(* IEC 61131-3 sources: ml2plc/benchmarks/st (part 7) *)

    weights_7 : ARRAY[0..191] OF REAL := [0.688684464, -0.251728266, -0.865464985, -0.106039852, -0.342710823, 0.691397548, 0.545316637, 0.451106936, -0.972581029, 1.01049495, -0.46521771, -0.194902733, 0.047600802, 0.219640687, -0.898541093, -1.06958103, 0.576955795, 0.662654877, -0.551774442, -0.393089443, 1.25733566, -0.102036051, -0.33817184, 0.573561192, 1.02358389, 0.0429671332, -0.451354206, 1.01461709, -0.512437761, -0.405483395, -0.904772937, 0.0525284261, 0.531825364, 1.37226915, -0.355399728, -0.68238759, 0.599305511, 0.39647612, -1.08820724, 1.2778101, -0.0734612197, -0.358505845, 0.813616991, 0.21143426, -0.601562083, -0.720784783, 0.119864009, 0.748160541, -0.00713000586, 0.244366869, -0.894774139, -0.781875014, -0.0933139026, 0.823451638, -1.0571214, 0.397565454, 0.221330047, 0.794143915, 0.0579137206, -0.834286153, -1.02714491, 0.4435018, 0.325868577, 0.0499007814, 0.244628534, -0.956271648, -0.811831295, 0.113917887, 0.623460889, -0.901144326, 0.656858027, 0.285817534, 0.424304128, -0.158880517, -1.02905571, 1.03020906, -0.499804497, -0.475916564, -0.337449938, -0.158021986, 1.40593672, 0.95926398, -0.595809937, -0.287213802, -0.47090137, -0.392327726, 1.09143257, -0.364193618, -0.291908026, 1.43915653, -1.03929389, 0.432665855, 0.234065458, 1.08598685, -0.368728101, -0.609597504, -0.233271882, -0.42965731, 0.926180065, 0.188584849, 0.223465264, -1.11406386, -0.50280422, -0.178945631, 1.10107863, -1.26540232, 0.234013259, 0.419472396, -0.618463218, -0.307608634, 1.32427752, 0.952789187, -0.563809812, -0.25738892, -1.16513908, 0.324054241, 0.353279918, -0.750201344, 0.0481031314, 0.692657232, 0.545174181, 0.144862831, -1.10333705, 0.573349059, 0.272133052, -1.33604789, -0.165077209, -0.424486279, 0.880616426, 0.664759457, 0.357302666, -1.25569296, -0.0329220407, 0.482446015, -0.317285031, 1.13552487, -0.381064355, -0.586573541, -0.733967721, 0.152410552, 0.860239148, 0.990790427, -0.491253883, -0.512532234, 1.046013, -0.51024735, -0.624616563, 0.882700682, -0.114194848, -0.756001472, 0.88511467, -0.404787958, -0.668740392, -0.692761958, -0.321748972, 1.15619385, -0.657764494, -0.166892812, 1.11973906, -1.07256877, 0.377563357, 0.286821365, 0.385569185, 0.258302331, -1.33617496, 1.14878833, -0.584546626, -0.583055913, -1.05693662, 0.504781961, 0.443913162, -0.114870973, -0.384501725, 0.897702992, 1.03910887, -0.165579304, -0.616232336, 0.463422328, 0.441405088, -0.974973619, 0.627231061, 0.212427795, -0.956863701, -0.648825645, -0.309565783, 1.04708552, 1.24038255, -0.20401369, -0.22858876, -0.200083375, -0.332850873, 0.897526622];
    bias_7 : ARRAY[0..2] OF REAL := [-0.0229109377, 0.115018375, -0.164126784];

END_VAR

VAR
    (* Merged variables from all regions *)
    buffer_0 : ARRAY[0..63] OF REAL;
    buffer_1 : ARRAY[0..63] OF REAL;
    h_new_0 : ARRAY[0..63] OF REAL;
    h_new_3 : ARRAY[0..63] OF REAL;
    h_state_0 : ARRAY[0..63] OF REAL;
    h_state_3 : ARRAY[0..63] OF REAL;
    r_gate_0 : ARRAY[0..63] OF REAL;
    r_gate_3 : ARRAY[0..63] OF REAL;
    u_gate_0 : ARRAY[0..63] OF REAL;
    u_gate_3 : ARRAY[0..63] OF REAL;

    (* Temporary computation variables *)
    i : DINT;
    j : DINT;
    t : DINT;
    sum : REAL;
    (* Computation helpers *)
    max_val : REAL;
    exp_val : REAL;
    exp_sum : REAL;
    (* Spatial loop variables *)
    oc : DINT;
    oh : DINT;
    ow : DINT;
    ic : DINT;
    kh : DINT;
    kw : DINT;
    ih : DINT;
    iw : DINT;
    (* Transpose loop variables *)
    t2_d0 : DINT;
    t2_d1 : DINT;
    t2_d2 : DINT;
END_VAR

(* Forward pass execution *)

(* Region: r0 [ACYCLIC] *)
(* Acyclic Region r0 *)
(* Layer 0: GRU (hidden_size=64, input_size=1, seq_len=1) *)
(* Generating output: Y, linear_before_reset=1 *)

(* Initialize states to zero *)
FOR j := 0 TO 63 DO
    h_state_0[j] := 0.0;
END_FOR;

(* Process 1 timesteps *)
FOR t := 0 TO 0 DO

    (* Reset Gate *)
    FOR j := 0 TO 63 DO
        sum := 0.0;
        FOR i := 0 TO 0 DO
            sum := sum + input_data * weights_0_r[j * 1 + i] ;
        END_FOR;
        FOR i := 0 TO 63 DO
            sum := sum + h_state_0[i] * recurrent_0_r[j * 64 + i] ;
        END_FOR;
    sum := sum + bias_0_r[j];
    r_gate_0[j] := 1.0 / (1.0 + EXP(-sum));
    END_FOR;

    (* Update Gate *)
    FOR j := 0 TO 63 DO
        sum := 0.0;
        FOR i := 0 TO 0 DO
            sum := sum + input_data * weights_0_u[j * 1 + i] ;
        END_FOR;
        FOR i := 0 TO 63 DO
            sum := sum + h_state_0[i] * recurrent_0_u[j * 64 + i] ;
        END_FOR;
    sum := sum + bias_0_u[j];
    u_gate_0[j] := 1.0 / (1.0 + EXP(-sum));
    END_FOR;

    (* Candidate (lbr=1): h'_t = tanh(Wx + r_t * (Rh + Rb_h) + Wb_h) *)
    FOR j := 0 TO 63 DO
        sum := 0.0;
        FOR i := 0 TO 0 DO
            sum := sum + input_data * weights_0_h[j * 1 + i] ;
        END_FOR;
        exp_val := 0.0;
        FOR i := 0 TO 63 DO
            exp_val := exp_val + h_state_0[i] * recurrent_0_h[j * 64 + i] ;
        END_FOR;
        sum := sum + r_gate_0[j] * (exp_val + bias_r_0_h[j]);
        sum := sum + bias_w_0_h[j];
    exp_val := EXP(2.0 * sum);
    h_new_0[j] := (exp_val - 1.0) / (exp_val + 1.0);
    END_FOR;

    (* Hidden state: h_t = u_t * h_{t-1} + (1 - u_t) * h'_t *)
    FOR j := 0 TO 63 DO
        h_state_0[j] := u_gate_0[j] * h_state_0[j] + (1.0 - u_gate_0[j]) * h_new_0[j];
    END_FOR;

    (* Y output: Full sequence *)
    FOR j := 0 TO 63 DO
        buffer_0[t * 64 + j] := h_state_0[j];
    END_FOR;
END_FOR;

(* Layer 1: Squeeze *)
FOR i := 0 TO 63 DO
    buffer_1[i] := buffer_0[i];
END_FOR;

(* Layer 2: Transpose perm=(1, 0, 2)  (1, 1, 64) -> (1, 1, 64) *)
FOR t2_d0 := 0 TO 0 DO
    FOR t2_d1 := 0 TO 0 DO
        FOR t2_d2 := 0 TO 63 DO
            buffer_0[t2_d0 * 64 + t2_d1 * 64 + t2_d2] := buffer_1[t2_d1 * 64 + t2_d0 * 64 + t2_d2];
        END_FOR;
    END_FOR;
END_FOR;

(* Layer 3: GRU (hidden_size=64, input_size=64, seq_len=1) *)
(* Generating output: Y, linear_before_reset=1 *)

(* Initialize states to zero *)
FOR j := 0 TO 63 DO
    h_state_3[j] := 0.0;
END_FOR;

(* Process 1 timesteps *)
FOR t := 0 TO 0 DO

    (* Reset Gate *)
    FOR j := 0 TO 63 DO
        sum := 0.0;
        FOR i := 0 TO 63 DO
            sum := sum + buffer_0[t * 64 + i] * weights_3_r[j * 64 + i] ;
        END_FOR;
        FOR i := 0 TO 63 DO
            sum := sum + h_state_3[i] * recurrent_3_r[j * 64 + i] ;
        END_FOR;
    sum := sum + bias_3_r[j];
    r_gate_3[j] := 1.0 / (1.0 + EXP(-sum));
    END_FOR;

    (* Update Gate *)
    FOR j := 0 TO 63 DO
        sum := 0.0;
        FOR i := 0 TO 63 DO
            sum := sum + buffer_0[t * 64 + i] * weights_3_u[j * 64 + i] ;
        END_FOR;
        FOR i := 0 TO 63 DO
            sum := sum + h_state_3[i] * recurrent_3_u[j * 64 + i] ;
        END_FOR;
    sum := sum + bias_3_u[j];
    u_gate_3[j] := 1.0 / (1.0 + EXP(-sum));
    END_FOR;

    (* Candidate (lbr=1): h'_t = tanh(Wx + r_t * (Rh + Rb_h) + Wb_h) *)
    FOR j := 0 TO 63 DO
        sum := 0.0;
        FOR i := 0 TO 63 DO
            sum := sum + buffer_0[t * 64 + i] * weights_3_h[j * 64 + i] ;
        END_FOR;
        exp_val := 0.0;
        FOR i := 0 TO 63 DO
            exp_val := exp_val + h_state_3[i] * recurrent_3_h[j * 64 + i] ;
        END_FOR;
        sum := sum + r_gate_3[j] * (exp_val + bias_r_3_h[j]);
        sum := sum + bias_w_3_h[j];
    exp_val := EXP(2.0 * sum);
    h_new_3[j] := (exp_val - 1.0) / (exp_val + 1.0);
    END_FOR;

    (* Hidden state: h_t = u_t * h_{t-1} + (1 - u_t) * h'_t *)
    FOR j := 0 TO 63 DO
        h_state_3[j] := u_gate_3[j] * h_state_3[j] + (1.0 - u_gate_3[j]) * h_new_3[j];
    END_FOR;

    (* Y output: Full sequence *)
    FOR j := 0 TO 63 DO
        buffer_1[t * 64 + j] := h_state_3[j];
    END_FOR;
END_FOR;

(* Layer 4: Squeeze *)
FOR i := 0 TO 63 DO
    buffer_0[i] := buffer_1[i];
END_FOR;

(* Layer 5: Slice starts=[0] ends=[1] axes=[0] steps=[1] *)
FOR i := 0 TO 63 DO
    buffer_1[i] := buffer_0[i];
END_FOR;

(* Layer 6: Squeeze *)
FOR i := 0 TO 63 DO
    buffer_0[i] := buffer_1[i];
END_FOR;

(* Layer 7: Fused Linear + SOFTMAX *)
FOR j := 0 TO 2 DO
    sum := 0.0;
    FOR i := 0 TO 63 DO
        sum := sum + buffer_0[i] * weights_7[i * 3 + j];
    END_FOR;
output_data[j] := sum + bias_7[j];
END_FOR;

(* Softmax: find max *)
max_val := output_data[0];
FOR i := 1 TO 2 DO
    IF output_data[i] > max_val THEN
        max_val := output_data[i];
    END_IF;
END_FOR;

(* Softmax: compute exponentials and sum *)
exp_sum := 0.0;
FOR i := 0 TO 2 DO
    output_data[i] := EXP(output_data[i] - max_val);
    exp_sum := exp_sum + output_data[i];
END_FOR;

(* Softmax: normalize *)
FOR i := 0 TO 2 DO
    output_data[i] := output_data[i] / exp_sum;
END_FOR;

END_FUNCTION_BLOCK

(* ---- GRU3_straton.st ---- *)
FUNCTION_BLOCK GRU3_FB

    (* Model Inputs/Outputs *)
VAR_INPUT
    input_data : REAL;
END_VAR

VAR_OUTPUT
    output_data : ARRAY[0..2] OF REAL;
END_VAR

VAR
    CONSTANT weights_0_u : ARRAY[0..63] OF REAL := [-0.439286172, -0.480953246, -0.870120704, -0.69075644, -0.657077134, -0.589701712, -0.481989682, 0.11155279, -0.595970333, -0.522424638, 0.066479668, -0.477147967, -0.548775792, -0.440251201, -0.581660211, -0.851885259, -0.447049588, -0.158783153, -0.671791077, -0.790636778, -0.670549393, -0.228230864, -0.573410928, -0.463102937, 0.294410557, -0.154226393, -0.428246915, -0.419357181, -0.580893517, -0.450942427, -0.434489578, -0.354421765, -0.500179946, -0.272357315, -0.211979702, -0.347913235, -0.509638548, -0.571337163, -0.666850746, -0.102425002, -0.464207053, -0.692536592, -0.576414764, -0.25179112, -0.587422669, 0.197722241, -0.440594107, -0.0186067764, -0.233214989, -0.485925347, -0.624329388, -0.464201093, -0.771930814, -0.648595512, -0.712386131, -0.865132749, 0.0861109644, -0.699016631, -0.64285028, -0.76548481, -0.601012945, -0.522387683, -0.408631802, -0.428571761];
    CONSTANT recurrent_0_u : ARRAY[0..4095] OF REAL := [-0.0650523901, -0.129474998, 0.0260338224, 0.0695474148, -0.0666072816, 0.0774139315, -0.0643586814, 0.0473090038, 0.0519357473, 0.0531803295, 0.0508824363, 0.156312734, 0.0510548055, -0.0783398449, 0.0161208138, -0.0254090969, -0.0333776586, 0.0407715552, 0.0384992361, -0.00284529058, 0.0996260718, -0.0809974, -0.0287103504, 0.0288348049, 0.121645145, 0.129295856, -0.121905953, -0.0567066036, -0.0332944021, 0.10126324, -0.0619100034, -0.0120835379, -0.0321507938, 0.152141571, 0.0557904243, 0.0295200478, 0.0753500834, 0.0523380376, -0.045079913, 0.0743025169, 0.03919724, -0.0464075021, 0.0460194834, 0.0400504917, -0.0186564252, -0.0811230615, 0.0205100551, -0.0494997241, -0.0123350881, -0.0521072671, 0.0318819955, 0.0125074722, 0.086325638, -0.14838697, 0.0729614198, -0.123611242, 0.0608778223, 0.136695266, -0.0275732893, 0.103986211, 0.0964937732, 0.0746636614, 0.0518375002, 0.0131850429, 0.0481536575, 0.080832839, 0.00456657633, -0.0930995643, -0.0926894546, -0.104142435, -0.0113655347, 0.0689256042, 0.0391013213, -0.145912498, 0.0662881434, -0.125198483, -0.0359372757, 0.0683884099, 0.0814840198, -0.0467883013, -0.0385110751, 0.0412478335, -0.026082132, 0.00598589424, -0.0733542442, -0.0616489351, 0.0599563681, 0.0975151584, -0.102699503, 0.0168768093, 0.0567795113, -0.109472096, 0.0479807556, -0.0641779676, 0.0252187103, 0.0170151237, 0.052396398, -0.00687042344, -0.0297337286, 0.052699931, 0.0299865901, 0.0428941771, 0.143816575, 0.0724755228, 0.0308377538, 0.0377355814, 0.073744677, 0.100715749, 0.0200833306, 0.00330035621, 0.0808146596, 0.0683915466, 0.00292335614, -0.0387148745, -0.0278775394, 0.0165898427, -0.0266524255, -0.0119600557, 0.0607938841, -0.171499431, 0.00670967251, -0.0278419442, -0.0198536664, -0.0489947647, -0.0504177436, -0.0603820346, -0.0319245569, 0.0403733216, -0.0657449737, -0.0835127532, 0.074783206, -0.0822283328, 0.0527420714, 0.025356207, 0.00193200377, 0.0403062142, 0.011863322, 0.0911065713, -0.0981498286, 0.0448010042, 0.00674223201, 0.0832657516, 0.0133088445, -0.0096457703, -0.126930133, 0.0133038349, -0.0605163276, 0.0315002874, 0.163095102, 0.0627945811, -0.0319333449, -0.0184467398, -0.0260825343, 0.1507947, 0.0180257969, -0.113473095, -0.00113128126, 0.034390863, 0.158128366, 0.0736147836, 0.00302845053, -0.0366435051, 0.0202366989, -0.0454519801, 0.027544789, 0.00827108417, -0.116445266, 0.136078835, -0.0322153643, 0.0859275237, -0.0495595485, -0.0305913445, -0.0528560281, -0.0197725855, 0.0479791425, -0.0321966782, -0.0912050977, 0.08009094, -0.131073937, -0.073050648, 0.0158983283, -0.0129424734, 0.0236992333, -0.0654924586, 0.00780409761, 0.0303560495, 0.0224402416, 0.195856482, 0.104409501, 0.00386209786, 0.0270838067, -0.0308708213, 0.0765376315, -0.144475698, -0.00663482724, -0.0773844719, -0.0756781921, 0.0114769517, 0.07947056, 0.0525699407, -0.0490815043, -0.0797774196, -0.0738181025, 0.00899818353, 0.00655652676, -0.0247584134, -0.142790094, -0.0536906458, 0.0891067088, 0.0319167599, 0.0273121186, -0.0111009832, 0.0738681182, -0.0465159416, 0.10495235, 0.0167910457, 0.0170945786, -0.0259337351, -0.0238404684, 0.105175085, 0.0262874551, -0.0252160784, 0.0407399312, 0.0396488942, -0.000441844575, 0.0779087767, -0.101633228, 0.00611562654, -0.138864547, 0.0793924779, 0.0318161361, 0.00487799011, -0.0742631257, 0.0282261875, -0.0452414677, 0.103862561, -0.233050048, 0.0166822113, -0.0502803773, -0.105138443, 0.00815397315, 0.075144209, -0.000656956807, 0.00553116389, -0.0327767022, 0.0563323051, 0.00168130081, -0.0347454548, 0.0447669849, 0.0809304044, 0.0181033891, 0.0829547346, 0.0445744358, 0.0685421899, -0.0522269495, 0.10767854, 0.0401147828, -0.0274171568, -0.0556086302, -0.0181052946, 0.0614649057, 0.15146631, -0.107644446, -0.0519810207, -0.0192557313, -0.050705526, -0.00130558573, -0.00449152011, 0.0586461015, -0.00949175656, -0.161170155, 0.0415757112, 0.0234208908, 0.0994374529, -0.107094176, 0.0798551813, 0.00859866291, 0.00905988738, 0.17884995, -0.052185487, -0.00788529217, -0.0128635718, 0.0425841771, -0.0781655982, 0.0738354772, -0.0700388551, -0.0454497337, -0.0581207834, 0.0587512478, -0.129331231, 0.089504689, 0.0157049354, 0.0867228657, 0.0273658019, -0.0242159963, -0.0269595832, -0.0785825849, -0.0127460342, 0.0726092383, -0.0813473612, 0.0418060534, -0.098036088, -0.0871397629, 0.12796244, 0.115513436, -0.0840419456, -0.0282502882, 0.0339900963, -0.0615085512, -0.0237938426, 0.14066948, 0.0103495289, 0.0563306212, 0.0128910914, 0.0566199236, -0.0431611128, 0.0414758436, -0.0598706417, -0.00455367938, 0.010008106, 0.0502123758, -0.0128066251, 0.119871259, 0.169338882, 0.0573619083, -0.00254678726, 0.0632556081, 0.0658841059, -0.0489678681, -0.0136197284, 0.0332296528, 0.0304199178, -0.0101228859, 0.0340865031, -0.1463456, -0.0561735369, -0.078145586, -0.105770409, 0.021583017, 0.0442470424, -0.0132950321, 0.0343763754, -0.131868333, -0.0834302157, 0.0234229043, 0.0955413878, -0.00966519676, 0.133738831, 0.0799299628, -0.0209413245, -0.0201649163, -0.078094773, 0.00760632753, 0.10674265, -0.0504244342, 0.130076349, -0.0765756071, 0.0406672917, -0.0677179396, 0.0489641167, 0.0178483911, 0.0639283434, -0.0072317142, 0.0689901859, 0.0284034405, 0.0447224788, 0.080589503, -0.0753613785, -0.0883018747, -0.209824249, -0.025372155, -0.0194213465, -0.121756315, -0.0405391641, 0.0252318978, -0.113081403, 0.00984102953, -0.0379814059, -0.0696330816, -0.0607138053, 0.00136227917, -0.0684736297, 0.084016636, 0.0580409989, 0.0783514529, 0.038732525, -0.110764012, -0.184509531, -0.0218135417, 0.0410628468, 0.0143347979, 0.0210808329, 0.0938048959, 0.0952843726, 0.0369632132, -0.036689274, 0.0596370548, -0.101092562, 0.021979671, -0.00666903984, -0.0002728533, -0.102687143, 0.101846725, -0.0270557068, -0.0740891248, 0.0451480709, 0.0244468898, 0.0135530774, -0.0656716228, 0.126964301, 0.046734333, -0.0135823097, 0.104897536, 0.0116401128, -0.0351510793, -0.0270920806, -0.0317737125, -0.0427896604, 0.0606436953, -0.055717431, 0.0877809376, 0.0525183901, 0.0816646814, -0.123816505, 0.0268022101, 0.0949827731, 0.0286988262, -1.17924064e-05, -0.107156947, -0.0325826406, -0.176235095, 0.0207939055, 0.140304744, 0.0597819574, -0.0181577466, 0.117161281, 0.0191873126, 0.0420570076, 0.0174266361, 0.0642305687, -0.0820301622, 0.0203213636, -0.0772711709, 0.0149432123, 0.078445442, -0.031391941, 0.0178297423, 0.0258787423, 0.105060086, -0.185030684, -0.0465904325, 0.033022128, -0.0522077605, 0.18817015, 0.17154251, 0.0908443928, -0.114609689, -0.0463253893, 0.179783046, -0.0138813183, -0.0250236578, -0.0397495851, -0.0401404127, 0.0414455384, 0.00421553105, 0.00501056761, -0.0355476104, -0.0948569328, -0.0180768073, -0.0929266214, -6.38996717e-05, 0.0402616151, -0.04017644, 0.0292976033, 0.122893214, -0.0101269074, 0.0949848741, 0.0924490988, -0.0142561533, 0.034249723, -0.0345417485, -0.0720876306, -0.116285995, 0.0757803917, 0.0925265029, 0.0501283891, 0.0556523763, -0.0871114284, 0.063929759, 0.111392535, -0.0113485595, -0.0560661219, 0.0588565171, 0.0202990752, 0.0169391409, 0.0079346532, -0.0346361771, -0.0971538872, -0.107799433, -0.0225640163, -0.104902133, 0.0540932752, -0.0481065586, 0.0236067846, -0.135952473, 0.105642021, 0.0632608011, -0.0237644296, 0.0115678804, 0.0341430977, 0.00839798432, 0.00526432134, 0.00430205092, 0.063617371, -0.0232296586, -0.0100963581, 0.0232974347, -0.00805089623, -0.0783473253, 0.0837393031, 0.0119392872, -0.171118468, 0.0533629246, 0.0270157438, -0.0287604984, -0.024254458, -0.0379126333, 0.0377461091, -0.129247546, -0.0196368489, 0.121421359, 0.141241029, -0.0185492001, -0.0607114322, -0.118905656, 0.0243493672, 0.00225942954, -0.02267823, -0.114327833, -0.00651719887, 0.0233639106, -0.0216970742, 0.181706235, 0.0208011288, 0.019147085, -0.046965789, -0.0224242695, 0.170098603, -0.0381373689, -0.0911064297, 0.0361324437, 0.0604973882, 0.0523151048, 0.00412818976, 0.0810551196, -0.0951434225, 0.0870590508, -0.0168896336, -0.128554851, -0.0098116193, -0.0513504371, 0.0390418544, -0.0403953195, -0.101676092, 0.0051176697, -0.00728737004, 0.0545737594, 0.0803038031, -0.106364466, 0.0805499181, -0.0291947313, -0.0313916355, 0.00281906407, -0.00804035645, 0.0905895531, 0.138566479, -0.0726417452, -0.0388255194, 0.0526182652, 0.0332292169, -0.0458627641, 0.0337294526, 0.00538110361, 0.140382588, 0.0673478395, -0.0970090628, -0.0075024087, -0.0495187268, -0.0802161619, 0.123421639, -0.0669697523, 0.0695282966, 0.0278533436, 0.0633659065, 0.00612806296, -0.0442293584, -0.0825438574, 0.102498822, -0.0788070858, -0.00543309376, 0.00251733419, -0.112787522, 0.0541282296, -0.167338938, 0.0514628179, -0.0181294475, 0.00405258778, -0.144672319, 0.0080318721, -0.0168379508, 0.0630492195, -0.0291489959, 0.0451016501, -0.0668138266, 0.0430565365, 0.0430122651, -0.0329513662, 0.000115959905, -0.155294836, 0.0717644468, -0.0975336134, 0.0627146736, 0.0671754926, -0.0245223772, -0.0847209394, 0.103243671, -0.0160844456, -0.0769205019, 0.0603941306, -0.0861880928, -0.124118626, -0.0407451317, -0.0479636192, 0.0243864693, 0.0225671809, 0.0300183278, 0.0491476469, 0.0137792621, -0.101849571, 0.0899749994, -0.147746086, 0.00454038568, 0.0589881316, -0.0145919751, 0.135418221, -0.0641773641, 0.00270533562, -0.0761346892, -0.0119857313, -0.0468325913, -0.0362873077, -0.131199926, 0.0103873778, 0.119403817, 0.0133330058, 0.0119966101, 0.0999416485, -0.0672517344, -0.0058638826, -0.00583216175, 0.0140269175, -0.068311438, 0.03253185, 0.103045583, -0.0298009366, -0.0424585715, 0.049341809, 0.0334219672, 0.0674507618, -0.0598343313, -0.0709823295, -0.00613911822, -0.0969725773, -0.114717588, 0.0991245732, 0.0570561923, -0.019426886, 0.052425161, -0.0514192283, 0.0795131326, -0.0747317523, -0.0695499405, 0.0674568191, 0.0873003826, 0.183561474, 0.0483771265, 0.00801333692, -0.0329486541, 0.118730754, -0.024188403, -0.00475108158, -0.102296896, 0.0118699996, -0.0566260032, -0.00249518454, 0.0371045657, -0.0271308124, 0.0527189821, 0.0894352719, 0.186274648, 0.0990155637, -0.0390276238, -0.102149099, 0.0725147501, 0.0395716839, -0.0627084598, 0.0174233504, -0.118221872, 0.057125818, 0.00148172863, -0.0975891799, 0.0914200917, -0.0564012453, -0.00408087857, -0.115551151, 0.0542268753, 0.019407969, -0.04010031, -0.0751183033, 0.0519157983, 0.0462308973, -0.00663706008, -0.0179555975, 0.128559679, -0.0160329398, -0.0250887014, 0.0124615263, -0.0278950725, 0.0723621994, -0.0639792681, 0.0245549679, -0.0128075834, 0.0482278317, -0.00473110611, -0.0172997359, 0.0275737233, 0.0381074212, -0.0479229614, 0.15075548, 0.236614883, -0.12308903, 0.0457972996, -0.0270488337, -0.0401842594, 0.0367866941, -0.0665339977, -0.124880955, 0.0096321106, -0.0183932558, -0.0149384877, -0.0207794402, -0.0273507237, 0.0092713302, -0.137307942, 0.124376148, -0.000531716272, -0.0697186887, 0.0233710855, -0.0879249945, -0.0595673844, -0.0753096193, -0.10940744, -0.0863983482, 0.0678732842, -0.0699944496, -0.0533968322, -0.0598150305, -0.109890275, -0.0255937222, 0.0414171703, -0.028406553, 0.0625951141, 0.0562955327, -0.040136572, 0.102456421, -0.094027251, 0.0563254878, 0.0507630631, -0.100891739, 0.0114759067, -0.0276399851, -0.0600263849, -0.0218528342, 0.0106363287, 0.0762119591, 0.0472210646, 0.0182249043, 0.0761318132, -0.0902465209, -0.0155644314, 0.0497058667, 0.00891689677, -0.0575596653, -0.063269861, -0.0369747803, -0.0418471023, -0.0446194261, 0.0618177094, 0.163427904, 0.0439322591, 0.0151975229, -0.139614716, 0.0382574834, 0.0647403747, 0.0044741584, 0.0366933271, -0.0847294405, -0.098235622, -0.102225974, 0.0730303079, 0.0709254742, 0.114724368, -0.058182843, -0.0275532752, 0.0699310824, 0.073567912, -0.118505709, -0.0922444239, 0.0654501319, -0.0442147106, -0.0973261297, 0.0649150908, 0.0473677218, -0.0438311286, -0.0123466263, -0.0506518409, -0.00112013146, 0.0114555079, -0.225004256, 0.0179542284, 0.00154356682, 0.0197916869, -0.0964033976, -0.0149603887, -0.0931083262, -0.0858175233, -0.0240392219, -0.0473877937, 0.0356729813, 0.0953858122, 0.0516837016, 0.000944763422, 0.000391166657, -0.0161546711, 0.0617823638, 0.0323178768, 0.0746243447, -0.0289416965, -0.132081941, 0.0347845852, -0.00957541913, -0.146093175, 0.00121896248, -0.088182658, -0.0529079251, 0.00144353509, -0.10963767, 0.0711052567, -0.130099729, -0.127687454, -0.0238898639, 0.0237303749, -0.0463271476, -0.0377245843, 0.146435305, 0.0406003967, -0.00347847119, 0.0402232558, 0.0606766082, -0.0170659591, 0.00456166919, -0.0581656583, -0.0257244669, -0.114303187, -0.109322034, -0.000124797225, 0.0906794146, 0.0998297706, -0.0660899505, -0.0273227766, 0.00623180624, -0.0511037856, 0.0518054552, -0.130383685, -0.104795009, 0.00977518409, 0.0961738452, 0.0406313278, 0.0335147977, -0.0768964514, -0.021825349, 0.114472322, -0.0201997422, -0.0598041527, -0.0629845262, 0.105795145, -0.0276378486, -0.0260668173, -0.0237419959, -0.0401881412, 0.0480453372, 0.0071930117, 0.00337004848, 0.0128219994, 0.067926839, 0.102826566, -0.0290449653, 0.123585209, 0.0586936176, -0.129759327, -0.0223709345, -0.116297573, -0.0687413886, 0.109364361, -0.016150102, 0.0699984133, 0.0204590037, -0.0488001369, -0.0933896229, 0.11484497, 0.146208376, -0.0152992923, 0.0223931447, 0.0693335161, -0.126214027, -0.0157451089, 0.020451, -0.0159052685, 0.0770635083, -0.165799066, -0.0527213998, -0.080435276, -0.0827942193, 0.0621753186, 0.00343356607, -0.0961636975, 0.0286911149, 0.0452868044, -0.0499980301, -0.0868136883, 0.050965365, -0.0764427632, -0.0663457513, 0.0639655739, -0.121900126, -0.0106822588, 0.0629351214, -0.0268343873, -0.0563602373, 0.0208010022, -0.0950316712, 0.0376925468, 0.0941148102, 0.0284186527, 0.0386470295, -0.0649496838, 0.00324150547, -0.0536398701, 0.0218845457, 0.101267442, 0.00504809991, -0.0866092741, 0.0529379621, 0.0938520655, 0.0396423154, 0.127945945, 0.11368385, -0.0549047142, 0.114498168, -0.0241714753, 0.0520189852, -0.0362896509, 0.0509226546, -0.165635839, 0.0881007984, 0.0160411, 0.024631137, 0.0659909099, -0.0762100443, 0.0427479185, -0.00694125425, 0.143184051, -0.149732918, 0.0110863149, -0.0155461309, -0.13748844, -0.0504982434, 0.025665462, -0.0429363698, -0.0277443547, -0.0475423895, 0.0285833944, -0.0735700205, -0.144904912, -0.0755529851, -0.0403888598, -0.0527475253, -0.000688489527, 0.101409346, 0.0988431573, -0.0909979939, 0.0660976842, 0.063818492, -0.00707271695, -0.00301229395, -0.0202014614, 0.0212209262, -0.0612271912, 0.142480314, -0.102822497, 0.121017784, -0.0435582623, 0.100066409, -0.0312062576, -0.0822519436, 0.057339862, 0.0568015501, 0.0269984789, -0.0163367614, -0.0477057099, -0.101986229, -0.00421534479, -0.179487348, -0.0764475316, -0.0430073664, -0.0425812863, 0.0527436584, -0.13650541, -0.00514466688, 0.00624288665, -0.0491546728, -0.0670409873, 0.0240444243, 0.035694059, -0.0549894422, -0.0163852815, -0.0803953186, -0.0258201156, -0.0284036025, 0.0236114748, -0.0177096128, 0.0899664611, -0.136392832, -0.0611273237, 0.0208600666, 0.0675291047, -0.033409629, 0.183402792, -0.0179462973, 0.0402268246, 0.0538903326, 0.0605378859, -0.00444559008, 0.00593124051, 0.0584437177, -0.0465901792, 0.0367346182, -0.00531690102, -0.0891991258, 0.108523466, -0.000754443929, 0.0853905827, 0.0139564294, -0.0571048073, -0.0341003574, 0.0744261444, -0.0160620511, 0.0420818552, -0.072983481, 0.105422221, 0.0132888965, -0.156731457, 0.0509976372, -0.00400068983, -0.0257125702, -0.010336509, -0.0466502346, -0.0191403441, -0.0370061398, -0.0619829483, 0.0589080006, 0.085831672, -0.0815126747, -0.148456261, 0.035992898, 0.00954711344, -0.0224743038, 0.0770518929, -0.0347290412, 0.0506613515, -0.0776980445, 0.0472105034, 0.206908733, 0.0290955547, -0.113211304, 0.146189138, 0.0581367761, -0.0555344708, 0.0266725048, 0.0476324111, -0.0754805133, 0.0204973966, 0.0354307257, -0.0414481908, 0.0941888317, -0.142457843, 0.01902714, 0.00608063489, -0.142902017, -0.00904501975, -0.0471438207, 0.0187765174, 0.0261135101, -0.0300621614, 0.0145887854, -0.0236850809, 0.0117516052, -0.0394856744, 0.0042070318, -0.094953917, -0.107410148, -0.0374321714, -0.0109713413, -0.0557455085, -0.0535232276, 0.0823234618, -0.0228107423, -0.145991802, -0.142637998, -0.0141612738, 0.0681499764, -0.0601133108, -0.048684977, 0.028852893, -0.0919774398, 0.0113884229, 0.0250541884, 0.108147934, 0.125753194, 0.040229924, -0.0862782151, 0.0393346809, -0.0627611578, -0.0139939766, -0.0519772731, 0.0389488079, -0.0385627151, -0.0904045478, -0.0797261447, -0.0159214437, -0.00528162252, 0.00593003258, -0.0402139761, -0.100702733, 0.0729726627, -0.0694422498, -0.101501249, 0.026667282, -0.0488509983, -0.0981456414, 0.0895740688, -0.0577398948, -0.0186711848, -0.00111833401, 0.000157465227, 0.070121713, 0.110388353, -0.0305795819, 0.00751299458, -0.159779117, -0.0279579163, 0.0977309942, -0.00896156579, 0.0305966716, 0.0786327869, 0.0876243636, -0.0386611111, -0.0101302303, -0.160905316, 0.105016418, -0.0753878355, -0.0497038662, -0.0164555032, -0.0430143699, -0.045727957, -0.0521295182, -0.00294361566, 0.0361426473, 0.00889566541, -0.0249266233, 0.0799256191, -0.0287304316, -0.0792678446, -0.0854634121, -0.050208319, 0.0208053384, -0.0348147191, -0.114404887, 0.0125034805, -0.0298862718, -0.0686926022, 0.0476176292, -0.0698538199, -0.0111048371, 0.0644094273, 0.0129547417, -0.0727717876, -0.0681286678, 0.13020657, -0.027219126, 0.0698305443, 0.0116916075, 0.14363949, -0.113594539, -0.000844738446, 0.0082028266, 0.0454428382, -0.00381363602, 0.0126697449, -0.187009782, -0.0268669054, -0.128417894, 0.0594988614, 0.0632686764, -0.138941869, 0.107257128, 0.112114236, 0.0334792137, -0.0564817488, 0.000689910725, 0.110511348, -0.116754688, 0.00211306289, 0.0736983195, -0.00167888403, -0.0343024731, 0.0968845412, 0.0107437428, -0.0036681965, -0.0132405106, 0.0795757398, -0.0983074009, -0.17490913, -0.0407146737, 0.129254073, -0.00595551729, -0.0102427769, -0.0578140169, -0.00301308557, -0.0852808505, -0.00178171322, -0.0460724831, 0.0447371192, -0.0961295962, 0.028552942, -0.0433705673, -0.0627188534, 0.0271210223, -0.0610382147, 0.0640244409, -0.00287532061, -0.0704336017, -0.145652339, -0.163796186, -0.157491252, 0.0173620582, 0.234602943, 0.0841561556, -0.00848647393, 0.0434717573, 0.148942828, 0.0672514886, 0.0184065942, 0.0249046497, 0.0132941119, -0.065047577, 0.0867860764, -0.0353404805, -0.0038694879, -0.00896554533, -0.030097058, -0.0858454853, 0.0279321168, -0.0583353005, -0.114406154, 0.0291701369, -0.103932366, 0.10427992, -0.0508416221, 0.0617097132, 0.0285572838, 0.035257943, 0.0155800534, -0.174241856, -0.0110836942, 0.0528832301, 0.170236602, -0.0480959341, 0.0568181984, 0.0429964401, -0.0398594141, 0.142875105, 0.0198408999, -0.0234815422, 0.0413020328, 0.0316126868, -0.0242498852, -0.085475266, 0.064656049, -0.091913268, 0.00903178845, 0.0966716036, 0.0519700944, 0.050653033, -0.171772823, -0.0414884649, 0.0218126774, 0.0484813899, -0.0342098139, 0.0431513302, -0.0775837302, -0.0194175802, 0.0608915053, -0.0958085358, -0.0525278524, 0.172223568, 0.0520742238, 0.0220057666, 0.108987883, 0.130237713, -0.107932687, 0.0317093804, -0.0324443653, 0.0835223198, 0.199562863, 0.148373321, 0.112411663, -0.0236171074, -0.0052724164, -0.0620609745, 0.0111017656, -0.0111301467, 0.0467493832, -0.0206472725, 0.00297360634, -0.0119733168, -0.0970944092, -0.0316341296, -0.0132295629, -0.0338335037, 0.0520780794, 0.12766394, 0.068843931, 0.195665359, 0.0558646694, -0.0955600888, -0.077448085, -0.0211934205, -0.0296740029, 0.00166139007, 0.0591102466, 0.0120509472, 0.0354253165, 0.157639459, 0.0244942661, -0.189979553, 0.0354224183, -0.0612734891, 0.0376649685, 0.205627829, 0.00432812702, -0.02739764, -0.0818298906, -0.120526254, 0.0180814825, -0.000375784934, -0.00592299784, 0.106825203, 0.0165459365, -0.0205880832, 0.111172318, 0.0138723217, 0.0164856389, 0.0165480785, 0.062894091, -0.0380115025, 0.0288346447, 0.0361645594, 0.0495932661, -0.0227110572, 0.075070098, -0.0742200911, 0.0544882938, -0.100449175, 0.0435093604, -0.0736430958, -0.037141487, 0.0257380009, -0.0985285342, -0.0582001545, 0.0263903867, -0.133239761, 0.105293542, 0.0509466119, 0.0149480924, 0.00264212303, -0.0803615153, 0.016234152, 0.059326943, 0.0166629646, 0.129690155, 0.00954441354, -0.089779377, 0.00573088974, -0.00493869651, 0.0591944307, 0.104186028, -0.0218419582, -0.00641731732, -0.0487543717, 0.0456377119, 0.0427142642, -0.0505627245, -0.0945144147, 0.0202183761, -0.0657929033, 0.0831303746, 0.0750920549, -0.0910624713, -0.0225744545, -0.124150276, -0.152486816, -0.0330677181, 0.0442869589, -0.0471795797, -0.134105518, -0.0558637902, 0.0834738016, 0.0108987726, 0.0160592347, 0.108882993, 0.0598439351, -0.0831453726, 0.0973557979, 0.0623315871, 0.0383794159, -0.00982961245, 0.0576453581, 0.0494841523, 0.0718243048, -0.0572519116, -0.0411631241, 0.0534142479, 0.0589003153, -0.0547911972, 0.0755654052, -0.0815965533, -0.0117946044, 0.103706859, 0.0667564943, 0.0903166533, -0.038736023, 0.018129129, 0.060453929, -0.0346493199, -0.0850336775, -0.00476394966, -0.046710752, 0.0143833831, -0.015953254, 0.0134185404, -0.0532437861, 0.017363999, -3.44109721e-05, -0.149937063, -0.0611102469, -0.0427428, -0.00926883332, 0.0374133512, -0.0711838678, 0.0258399993, -0.00872873422, 0.0366705805, -0.0147527959, 0.057190951, -0.0818497464, -0.0571168959, -0.0519183539, -0.0537600778, 0.0200558268, -0.0356059968, -0.0514560342, -0.115551762, 0.0614381582, 0.0904121846, 0.0550923347, 0.09433157, -0.0337151326, 0.0622163899, 0.0612645894, 0.0891919881, -0.0207224004, -0.0534750856, -0.0296462215, -0.0158423334, 0.0887120888, -0.0703074336, 0.00989756919, 0.130590975, 0.0778346881, 0.00399551541, 0.108989477, -0.00454995502, 0.0528934747, 0.121316366, 0.0511680767, 0.0755439252, -0.0733139291, 0.0752391368, 0.0770118833, -0.000957053155, 0.0114189107, 0.0590100586, 0.00575780775, -0.0877712369, -0.0187948812, -0.0657808185, 0.0406781025, 0.0595240593, 0.00684884563, 0.0149538293, 0.00922561437, 0.114996634, -0.0660880059, 0.00837289169, 0.0117377583, 0.0296314899, 0.0261435769, 0.14703317, -0.0287333839, -0.0299690161, 0.00223761285, -0.0870166644, 0.0896945298, 0.0500493981, 0.0744577274, 0.013104694, 0.0748228654, -0.0941333324, 0.0413618535, 0.0238855034, 0.0836726874, -0.0697423667, -0.121260516, 0.0637812093, 0.0396960527, 0.0819698572, 0.0435053259, 0.0501765572, 0.00983571447, 0.0299814939, -0.0600497648, 0.04743848, 0.0918345079, -0.192011252, 0.185129195, -0.132771015, -0.0218426287, 0.0106724147, 0.0418993495, 0.07511691, -0.0415916629, 0.0514673628, 0.0512605757, -0.101605847, 0.0378510244, 0.167794362, 0.0514133871, 0.0400778428, 0.0447239429, -0.0781334937, 0.0273859277, -0.0525638573, 0.0734867603, -0.0286831781, -0.0886658579, 0.0515142232, -0.117384307, -0.161638945, 0.110049561, 0.0852481127, 0.035481941, 0.0158129036, 0.088354513, -0.00556714088, 0.0537756681, -0.0467627533, -0.00163430907, 0.0605735257, 0.109923393, 0.0235946123, -0.0543056205, -0.0435014889, -0.0780219436, 0.0887052789, 0.0288573951, 0.0956314802, -0.119991414, -0.0950825363, -0.0577025861, -0.00233832374, 0.0321475305, -0.0296782143, -0.13685973, -0.0840527713, -0.115250856, -0.086614266, -0.0719218403, 0.0350063443, 0.0287500955, -0.0230677407, 0.13799727, 0.0648974031, -0.0969269872, 0.0105827358, 0.0187805891, -0.0817399919, 0.134309664, -0.0834898725, 0.0636503398, 0.0892517194, -0.0689574108, -0.0209724437, -0.00819023326, -0.00418700883, -0.0096282959, -0.0291463416, 0.0508619435, -0.0297213681, 0.0173015445, 0.00606717542, 0.0537274331, 0.041289378, 0.00145007065, 0.0465077683, 0.130988643, -0.0168933291, -0.0218317695, 0.0134224519, 0.00168778002, -0.00168193318, -0.0929443315, 0.0933136791, 0.0271413755, 0.0012512356, -0.0429633558, 0.00577729195, 0.0381182507, 0.0506631732, 0.0104230382, -0.0946019739, -0.146492317, -0.0122778527, 0.0851407722, -0.00430129794, 0.0286120772, 0.0544554926, 0.000575783662, 0.0418614075, 0.0509960353, 0.235207349, 0.0231721811, 0.03219245, 0.0219864137, 0.0771256983, -0.0475538969, 0.0167042073, 0.043224901, 0.0525902212, 0.0109413685, 0.0310349781, 0.0262097772, -0.0763660222, 0.0886459798, 0.0879353359, 0.0266202651, -0.012050109, 0.0364502966, 0.110469103, -0.0649368986, 0.137989163, -0.00345457532, -0.00076057855, 0.0495130271, 0.0963264555, 0.0292368587, -0.0136958137, -0.0916326419, -0.09134987, -0.143160895, 0.0552338138, 0.0943126529, -0.0341492742, -0.046550639, 0.0415712446, -0.190018594, -0.0170447789, 0.0271576829, -0.0791434646, -0.0259393826, -0.0358110107, 0.114700861, -0.0451665968, 0.00859330222, -0.0176053625, -0.0665916502, -0.10659565, -0.0103667611, 0.0607822947, -0.0335317552, -0.0578957722, -0.0600993, -0.0143982824, -0.0169818364, 0.0747436732, -0.0824175626, 0.0734613463, 0.0172847919, 0.0679807961, 0.0354374871, 0.0221069511, 0.0698141977, 0.103264622, -0.0643693283, -0.0904196575, 0.0209124722, 0.0533089563, 0.138175309, -0.0808143616, 0.0518090576, -0.04021056, 0.0328150876, 0.0717661381, 0.0629613996, 0.104841411, -0.0416442491, 0.0719090104, 0.059182696, -0.15314886, 0.0215544775, -0.0130644813, 0.114227138, 0.00902843848, -0.0153322266, -0.13713704, -0.0476132631, -0.119293369, -0.0679454356, 0.122949339, 0.0693741217, -0.0994557068, 0.0399324894, -0.0314740613, -0.000461213291, 0.00562566333, 0.140679166, 0.0478050821, 0.108278081, -0.0659516081, -0.00195731036, 0.0559609048, -0.0145426169, -0.0347096696, 0.0258138534, -0.0312658995, -0.0548630729, -0.0697729737, 0.0109880194, -0.0809436738, 0.0592633858, -0.00464516133, -0.107980013, -0.0189933032, 0.0685023963, -0.0257080533, 0.074374266, 0.0587298237, -0.056436114, 0.0454883464, 0.0601172373, -0.0381640494, -0.0409820527, 0.00114455202, 0.0928920731, -0.0341993608, 0.01902242, -0.0319391079, 0.0252930373, -0.0232422352, 0.00733191008, -0.0100106141, -0.056417428, -0.0364283621, -0.0677095577, -0.0730913579, -0.0449670255, -0.112897381, -0.0383246988, 0.0491045266, -0.00531547517, -0.069094345, -0.0260258541, -0.069829613, -0.0624606349, -0.133198172, 0.0081421202, 0.0548977219, -0.0505369082, -0.021252159, -0.0689540803, 0.0545859337, -0.00222222786, 0.0334032364, 0.0678267553, 0.0439778864, -0.0222215448, 0.0925648957, -0.0336760692, 0.0680503026, 0.067150943, 0.169242263, -0.127817169, 0.0840600431, 0.0119890599, 0.0408258699, -0.0424239263, 0.0234956034, -0.0822051615, 0.127012193, -0.018799413, -0.0460282192, 0.00472665858, 0.0129743032, 0.00426072115, 0.0703843161, 0.0145993857, 0.119512692, 0.0195069741, 0.0493210033, 0.0875848681, 0.100930437, -0.0486361198, -0.0475119352, 0.0138504477, 0.208870143, 0.0598653406, -0.120691441, -0.0283632614, 0.0474334285, 0.00298458477, 0.067226842, 0.150975302, -0.0541105792, 0.0256627742, -0.0438354947, -0.0542730018, -0.00181115232, -0.105021812, -0.0556066297, 0.0338146091, -0.0549245104, 0.0143369175, -0.0539371893, 0.0432943441, -0.0535181016, 0.0258672144, -0.0821818784, -0.0270294957, 0.0225534495, -0.0127259865, 0.0120830201, 0.0125242695, -0.0619680323, -0.087769866, -0.011979159, 0.15043509, -0.10600248, 0.0364335105, -0.061168395, 0.0152373658, -0.0460021645, -0.109346926, 0.0364494249, 0.00472447462, 0.102088474, 0.0257884748, 0.0533271991, 0.0729068294, 0.00768535864, 0.112634815, -0.0691387504, -0.0601366162, 0.0453425571, -0.0314094163, 0.0349893384, 0.0256387182, -0.00378753617, 0.0768208951, -0.0505088195, 0.0269892886, -0.00966024026, 0.043255616, 0.00924504176, -0.00864656642, -0.0591106378, 0.0949935094, 0.0487293713, -0.0323852487, 0.0252678767, -0.0076211039, 0.111468486, 0.0816216171, 0.037076585, 0.00846009329, -0.0315636173, 0.0731508285, 0.10651087, -0.034380503, 0.11133229, -0.00250713434, -0.0430554636, 0.165012404, -0.0231795907, 0.0274878461, 0.0483577475, -0.0599443391, 0.0668406785, -0.0761960298, 0.0266923569, 0.00958470255, -0.0702683628, 0.0497920513, 0.0786102861, 0.0636078268, 0.021653505, -0.0515439399, 0.0863124654, 0.0131225679, 0.054686375, -0.0462396704, -0.0317671299, -0.0549215488, 0.0526956804, 0.0599532798, 0.0697892085, -0.0464518778, 0.0786490142, 0.0801427364, 0.135556832, 0.0811728388, 0.0162178427, -0.100880146, -0.0164203923, -0.09579698, 0.00686951773, 0.0556715578, 0.154748037, -0.0384738967, -0.0697567761, -0.0658533126, 0.0563082471, -0.0837014914, -0.120353431, 0.0157528166, 0.11380288, -0.0509812795, -0.184196651, 0.140463933, 0.184002206, -0.0414622352, 0.156096339, -0.0566040725, 0.127726138, -0.135966212, 0.0285594333, -0.0718551874, -0.115175165, -0.0160157103, -0.0541006215, -0.0331212506, 0.0474987626, -0.0206688922, -0.0896792114, 0.0121970847, 0.0920595378, 0.0294709988, 0.00489335647, -0.0136370827, -0.0876406729, 0.0430216789, 0.040562436, 0.0644720495, -0.0303485282, 0.122684225, -0.165262386, 0.0237433817, 0.0427406877, -0.0989692509, 0.109646007, -0.00851122849, -0.00903640781, 0.0406889617, -0.0505370982, 0.0931062922, 0.0305767655, 0.062228322, -0.0525234826, -0.102460198, 0.0645387992, 0.0533145741, -0.206492513, 0.0133064939, 0.0559483878, 0.0906168297, -0.0595491901, -0.0381035544, -0.0209744722, 0.0858725533, -0.0881853476, -0.0829888582, -0.112644993, -0.0684021264, 0.0686395615, 0.0265239459, -0.131407306, 0.0274842456, -0.166530743, -0.0467720069, 0.01258785, -0.0204203501, -0.100700855, -0.110235199, 0.0999744534, -0.067055054, 0.0858595446, 0.0564401224, -0.0734795183, 0.0984800607, 0.000628214737, -0.100944236, 0.050260745, -0.0384647399, -0.117021114, -0.00581525033, -0.118169144, -0.0531625077, -0.110389993, -0.0503460653, 0.048195146, -0.0405612253, -0.0432871655, -0.0308589637, 0.0801219493, 0.022040328, 0.0507384911, 0.0382968932, 0.0698082075, 0.0641338974, 0.00569984969, 0.0396882296, 0.019232735, -0.0757699236, 0.0707999244, 0.0159386508, 0.0308304802, 0.0468344912, 0.0355247855, 0.0718743205, -0.0121067222, -0.0105456598, 0.0769912899, 0.0374626517, 0.0373739302, -0.0699928999, 0.0847563297, -0.0230606366, -0.0388202295, 0.103667095, -0.128558323, -0.046710927, -0.0857155696, -0.0199590083, 0.151113033, 0.121398017, -0.0511609092, 0.0720787272, 0.0295494981, 0.0245097131, 0.0487351418, 0.106066108, 0.0537618995, -0.0159866326, -0.156366274, 0.0242971852, 0.159070209, 0.00524867978, -0.0994271263, 0.0449088961, -0.0211867951, -0.0390554033, 0.077684395, 0.0779460743, 0.0523676053, 0.0588788539, 0.00485968869, -0.0598566197, 0.013074277, -0.0545727536, 0.0519137047, -0.0330678336, 0.0389791094, 0.0678062215, -0.125330731, 0.0168909654, -0.0826457739, 0.0725395679, 0.123465694, -0.0158160534, 0.111778371, 0.0435737222, -0.0315076187, -0.101733088, -0.0460981056, 0.109187216, 0.0352550186, -0.0129180942, 0.171947062, 0.0519051552, 0.0502665862, -0.0938540846, -0.0937337503, 0.0209997464, 0.019742392, -0.0841773972, 0.065202415, -0.0252768025, 0.0767172575, 0.132501423, -0.041324053, 0.013803497, -0.0191468094, -0.0501539335, -0.0029412359, 0.0496336222, -0.0182176437, -0.0242415741, -0.0769018009, -0.0222259574, -0.0599570423, -0.0785850957, 0.0483198538, -0.158214718, -0.102507047, 0.0461308062, -0.0683883056, -0.0411389247, -0.0950894877, 0.100902207, -0.00471645314, 0.00992084574, 0.0858963057, 0.0614297986, 0.117100388, -0.0240918137, 0.0707100406, 0.132806167, -0.116088726, 0.00466614868, 0.0599054582, -0.0183604769, 0.0550542325, 0.0614843927, 0.00322095677, 0.0649169087, -0.0379064046, 0.0497901775, 0.0719092637, -0.154971763, 0.117400832, -0.0427108631, -0.0316413231, 0.0339113027, -0.023429919, 0.0100743826, -0.0608712286, -0.0393153466, -0.0721224099, -0.019769663, 0.0305335447, -0.00641385559, -0.0616339706, 0.0896052122, -0.0450256616, -0.0206921622, 0.0356086567, -0.0749701783, -0.0147821922, 0.0112537732, 0.097909674, 0.0569019616, 0.0509603657, -0.072360158, -0.0678833127, 0.0768040866, -0.110155649, -0.0740643889, -0.094099097, -0.0108416183, 0.060312368, -0.0583655126, -0.104549289, -0.218230203, 0.0970755219, -0.0179643556, 0.100377582, -0.0316814184, 0.0642254949, -0.0426855683, -0.0397533514, -0.0256710351, 0.0136024654, -0.0055637476, -0.200856268, 0.0169277843, 0.078002885, -0.14920415, 0.0111826845, 0.0809670985, -0.052739054, 0.0624899492, 0.0306037925, -0.0699668303, -0.0787069276, 0.0403862, 0.0614282824, -0.00977569167, -0.0857097507, 0.103655919, 0.124205105, 0.0120967291, -0.0551354587, -0.042931851, -0.0854013264, -0.0685761273, 0.0644985661, -0.0383845717, -0.0024125278, -0.063759163, 0.0521320626, 0.124909475, 0.111597076, 0.0148241296, -0.0615106374, 0.0415096581, -0.0933477953, 0.0717638135, 0.0793121159, 0.0742387325, -0.0539873391, 0.00332836807, -0.0300874971, -0.0831861719, -0.0381114557, 0.0751383677, -0.113011718, -0.0112683401, 0.0606956668, -0.172200784, 0.00429096073, 0.0602080822, -0.137329713, -0.090002872, 0.0323414132, -0.0719932467, -0.140211582, -0.0128612556, 0.0361765325, 0.0980945751, -0.010059149, -0.0461915061, -0.0139733413, -0.0086908564, 0.0273868591, 0.0861311108, 0.0443583541, 0.0680558532, -0.0228823051, 0.0917587876, -0.100482099, -0.0359601751, 0.122452661, -0.0542502478, 0.027852837, 0.0694331974, 0.00141336536, -0.109030351, -0.131108165, -0.162553549, 0.0753331035, 0.0134982076, -0.0366807505, -0.0386078581, -0.00658005895, -0.0914643705, -0.0252701417, 0.0801979229, 0.0021053683, 0.0746067539, 0.0221132264, -0.00809657201, 0.12774621, 0.0647266284, 0.0584487692, -0.064717263, -0.0277714748, 0.0883828104, -0.110183463, 0.0370126292, -0.0138474237, 0.0159780867, -0.016058648, -0.0404856317, 0.0766953677, -0.10419903, -0.141589358, 0.144594938, -0.109949932, 0.0647953376, -0.0917214304, -0.0102576986, 0.0803454667, -0.0682678446, -0.0576918498, -0.00570382923, -0.0834980905, -0.00225776061, 0.0470857583, 0.0150479516, 0.042511303, 0.0727005824, -0.128937468, -0.0655451864, -0.0340349115, -0.0954819322, -0.0620098263, -0.172165602, 0.0282320231, -0.0634708181, 0.0287884995, -0.171313956, -0.152317584, -0.0844539329, -0.0112288594, 0.120956585, -0.0573068708, -0.0637781844, -0.0221945029, 0.0527748689, -0.0105367936, 0.0755724683, -0.0467769243, 0.0614911839, -0.135969311, 0.105225481, 0.156952262, 0.0370586067, 0.15616776, -0.0840421766, -0.0951181725, -0.0149632134, 0.0322490297, 0.0670348257, 0.130084842, 0.0266189165, -0.0625972375, 0.00457772799, 0.0979716629, -0.00742265768, 0.118027046, 0.0416464359, 0.0718041658, -0.0798822492, 0.0614944771, -0.091669254, 0.00349572115, 0.0355406329, -0.0315599367, -0.0384840742, 0.0917298421, -0.0112617295, -0.0501065403, 0.0413927324, -0.0128761344, 0.0815452337, -0.0172406044, 0.130260676, -0.0188278407, -0.0011760518, -0.0579140298, 0.0338388719, 0.112019926, 0.0727667958, -0.00672438648, 0.00536828581, -0.0465201363, 0.00503383111, -0.0678088143, 0.0614547953, -0.106527671, 0.108292408, -0.0248407945, -0.0236443058, -0.0199482255, 0.0271114185, -0.0999043509, 0.0715598539, -0.0604586042, 0.0159977283, 0.101002097, 0.0251209512, -0.0435456298, 0.0404220521, 0.0287586413, -0.00336176204, 0.00109383767, 0.188423753, -0.0121071227, 0.0344866551, 0.0340253003, 0.0281979404, -0.020309411, 0.112903818, -0.0353781506, 0.0142767709, -0.0821403638, 0.0994499773, -0.0324760824, 0.108188063, -0.000992564484, 0.0135587398, -0.13331835, 0.0263649207, 0.0262281783, -0.0107785314, 0.0589572713, -0.0244767591, 0.0194578413, 0.0756996647, -0.124957405, 0.0433721058, -0.0131629705, 0.00946621597, -0.0793711543, 0.0270108059, -0.0341884941, -0.0752030089, -0.104312092, 0.0887307227, 0.0835861564, -0.0330076404, 0.162407339, 0.0132059641, 0.0758589134, -0.0445123538, 0.0380469374, -0.000802192837, -0.0470603779, 0.135118589, -0.0318722017, 0.000692218542, -0.0302473344, 0.114358984, 0.00851656124, -0.126637205, 0.0359836593, -0.00687000901, -0.0121891778, 0.0134458765, 0.0366071984, 0.0142765157, 0.0222175159, 0.000126404688, -0.0124760196, -0.0359021425, -0.0431295522, -0.0966509655, -0.0100903204, -0.0353743173, 0.0715210587, -0.081053026, 0.0999638587, -0.019016372, -0.0239935089, 0.00648718514, 0.0153071349, 0.012509536, -0.0589868091, 0.0743578523, 0.0191438161, -0.0187446624, -0.0208187737, 0.00617905706, 0.160369337, -0.025553029, -0.164978892, 0.0432493463, 0.052146554, 0.00317490846, -0.0926495492, 0.0303232074, 0.125212759, -0.0296045784, 0.024818765, -0.0604889244, 0.0330986381, -0.0673882589, 0.0580419749, -0.103213176, 0.0422696471, 0.0958758742, -0.0965849459, -0.00950852036, 0.0918902084, -0.068486914, -0.12186332, 0.0030031316, 0.131197795, 0.00548650976, -0.00403932016, 0.0173820686, -0.0290936418, -0.0979100466, 0.0117043052, -0.118052997, 0.0237339474, 0.0828405619, -0.103721827, -0.0860361904, 0.065347068, -0.0213578418, -0.00391968619, 0.0236401204, 0.0144597851, 0.054736048, 0.0231402628, -0.0840564817, 0.0548789054, 0.130872041, 0.00752765685, 0.0240224563, -0.00454153167, 0.0319019519, 0.063471444, 0.0219805893, -0.0952587053, 0.0340296663, -0.00117000053, 0.0152508952, -0.0606811643, -0.047678858, -0.0131933, 0.0261857826, 0.0161818042, -0.0327050351, -0.000714013353, 0.062065091, -0.00254658936, 0.0433586389, -0.0278949924, -0.0263456665, -0.0698257834, -0.0431765653, -0.0144449733, 0.126253545, 0.0126124537, -0.0509497039, 0.000468326733, -0.00036503002, -0.0447247848, -0.0417972095, -0.0157134756, 0.025018584, 0.0699072331, 0.0882948413, -0.0929879695, 0.00265961373, 0.00323988311, 0.00498005841, 0.00374827161, 0.0459985994, -0.0181076191, 0.0145163927, -0.0408614576, 0.0804381892, 0.0233130399, 0.00467471313, -0.0549203008, -0.0559486635, -0.0105915256, 0.0502482392, 0.0795770064, -0.162366003, 0.000561785651, 0.00131846406, -0.0867253095, -0.0644728467, -0.0526860952, -0.0904279724, 0.0680651143, 0.0549977012, -0.0198836289, 0.0226633139, 0.124892376, -0.0483702384, 0.025002405, -0.00761365099, -0.193545878, 0.116730005, 0.0593729913, -0.0828391612, 0.159838334, 0.0629694685, 0.0573315881, 0.034116488, 0.122743621, 0.00297184102, 0.0652865767, 0.0233377926, 0.0117186205, 0.00482350402, 0.00210875086, -0.133521438, -0.00392506085, 0.0866617113, 0.0794988349, 0.0499842316, 0.123910151, 0.111768797, 0.00231364276, 0.0588010177, 0.0367658734, -0.0292860344, -0.0044385083, 0.0357940495, -0.000611573458, -0.0268944241, 0.0574458987, -0.0747600868, -0.095133923, -0.0577830747, -0.0673853606, -0.0535354726, -0.000596318394, -0.035483066, 0.0208486263, 0.0316488817, -0.195054889, 0.0611732341, -0.0187134333, -0.0486381464, -0.0301590897, 0.0133740138, 0.068864353, -0.140572727, -0.0387248173, -0.0527053252, 0.108385712, -0.0978539661, -0.0396942608, 0.055108171, 0.155904785, 0.128576532, -0.0461218059, -0.00189863332, 0.0483641289, 0.0793901011, 0.0244574696, -0.0248883814, 0.108808123, -0.118639104, 0.0368720591, 0.0476099178, -0.0547937602, -0.126454487, -0.10340786, -0.131127492, -0.0437266976, 0.0529951043, 0.0883525163, 0.0980372503, -0.0825529173, 0.102423966, 0.163403392, 0.0976418331, 0.0313921869, 0.0288433321, -0.0276666954, -0.0106668435, -0.00334626157, -0.0132831838, 0.0184611958, -0.0464694872, 0.0805625767, 0.0173439197, 0.0262606516, 0.126519099, 0.138395324, -0.00254166313, 0.119938344, 0.0573389977, 0.0542154163, 0.0692043006, 0.0597935244, -0.0188125204, 0.049818065, 0.0757564455, -0.0483031236, -0.193337351, -0.00217950717, -0.0817932785, -0.106830128, -0.0650802255, -0.0446323194, 0.0341032632, 0.080365479, -0.0988180935, -0.0450610071, -0.0722491369, 0.0166641083, 0.127055496, -0.103618376, 0.0380277, -0.0759299994, -0.0933069065, 0.0111208772, 0.155003533, -0.0709212944, -0.0932924896, 0.0226059556, 0.0122168204, -0.114529938, -0.103299066, 0.0415850468, 0.00406396575, 0.0625993013, 0.00801790785, 0.0511501096, -0.0501103476, 0.1241448, -0.0662367791, -0.00844532624, 0.177476555, 0.0625147074, -0.0147227608, -0.0120679624, 0.0353377983, -0.046898514, 0.0142605919, 0.056622006, 0.172268614, -0.0329496637, -0.231005609, 0.0563728623, 0.080097951, -0.00894291885, -0.151174337, 0.0251428112, -0.0579357818, -0.0256807655, 0.0514307618, 0.0262518115, 0.0426398553, -0.001229716, -0.0286666676, -0.0170986764, -0.125903815, -0.0690000802, 0.0786091909, 0.0171093177, -0.00777454674, -0.00667924713, -0.0768917128, 0.0167301055, -0.0605392531, -0.00799709186, 0.0590173975, 0.039383892, -0.0531835444, -0.0277832299, 0.0562856458, 0.0160953552, -0.103994332, 0.0460520945, 0.190410435, 0.122205824, 0.0989888832, 0.119691916, 0.142407835, -0.022124365, -0.00849366561, 0.0506508723, 0.0850793868, 0.0271743592, -0.0376036167, 0.0482522696, 0.102856554, -0.0496400036, 0.0277350806, 0.103806086, 0.0148996105, -0.0158420596, -0.0316775106, -0.0387260206, -0.0233267397, 0.0821134523, 0.0401642285, 0.0917946175, 0.0671747178, 0.0684598088, -0.000702465884, -0.0451893173, 0.0517121479, 0.00471234322, 0.0793196112, 0.00699635781, -0.131860629, -0.0368878245, 0.104009926, -0.0268972032, -0.0428332537, 0.113431826, 0.0198208876, -0.0664840862, -0.0546237454, -0.019905258, -0.00254343264, -0.036215134, -0.0554769486, -0.0181054473, 0.140997991, 0.0111484537, 0.0367606059, -0.0674065724, 0.0212049112, -0.0561227873, 0.0290108286, -0.00833883137, 0.00222712872, -0.0847283453, 0.0431756042, -0.109141119, -0.0129319951, 0.0333293751, 0.00531570101, 0.097147122, 0.0388240851, -0.0354440808, -0.0885681733, -0.213006049, 0.0727706179, 0.036135029, 0.102887303, -0.0465593152, 0.0640048981, -0.111603916, 0.094097659, -0.0586705655, -0.075268656, 0.052961275, -0.135893717, -0.0614549555, -0.0569578558, 0.0523011349, 0.0330762491, 0.0435143337, 0.0344756283, 0.0671566129, 0.10543716, 0.0944586769, 0.0153974276, -0.050820291, -0.0458775647, -0.0345414616, 0.0962239429, -0.096707724, -0.0452955365, -0.0182661228, -0.0212264918, 0.069447279, -0.0450920016, 0.100490421, 0.0278961621, 0.0882038102, -0.0678256229, 0.0138143562, -0.0689106062, -0.00360275386, 0.0663605928, -0.0607298799, -0.0621103942, -0.0543092974, 0.0128324572, -0.0431163646, 0.0219562948, 0.00678311661, -0.0441136137, 0.0982432887, -0.0705860108, 0.182194039, -0.108619966, 0.0207179412, -0.122581631, -0.0929343551, 0.0586816929, -0.0232572667, 0.00806567539, 0.0225188695, -0.0365971811, 0.102062739, -0.055163864, 0.0595620796, 0.193907857, -0.0719701275, -0.0325663052, 0.0913035646, -0.0724671558, -0.0490570292, 0.0606238581, -0.00221333839, -0.0208245013, -0.18978031, -0.0184468329, 0.0584079362, 0.0619091392, 0.0283486024, 0.00343166548, -0.0329216793, 0.102478705, 0.0746710822, 0.042023275, -0.00857234187, 0.02867046, -0.037411008, -0.00556871109, -0.0417560525, -0.123214625, -0.00407732744, 0.0280542225, -0.115010217, 0.0420889705, -0.0983415693, 0.033393234, 0.0291160401, 0.0999559239, -0.037810795, 0.0574650541, 0.0249308553, -0.0111770369, 0.0586905405, -0.0181362778, 0.129456714, -0.028140679, -0.0116888974, 0.0460940041, -0.183939517, -0.107369378, 0.0142709417, 0.0799058527, -0.0281989574, 0.00468265638, -0.00359648839, -0.00181956217, -0.00247250684, 0.0800077394, -0.0349083468, -0.0869949088, 0.030391261, 0.0290568061, 0.0480341166, 0.0350300148, -0.218458921, -0.0633597374, -0.00389631395, 0.0858308673, -0.165539861, -0.0115812551, 0.110183015, 0.0742593631, -0.0190524422, -0.0575886704, -0.0105343126, -0.0458830781, -0.0268041249, -0.0500699021, -0.0974797457, 0.142067999, 0.00756507739, -0.0139123565, -0.219773516, -0.192728773, 0.0831120834, 0.0301636811, 0.0989038795, -0.0733708888, -0.00122421142, -0.0823754147, 0.134696111, 0.064505741, 0.099184759, 0.0629062727, 0.215615958, -0.0425261408, -0.0731833428, 0.0291134324, 0.0813642889, 0.0460265577, -0.0210361108, 0.0383235291, -0.090638876, 0.00868848525, 0.0973384976, 0.0863050148, -0.126141474, -0.0671756789, 0.0142485201, -0.00345332734, 0.085107848, -0.0468325168, -0.0311242789, 0.0531625003, 0.0203431584, 0.0540217683, 0.0213960689, -0.0126134809, 0.0620418936, 0.0049791839, 0.094513759, -0.00577996671, 0.142208964, 0.0486403853, 0.00964468438, 0.0353494138, -0.0813095719, -0.0396264419, -0.0299608354, -0.0700816289, -0.0436064377, 0.0170924012, 0.0520251021, -0.0128122233, -0.0186763313, -0.0422864184, 0.0751069486, 0.0735050514, 0.0184059013, -0.14228113, -0.0401629582, -0.0588053875, 0.110950388, 0.113210753, 0.0271767527, -0.0060010571, -0.0826001614, -0.0834111571, 0.017040506, 0.0191633068, 0.0121653015, -0.0290833972, 0.0624605678, -0.0357175432, -0.0785514563, -0.0902193189, -0.0996724367, 0.0230609588, 0.0412896797, 0.0997388065, -0.0565732531, -0.00927331299, 0.138090402, 0.0513459668, 0.142254293, 0.128031746, -0.0142473355, -0.00695161195, -0.0359653533, 0.102160811, 0.0172250327, -0.0224740561, -0.0615768358, 0.0354183391, -0.141508907, 0.00267085433, 0.0222913697, -0.133883581, 0.0196404234, -0.0762126669, -0.0453807004, -0.0193437468, 0.0606390536, 0.140449613, -0.0485979468, -0.0578757189, 0.130762786, 0.0309764072, 0.0085640084, -0.0317615718, 0.0492270291, -0.04021018, 0.0889722332, -0.0266411975, 0.0901532173, 0.132348806, 0.0413502529, 0.0548291393, 0.0590111315, -0.0898910612, 0.0582996011, 0.065266408, -0.0744625032, -0.0377952904, -0.0368359089, 0.0469830334, -0.116807431, -0.115320541, -0.0879266933, 0.00238024257, 0.0103788227, -0.069691278, 0.00391908037, 0.024099797, 0.0738078877, 0.0303493738, 0.0550419018, -0.121972822, 0.0200210288, -0.0166991334, -0.0649560243, 0.0218866523, 0.0012789527, -0.071845673, 0.120481841, -0.219442159, -0.0388041958, -0.0489232615, 0.0408151038, 0.0525902323, -0.0625492558, -0.0334295034, -0.179259941, 0.0485134721, -0.00684842002, -0.172918841, 0.0152828321, -0.00353746861, 0.0797556043, 0.171828106, -0.0856639072, 0.0483391657, 0.106606655, -0.0346524417, -0.0662102997, 0.000548389042, -0.0723318458, -0.0226519592, -0.0298163742, -0.00970225781, -0.00914438255, 0.0463590994, -0.0031957943, 0.0499412045, -0.0235150084, -0.0300997011, 0.0376598649, 0.198073745, 0.0993624479, -0.0572848916, -0.109548002, 0.0868605822, -0.0564789772, -0.113025799, 0.0835291892, -0.0292221382, 0.0901703537, 0.108187534, -0.0882775038, 0.0816135556, 0.0239357501, 0.0677815974, 0.00296494737, 0.0748788863, -0.0120913768, 0.0256078783, 0.0664716363, 0.0385060161, 0.0163188521, -0.0646069273, -0.0842390433, -0.0362252221, 0.0761245117, 0.0370759107, 0.162758842, -0.119829409, -0.015496552, -0.0286020041, 0.127342939, -0.00396361947, 0.0463322103, 0.0827808231, -0.0372733176, -0.0234975945, -0.0555949658, -0.05986543, -0.0525532961, 0.0899257213, -0.0632371083, 0.00453333929, 0.139113203, 0.0346173048, -0.00875579193, 0.0369689353, 0.116822541, 0.000411467627, -0.0311805699, -0.0324053466, 0.042315729, 0.0325569808, 0.0705077425, -0.158490002, -0.0692853034, 0.014626611, 0.127531514, 0.085432902, -0.0120464228, 0.0703074709, 0.0510105826, 0.0701586604, -0.0554094948, 0.0482138582, 0.124873832, 0.0997996107, 0.00841645058, -0.0322865173, 0.00332034309, -0.0512876958, 0.00796328858, -0.0496845655, -0.0817840248, -0.0284804404, 0.207782403, -0.00811658893, 0.0207694601, -0.0552041009, -0.00310244411, 0.0468787253, -0.133973569, -0.155573621, -0.118333511, 0.0644147024, 0.0424428135, -0.0530001745, 0.0445820577, 0.0557935536, 0.0129037797, -0.0369238518, 0.127312809, -0.0277343579, -0.0698076189, 0.15275225, 0.0398202725, -0.0484452844, -0.0406120904, -0.0565820746, 0.00224541454, 0.0964962691, 0.00645267218, -0.0306327064, -0.118842952, 0.0958830044, 0.0555735417, -0.0384260118, -0.00305845402, -0.0558330007, 0.0854666829, -0.0205603279, -0.035670273, 0.0723932087, 0.0588418469, 0.0438152626, 0.0188954454, 0.101422183, 0.0711393803, 0.111880019, -0.0488751605, 0.013999437, -0.048159752, -0.0452164672, -0.0451781154, -0.00924299285, -0.158946276, 0.0276355017, -0.019252412, 0.050336957, 0.0381732211, 0.0468685105, -0.100663327, 0.0153418193, -0.0391150564, -0.057868544, 0.107873701, -0.00606214022, 0.0402068198, 0.112427071, 0.055900462, -0.00954103004, -0.0631262213, -0.0752608627, -0.121419631, 0.0537686422, 0.0702112317, -0.0317528136, 0.0155923311, 0.0643391088, 0.0823150501, 0.011424928, 0.0866788924, -0.0557377785, 0.0242005736, 0.0581678934, 0.0170797296, 0.0112792905, -0.029697597, 0.0732057691, -0.153560072, 0.0463197939, 0.00305291638, 0.187867433, 0.0859213769, -0.0525866076, 0.0788777024, 0.0505607501, -0.0339050591, 0.00377000868, -0.0081246607, -0.0502759106, -0.0199783258, -0.0896850973, 0.0376046449, -0.159608096, -0.0208158493, -0.0547869429, 0.140949667, 0.00822881982, 0.0426262915, -0.00746865384, -0.0208673328, -0.0236783735, 0.0556462817, 0.0360817984, 0.00203144737, 0.0328801721, 0.0383945853, 0.0120557062, 0.00986700132, 0.138688341, -0.0186713263, 0.0991785973, -0.0621830449, 0.102392785, 0.196683288, -0.113352746, 0.0307539217, 0.160915852, -0.00642421097, -0.0744954497, 0.0174026955, 0.0922159851, -0.00581721589, -0.104899362, 0.0780781731, -0.0671591014, -0.00771567598, 0.0277557056, -0.0648308918, 0.128763229, 0.0467619039, 0.035747759, -0.0413503721, 0.15562813, -0.0232945103, 0.125851959, -0.230834201, 0.0893382207, -0.0495846346, -0.0385772809, -0.0353227928, 0.0507783592, -0.035266526, -0.047131449, -0.0176881682, 0.0360539183, -0.0857599825, 0.0258405209, 0.0694242418, -0.00353942811, -0.0398704633, -0.0827132091, 0.0523384586, -0.117656805, 0.0172490813, -0.0411410183, -0.0999691635, -0.0979274511, -0.114667013, 0.0348461792, -0.0144496374, 0.058701843, 0.0706167221, -0.0642464906, 0.119065277, 0.131035864, -0.0304263122, -0.0137733072, -0.0363757685, 0.0266923793, -0.0455352701, 0.0286264122, 0.00583955739, 0.00585118961, 0.175062031, 0.00927729532, -0.0204659514, -0.0332344584, -0.0079884883, -0.0494965687, 0.0365244783, 0.0589441247, -0.0634012818, 0.0168215558, 0.00974214636, 0.0313278846, -0.0947920382, -0.0776266083, 0.0622960627, 0.0688989311, -0.0952006131, -0.0346632153, -0.0338409357, 0.0726115108, 0.197687849, 0.007835133, 0.00582121126, -0.00569648948, -0.00252835872, -0.0110833589, 0.0878808126, -0.00196283776, 0.165228099, 0.0459995419, -0.00982443895, -0.0796034783, 0.00905897189, -0.153510392, 0.108211473, 0.158081084, -0.0377744958, 0.0505883135, -0.0575247556, -0.075220719, 0.0338324197, -0.130541414, -0.0906890631, 0.0591744483, 0.0738413781, -0.149436235, -0.0250280201, -0.0346436054, -0.0141798705, -0.108943425, 0.00232343376, 0.00533589954, -0.127761394, -0.032311108, -0.0971097201, 0.0150812231, -0.0370598696, -0.00486735255, -0.0548874661, -0.0815641657, -0.0441496521, -0.130818218, -0.0627015531, 0.0333955213, -0.0187171474, 0.0680370629, 0.0568083078, 0.0401994251, 0.0638009235, 0.00617516972, -0.0177865513, 0.0456849448, 0.0413590893, -0.0400048085, -0.00927871279, 0.122263268, -0.0846701115, 0.0735645965, -0.0731005818, 0.0534018949, -0.0490769558, 0.07646323, -0.0171432532, 0.111487597, -0.0126327146, -0.0667313784, 0.0441563725, 0.0396787003, -0.0108370492, 0.0236835256, -0.0392706022, -0.102848731, -0.0621793605, -0.0423569158, -0.0354129225, 0.0208173264, 0.0364403203, -0.142889783, 0.0237936713, -0.0149820875, -0.145569399, -0.0394799598, 0.0969427079, -0.054175701, -0.134356916, 0.0276410729, 0.0506090187, 0.0710193217, 0.0870926604, -0.0606542602, -0.0026505813, -0.160247087, 0.0402680226, 0.0271979403, -0.0864291713, 0.0413569026, -0.0622934103, -0.0218009725, 0.089244321, 0.0332072489, 0.0657498166, -0.00505386665, -0.0492895395, -0.0890076309, 0.0782933906, 0.0204010755, -0.0450760461, -0.0718519688, 0.0547425337, 0.0627222061, 0.0665706843, 0.0384123474, -0.00860513374, 0.012388546, -0.0839210823, -0.0487274155, -0.0539148673, 0.0449279994, 0.078998886, -0.0950290188, -0.050470002, -0.0429880768, -0.0437469818, -0.048291862, 0.10736306, -0.0979295671, -0.0811112747, -0.0530942306, -0.153853074, -0.16854775, -0.0392187871, 0.0121662412, 0.00176871335, 0.0253451467, -0.0658509582, -0.0616914257, 0.0228686966, -0.10971415, 0.135989681, -0.0335242748, -0.000956429169, 0.0553396866, 0.126581058, 0.0474915504, 0.0211014152, -0.0707104206, 0.119461305, -0.0858744234, -0.0533777773, -0.206835583, 0.0496135354, -0.0852625817, 0.0548041314, 0.108932175, -0.0661319047, 0.00594475213, -0.0798635483, -0.00666934438, -0.00316115795, -0.0238929577, 0.0638570264, -0.0389510468, 0.0643313378, -0.0307526607, 0.0883754566, -0.0476251803, 0.00247806869, 0.0990912765, 0.0571272932, -0.0656959936, -0.0876581669, 0.0539998636, 0.0428763889, -0.0565429293, 0.0822702497, -0.0976557434, 0.0224922448, -0.137141794, 0.0516681969, -0.173518211, 0.00714187324, -0.0489615425, -0.0682698637, 0.0697755441, -0.0377197936, -0.0324800834, 0.0682256967, -0.0459169932, 0.16174911, -0.00530527253, 0.0351424366, -0.0741646439, 0.0660107434, -0.0197895616, -0.141294301, -0.07206662, 0.0847613141, -0.0939313322, 0.0219362117, -0.153947011, -0.0551418439, 0.154210478, 0.04822056, 0.0734988078, -0.0403701477, -0.138773963, 0.0329378285, -0.00727817742, 0.0566106662, -0.0855385438, -0.0894598365, -0.0608090162, 0.012729533, 0.0434634276, 0.0687907189, 0.148822874, -0.0516477674, -0.0554004386, -0.0936880261, -0.0658270121, 0.0839076266, 0.0431993119, -0.00819264818, 0.0264952667, -0.016709324, -0.00969122909, 0.138044655, -0.0653872341, -0.0255857483, -0.0257683992, 0.0354169458, -0.169573903, 0.0797453597, 0.0307036862, -0.0552977026, -0.136601239, -0.0300603788, 0.050477773, 0.070897989, -0.00995214283, -0.0248042196, -0.066885978, 0.0727180913, 0.0737626031, 0.0173303485, -0.025581304, 0.0635150671, -0.0901748165, -0.0042982474, -0.0772284865, -0.0734660327, -0.0484250672, -0.0562392324, -0.0777136534, -0.142158046, 0.118982479, -0.122404516, 0.0402211547, -0.0368508734, 0.029629685, 0.0634636134, -0.0273319464, 0.0272786859, 0.0352585874, -0.0379413068, -0.0257819872, -0.0336226448, -0.0354589596, -0.0424527749, 0.102676675, -0.0579748675, -0.0432516821, -0.0110586304, 0.123912379, -0.0254480392, 0.0900846422, -0.0209755339, -0.0430043302, -0.0256560706, -0.0365977176, 0.0179417226, 0.050363481, 0.127457201, 0.0994190574, 0.0845612884, -0.0200168267, -0.104750745, 0.239868566, 0.0186115988, 0.178199813, 0.0310933404, 0.062885955, -0.0562206246, -0.0392183103, -0.0526602902, -0.0727086812, -0.0366779007, -0.122839846, -0.0177269597, -0.020671878, -0.0447096899, 0.112125948, 0.0552616157, -0.0793292597, 0.11010053, 0.0566014536, 0.0105314925, 0.0649300516, 0.0124685336, -0.065028511, -0.0814464539, -0.0535159707, 0.075172931, 0.0512848869, 0.124607354, -0.0304890964, -0.0202325247, -0.0133397505, 0.00607856037, 0.0542979315, 0.0357338227, 0.0694069266, -0.0883907303, -0.0505184866, -0.0274258684, -0.0451109298, 0.0880140737, 0.0571361668, 0.0118459854, 0.0533859767, 0.101867095, 0.00520355441, 0.12812005, 0.200060204, 0.120280221, -0.0197006054, -0.0587520935, 0.0717615932, 0.166860014, -0.0882551745, -0.0660146177, -0.0328773782, -0.137794584, -0.0938184783, -0.00144285941, -0.118490122, 0.023691915, 0.0282468814, -0.0695485622, -0.0863662213, -0.104297206, 0.0190177113, -0.00720984489, 0.0746551752, -0.054489132, 0.16164881, 0.127069384, 0.0143358847, 0.0857696831, 0.0835655481, -0.0396123752, -0.116242573, -0.0264006965, -0.0861118883, -0.0320002288, -0.0515784696, 0.0245875269, -4.10219654e-05, -0.0561805964, 0.0511259586, 0.0491109192, -0.0950999707, 0.0726895705, -0.108802855, 0.018060118, -0.133699417, -0.00267339405, 0.0589299276, 0.0167818218, 0.0702794045, 0.000833958387, 0.0499559194, 0.0545615032, 0.162329838, -0.0680439919, -0.0699060559, -0.15240258, -0.0243935026, -0.00303140096, 0.00623072311, -0.020528052, 0.00236353464, 0.0902205631, -0.0367763489, 0.0199145116, 0.0212102402, -0.0352000743, -0.00631831959, 0.0320474952, 0.0281665921, 0.0808550641, 0.0251082182, 0.0282254033, 0.0036831554, -0.0160769746, 0.0233788732, 0.0261787195, 0.0226513185, -0.0150998672, 0.0153304236, 0.0188213531, 0.0503936633, -0.045406118, 0.0820774511, 0.0189963859, -0.0735352412, 0.0783244967, 0.0159697533, 0.123810753, 0.0472124331, 0.0501417145, 0.0643201843, -0.0742305368, -0.0364033878, -0.054758314, 0.0295691304, -0.00533509441, -0.0248704236, 0.0944912434, 0.0813809186, 0.0800662935, 0.0420621634, -0.104065731, -0.00707397517, 0.0386740789, 0.168509588, -0.0944282636, 0.0742100775, 0.121663205, 0.0613658726, 0.0363074765, 0.138406873, -0.078356795, 0.0452519581, -0.0600139759, 0.150149718, 0.023582831, 0.0457559377, -0.0855897516, 0.0482263267, 0.00215817336, 0.00113095716, 0.0506576933, 0.0123284925, 0.0568627268, 0.00802153349, 0.133727148, 0.0333910063, -0.023536358, 0.141339049, 0.0279657394, -0.105808012, -0.00864004344, -0.012913486, 0.0723010227, -0.0580282882, -0.0980359167, -0.121762902, 0.0335033461, 0.0492193848, -0.00799391884, 0.0229605138, -0.0465496927, 0.0366377011, -0.0190207548, -0.0344992056, -0.0638491586, 0.19049722, -0.0673196018, 0.163322881, 0.0370728299, 0.0201039165, -0.117321387, -0.0258302167, -0.021659717, -0.0786858648, -0.042272266, 0.082426101, 0.0618773587, -0.00105269952, 0.0102046933, -0.0235174112, -0.0510242581, -0.116305858, 0.0226745121, 0.0556324944, 0.120265208, 0.0731783137, 0.0661707222, -0.0280066542, -0.0199447945, 0.0128385788, 0.0226939432, 0.0104000568, 0.00935876649, -0.213882118, 0.043200016, 0.0241836477, -0.13518852, 0.140135095, 0.0253206324, -0.089445211, 0.00240788609, -0.0890551805, -0.0191624686, 0.0517471433, -0.0367655568, 0.0598453246, 0.112564206, -0.116867706, -0.0396824777, -0.0163099933, -0.118076362, 0.11046911, 0.0247966498, 0.0313623138, -0.108059898, 0.0364985466, -0.0730506554, -0.0836252645, 0.0544317178, 0.0144574177, 0.0365974307, -0.0178850703, -0.055263631, 0.130582184, 0.0158302486, 0.0212825127, 0.0239027031, -0.0166860893, -0.0275060162, 0.0294779949, 0.0809956118, 0.0361995175, 0.0210323408, -0.0460734852, -0.0791156143, 0.0205498245, -0.0106738573, -0.00989503041, 0.0165876858, -0.0203668587, 0.0815822035, -0.0239934083, 0.0604061931, -0.00175664946, 0.0208463781, 0.0540469699, 0.174571007, -0.0146036129, 0.0423222333, 0.0977733657, -0.0425417535, -0.0710100755, 0.0760513246, 0.113821641, -0.0535171703, -0.00542533398, -0.0697968975, -0.0428297296, 0.0674038902, -0.0297512412, -0.066744484, 0.0181291327, -0.00508406153, -0.0266535934, -0.0606855378, -0.0260272212, -0.029811386, -0.107172653, -0.150785118, -0.0542859547, 0.0356353149, -0.122487269, 0.0750695467, -0.0401163846, -0.0629263371, -0.0792647377, 0.104086034, -0.0047227107, 0.103974536, 0.0502419882, 0.0476147234, 0.052882392, 0.081533879, 0.0924756974, -0.0315656103, -0.0200783983, 0.130904391, -0.0245863274, 0.0448258296, -0.0867705271, -0.0143366829, -0.0240080208, 0.0499560311, -0.00190844573, 0.0032625813, -0.000506900251, -0.0229720958, 0.0386845991, -0.0575748906, 0.00777366385, 0.0670741051, 0.065418154, 0.149928927, 0.0400025733, 0.124139905, 0.0728096142, 0.00236796588, -0.120325178, 0.16046533, -0.0657965019, -0.0568519235, -0.00610711426, 0.0497483648, -0.00804714486, 0.0444892272, 0.0504619479, -0.133039102, 0.00865272805, 0.0114317089, -0.00698417053, 0.0169084482, -0.0348446779, -0.0723827779, 0.0108677205, -0.00218051486, 0.0390979648];
    CONSTANT bias_0_u : ARRAY[0..63] OF REAL := [-0.931392431, -0.669652343, -1.55073643, -1.15129042, -0.928060949, -0.835326016, -1.05773425, -0.809125721, -1.0343436, -1.36020243, -0.812485695, -0.596730828, -0.800589681, -0.83492893, -1.23361444, -1.4201777, -1.06900442, -1.04275012, -1.86629462, -1.68873703, -1.34019673, -0.945544183, -0.886029959, -0.729185879, -0.675665855, -0.875132143, -0.690106928, -0.763296306, -0.747061849, -1.10096192, -0.758312643, -1.23618972, -1.4139967, -1.28251481, -0.887215853, -1.12884796, -1.17651927, -1.66531849, -1.57700455, -1.01120985, -0.878331959, -0.872978032, -0.621329427, -1.0162462, -0.99940753, -0.698668599, -1.47800922, -0.852591813, -0.93049854, -0.788715541, -0.874885857, -0.572944462, -1.31330848, -0.807830811, -0.895757496, -1.79783428, -0.845625222, -1.08024359, -1.43994868, -1.82642233, -1.50900924, -0.701206744, -1.07954109, -1.05142236];
    CONSTANT weights_0_r : ARRAY[0..63] OF REAL := [-0.301351488, 0.191772759, -0.403094679, -0.385009229, -0.325696975, -0.344430864, -0.430924505, -0.490683407, -0.380927861, -0.361935526, -0.291825026, 0.270645022, -0.557896674, -0.624442339, -0.570287347, -0.547084689, -0.328458816, -0.604146957, -0.345501393, -0.616985977, -0.625005603, -0.563085496, -0.468810678, -0.398420662, -0.227860957, -0.486180753, 0.0191694256, -0.046916645, 0.234420627, -0.389543176, -0.00718040438, -0.374701381, -0.612858176, -0.358533949, -0.574734867, -0.603802323, -0.283780545, -0.357478797, -0.447851956, -0.458725035, -0.410655737, -0.376305223, 0.303187847, -0.553753257, -0.386509717, -0.504178882, -0.474493176, -0.238366574, -0.448695511, -0.551571906, -0.411650151, 0.404194504, -0.465952367, -0.147349313, -0.468469918, -0.304423511, -0.4342767, -0.47622183, -0.525499105, -0.457058758, -0.439959496, 0.0408562459, -0.552530468, -0.292028844];
    CONSTANT recurrent_0_r : ARRAY[0..4095] OF REAL := [-0.0834894925, 0.0467989594, -0.0922519863, 0.0892271101, -0.0968513042, 0.0679784194, -0.0419990122, -0.0955153108, -0.0172851142, -0.0447769873, 0.0400388502, -0.0478489809, 0.0498131029, 0.0975087509, 0.103417948, -0.0618524924, 0.138862789, -0.0484442562, -0.106181331, -0.132875144, 0.0242299326, 0.0707813576, -0.0631774291, 0.0927816704, 0.146799028, -0.0673606545, 0.0149163306, 0.158295408, -0.0541859716, -0.0671267807, -0.00778596848, 0.000831183046, 0.0179751236, 0.0616365261, 0.0552535653, -0.11939618, 0.00227971375, 0.0860660523, 0.0384575725, 0.0739784613, 0.00518694334, -0.0637862906, -0.00229425658, -0.0886000842, 0.119190097, -0.0505612381, -0.100778803, -0.11373806, -0.046051234, 0.0172212869, 0.00996381789, 0.0867178142, 0.00406045653, 0.0659313872, 0.0901537985, 0.00407537259, -0.155829459, -0.0182549451, -0.0341455899, 0.124589838, -0.0760684684, 0.0296373926, 0.00549710728, 0.0332801342, 0.0679366067, -0.0555260926, 0.0819408521, -0.0728703663, 0.020875264, -0.0447206348, -0.024039913, 0.0543668233, 0.0924990252, -0.0224341024, 0.0680758804, -0.0131752398, 0.0171246715, -0.0379354954, -0.118314825, -0.0296662319, 0.0103624333, -0.150564685, 0.0755786151, -0.0666730851, -0.0181739815, -0.0342114717, 0.0339080915, -0.0595367178, 0.0309331622, -0.0153474286, 0.0614931062, -0.0788206384, -0.0491645597, -0.0551766492, 0.110275842, -0.0309414417, -0.087802209, -0.0610899068, -0.00560984015, 0.0977157503, 0.00970546156, -0.156553969, -0.0635337755, 0.00846432708, -0.0481569208, -0.156108454, -0.0311011374, 0.0380924568, 0.0604931377, -0.106866658, 0.0386045091, 0.0167547446, -0.0975543559, -0.0810313448, -0.00664621964, -0.0154656004, 0.0141974762, -0.0400947481, 0.0326277912, -0.0616046824, -0.0670897216, 0.163002104, 0.01041748, 0.0679064617, -0.0368735157, -0.0427763127, -0.0614703819, -0.0516258851, -0.0362892523, -0.0502930507, -0.0644264519, 0.040134564, 0.163039222, 0.0453167073, 0.0265058093, 0.0309302956, -0.0310254358, -0.0870743915, 0.0869462565, -0.0102094412, 0.02950841, -0.0191445109, 0.0157393347, 0.112097934, 0.142738387, -0.0986512154, 0.101732939, 0.0275557972, -0.0516387671, -0.024218658, -0.00215544179, 0.0165637061, 0.0156634506, 0.0115557984, -0.0915465057, -0.0172377117, 0.0396726206, -0.0412831642, 0.0991871059, -0.0850381553, 0.122572176, 0.059342213, -0.0229966789, -0.0314630009, 0.00477001816, -0.0216304138, -0.0459695496, -0.0558857583, 0.0364166088, 0.0599161908, -0.0168819502, 0.155651927, 0.141873583, 0.126577303, 0.0584061071, -0.0245434716, 0.07191585, -0.125751734, -0.096313253, 0.0990332961, 0.0953751877, 0.0237817224, 0.0773518533, -0.0857243687, 0.138499305, 0.0413452238, -0.00136547722, 0.0418496765, -0.00384547003, 0.0725840926, 0.0687962323, -0.221241683, -0.0535463355, -0.0130795371, -0.152106091, 0.00108890608, -0.0629126653, -0.109754905, 0.0672944188, 0.0458643995, -0.127328977, 0.0779956579, -0.0260329992, -0.0222704634, 0.0060250815, 0.0342492759, 0.0469465703, 0.0682547241, 0.0466573387, -0.0317380279, 0.118174516, 0.0363855176, 0.0165183749, 0.216430724, 0.0503736399, -0.0601224527, 0.047193028, 0.131177261, -0.0908262208, -0.15726164, 0.0594424009, -0.0204188749, -0.0278644171, 0.101016611, -0.0298268441, -0.080154486, -0.0577925071, -0.106108546, 0.00219925866, 0.0538200289, -0.000312333927, -0.0564782694, 0.0101036718, 0.00516057666, 0.00766485184, 0.0177538376, 0.00237444974, -0.0577772781, -0.127201959, 0.0181556642, -0.00818925537, -0.0185058136, -0.0378008261, -0.0132604018, 0.0929510295, 0.0808474272, -0.0706657469, -0.113311686, -0.0553113446, 0.0279085524, -0.105972864, -0.0372796655, -0.0130742528, 0.0488647111, 0.0226176027, 0.0247713439, 0.0545698255, -0.0249881856, -0.0808280632, 0.0343040675, 0.0220307633, 0.0778453946, 0.00909530744, 0.00474842079, 0.0245809406, 0.027137503, -0.0232185125, 0.140213117, 0.0256274082, 0.0719716772, -0.0154388361, -0.0446083136, 0.0152545236, -0.0324217938, 0.0500168242, -0.114832193, 0.0540725663, -0.201761976, 0.0459797718, 0.0488682203, -0.0374526232, -0.0756408647, 0.0282250922, 0.0548831299, -0.151702717, 0.0439265333, 0.0316746458, 0.0101707652, 0.0837145448, 0.0808735639, 0.0973392278, -0.0686043128, -0.0390135162, -0.037535198, -0.0250067096, -0.0664628521, 0.0204570256, 0.0354304649, -0.057973817, 0.0578858256, 0.0356692336, 0.0886768922, 0.0543263741, 0.0420739315, 0.084652096, 0.180876732, -0.0387669355, 0.0118383123, 0.0290507115, -0.0599402376, 0.0485393032, -0.0703626052, -0.0345942751, -0.0286344141, 0.0617277063, -0.0411391258, -0.0778558925, -0.0121396091, 0.0011215657, 0.0436940789, 0.000647306093, 0.0169583671, 0.0537803844, 0.0782520995, -0.0194653235, -0.0218962058, 0.00249565719, -0.010981407, -0.0674014688, -0.0330897793, 0.018824378, 0.157535002, 0.0308090374, -0.0746396407, -0.0875643045, -0.00356309139, 0.00969221443, 0.0921113268, -0.0434736833, 0.0130275963, -0.0466789939, -0.0251713507, 0.10718137, 0.155800402, 0.0190462153, -0.0899385735, 0.137247831, -0.0866682157, -0.0320754685, -0.0946900174, -0.0161404721, 0.0882564411, -0.112924516, -0.088722147, 0.192345887, -0.0126325535, -0.0174161885, -0.0645587966, 0.0146739678, -0.0393769257, 0.0789906681, -0.0809244365, 0.0494276024, 0.0675513595, 0.0875197873, 0.168436021, 0.0236752108, -0.0369569995, 0.0797938108, -0.119467117, -0.0492167324, 0.0533705875, -0.000214729458, 0.0990879759, 0.0621759742, 0.0427966863, 0.0239031687, 0.0799559504, -0.0621714219, 0.0745402873, 0.0781922266, 0.0327110179, 0.0261501111, 0.011958912, 0.106199577, -0.0313672908, 0.0454588458, 0.0187561624, -0.0123822438, 0.0570373051, -0.0774810463, -0.0445477366, 0.195391595, -0.0160081312, -0.0467466153, -0.15215385, 0.0304640979, 0.0530834794, 0.0519628152, -0.142502248, 0.0521924794, -0.0213847924, 0.137605369, -0.0943483561, -0.0639615729, 0.0294855349, -0.000336129218, -0.104782604, 0.0927328095, -0.028684549, 0.132814825, -0.0141541846, 0.0926760733, 0.0494773462, -0.0836238563, 0.0119094858, 0.0856154338, -0.139292598, 0.0450100079, 0.0095192045, 0.0648575351, 0.0879206955, -0.0362641513, 0.0149863679, -0.093047604, 0.0910623372, -0.0729507431, 0.099900797, 0.00975495018, 0.10402672, -0.0265085027, 0.00896766782, -0.0797617286, 0.0680103824, -0.00225491449, -0.111769781, -0.0673333183, -0.107364029, 0.0766148716, 0.0842316598, 0.0189867634, -0.139816821, -0.0133126192, -0.125086024, 0.0900506675, 0.107696734, 0.0128689855, -0.0446564034, 0.0704938099, -0.0910163745, 0.120799132, -0.0846302807, -0.0124115273, 0.010663012, 0.0126034543, -0.0300969128, 0.0170655474, 0.0514482073, 0.0689900517, -0.00158789381, 0.149908528, -0.0603792854, 0.0131468186, -0.0535668321, -0.118181631, -0.025183931, -0.109207809, 0.00673588412, -0.124501571, 0.0124984011, 0.0683000535, -0.0511983112, -0.0355482064, 0.0124112274, -0.105003238, -0.0914214924, -0.037354432, -0.0406142324, 0.0181756504, -0.0504919142, -0.0960488319, -0.0375996903, 0.0391708873, -0.0349344909, 0.0847899988, -0.0085113775, -0.0851751342, -0.0951333269, 0.0153997168, -0.0674072206, 0.0236242227, 0.0501294322, -0.0528307669, 0.131298378, 0.0220658295, -0.0347023904, 0.029442694, 0.0483123884, -0.16232118, 0.0271872394, 0.0621333644, -0.0257400814, 0.0729334578, -0.0658665001, -0.105266467, -0.171774209, -0.0453840047, -0.0155880339, 0.0938720107, 0.0879871398, 0.0643682331, 0.0427748635, -0.0361816436, -0.0438858196, 0.0104101989, -0.134780109, 0.0869414657, 0.00118048675, -0.00513844192, 0.0182014499, -0.0240692645, -0.0398045331, -0.0146628786, 0.0358414315, -0.0180199072, -0.0287214592, 0.0866206288, -0.0701739937, 0.000415597111, 0.0721387342, -0.0679822639, 0.171161994, 0.0371262208, -0.0477780961, 0.0761367232, 0.00384224392, 0.130283386, -0.0281605236, -0.0999097824, 0.00152361393, -0.0915167928, -0.0212306529, 0.0126610585, 0.0154684512, -0.0978761613, 0.0650571138, 0.107376486, 0.0881768167, 0.0337237157, 0.054977864, 0.0540641472, -0.134753376, -0.131919801, 0.0537733622, -0.0841272324, -0.0393206924, 0.0709122196, 0.102772944, 0.156615913, 0.0902129337, -0.0831259787, 0.0207677744, -0.0577425808, 0.0763535425, 0.0751461163, 0.0386200547, 0.0937433094, -0.0476259813, -0.0373367108, 0.0155079169, -0.0248294845, -0.120135389, -0.0352638401, 0.145516515, -0.100795284, -0.0410206988, -0.141030952, -0.0106899496, -0.0759382918, -0.0494840071, -0.0805307701, -0.0583564751, 0.0285217259, -0.0824788734, -0.000849559903, 0.0188932419, -0.0336842611, -0.0506386012, 0.0203082673, 0.0773929581, -0.0287808534, -0.06769678, -0.0738249421, 0.155622259, 0.0350486711, 0.0308453329, -0.0915696025, 0.0791843161, -0.0964923128, -0.00887560379, -0.0208047107, -0.133802965, 0.0323152542, -0.026939515, -0.0812889114, 0.0496312641, 0.0404926501, -0.1019504, -0.0131298713, 0.100097105, 0.115483843, -0.00638710242, 0.163589418, -0.0991462022, -0.0362230949, -0.0176009014, -0.0313397944, -0.0212460831, -0.0176329389, 0.0253308993, -0.0264203008, -0.0197697654, 0.0765542611, -0.0138612632, 0.0492661186, 0.00846538972, -0.0992811099, 0.120879501, 0.0574992225, 0.0359927192, -0.0615425259, -0.0063858442, 0.0557737239, 0.0424413607, 0.130089223, -0.0444395095, 0.107088849, -0.0397110581, -0.053124819, 0.011124542, -0.0532939099, 0.0410669371, 0.0292511564, -0.101436161, -0.0138421534, 0.261617333, 0.0745773017, -0.00261045154, -0.0530744269, 0.0931384563, -0.041711852, 0.0388382412, -0.0277338717, -0.137989819, 0.0612927973, 0.104822055, 0.0361424498, -0.081897676, 0.082424067, -0.0292748399, -0.0650308207, -0.0574782565, -0.0816696733, 0.115542442, 0.108364627, 0.150625765, 0.0555263087, 0.000987943262, 0.0676554143, -0.0174685903, -0.019615002, -0.095944263, -0.0548800603, -0.0220668316, 0.0540091395, 0.040932171, 0.0198501125, -0.0563352332, -0.0535954833, 0.0527449995, 0.157754645, 0.00486304238, -0.177564219, -0.0268895626, -0.0191486217, -0.0552683026, -0.0416013673, -0.147009224, 0.0570645519, 0.114052191, 0.0689847618, -0.00186852366, -0.0354810581, -0.0787176266, -0.0754320398, -0.0211988557, 0.00642943941, -0.0388428755, -0.0820757076, -0.0232652538, -0.0523139276, -0.192835316, -0.0925032943, 0.0320784673, 0.0165662523, -0.050621748, 0.048093807, -0.0466006622, -0.0441171862, -0.0852081925, 0.0172305536, -0.0356022976, 0.125120699, 0.00274382625, 0.0296839103, 0.0180109572, -0.00339450128, -0.200602382, -0.0330988802, 0.00348684168, -0.143698916, 0.0309801847, -0.0543181002, -0.0799558908, 0.190914512, -0.0614015609, 0.00774812885, 0.0226198081, 0.0531787537, -0.0618811138, -0.0585327186, -0.0788292214, -0.00366556738, 0.0347583294, -0.0325671248, -0.134057224, -0.0463110805, 0.0597175434, 0.0521154925, 0.00114774657, -0.0531816185, 0.019560026, 0.0392225087, -0.00842877384, -0.101296403, 0.14710924, 0.0299691372, -0.0620323084, 0.10974852, -0.0141659304, -0.0494842306, -0.0295206457, 0.0119519308, -0.0382294469, -0.139502227, -0.131658226, 0.0115597174, 0.0770779178, -0.0218290314, -0.0121306516, -0.0382104144, 0.060878098, 0.142750472, -0.0589798763, 0.0676200837, 0.0185247324, -0.0410691239, 0.0299137048, -0.127572939, -0.0378006473, -0.100536868, -0.0363167077, 0.00676896796, -0.167191088, 0.0212077759, 0.0868244767, -0.132884994, 0.0342110395, -0.0611182749, -0.0260481872, 0.102945745, 0.0365496017, 0.0234432518, -0.0248310417, 0.175976261, 0.0216019899, -0.00532627665, 0.00764858723, 0.027753979, 0.0405078456, -0.0206162166, -0.00527708791, 0.0114256972, 0.0365030132, 0.0336980522, 0.0692263246, -0.0243159756, 0.0986577272, 0.10393206, -0.0943767056, 0.00742093101, 0.0436499268, 0.0341592506, 0.0456877351, 0.0279276185, -0.039765738, 0.135489181, 0.233778447, -0.0658682585, -0.0471731834, 0.000448940322, 0.00922876596, 0.117229208, 0.011610589, 0.0243017413, 0.031091243, -0.0900265202, 0.0601132065, 0.00408360083, 0.0275879912, -0.118830316, -0.0615517758, 0.0681044236, 0.158631369, -0.0484357812, 0.124020174, -0.0326664746, 0.0409314819, -0.00422460213, -0.0324111953, 0.0290527269, -0.103400938, -0.107562162, 0.0932063311, 0.0250069126, -0.124122925, 0.03050589, 0.102034807, 0.138139054, -0.0296162739, 0.0276926365, -0.0569745451, 0.129586026, 0.0547338687, -0.116471387, -0.0195134766, 0.0506814942, 0.0076626474, -0.0558482297, -0.101829417, 0.069013834, 0.0300411563, 0.0648475587, 0.166248247, 0.101213507, 0.0444345027, 0.147666112, 0.0086207306, 0.0374275669, 0.0151421484, -0.0581510216, -0.0248833448, -0.0628596321, -0.133901253, -0.0859556645, -0.0856730938, 0.045230452, -0.0480204336, 0.033454746, 0.0220677182, 0.054104574, -0.0845751017, -0.00932334457, 0.0160639696, -0.0344653763, 0.0510070175, -0.0676326752, -0.034518566, 0.00499220565, 0.0302092172, -0.0518940836, -0.00955612399, 0.00382014737, -0.0239019413, -0.115307562, -0.0828005672, 0.0636793822, -0.0738432407, 0.0954737216, -0.109313734, -0.0578072183, -0.012398852, -0.0527146682, 0.0275513027, -0.0815594122, 0.00507738208, 0.045145262, -0.0461822748, 0.0274811871, 0.0118764099, 0.0133302175, 0.133594975, -0.0398499705, 0.065370582, 0.0196005814, -0.114700183, -0.107491247, -0.030636169, -0.0373892598, -0.00918629952, 0.129107028, 0.0423830003, 0.0965084732, -0.100005589, -0.115171194, 0.00263285707, 0.060572587, 0.0379161015, -0.0931825787, -0.116522536, 0.0266920701, -0.0241217595, 0.00282175466, 0.0295968801, 0.000478329137, -0.110135563, -0.0414175317, -0.0636743531, 0.0197038241, -0.00920526311, 0.0625352487, -0.0236603841, -0.138025969, -0.0883734673, 0.0917572156, -0.11933253, 0.0258444548, 0.0710579157, -0.0780234337, -0.0148170441, 0.0312691033, -0.00566856563, -0.0145191867, -0.0349283367, -0.00670860149, 0.105804041, -0.0641736388, -0.0366437323, 0.0522898138, 0.115683272, -0.0386916995, -0.215895638, 0.0518536642, 0.0728991702, 0.0477389321, 0.0112064974, 0.0782056302, 0.0881057382, 0.024451958, 0.120363623, -0.0709322169, 0.06867598, -0.0660766438, 0.00340095931, 0.149231806, 0.0184066538, -0.0856160894, -0.0739547834, 0.0312558375, -0.0619605556, 0.0516609736, 0.0347899199, -0.15554671, -0.0294578224, -0.0578455925, 0.0576982014, 0.036413908, 0.0532127656, -0.0513671227, -0.030536525, -0.0260005239, -0.0207533687, -0.01641028, -0.116865128, 0.124191687, 0.114527084, 0.0870671272, 0.119564414, -0.0358877964, 0.0894882455, -0.0142037831, 0.0589610264, -0.00495830178, 0.0118975155, -0.0367976651, -0.106736168, 0.0531613529, 0.00647791289, 0.0446007475, -0.0617889166, -0.0287456177, -0.124598369, 0.0289232414, 0.128152966, 0.0362791494, -0.0292951427, -0.0408745706, -0.0576321818, -0.0480503216, 0.161305472, -0.00748889893, -0.0536159575, -0.019543618, 0.0229161847, 0.038694039, -0.00959399343, -0.036313355, -0.0360907875, -0.0258969292, 0.0174424201, 0.005995363, 0.0753622204, -0.0476423204, -0.0331449658, 0.0135375774, 0.0225478727, 0.079924807, -0.0982389003, 0.100322366, 0.0484079532, 0.0593880564, -0.104930677, -0.0233237967, -0.121263564, -0.047104951, 0.0493723154, 0.0864522606, -0.00893124938, 0.0428383239, 0.0720678344, -0.0713310167, -0.00386607088, 0.093112953, 0.00370634254, -0.0390104242, 0.0295266621, 0.184043735, -0.00185719877, 0.0377220772, -0.0604721606, -0.0894271433, -0.10692969, -0.0459658429, 0.00398916379, -0.0968620628, 0.0383661166, -0.0810789838, -0.0860629678, -0.109189242, 0.169216365, 0.1289244, 0.0566616319, -0.0316038765, -0.0574379712, 0.0202376135, -0.0542436466, -0.025901895, -0.018552348, -0.00465473533, 0.0463921055, 0.00306424685, 0.0593580268, -0.0218768641, 0.0863000751, -0.00658572465, -0.0336344652, 0.0975641906, 0.0272094943, -0.167632833, 0.0712785348, 0.0234816838, 0.0755730569, 0.121718504, -0.0777702406, 0.0686770678, -0.050026767, 0.0416301936, -0.0960736573, 0.0664560124, 0.102550723, 0.0625562221, 0.110591643, -0.113259137, 0.0022691451, 0.0703474581, 0.0666949004, -0.0071596792, 0.061394833, 0.0293247029, -0.0631409734, 0.020673316, -0.0263614226, 0.0982172564, 0.00699460227, -0.0455927588, 0.0802026019, -0.10190887, 0.0846148133, -0.11210525, -0.0350118726, -0.0242762193, -0.000193818472, 0.0546705574, 0.0366264507, 0.134070396, -0.0260837413, -0.0177230798, 0.0196370408, 0.0894785747, -0.0395769067, -0.107305057, 0.0529573187, -0.081204012, -0.152088001, 0.0303028487, 0.0674561337, -0.0395990945, 0.0461127982, -0.0541351065, 0.00466474006, 0.00836414658, 0.104049645, -0.00101429038, 0.13354446, -0.0696410462, -0.0254141055, 0.00835372508, 0.000807271339, -0.0187259577, -0.0563195646, 0.105594195, 0.0708100349, -0.0317827202, 0.0994293988, -0.0434136167, 0.102707855, -0.0394269079, 0.0146331284, -0.00732005015, -0.0310396105, -0.0530030057, -0.0496953093, -0.0778527483, 0.00890290551, 0.023694545, -0.0329473205, -0.0327186771, 0.023676496, 0.0597901158, -0.0215158965, -0.0325211063, 0.0834325701, 0.0684324652, -0.0814330131, -0.0691422001, -0.0356172249, -0.0329068005, 0.0185153484, -0.0137839317, -0.0288640819, 0.136546835, -0.037425831, -0.0333168395, 0.0422376283, -0.0332692713, 0.0755482465, 0.0192054361, -0.0823622718, -0.0410633124, -0.0412313119, 0.138509929, 0.0316699706, 0.132271022, 0.0183287039, 0.0480044708, 0.147155046, -0.0573583022, -0.0365737379, 0.107809931, 0.0909634158, -0.0412379578, -0.123732083, 0.0469360687, 0.111640856, 0.0569434911, 0.0930527151, 0.140695393, -0.0894969255, 0.00256445911, 0.0125999935, -0.0562401563, -0.114302367, -0.0382896215, 0.0104759187, -0.0232379213, 0.0542952791, -0.034059599, -0.146358714, 0.066709727, -0.0732627437, -0.00571516529, -0.0198372602, 0.120803088, -0.105709523, -0.100433663, -0.0215995014, -0.0400962122, -0.0655378699, -0.0331503414, 0.0164581686, -0.0318296552, -0.100893125, -0.181700885, 0.120456025, -0.0762417614, 0.0831995532, -0.00903397053, 0.143906787, 0.0352139436, -0.0112549327, 0.0669031441, -0.0417459607, 0.00541909691, 0.0642425418, 0.116839305, -0.179413512, -0.067691505, -0.00389492046, -0.00482019968, 0.00230792724, -0.0782617629, 0.0633524507, 0.0558453351, 0.0827809349, 0.108852305, -0.0359224975, 0.0284109451, -0.0222191606, -0.101449154, -0.127913833, -0.109366447, 0.146415055, -0.0545229688, 0.157297999, -0.0392694511, -0.136351794, 0.0631641373, 0.0868870541, -0.047785867, 0.128236473, -0.0711336285, -0.0256616995, 0.125207156, 0.073627241, -0.0366111249, 0.0887460783, -0.139744967, -0.0566972345, 0.0924156308, -0.00253159087, 0.0565007627, 0.0418369919, -0.119484343, 0.0318732932, -0.0316493884, 0.00976659823, -0.0111968163, -0.123742029, 0.0509138629, 0.0725260526, -0.0395703204, -0.00607385579, -0.00724574691, -0.0408083349, 0.0192282572, -0.0687208474, 0.00142038311, -0.125461325, 0.0599353909, 0.084194988, -0.057588283, 0.00553785916, 0.0209137872, 0.00708530564, -0.064549908, 0.000950800255, 0.0361906178, 0.106690891, -0.0902081355, -0.010964714, -0.0176610649, -0.0183612779, -0.0169377495, 0.0292202812, -0.00526601076, -0.0592814647, -0.0923140794, 0.0702977553, -0.0418194905, -0.00336346775, 0.0736140683, 0.0709515214, -0.0671726838, 0.119039156, -0.044654049, -0.0310713947, -0.058872927, -0.0735617876, 0.111595832, -0.000629011542, 0.0473766737, -0.0703351051, -0.103621587, -0.062163122, 0.0484706573, 0.0491833352, -0.0284291729, 0.120324776, 0.0621699095, 0.0961769968, -0.112067148, 0.0347730964, -0.126400009, 0.0318991877, -0.0962366164, -0.0341994688, 0.0218884982, 0.0080213882, -0.0774020925, -0.0732281432, 0.00689242594, 0.0167558584, -0.0840547979, 0.0384579897, 0.0810027942, -0.145067349, -0.100323461, 0.00845299568, 0.0601886511, 0.0302432552, 0.0088377092, -0.153663918, -0.0154264988, 0.00787600968, 0.0539445095, -0.164799377, -0.0100836325, 0.00179879088, -0.0612194575, 0.0524255112, 0.0441213287, 0.042193003, -0.0278313346, 0.0382799134, -0.00075703254, -0.0351711512, -0.00383648649, 0.0892538652, -0.120289706, 0.0880583376, 0.0809447318, -0.0352157615, -0.0152201615, 0.0262710433, -0.108669877, 0.0415507369, 0.019583337, 0.161030442, 0.0468844399, 0.00803215057, 0.00341675803, -0.0586863384, -0.127230674, 0.0464866236, 0.020540949, -0.0430138856, -0.194104955, 0.00367502496, -0.0318855755, -0.134010583, 0.0450272001, 0.0145560429, -0.246621549, 0.0988970846, 0.0510415658, 0.0687515289, -0.0536560044, -0.0625091419, -0.0327615403, 0.0907914191, 0.0783033073, 0.0203253068, 0.0194462538, 0.0553661026, -0.0425359383, 0.0350326747, 0.128417015, 0.0408646986, 0.026424367, -0.105355956, -0.113743819, 0.126335546, -0.00976781547, -0.0702449083, 0.0934237987, -0.0495629832, -0.120837845, 0.140801162, -0.0129696168, -0.0515523106, 0.0654594451, 0.0878215879, 0.00559131615, -0.0391941629, -0.110382959, -0.0833658129, -0.0678980723, -0.121550776, -0.0277186874, -0.0747896284, -0.0528696813, 0.062489666, 0.0258378275, 0.14689526, 0.0139871612, -0.0774390623, -0.0257221013, -0.133306846, -0.027471479, -0.0779962316, -0.0114445668, -0.0644760877, 0.0602955893, 0.0901463851, -0.0512889475, 0.0411484092, -0.0123691522, -0.0285694972, 0.0619165599, -0.0283145756, 0.0895031691, -0.0317250974, 0.0182393733, 0.0494113527, 0.0265502576, 0.0284394547, -0.109676167, 0.106926247, -0.00997429341, 0.0960271582, -0.0780220181, 0.0630786344, 0.0139888963, -0.0320418403, 0.0691434443, 0.0730710551, 0.0373421013, 0.109231554, -0.0456483439, 0.188781306, 0.0167414919, 0.0248027481, 0.0556567833, -0.131824747, 0.0671918541, -0.0238614921, 0.0298387464, 0.0921626911, -0.043094404, 0.078622967, -0.0343140215, 0.0269713774, -0.0172435343, -0.0108120041, 0.0982474908, 0.0519196466, 0.0162194744, 0.118766591, 0.0149338562, 0.0667814463, 0.032377176, -0.115251333, 0.0373098627, -0.0259436853, -0.0307341777, -0.11223197, -0.091855742, -0.115036793, -0.0118110599, -0.0412412398, -0.104448631, 0.0298828408, 0.054202266, 0.0600945503, -0.0280554015, 0.0998843983, -0.0229049902, -0.0153931035, -0.0195422284, 0.0835999846, -0.00953147747, -0.0565470383, 0.107559517, -0.0194214284, -0.0247669406, -0.0479892194, -0.0300220288, -0.0323037095, 0.0216859505, 0.0141581837, -0.0876181722, -0.00716956332, -0.16756773, -0.0205360614, -0.046861358, 0.0352517217, -0.0290013291, 0.124769107, 0.0261376947, 0.0112239327, -0.0346608944, 0.062852174, -0.0236231424, -0.153502658, -0.19097279, -0.106461793, -0.0408299826, -0.125152305, -0.0721943304, 0.0340681151, -0.0453003272, -0.061441943, -0.102795735, -0.0569854006, 0.034737654, 0.0421225093, -0.0153091736, -0.0218936522, -0.146173477, -0.00829258747, 0.184158102, 0.122241288, -0.084177345, 0.168531835, -0.00641076453, 0.0334824249, -0.0122941528, 0.032062754, 0.059957698, 0.0355172753, 0.107312627, 0.0144212283, 0.0861650929, 0.0188808516, 0.0193134509, -0.145267516, -0.0889582932, -0.0842778534, 0.0916769803, 0.0411723703, 0.00554753607, 0.0037490651, -0.10848517, 0.051846154, 0.0776569173, 0.101116732, 0.112386301, -0.0098252669, -0.0481179878, -0.0171496551, 0.0795148313, -0.0189479142, -0.018890053, 0.178836018, 0.0138866231, -0.0821822882, 0.0711538345, 0.0129677355, 0.146517605, -0.0250943117, 0.0803776085, 0.0770965517, -0.0571847223, -0.00601102784, -0.0542757064, -0.0443117172, -0.0133484909, -0.102817506, 0.0237798542, 0.00735295052, 0.0711276382, -0.0795218721, -0.0454166718, 0.0172596034, 0.0610119589, 0.0483013652, 0.0160205476, 0.0464293063, -0.0604674481, -0.0779783204, -0.089457497, 0.0523129627, -0.0215199031, -0.0400521234, 0.125532493, 0.00734655932, -0.0142266527, 0.17185384, 0.0890401602, 0.0309686381, -0.00859410036, -0.00727661327, 0.0869946256, 0.0273250788, 0.0912422165, 0.0242036991, 0.0311453603, -0.020802971, 0.16884917, 0.023390457, -0.011494942, 0.0450326912, -0.0799407959, -0.0613714755, 0.0293006413, -0.0254077837, 0.0961817577, 0.0673164576, -0.106642745, 0.0756556317, -0.119609937, 0.00969868712, -0.0904721096, -0.0404048115, -0.0239201784, -0.0613796264, -0.0403573252, 0.00890928507, -0.0665615574, -0.026793398, 0.00395689905, 0.00609805994, -0.0335235782, 0.0222840495, 0.0283607394, -0.0275544729, 0.080691807, -0.0175271239, 0.0861111283, -0.101052701, -0.0350018553, -0.0074343998, 0.0489694923, -0.04479919, -0.0272994488, -0.000515452353, 0.11313732, 0.00529505312, 0.0637723953, -0.0843197331, -0.0343549028, 0.0817853212, 0.0610746928, -0.0720800161, -0.0684199333, 0.0722889081, 0.0581635833, 0.0892965198, 0.0583080053, -0.000900680199, 0.0381048024, -0.0110369334, 0.0662589222, 0.059857443, 0.0375354849, -0.0301726814, -0.0731346235, -0.0929167867, 0.054312624, -0.0291669834, 0.0284009241, -0.0290024541, 0.0465549082, -0.11410591, -0.139297336, 0.0127172079, -0.0130840633, -0.0452667475, 0.12527664, 0.00445348769, 0.112321369, 0.109566353, -0.0398729518, 0.0398472846, 0.151911288, 0.0120465476, 0.0567985326, -0.0720740855, -0.0592865236, -0.0561313517, -0.163934529, -0.0104121789, 0.0304081552, -0.0932850093, -0.0522189215, 0.045732826, -0.066893436, 0.0734580308, -0.0794622451, -0.00772430375, 0.0656402558, -0.00430299528, 0.0265939385, -0.0601608455, -0.0750281513, 0.00693067675, -0.00672144443, -0.0678872094, 0.0953256115, 0.121188894, -0.0479607396, -0.000628431328, 0.0833768621, -0.044921536, 0.0608398728, -0.0442973524, -0.0231449939, -0.0572286695, -0.0221622698, -0.0162954461, -0.041878514, -0.192133889, -0.0224961266, -0.0339366198, -0.0900944024, 0.0720057562, -0.0412492082, -0.0521879941, 0.00318414159, 0.028346613, -0.0885099247, -0.000461629592, 0.103174105, 0.0511165485, -0.0606587902, -0.033228077, 0.0603607632, -0.06066975, 0.00644999929, 0.0252265558, -0.0471164212, 0.0586018898, -0.0240608919, -0.0429954156, 0.166241214, 0.0847603455, -0.0853525251, 0.11635372, 0.0768302977, 0.0145210586, -0.12955749, 0.00712409057, -0.0659702271, 0.0281008687, 0.0699765086, -0.013855814, -0.0146459248, -0.0388546735, -0.00915924273, 0.0566541813, -0.0674254894, -0.0491815172, 0.0648297444, 0.0113611426, 0.00847549736, -0.00886135548, 0.0137894098, 0.0638384819, 0.00420870353, 0.090354532, -0.0619390905, 0.171965525, 0.187458158, 0.0527163669, -0.043487113, -0.147247821, 0.033757668, 0.0188759882, 0.00401037186, 0.0405628979, 0.0586508065, 0.0865700543, -0.152879521, 0.0159267597, 0.0652434751, 0.0097250808, -0.0354112461, 0.084558472, 0.0526328981, -0.0632263646, -0.00106894691, -0.00946753658, -0.100315794, 0.0185935926, -0.14264448, 0.0788547918, 0.0478432029, -0.0242307168, -0.0160921402, 0.0731759369, -0.112183109, 0.0706517175, -0.0978575125, 0.0518998057, 0.0293896683, -0.00136082526, 0.120696381, -0.0453348346, 0.091407612, -0.0290567577, 0.074232772, 0.0126435924, 0.0418775305, -0.0812566578, 0.105791613, 0.0246349741, -0.0152652264, 0.018106509, -0.0737674311, 0.150271326, -0.215129614, 0.0300735831, -0.113408081, 0.0650518909, 0.0222016051, -0.0797848776, 0.0827352777, -0.00763365626, -0.0335478373, 0.0528862737, -0.0798040032, -0.0421789326, -0.0122761875, 0.0529228002, -0.0549547821, 0.100646958, -0.00234978111, -0.00746429106, -0.0555395149, -0.173543662, 0.0105401687, 0.00531535782, -0.0594168641, -0.129437089, -0.00683795381, 0.108063489, -0.00755071267, -0.109399363, 0.114717439, 0.104691789, -0.0698268041, 0.028761737, -0.0772326216, -0.044201903, 0.0836420134, -0.0357559994, -0.0959446877, 0.016582489, 0.104911201, 0.0475973561, 0.0710235164, 0.0856918842, -0.0608736686, -0.00993047655, -0.0893506557, 0.0339855142, -0.0493616611, -0.137649253, 0.130620331, 0.0248426832, 0.034240786, -0.0214420035, -0.0842188001, -0.0435745195, 0.115031354, 0.0328332856, -0.0987135395, 0.0862497985, -0.0302738771, -0.0708632991, 0.0572016239, -0.0762674138, 0.0691025257, -0.037434496, 0.0217761323, -0.0370992795, -0.0456319712, -0.0147401839, 0.0181538314, 0.0726551414, 0.00899257138, -0.0270052366, -0.0836559385, 0.0980546325, 0.061095994, 0.000828944147, -0.057132408, -0.0950826257, -0.0256363545, -0.0929112732, 0.0425492786, -0.0024689571, -0.0306376722, -0.0523114949, 0.101528853, -0.0523844846, 0.0640822276, -0.0737137944, -0.137838081, -0.0076995492, 0.136963502, -0.0478355587, 0.0325510614, 0.111381933, 0.117927238, 0.10202948, -0.0806948617, -0.0648256764, 0.133120418, -0.00224611163, -0.0104684122, -0.000627145171, -0.0603796095, -0.0283243842, 0.0665622652, -0.142835289, -0.0274916962, 0.00142771378, 0.0558498278, -0.0643476769, -0.00676162913, -0.053988494, -0.00484051928, 0.0715775266, 0.0154943559, -0.00997336302, -0.0383435152, -0.0402208492, -0.0872833431, -0.0233834311, 0.145907968, -0.0435767137, 0.0957608968, -0.028151758, 0.0649675578, 0.190936983, 0.06481345, -0.000855347142, 0.162423104, 0.0394274928, -0.0496312082, -0.0455062985, -0.222967058, 0.0792990401, -0.137906283, 0.149159878, -0.0124643315, -0.0468844511, -0.102703512, -0.0351455733, 0.117990598, 0.106325418, 0.0819974691, 0.0866898969, -0.0903978422, -0.0957485512, 0.0534124188, -0.0865085721, -0.0171378478, -0.0201135948, 0.065308623, -0.0143852551, -0.102555662, 0.0376451202, 0.00103474874, 0.0305470023, -0.0194290355, 0.0443652645, 0.0108052883, -0.050805755, -0.0560781658, -0.0568571538, 0.0239526071, 0.0536852479, 0.0659016892, -0.00530015863, -0.113984883, 0.00188809633, -0.00598471193, -0.0527855679, -0.00734733976, 0.0682486147, 0.0730547756, 0.074361369, -0.0592212304, 0.123616904, -0.0555166192, 0.0351577625, 0.0318785086, -0.0688275099, -0.0140260011, -0.113746852, 0.0592081994, 0.0959497392, 0.0216836743, 0.0712018013, -0.0673099607, 0.103493616, -0.0469349474, -0.0424249321, 0.0547314994, 0.111671314, 0.0592016429, 0.0379485413, 0.083008185, 0.0462957546, -0.00969570689, 0.14310959, 0.0635819286, -0.120568633, -0.105409615, -0.0384053178, -0.0211726725, 0.0320640057, 0.0474545248, 0.00662817247, 0.0142514175, -0.0209808461, 0.0332401618, -0.048783768, -0.0646389797, -0.0202070791, 0.0606515482, -0.0727318227, -0.0261643417, 0.0628451109, 0.011384422, 0.0278099049, 0.0245810207, -0.0205679573, -0.080847986, 0.0436471552, -0.0715225264, -0.0238368548, 0.0790551603, -0.00950204767, -0.0530045927, 0.105068803, -0.00632932503, -0.0153049761, -0.0635962635, -0.00862434041, -0.0106838793, -0.0973426327, -0.0257954448, -0.124228589, 0.0763272569, 0.211909845, -0.0236179382, -0.0810620636, 0.0319620222, -0.002163684, -0.0705077499, -0.014357605, 0.0262934938, -0.0343292169, 0.0361409076, -0.103956789, -0.0340285748, -0.0602297559, 0.174030885, 0.0790194348, 0.0161414575, -0.0282022953, -0.0180360191, 0.0213341229, -0.00993218832, 0.0482341982, -0.0360355154, -0.0160495229, -0.0549918339, -0.0281617641, -0.215279579, -0.0329001322, -0.13107945, -0.0194422733, -0.0811705217, 0.0703393519, 0.0948659852, 0.0860955417, 0.00298020244, 0.0174867325, 0.104314342, 0.00757317059, 0.0873776898, -0.109705932, -0.00641422626, 0.0342337042, -0.0431328341, 0.140281439, -0.0141475201, -0.00715182908, -0.0821413025, -0.166424349, 0.0175308995, -0.00971734151, -0.0294843055, 0.024879612, -0.0663464367, 0.0145991985, -0.113094434, 0.0108234081, -0.0424563773, 0.0702047348, 0.146885216, 0.0739716291, 0.0807786584, -0.0294531658, 0.0644897372, 0.0465509035, -0.140208289, 0.0105558988, 0.061719127, 0.119625054, 0.122069746, -0.00659644231, -0.0888892189, 0.0391467549, 0.0318171196, 0.0392123535, -0.0693224147, 0.03465968, -0.0476835184, 0.0632190555, 0.00752518512, -0.0693088621, 0.0556228012, -0.034609288, -0.0562940314, -0.0935908407, 0.0894165337, 0.0460318811, 0.0946106911, 0.0970253497, -0.0378115699, -0.0580373146, 0.00685130805, -0.0240787845, -0.0655495301, 0.0920475721, -0.0572968684, 0.0907118097, -0.000337135047, 0.0958020017, -0.00220216811, -0.105195656, -0.00343512697, 0.135109693, -0.0170508716, -0.0159937311, 0.0629626587, 0.038738329, 0.043182198, -0.149704367, -0.0275805071, 0.0830653906, 0.135414079, -0.0911396965, 0.0255063958, 0.0678325221, 0.117846638, -0.0977108777, -0.0146968234, 0.0410707369, -0.0079479944, 0.00758772902, -0.0975005254, -0.0584881231, -0.0411358178, -0.0954357386, 0.0131467246, 0.0884373337, 0.0314341597, -0.0540474504, -0.131020159, 0.00755074248, 0.00428653974, -0.0513308756, -0.144464895, -0.0465611182, -0.0106990952, 0.166800812, 0.0565037616, 0.0638967529, 0.0368259996, -0.00591901131, 0.0741597861, -0.0822639316, -0.0216166861, -0.0142547525, -0.105811425, -0.129464537, 0.00880646706, -0.124055475, 0.0486171208, -0.0312933289, 0.0335986391, -0.0956721902, 0.0666646883, 0.00134075899, -0.0241167396, 0.0286073964, -0.0168476515, 0.0488022156, -0.204614803, 0.119252726, 0.0173368528, 0.0164972693, 0.0484212488, -0.00370501354, -0.0814251751, 0.0140291722, 0.0981728882, 0.0892434344, -0.0246675052, 0.0102536585, -0.0505557954, -0.0823860988, -0.132501259, 0.0507950634, -0.0830733478, -0.0402466208, -0.121927015, 0.0505604818, -0.0569023155, -0.217993006, 0.0493810214, -0.069898285, -0.109336302, -0.00529927202, -0.0074481531, 0.00809708796, 0.0706185475, -0.0761374906, 0.0308077484, -0.0390697792, -0.0364637785, -0.120178454, 0.0378564, -0.014556909, -0.0459425524, 0.0791534483, 0.00495853275, 0.100030519, -0.0384478159, 0.0553810075, 0.0197767988, 0.0948791057, 0.0416829251, -0.0923174024, 0.0716896504, -0.0207008142, -0.128450945, -0.00730367564, 0.0726294816, -0.0313276686, -0.143590629, 0.0255806707, 0.0434266813, -0.0224328507, -0.0891770571, -0.0527072251, 0.0488626324, -0.0659937114, 0.0346077457, 0.00469872728, 0.0800054744, 0.0616751239, 0.133224607, -0.0785946772, 0.0515422523, -0.0605530702, -0.0692069903, 0.0869517401, -0.113503605, -0.0688326433, -0.0344808921, 0.0939441845, -0.0693285838, -0.129364058, 0.0331576131, 0.00330016902, -0.060806904, -0.0473938957, -0.0382475108, 0.163586751, -0.0755013227, -0.00396516128, -0.0122583583, 0.0928661376, -0.0399830714, -0.0281913932, -0.0356783494, -0.0565432012, -0.174874783, 0.00862659141, -0.0120314248, -0.10457021, -0.0178394355, -0.0528360493, 0.0537608564, 0.00123192556, 0.00244560465, 0.12382669, -0.119202323, 0.0578210056, 0.0637606233, 0.00625109719, 0.0115161706, -0.0988153443, 0.056037128, 0.0449979082, 0.0104337549, -0.0543784313, 0.0196551364, -0.0442993864, 0.0959204882, -0.10798794, -0.116974369, 0.0091380924, -0.0100636166, -0.0393831953, -0.0654226393, -0.0669216812, 0.0244851075, 0.0065101916, 0.00610528141, -0.106983304, -0.106025919, 0.00486871041, -0.0126079768, -0.0479022302, 0.023387013, 0.0537120663, -0.0453917272, -0.0491301902, 0.0628812015, -0.00236194581, -0.00814808439, 0.0227814056, 0.0942559615, 0.020572044, -0.116628557, 0.025704002, 0.0473104045, 0.00108542852, -0.0587278195, 0.0383057073, -0.0542852655, -0.0688491538, -0.0918664262, 0.00669162348, -0.10958086, 0.122720167, 0.0522697493, 0.0986699238, 0.106197536, -0.0432841703, 0.169561595, 0.117332898, -0.101258755, 0.0558797084, -0.125172824, 0.0544885956, -0.0112890974, 0.0185600091, 0.0578551888, -0.0466390587, 0.0376987047, 0.0864820108, -0.00115627423, -0.103971407, -0.00704975054, -0.0842340961, -0.204760641, -0.0627957657, 0.0418024473, -0.0980946198, -0.0473582223, -0.165247455, 0.0316605121, -0.00382990995, -0.0291041918, 0.0644813552, 0.0037751901, -0.0172346979, -0.0422124676, -0.0885811895, 0.0166758206, -0.0435407236, -0.0773774311, -0.0941780284, -0.0396579728, 0.0649015829, 0.0159331262, -0.0516304076, 0.0835015997, 0.00978837535, 0.0443133749, 0.0297001377, 0.02662565, -0.0238366965, -0.0462984852, 0.102302514, 0.0762243196, -0.0488283187, 0.0705497861, -0.0327157043, -0.11041598, -0.131304458, -0.0191016868, 0.0133641809, 0.0544066913, -0.0260483604, -0.0965383798, 0.0911923945, -0.0630287379, 0.0826769471, 0.133001104, -0.00473366678, 0.117705062, -0.0240012761, -0.00132794864, 0.0508191586, 0.0196961872, 0.159875497, -0.130224124, 0.0234762207, -0.0394301713, 0.018752683, -0.126942426, -0.0310703404, -0.0265759863, 0.0904723406, 0.0263345651, 0.000180898234, -0.00895390101, -0.139537156, -0.00722809602, 0.00720465649, -0.0559882782, -0.0860758871, 0.127098158, -0.0140588926, -0.0518677309, -0.0136835892, -0.0306002814, -0.0346528962, -0.0281581506, 0.0666721463, -0.115534246, -0.0981145948, -0.0289623868, -0.042298682, 0.0434158035, 0.0336587578, 0.0614327639, 0.0575813316, 0.0614780337, 0.0796466991, -0.0453872308, -0.0191985294, 0.135225505, 0.123685859, -0.0242740791, 0.0496836677, -0.0200163014, -0.00225748867, -0.0373399705, 0.00826786831, -0.014817981, 0.0557427146, -0.0234015342, 0.0436130874, -0.00313477032, 0.0691500381, 0.0741273835, 0.0460153595, 0.0242686737, -0.104999177, -0.0285043865, -0.171705365, 0.145800456, 0.0221375152, -0.00735259522, 0.0132935327, 0.0232473984, -0.112734877, -0.0114636961, -0.0499154553, 0.0371822603, 0.144290581, -0.0236323997, 0.0746450275, -0.00084541738, 0.0358160064, -0.0982175469, 0.0101916995, 0.0164498053, -0.0282862056, 0.112586729, -0.0157094374, -0.0454060249, 0.0233968291, -0.048598811, -0.071312651, 0.0603617281, -0.0299381651, -0.001147056, 0.0363889188, 0.0820527822, 0.0915727168, 0.00140509382, -0.0425595418, 0.0359408632, 0.0342875011, -0.0242629163, -0.0147682372, -0.0239619911, -0.0616740361, -0.106484808, -0.00417627115, -0.0359819755, 0.178155974, 0.0617378056, 0.00666147145, 0.07771945, -0.128619179, -0.063391149, -0.0276715122, 0.02143934, 0.112703092, -0.048061125, 0.0585327521, -0.0517405607, -0.0120576713, -0.0157191195, -0.14012593, -0.0363316238, -0.0819730535, 0.027305495, 0.0567959249, -0.00592879578, 0.0371960476, 0.0609055422, 0.0134695498, -0.0132031692, -0.0557713658, 0.015527321, 0.0689506158, 0.104819506, -0.014489511, -0.0784410834, 0.0254593417, 0.0180023275, -0.0046950113, -0.147947267, -0.0200401265, 0.106144421, -0.0275860094, -0.0517215878, 0.0516379327, 0.112819403, 0.0810719505, 0.034373235, -0.0147770941, 0.0814909488, -0.119913943, -0.0797332674, 0.018588502, -0.0902142748, 0.0192847736, 0.0663855523, -0.00207715854, -0.0844640508, 0.0395605639, -0.0880021155, 0.0426400639, 0.0728933513, 0.0677083433, -0.0474901125, 0.00312681869, -0.14532721, -0.111008584, -0.0410129428, 0.0849896818, -0.0987597853, 0.0398582518, 0.0964793861, -0.0304511748, -0.153164774, 0.00261903834, -0.0031320611, -0.0169175528, 0.014321099, -0.0595640317, 0.0555091128, -0.0140340831, -0.134952247, 0.00902788155, -0.108637534, -0.0187828317, 0.115464345, -0.0165707469, 0.119169354, -0.0362934433, 0.00672626123, 0.0907325149, -0.00682189502, 0.146521851, -0.0830077678, -0.120897137, 0.127929941, -0.115087472, 0.0116726132, 0.0962724537, -0.045083411, -0.15104124, 0.0840260535, 0.0407922938, 0.0877076387, 0.0777267292, 0.0350440107, -0.0656366274, 0.0713185966, 0.0618479177, -0.10615126, 0.0526302494, -0.0329756998, 0.160746917, 0.0684841126, -0.0272260159, 0.0634056702, -0.1046855, -0.0855556726, -0.0170933641, 0.000779412687, 0.0131857395, 0.0752171651, -0.048603531, -0.0176196843, -0.021763932, -0.0501052067, 0.0336745158, -0.0360268988, -0.0449153185, 4.29404899e-05, 0.0571754873, -0.0033179298, 0.0603400432, 0.168848693, -0.0462715253, 0.0458389819, 0.029579103, -0.0101604685, 0.033889018, 0.0622398555, 0.051276058, -0.0375341959, -0.0438668318, 0.0143896788, -0.0366873965, -0.00446784124, 0.0593102835, 0.0402583517, -0.0951602682, -0.180572614, -0.0796765611, -0.190664366, -0.0470530353, -0.0576060265, -0.0824119672, 0.0122747859, -0.110321932, 0.03454623, -0.0523498654, 0.0735493973, -0.0132928854, -0.00104576163, -0.0827548802, 0.0604652017, 0.0155662512, -0.0757914558, -0.0429328866, 0.0148150176, -0.0697317421, 0.0528019294, -0.0969544649, 0.111104771, -0.196005717, -0.0987585634, 0.0712072104, 0.00649388041, -0.0332998447, -0.0260967277, -0.0369820669, 0.0213686749, 0.0171974748, 0.123341791, 0.000567279756, -0.056413956, 0.0690545887, -0.0805647224, 0.00467581116, -0.0327795148, 0.0471625067, -0.0631929487, -0.0601705611, -0.0225944482, 0.0228578821, -0.0516695455, -0.0419914871, -0.0148608834, 0.196023926, -0.0900745094, -0.0365177616, 0.0983268544, -0.0211878717, -0.00590895489, 0.0804941356, 0.0306762606, -0.0259889401, 0.0064141457, -0.0201188475, 0.045681648, 0.116616346, 0.031765677, -0.056428425, 0.0712942854, -0.0335800052, 0.124227926, 0.135445073, -0.103780881, -0.0415219292, 0.0239031091, 0.0332115144, -0.0683033392, -0.112730265, -0.013637932, -0.0741279274, 0.1100403, -0.0143038603, 0.111749701, 0.0307638887, 0.0331706181, 0.0272779148, 0.0609667897, -0.055300042, 0.0078124404, -0.0154411234, -0.0340315588, 0.0390034989, 0.107351936, 0.0303496346, 0.00232033804, 0.0530956686, 0.0861958787, -0.0758782923, -0.015927013, 0.0752552003, -0.00799689069, -0.0265250653, -0.010232335, -0.0755146593, -0.0187492482, 0.0497631207, 0.0227313042, 0.086643979, -0.0903109387, 0.0361445211, 0.0851439014, -0.0371047631, 0.0125641655, -0.0443306118, 0.0184564423, 0.0641649738, -0.00154084526, -0.0506638959, -0.0268343985, -0.0993898287, -0.132515728, -0.0298210531, 0.031581834, -0.0476533435, -0.0211789683, -0.0385781489, -0.0643052086, -0.102327302, -0.0622971244, -0.0804271996, 0.0161505565, -0.083058618, -0.0220388602, 0.0415044576, 0.00775893964, 0.100917056, 0.0302919801, 0.0594701506, -0.032192573, -0.109479927, 0.00380911306, 0.0257576611, -0.0429031029, -0.0120052826, 0.0295684189, 0.132145762, 0.0901322439, -0.0651533455, 0.0392933302, 0.0356644392, -0.0225292798, -0.1250287, 0.0637708455, -0.12362133, -0.0713968426, -0.00440163491, -0.129764214, 0.0308040008, -0.123995245, 0.0727155209, 0.0359779857, 0.0557515621, -0.00788295828, -0.0418291837, -0.0556169599, 0.0073938407, -0.0131131299, -0.09903799, 8.13147053e-05, 0.0302125141, -0.0278899334, 0.0535467304, -0.0798689798, -0.0573887378, -0.0173641667, -0.00622116029, 0.0335880443, -0.0624668077, 0.0515625998, 0.11595048, -0.0661625415, 0.10432899, -0.11084725, 0.0875949562, 0.0392709337, -0.0364517421, -0.0743830502, 0.00235208124, 4.60073352e-05, -0.0377354324, -0.0205002762, 0.139248654, -0.00987232476, 0.0279238559, -0.0376371965, -0.0748126581, -0.14912799, 0.0279988665, -0.0754584074, 0.0367791727, -0.0684543997, -0.120797753, 0.210929647, -0.0683470666, 0.0416743346, -0.00167389307, -0.03560495, -0.0740633756, 0.0182297807, 0.0579238199, -0.0464916304, 0.0312767625, 0.0230260603, 0.00420898199, -0.00905129593, -0.0361692533, 0.0551778674, 0.0748246461, 0.0900884718, 0.106486678, 0.046182286, -0.0436386056, 0.0318417326, -0.0593780093, -0.0390714593, -0.00232599862, 0.0168671533, -0.00128097087, -0.0234770365, -0.207413524, 0.091397658, 0.0404496193, -0.0955121964, -0.0953916684, 0.0376782902, 0.0643178821, 0.0802147463, -0.069396995, -0.00916909426, 0.0369172953, 0.0255105644, -0.0491899848, -0.032136552, -0.107756861, 0.0107436292, 0.019768646, 0.0980418399, 0.0568639934, 0.0204656459, 0.0187228061, -0.00544637628, 0.0828665942, -0.00240248069, -0.0522129759, 0.0143650025, 0.0482954122, 0.0405194908, 0.117483482, 0.0239349958, 0.00080441311, -0.0541618094, 0.0940204933, -0.105444238, 0.118430451, -0.0870203078, -0.123753317, 0.0329259448, 0.0420681946, 0.132282391, -0.0484123155, 0.000465761404, 0.146358669, 0.177483767, -0.0771356225, -0.0731008649, 0.0138120726, -0.0384135433, 0.0724786445, -0.0743359923, -0.034141764, -0.0258353278, 0.0891263932, -0.0614453405, 0.149894118, -0.0627272725, -0.0523161069, 0.0335989147, -0.041771844, 0.0213093907, 0.0459769294, -0.00445639715, -0.0234814584, 0.103136525, 0.0533659272, -0.022723956, -0.0382430181, 0.0330411904, -0.147755891, -0.0439336523, -0.10285791, 0.0145746469, -0.0746227801, 0.0824759454, -0.067650646, -0.11463163, -0.136612028, -0.0311640576, 0.00981829129, 0.00207894668, -0.0804388374, 0.0687851235, -0.00379346497, 0.0771161541, -0.130354851, -0.0437753089, 0.00205173716, 0.0463164002, -0.0175507255, 0.0375224687, 0.10031689, -0.0767227262, 0.0601984486, 0.0444888584, -0.0265136808, -0.084761098, -0.000143888872, 0.0326584131, -0.0210909694, -0.0118333716, 0.118986979, -0.00320465397, -0.0930535793, -0.0411692336, -0.0462614559, -0.0252511725, -0.0238584261, 0.0695445091, -0.00723118708, 0.0638550073, -0.0812215209, -0.171835899, 0.055236809, -0.0854737982, 0.00169022381, 0.108785376, 0.0245490521, -0.0220617913, -0.121044368, 0.0211217031, -0.0161820352, 0.151667625, -0.092914477, -0.110812977, -0.0416993797, 0.0688993037, 0.0716673583, 0.0323226042, 0.0435284115, 0.0607336052, -0.048121959, -0.0266444664, -0.0232259948, -0.012700025, -0.107227765, -0.0672004223, -0.207843721, 0.037615329, -0.0249993652, -0.0910415351, 0.157347187, -0.0610164329, 0.191035032, -0.0491201542, -0.0428905301, -0.0213949382, -0.0874956697, 0.10035333, 0.0531928726, 0.0230856277, -0.0840579718, -0.0603243746, 0.0622626655, -0.0587715544, 0.0670978352, 0.0656613708, 0.00271900184, -0.0609509796, -0.0492823869, -0.0401115902, -0.0509398505, -0.0496883169, 0.065441981, -0.0381773636, 0.0243011992, -0.00364368455, -0.00995516777, 0.0427191481, -0.127105564, 0.0633584261, -0.0931454301, 0.049144771, 0.0516123921, 0.0413496122, 0.00990300626, 0.048000738, -0.0535469465, -0.0971256196, -0.0142761804, 0.0540780574, 0.0527291261, -0.0447016656, 0.081862554, -0.0444602482, 0.0722750202, -0.0399135537, -0.0010391192, -0.0163113624, 0.0631549135, 0.0347271562, -0.0251329131, -0.0387175083, 0.0111792628, -0.0346063338, -0.071156919, -0.046510119, 0.107706293, 0.0824263543, 0.0127300788, 0.127644643, 0.016475996, -0.0238917824, 0.151583269, 0.114829041, 0.0530352108, -0.0179952569, 0.0800536871, -0.070317775, -0.152198091, -0.04821942, -0.0494440272, -0.024356192, -0.0940830857, 0.0912103504, -0.119127162, 0.066063486, 0.00056592375, -0.011524695, -0.00827786606, 0.0117728822, -0.0889376029, -0.00546765141, -0.0990630835, 0.145165592, -0.00199469179, 0.12126606, -0.0608006977, -0.124840729, -0.0649535656, -0.144844249, 0.0948657542, 0.0110113937, 0.0435435511, 0.0776191503, 0.0173303783, -0.0691903085, -0.0406034701, 0.0872050077, -0.0880143195, 0.021160692, 0.114508845, 0.157790467, 0.0701552182, -0.140762731, 0.0232453775, 0.0812149644, 0.0195620134, 0.0553476885, 0.00700753927, 0.0144191021, 0.0325794406, 0.00836092979, 0.00485529378, -0.150897592, 0.137030959, -0.0338992923, -0.00199312624, 0.0158948619, 0.0711862817, 0.0803703815, 0.00394163653, 0.0166742392, -0.0637132823, 0.0576172471, 0.0989794806, 0.0588038862, -0.017602291, 0.0131374076, -0.103191964, 0.149016008, 0.0303576104, -0.00741250627, 0.0757397935, -0.014678305, -0.0112621728, 0.03361753, 0.0766832829, 0.0150260366, 0.0720072687, 0.140976176, 0.0125573575, 0.0717029348, 0.00362505531, 0.0787613168, -0.084628731, 0.044434987, 0.0376896113, -0.0569761284, -0.0480788872, 0.0425903611, 0.0584106147, 0.149757862, -0.00124625303, 0.0625538826, 0.0381772146, 0.00189108262, -0.0102716405, 0.147797242, -0.0874876529, -0.0679499805, -0.00844030268, 0.0668255314, -0.0102202641, 0.0443724021, 0.00881034881, -0.0599477515, 0.0419975035, -0.109376848, 0.031993825, 0.175400287, 0.0698224381, 0.0410628542, -0.150160089, -0.0284209065, 0.022347793, 0.00905410666, -0.0653152615, -0.0166206267, 0.21127218, 0.0454411879, 0.103180595, -0.0458617359, -0.0995125696, -0.0363291949, -0.0063140206, 0.0859165043, 0.0356240943, 0.0178990569, 0.0507258661, -0.0424911156, 0.032425534, 0.0798085704, 0.013637729, -0.072872974, 0.0755365044, -0.15487203, 0.0912024528, -0.121919304, -0.0774344206, 0.0649062693, -0.047781039, -0.0749223232, 0.114782691, 0.0160173289, -0.00308426097, -0.0619944185, 0.0919422507, -0.0676485077, -0.0958780199, -0.0106051993, 0.10275393, -0.0781324804, 0.0431928039, 0.00466829911, -0.0837497413, -0.017176494, 0.0481531695, 0.138138577, 0.105663054, 0.00645310851, -0.0261352975, 0.0743861869, 0.0354747064, -0.0858714581, -0.109296694, 0.069152981, 0.029206302, -0.17600356, 0.0795082301, -0.0715349987, -0.0060289707, 0.0259194784, -0.0387955941, 0.0371407866, 0.170553535, 0.0257288963, -0.0508159474, -0.0873826891, 0.0374071039, 0.0141317174, 0.00928837713, -0.0462122709, -0.0323836878, -0.111822888, -0.0685174242, -0.11734613, -0.0474074483, -0.0817076787, 0.0350165591, -0.154563427, 0.0498186871, -0.0998867452, 0.0855002999, 0.0407505259, -0.0847005695, 0.126987442, 0.00445590727, 0.148815557, 0.0157598257, -0.0677889213, 0.0678885877, 0.103936262, -0.0291266404, 0.108563244, -0.0531429797, 0.0151067507, -0.0193862207, 0.0237437859, -0.0711940601, 0.0665370151, 0.0799864382, 0.0235979799, 0.0302098636, -0.0391180962, 0.109693781, -0.0150751481, -0.0459537059, -0.123312064, -0.0431641638, 0.101107523, 0.0692357495, -0.0784172863, 0.0979446694, -0.029822316, -0.0326684006, 0.058933042, 0.0962768197, 0.0850250125, 0.032953918, 0.0947572589, -0.0437288508, 0.0137972319, -0.016414253, -0.00187447667, -0.0200755466, 0.0115629043, -0.0379117168, -0.0243147463, -0.0448954776, 0.0678378791, 0.000306433998, 0.0608597174, -0.0208371188, -0.0125763938, 0.00191673636, -0.0388574079, 0.0198504198, -0.0477382392, 0.0470644236, -0.0107967202, 0.173992619, -0.102686241, 0.0256157219, -0.0265013464, -0.163954511, -0.155132473, 0.12658456, 0.0500281639, 0.113883637, -0.00256442651, 0.0142556829, -0.0291736908, 0.0763308406, 0.0677200407, 0.0141491592, -0.0876829028, -0.0043666102, 0.0281589571, 0.0958286226, 0.0770577639, 0.0776152313, -0.0528775752, -0.0903838351, 0.0163058825, 0.00771669205, -0.0348566175, 0.0437220633, -0.0509710833, 0.0560960732, -0.00657285191, -0.0746331811, 0.0848636627, -0.0706262589, 0.104398347, -0.00784252677, -0.0019404497, 0.0469817668, -0.0435572118, -0.00113693834, -0.0457589179, 0.010874318, -0.0671563074, 0.024623489, 0.0105352551, 0.132269993, -0.0817873329, -0.0788935944, -0.040544644, -0.0617846958, -0.045770146, -0.0200390257, -0.145366877, -0.125423431, 0.0690955371, 0.0694849268, 0.0396142192, -0.0329445079, 0.0800578892, 0.0373657644, -0.0451677516, -0.0645712614, -0.0983189866, 0.00463890284, 0.0835429803, -0.0858966112, -0.0550517738, 0.0273464136, 0.0102375317, 0.0260891337, 0.0637064651, 0.00832006708, 0.0627907887, 0.0263583213, -0.0573627055, -0.0497084148, -0.123706594, -0.0853701085, 0.00854441524, 0.0208358113, -0.00285715237, 0.00765209273, -0.0266407281, -0.011619661, 0.0538106933, -0.120938472, 0.0332855321, -0.00340719614, -0.0140140066, -0.0576705113, 0.0325996391, 0.00708473613, 0.0657776147, 0.125871018, -0.0396783389, -0.0111825448, -0.0575863793, 0.101352975, -0.00209203176, 0.0176176727, -0.0766469836, 0.0313168392, 0.117277868, -0.0965819955, -0.103153199, -0.12177901, 0.0318619497, 0.0340569839, 0.0417677611, 0.205428436, -0.0218155142, 0.0979215279, -0.0488391891, 0.0437722132, 0.0320034884, -0.176868066, 0.0120335966, 0.0552526861, 0.13601996, 0.00721526891, 0.0537095554, -0.00682887249, 0.066698432, -0.0331088603, 0.058147911, -0.00401602685, 0.122633085, -0.0158447456, 0.142422378, -0.0176462829, -0.0290186554, 0.0217498466, 0.094007045, 0.0252387803, 0.00824793242, -0.0841873437, 0.122685328, 0.0434680283, 0.0487815365, -0.00721960329, 0.0800359696, 0.104408838, -0.0127684064, 0.0803305358, 0.0346615277, -0.032716807, -0.011786636, -0.0229381695, -0.0916494429, 0.0812630504, 0.0130644422, 0.027639389, -0.0231682099, 0.0505290926, 0.0093316352, 0.11424952, 0.0581807382, -0.0550244935, 0.0636840761, -0.0720747635, 0.10009405, -0.0246030726, -0.0192512758, 0.00266349874, -0.0312189572, -0.0594217815, 0.0872601718, -0.0480652973, -0.122673392, 0.0865379944, 0.137365401, 0.037465483, 0.0619018823, -0.0269445628, -0.0328418948, 0.110974364, 0.0480593592, 0.0864270777, 0.0263310969, 0.00914893672, -0.00284557976, -0.0217671227, -0.208772793, 0.0288814195, 0.082782194, 0.0077932477, -0.079423517, 0.0557791069, -0.003898561, -0.0291814711, 0.0399448611, -0.212592274, -0.126046807, -0.0656942427, -0.00784858316, -0.0898812488, -0.038078744, 0.00671042874, 0.0882877707, -0.106805675, 0.0206672121, 0.041465424, -0.0600041747, 0.0516393073, -0.0254743993, -0.00919895619, -0.0451346785, 0.0543551184, -0.0814894438, 0.0576454438, -0.0658828095, 0.104196236, 0.104056939, 0.0577372834, 0.0187297054, -0.1470038, 0.0328220278, 0.170873776, 0.0212486815, 0.00120717101, 0.0415091738, 0.0503896177, 0.0504891835, -0.114958778, 0.0143279154, 0.0389872454, -0.13502562, 0.104704447, 0.0744781494, 0.0312258564, 0.033509139, 0.00126305455, 0.0864359662, 0.0316561647, 0.0597085692, 0.111281879, -0.106449686, 0.0440641195, -0.0202647336, -0.0856270716, 0.0558689423, -0.0269347504, 0.0359246768, -0.00160080194, 0.125313014, -0.0114528965, 0.00402942672, -0.00101586059, 0.137872115, 0.0583958626, 0.00933099166, 0.124417253, -0.139215901, -0.0709310174, -0.147631377, -0.0317863114, -0.0459677838, -0.0470133126, 0.0606892928, 0.00546924025, 0.00531811826, -0.0243411474, 0.103531994, -0.0519852005, 0.0847287029, -0.044240281, 0.0635881126, -0.0433895402, 0.0413641483, 0.0175644141, 0.00655454025, 0.0130689368, 0.0702279434, 0.0816664398, -0.048228085, 0.13485229, -0.0109039508, 0.103604622, -0.0530207232, 0.048280403, 0.0366703942, -0.139046192, 0.0208499897, 0.0570953153, 0.0474857166, -0.0780786127, 0.0406286307, -0.023971118, -0.0951811895, 0.00127734989, -0.0205095876, -0.0751637295, -0.0296861902, 0.0369220525, -0.0240838528, 0.0758907795, 0.0400747061, 0.0179445073, 0.00428873487, 0.0070068296, -0.0846178532, 0.00317023322, -0.133584976, -0.0213891938, -0.010071286, -0.0526180975, -0.0439036749, -0.0216051992, -0.121510625, 0.0654005706, -0.0649946854, 0.0866615921, -0.00906985719, -0.11152412, 0.112167574, -0.0759050325, 0.0826534778, 0.0364894494, -0.0107544642, 0.0045947358, -0.0329279341, 0.159991831, -0.0640158802, -0.0484168828, 0.00337100029, -0.0512236133, 0.0678056479, -0.0402449071, 0.0908964649, 0.0604753233, 0.0151774399, -0.0899197906, -0.0495723039, 0.213968858, -0.00480384473, 0.0268741772, -0.107549869, 0.0347231999, 0.0437693372, -0.0361597687, 0.0470806845, -0.044883579, 0.0238408744, -0.0446516797, 0.0489419661, -0.0254730321, -0.0200302601, -0.104077362, 0.062718153, -0.0531329736, 0.0116707636, -0.117419451, 0.0254259072, 0.0750542581, -0.00397553854, -0.0665199682, -0.0184707958, -0.00270925183, 0.0763828158, 0.0337355435, 0.0279260315, -0.0583564714, -0.0531061068, 0.0229404271, 0.0293381512, 0.0615486503, 0.0824794471, 0.0113682449, -0.0790008307, 0.00741539523, 0.0823355466, -0.0864413232, -0.116274506, -0.000888613984, 0.0231170058, 0.0744010955, -0.000226739794, -0.0138292881, -0.0131120011, -0.0975422934, -0.0224729143, -0.0196888447, -0.140870899, 0.0356945992, -0.0985943973, 0.123549551, -0.000760247931, -0.0291051362, 0.0804991275, -0.0239255689, -0.0181377307, -0.0692903325, -0.0611725226, -0.0522443131, -0.134671256, 0.18177627, -0.110332564, -0.144453228, -0.106152989, -0.0792289972, -0.052244164, 0.00281627057, 0.0507592373, 0.0200824514, -0.0920186713, -0.142175823, 0.0308848098, -0.0685959309, -0.0735030398, -0.0047179726, 0.0742548928, 0.0716363564, -0.051056657, -0.000936691533, -0.0247088131, 0.0673220307, -0.103734247, 0.113195941, -0.0123151951, -0.0716323107, 0.0879234299, -0.0706144571, 0.0800992474, -0.116462201, 0.0710284188, -0.0274224319, 0.0911740512, -0.0591697395, 0.128571212, 0.00942194462, 0.0112342853, 0.0594393238, 0.122481525, 0.0518759452, 0.00391112827, 0.00459925085, -0.00107023492, -0.0406995639, 0.0181504153, 0.0787359923, 0.0413333066, -0.0773825496, 0.134060547, 0.105162509, 0.100520976, -0.0857238472, -0.0685628951, 0.0463460349, -0.128627837, -0.0599386021, 0.109882325, -0.00504093058, -0.0323709436, 0.0150102321, 0.039100565, 0.00190809369, 0.033697173, 0.00305089541, 0.00202031806, -0.146391481, 0.0123923076, -0.0165218934, 0.0793899894, 0.0192385539, -0.0389196128, -0.0517317243, 0.0559310243, -0.0768021494, 0.0226306207, 0.121306881, -0.0522455648, 0.00339139812, -0.0556291714, -0.0995496213, -0.0963014066, -0.0816042349, -0.11229635, 0.0557814501, -0.0740598366, -0.0173649304, 0.139369071, -0.0306224898, -0.0580060631, -0.091436848, -0.1747071, 0.118114039, 0.02228209, -0.0473897681, 0.0664613992, 0.0720168129, 0.0845688134, 0.0528362468, 0.000815280247, -0.102460355, 0.0476971269, -0.0671160519, 0.0525707528, -0.0415160656, -0.102914102, 0.0113827325, -0.083965674, -0.0490029082, -0.0314759016, -0.0968770608, -0.0548568815, -0.104666732, -0.0537175536, -0.0062415353, 0.10947898, -0.0233759973, -0.117974564, -0.0366625525, 0.0608506501, 0.0428013578, -0.0998068377, -0.118065089, -0.0119977761, 0.124744356, 0.0283070784, -0.0802738294, 0.0655657947, -0.0954824314, 0.0362423845, 0.0332849324, -0.0834430009, 0.0715879798, 0.0472209863, -0.0373611376, -0.0470067151, -0.0612793155, 0.0413198546, 0.0846912786, -0.0206781477, 0.148907751, 0.0997918695, -0.0374904834, 0.0923477262, -0.164048508, 0.0363637581, 0.12508589, 0.0251565874, 0.0373173356, -0.0349174105, -0.0210640188, -0.0291269049, 0.0575178042, -0.0673399717, -0.111204684, 0.000690751011, -0.0608374774, 0.0883233175, 0.0703906566, 0.00799492467, -0.0885908753, 0.0663681254, 0.00513501652, -0.0683957562, -0.0635244995, 0.0509348921, -0.045457378, 0.067822583, -0.0514202528, 0.0347993821, -0.105504952, 0.0464331098, -0.0200170074, 0.124304675, 0.00249845907, -0.139286578, 0.0419195741, 0.138129503, -0.137769043, -0.0693240017, -0.144727841, -0.0269639567, -0.0316476636, -0.00926445797, 0.0155554442, 0.0988779292, 0.0360196903, -0.11852254, -0.146118566, -0.141063496, 0.0180321112, 0.044023633, 0.0607468039, 0.0902918354, -0.0553643666, -0.0225360487, -0.0291328467, 0.120564714, 0.00701142848, 0.0940650702, 0.0386316068, -0.066673629, 0.0376338474, 0.0764669105, -0.0897704884, -0.0251525287, -0.00749431085, -0.0358690172, 0.0398492031, 0.0265903752, -0.0361888818, 0.125865638, 0.054716222, 0.0339330956, -0.0974758416, -0.0556336716, 0.0554950386, 0.0709042475, -0.0551284701, -0.150779456, 0.0356293619, -0.0151905287, -0.0415148139, 0.0461233035, -0.0375088528, 0.0776319429, 0.078568168, 0.0219056439, -0.0641739443, 0.0184024908, -0.0559999272, 0.00853113644, -0.0582099259, 0.0130015435, -0.000109020621, 0.0413256809, -0.0175708272, 0.00443046819, 0.0459968075, -0.0424706116, 0.00485516898, -0.139668763, -0.107954606, -0.033286605, 0.000858554617, 0.0112799844, 0.0316995755, -0.00445954315, 0.0098643275, 0.00362277031, -0.176973119, 0.0289542675, 0.0964407027, 0.0178754423, -0.0725989938, 0.0330223516, -0.0307930931, -0.136516929, -0.0208547302, 0.0932566077, -0.0433047451, 0.127082095, 0.0337875597, -0.0496471711, 0.0266216137, -0.0302028675, -0.0671077296, -0.069399491, -0.194116816, 0.107985169, 0.119947314, 0.116231322, -0.00947291963, -0.0721068382, -0.119167857, 0.0993771553, 0.0410175882, 0.0651499629, 0.113678746, -0.0722037777, 0.0489135459, -0.0615688562, 0.00746499747, -0.0885654688, 0.00774631463, -0.00619787909, 0.0144832283, -0.00118065253, -0.0396787487, -0.000157682225, -0.138799325, -0.094255127, 0.135156259, 0.0337659083, 0.0495264307, -0.00455174129, -0.098026149, 0.13226442, -0.00644892734, -0.0126878396, -0.119426385, 0.106981225, 0.0939402208, 0.0869578496, 0.0459269434, -0.0357407071, 0.0646807551, 0.067193076, -0.0493923053, 0.0898668766, 0.0236707926, 0.00805385411, -0.079227671, -0.087250486, 0.00157636264, -0.091030851, -0.0203078557, 0.0409940705, 0.0134612247, -0.0116334986, 0.0569527075, 0.0660834983, -0.13612771, -0.0281860009, -0.0982794464, -0.0445884764, 0.0251589492, 0.0647347793, 0.0288546849, 0.0464992821, 0.0603758171, -0.0300618839, 0.0956698805, -0.129332364, 0.0559479222];
    CONSTANT bias_0_r : ARRAY[0..63] OF REAL := [-0.173484892, -0.0675045773, 0.0491046086, 0.0463505276, -0.0815096349, -0.110554256, -0.0473120436, 0.437425762, -0.00653401855, 0.176917329, 0.370717168, 0.0396423079, -1.08117795, -0.0953554064, 0.150914401, 0.0577960424, -0.0104229543, 0.249676898, 0.0947834998, 0.126156241, 0.072207287, 0.261239588, -0.102599576, -0.646232307, 0.596568823, 0.280415773, -0.238218173, -0.300266802, -0.174425423, 0.181508452, -0.275678068, 0.177939966, 0.170858145, 0.144983739, 0.305772722, 0.21602802, -0.058799278, 0.16263026, 0.152120188, 0.226213232, -0.139869258, -0.26692462, -8.2628685e-06, 0.244418189, -0.0422431342, 0.486167401, 0.180008084, 0.371829987, 0.247329235, -0.39782384, -0.508523405, 0.0987078175, -0.00799489487, -0.575995445, -0.137379125, 0.00688174972, 0.359871328, -0.0202121828, 0.147642806, 0.0532373562, 0.141280323, -0.153836474, 0.204907924, -0.00387164229];
    CONSTANT weights_0_h : ARRAY[0..63] OF REAL := [0.511881709, 0.529895723, -0.477809012, -0.506132901, 0.537910998, -0.527767479, 0.491260558, -0.324178755, -0.548811018, 0.494253427, 0.363518178, -0.522180617, 0.508872926, -0.535762608, -0.393660396, 0.486902118, -0.543106973, 0.495763212, 0.534182966, -0.454969078, 0.549818516, 0.410422921, -0.523729563, 0.518692791, -0.241631955, 0.380803972, -0.511416197, 0.452509254, 0.450534821, 0.378833294, -0.505145967, -0.454468369, -0.521197736, -0.407331824, -0.358680755, -0.488305509, 0.447431266, 0.542436302, -0.509502351, -0.401503712, -0.546306491, -0.521000624, 0.419856697, -0.42881614, -0.506078959, 0.265747756, 0.523313284, 0.384962797, -0.367372096, -0.544435382, -0.486974597, 0.513249099, 0.413192004, -0.513616383, 0.459577471, -0.420617849, -0.35950458, 0.482437223, -0.450004786, 0.459671527, 0.469759375, 0.540518165, -0.404790819, 0.54321909];
    CONSTANT recurrent_0_h : ARRAY[0..4095] OF REAL := [0.0151014654, 0.0315691419, -0.00384554872, -0.105252482, 0.0954181105, -0.0486003868, 0.0757943094, -0.0748094544, 0.103059046, 0.0163525231, -0.0429565907, -0.0707249939, -0.123956338, -0.0394361317, -0.146633834, -0.103257373, 0.0837373883, 0.0299536027, 0.0506832749, -0.0691065937, -0.0754909143, -0.0278890803, -0.156872854, -0.0413584113, -0.137698248, 0.0687828958, 0.0563442335, 0.018389143, 0.0312211905, -0.0644816086, -0.0680799186, 0.102891371, -0.121650897, -0.0529458225, 0.092071712, -0.00170892943, -0.0130693149, 0.12133313, -0.124405108, 0.15404433, 0.0598416552, 0.0570201501, -0.0286285356, -0.0331414379, 0.0462406948, 0.0842860341, -0.0477161668, 0.0449983403, -0.0474944636, -0.0678177997, -0.0183854587, -0.0297140516, 0.106223077, -0.00322339637, -0.0999261439, -0.0824365318, 0.0240056701, 0.0590381622, -0.0936049968, 0.0295491889, 0.107780747, 0.080072917, 0.0176341012, -0.17420283, 0.0588149242, -0.0870779753, -0.134306341, -0.0692487508, -0.157706246, -0.0270572938, 0.0707601011, 0.149820372, 0.110426478, -0.00743779354, -0.0465169512, 0.0691735372, 0.111401349, -0.0139408177, 0.0205599926, -0.0962041765, 0.0503444895, 0.0740744546, -0.0419505239, 0.0196950305, -0.0837824196, 0.0464542881, -0.0288814493, -0.0535249971, 0.0254174136, -0.0666553527, 0.0397340655, -0.0178836547, 0.0203624424, -0.0447266363, -0.0661628321, 0.0150283603, -0.122055553, 0.0711871386, 0.0188331716, -0.109750815, -0.0493549854, -0.0550094284, -0.00762387738, -0.0353097506, 0.135499761, -0.015370369, 0.0184302274, -0.0249744803, 0.2203383, -0.0442610495, 0.0065962784, 0.0633476973, 0.0377533771, -0.0880632102, -0.0339279845, -0.0212823916, -0.0435293168, 0.0181129221, -0.0127849532, 0.110028744, 0.0964113325, -0.0344761126, -0.0126675069, 0.00523473881, -0.108181819, 0.129458338, -0.154461205, -0.0144926272, -0.0874574408, -0.0518219285, 0.0588002875, 0.014298114, 0.0187594295, -0.0174597241, 0.199162781, 0.134521887, -0.0472685322, -0.0397187695, -0.0142858475, 0.0857593864, -0.0718451291, -0.0385252982, -0.0189274848, -0.0534091666, -0.00660294015, -0.0306221731, 0.0354711525, -0.0566619001, -0.0506171137, 0.0256853756, -0.0265512876, -0.0473412536, -0.0894344822, -0.116834685, -0.0509595014, 0.0759056807, 0.0700788572, 0.00462372554, 0.089258492, -0.0152192153, 0.0457421429, -0.0269401558, -0.0140602961, 0.106877066, 0.123079993, -0.0989074409, 0.0320937112, 0.0529134832, -0.00390504859, 0.0247814283, 0.0754490569, -0.121886, 0.145266309, -0.121950209, -0.0752653405, -0.0901928097, 0.00366103277, 0.0372722931, 0.0210407581, -0.0174527131, -0.0353134423, -0.00717110001, -0.0354144573, 0.0215394534, 0.0330921113, 0.0686442032, -0.0344005786, 0.0645818338, -0.0111237355, 0.0727535784, 0.0465916693, -0.0652130917, 0.106176965, 0.0119006718, -0.0605614632, 0.0079497043, 0.0370872803, 0.00775675802, 0.0357049927, -0.126892924, -0.0222051032, 0.0738216713, 0.0740928352, 0.0294515938, 0.0681039169, -0.0378874578, 0.0758690089, 0.0175420642, -0.0628558099, -0.0672130585, 0.0307014622, -0.0804512277, 0.176019937, 0.132123068, -0.0889720023, -0.0831062198, -0.135356486, -0.143481523, -0.0899433345, -0.0380111784, -0.0449125469, -0.0193431079, -0.0362437889, -0.0266001876, -0.0325177684, 0.0157292224, 0.0499577671, 0.0174572486, 0.0536411963, 0.121578008, -0.0687552541, 0.0890867636, 0.0383188464, 0.0148758721, -0.0303913709, -0.00649094395, 0.0854870602, -0.102338418, -0.0666316673, -0.0281381235, 0.0549249165, 0.0424676798, 0.0872980133, -0.0456232056, 0.022293983, -0.148441434, 0.0569621846, -0.0632671192, -0.0296576694, 0.118491352, 0.0409092493, -0.054831367, -0.105856366, 0.0819140747, -0.128674701, 0.0155766308, -0.00430044997, 0.0650782585, -0.08370094, 0.0713149831, 0.0574905761, 0.0671258867, -0.0950446203, -0.0663676858, 0.0711896271, 0.00114663318, -0.00647407491, -0.119475968, 0.160537824, 0.0439400226, -0.0349544063, -0.012381129, 0.0524228588, 0.138963565, -0.100225538, 0.00670948718, -8.71550292e-05, 0.160157681, 0.0178130865, 0.02238499, 0.0803312287, -0.00828377903, 0.00724661164, 0.0321915038, 0.0242249686, 0.0313558206, 0.00169815496, -0.042619694, -0.0616292879, -0.0522229746, -0.0935247093, 0.153820843, 0.0857300758, -0.172498316, -0.021524474, -0.0319245197, 0.0929623768, 0.0532867275, 0.0314655602, -0.0274347682, -0.0879180729, 0.0986205786, -0.0337646529, 0.0416346788, 0.0332635641, 0.0381301343, 0.079621613, 0.0737273619, -0.0366122052, 0.119512878, 0.0474161692, -0.211196274, 0.0176645368, 0.0787715167, 0.0302956551, 0.0390346721, 0.00925036147, -0.0182805713, -0.041102685, -0.0138021689, -0.0270654373, 0.0491370782, -0.0514427237, -0.0751671568, 0.0477790311, 0.0277377404, -0.0619665608, 0.0156615973, 0.00482634781, -0.00682761334, 0.00939017069, 0.067990765, 0.137770802, 0.0574506521, 0.0701330528, -0.0982482061, -0.0862303302, 0.0904136226, 0.0466973111, -0.0325784385, -0.000851515681, 0.0318356156, 0.0433966741, 0.00800497457, -0.00970953703, -0.0271797776, 0.0797721297, -0.118577689, 0.0206320807, 0.017929947, 0.0955219716, 0.17246969, -0.0278012976, 0.0755585432, 0.079024449, -0.0478332341, -0.06807217, 0.0914565176, 0.20822309, 0.0121487696, 0.0471593961, 0.0288373716, -0.00932216831, -0.149716005, -0.0538578369, 0.0268720426, -0.0361705907, 0.117366888, 0.0253876261, -0.0262836274, 0.0496964678, -0.0192397106, -0.0702153593, -0.0391614847, -0.161675587, -0.136856928, 0.0672038645, -0.0700094998, -0.00911142305, 0.038635321, 0.0767850429, -0.0122583732, 0.183748305, 0.0132101532, 0.0678323731, -0.211896747, 0.0235066377, 0.0453544036, -0.0898434073, 0.103501424, -0.0940179378, -0.016603183, -0.00502588693, 3.42298299e-05, -0.013213018, 0.0565248802, -0.0319322944, 0.0672975481, -0.0400523022, -0.134900898, -0.0601539873, 0.0332695991, -0.0905719399, 0.0467153937, -0.0810768381, 0.127729416, -0.0900901854, 0.0902750939, 0.0299907867, 0.0586670302, 0.0495708399, 0.1158012, 0.0336007997, 0.00532219745, 0.123860262, -0.0363541022, 0.0275619552, -0.00662331656, 0.109502621, 0.0298098996, -0.00811201707, 0.0412303284, -0.0805860385, -0.0472148471, 0.102457054, 0.0257757008, 0.0102556758, -0.0890942737, -0.0421103425, 0.0365854949, -0.0659021437, 0.111958601, 0.0964360982, -0.046282202, -0.0126719587, -0.0458573662, 0.116932459, -0.0212433711, -0.0881072953, -0.00770005584, -0.0857032984, 0.0025970079, 0.0132948514, 0.0339403749, -0.0626496002, -0.0146684814, 0.0161503572, 0.000780121423, -0.032719072, 0.0686777085, 0.0906086937, -0.0502825528, 0.0462821573, -0.180640206, 0.00406896137, -0.0251903422, -0.11153277, -0.0614060163, 0.0169649497, -0.00545855705, 0.0387234055, 0.061546132, -0.0173524842, -0.0139072761, 0.0299902521, 0.00907874666, -0.00572424382, -0.0507996082, -0.0923170522, 0.0297425594, 0.0514120758, -0.0830440968, 0.0198585112, 0.0656371266, -0.0585631095, 0.0178769249, -0.0531284511, -0.0271281898, -0.140999585, -0.0196059793, 0.119963646, 0.111532696, -0.103885248, -0.100702703, -0.010400556, 0.0219070762, -0.0126086501, 0.0240438357, -0.060223829, 0.0423679128, -0.00986079872, 0.0329693109, -0.0818725005, -0.0714677423, -0.0257736444, 0.0543711409, 0.0940362662, -0.119938776, -0.0633669943, -0.116895951, -0.0374297909, 0.0153847542, 0.0372343957, -0.0610368811, 0.113813013, -0.0170616098, 0.00195942726, 0.00671724509, -0.0389183983, -0.0128870467, -0.113415472, -0.0129363602, -0.0356861092, 0.0534268841, -0.0288733747, 0.0418036468, -0.153400227, 0.0296305232, 0.0245947726, 0.066393964, -0.00165655045, -0.122910373, 0.0488593057, 0.0413906798, -0.0627416894, 0.0645338818, -0.026778372, -0.0406190902, -0.0442537032, -0.00246794894, 0.0225111302, -0.00398455374, -0.0284111463, 0.124458574, 0.130251542, 0.113397017, -0.0720993355, -0.0414232314, 0.0428066999, 0.0329683721, -0.0125187151, 0.115253933, -0.0684984401, 0.0104852254, -0.136497185, 0.00998436473, 0.0500208177, -0.0262930356, 0.0352597348, 0.0552926809, -0.134685189, 0.100826129, 0.0628324151, 0.0390063636, 0.010178389, 0.0558182113, -0.00302903913, -0.0310565364, 0.0949583054, -0.153061911, 0.0321237296, -0.051590357, 0.0456893779, -0.023379581, 0.0882194489, -0.0808342993, 0.093459636, 0.00758528709, -0.106659807, 0.00587938726, -0.0590616018, -0.0399960913, 0.00719778053, 0.108343609, 0.0468838401, 0.0391731933, -0.016234532, 0.0277812388, -0.0368827656, 0.00372426142, 0.0314919986, -0.0181080867, 0.0381364822, 0.112079777, 0.157007411, -0.0116896331, -0.0103837289, -0.155438438, 0.030527778, -0.114068605, 0.108232319, -0.0308927819, 0.117109597, 0.00867082179, -0.0103414804, -0.0227078237, -0.0242070407, 0.0158710014, 0.0176119618, -0.0023907884, 0.02301763, -0.172001734, -0.0185527913, 0.066018872, -0.00374495611, 0.00550355855, 0.0396729745, 0.0719289333, 0.0583389513, 0.228415847, 0.0289598331, 0.0523797348, -0.0487385169, -0.038304951, -0.0288884249, -0.0958547294, 0.0831411406, 0.00722385664, -0.0514185987, 0.0281225797, -0.0335371867, -0.0953213423, 0.0357710347, -0.00273016654, -0.0733452439, 0.0190322548, 0.0579749383, -0.0754311532, 0.0323413908, 0.130112335, 0.0591265336, 0.0263809413, -0.0889221877, 0.0362376422, 0.00274141366, 0.0602396727, -0.00956112519, -0.0633085221, -0.0705631971, -0.00269171223, -0.0227907635, -0.0692018792, 0.0450100601, -8.21100548e-05, 0.085006319, -0.0117384307, -0.178841949, 0.00916172564, -0.0331595391, 0.0488371365, 0.0309088267, -0.0520205721, 0.0543855466, -0.0609956905, -0.0151451491, -0.119706556, 0.0521327071, -0.0239361376, 0.0619983524, -0.0344233587, 0.0928516462, 0.123764999, -0.0510081723, 0.051918298, 0.134016812, 0.00433373079, -0.0399642885, -0.0476095639, 0.058590617, 0.0102138538, 0.0473462418, 0.0685652196, -0.00715079717, 0.0423923582, -0.123237118, -0.0599423945, -0.0193803404, 0.0810124949, 0.0482463613, 0.010171093, 0.0322510414, -0.0855225101, -0.0134441592, 0.0353776589, 0.0357695967, 0.0157995224, 0.00592060806, 0.0427856967, 0.019695485, -0.120965153, 0.0518125519, -0.025982812, 0.00440140441, -0.101803318, -0.00751397945, -0.0489026457, -0.110446945, 0.0387411118, -0.0329769477, -0.026433032, -0.0734259188, -0.0359849557, 0.0301200077, 0.0163871422, 0.00114649849, -0.10535416, 0.0533666052, 0.0522046946, -0.00681710057, -0.0213999078, -0.0203455649, -0.063229993, 0.0781266317, 0.0768756866, -0.0961050317, -0.065041244, -0.133748487, 0.0100543723, -0.0106222974, -0.0259819292, -0.0329633467, 0.0461320877, -0.0447794944, 0.003435269, 0.0207778122, 0.065288499, -0.028659109, 0.0149778146, 0.0349693224, 0.0478700735, 0.014303416, -0.0856329799, 0.10475678, 0.0338214226, -0.154605776, 0.00877577253, -0.132177755, -0.0806690902, -0.00436068373, -0.0136294104, -0.0454847552, -0.108277924, -0.0509702489, -0.10566017, 0.0186794251, 0.0360619947, 0.0443202034, 0.0150199682, 0.197757751, -0.0792406127, 0.126476422, -0.0556568801, -0.0213381834, 0.140827551, 0.0756311268, 0.0323015526, -0.0986557081, -0.0878089145, 0.0130598582, 0.0204975531, 0.0466922373, -0.0937384889, 0.0174807832, 0.0393661335, -0.0838654786, 0.014209413, 0.0197430924, 0.0545310043, 0.0844336376, -0.00396912917, 0.093169868, -0.159154788, 0.0605714992, -0.00325722061, -0.0306225698, -0.0325894691, 0.0413154587, 0.0223213788, 0.0820711106, 0.0751379952, -0.087409243, 0.0902555585, -0.0316079296, 0.00693639787, -0.0477129482, 0.0698177144, 0.0563609712, 0.150307685, -0.0405079909, 0.0418194234, 0.00745331962, -0.044603765, -0.0868503079, 0.0228795428, 0.0951327384, 0.145075753, -0.00281672552, 0.0819790065, 0.100366093, 0.120265633, -0.12336693, 0.097921811, -0.0526711382, 0.0146113727, 0.0517357066, -0.00685218349, -0.0323748961, -0.0437289886, -0.00333631411, -0.0126014203, -0.0984798595, -0.114890754, 0.0288062505, -0.0771140903, 0.0382514372, -0.0117044989, 0.126339108, -0.00630878564, 0.0530857854, -0.104100645, -0.00805898756, -0.0305066146, 0.105314784, 0.048034966, -0.00172337517, 0.0301087871, 0.165835604, 0.0267596543, -0.142763242, 0.181588918, 0.0551236197, 0.0679461434, 0.101056561, 0.0339270458, -0.073371917, 0.0601740666, -0.0367997475, 0.0108242445, 0.0693133548, -0.0234897546, 0.102104969, -0.0528279245, -0.0597027726, -0.0566084348, 0.0335544311, -0.205662742, -0.0541634336, 0.00158093637, 0.0658201575, 0.0301372595, 0.0693942308, 0.107268907, 0.0292246621, 0.128294975, 0.0263936706, 0.0309509225, -0.0775180459, 0.116698608, -0.0734690353, -0.0131640136, -0.0256189536, -0.062963888, -0.126585558, 0.0140708741, -0.0230707563, 0.109207697, 0.11241141, 0.0451781824, -0.0347523019, 0.0550954714, 0.0766290501, -0.0519221164, 0.0437252149, 0.102785774, -0.105436176, 0.10736078, 0.0210221633, -0.0217525065, 0.100014761, 0.0385276638, 0.0546158366, 0.0585203208, -0.0420682579, -0.171221569, -0.142569944, 0.0215001479, -0.023452919, 0.0635518059, 0.0205523521, -0.0221534446, -0.09596131, -0.0570831373, -0.0364792533, -0.117802076, 0.0533068553, 0.0692519322, 0.0763008073, -0.0444405191, -0.141365409, -0.0190920215, -0.0462770239, -0.116279766, -0.0336749479, 0.0318626389, 0.0286726728, -0.0309933089, 0.00509904884, -0.117549956, -0.0551077612, 0.00944215711, -0.0124984551, -0.0347758941, -0.0253979862, -0.0476573743, -0.0240106434, 0.0761979371, -0.00755198859, 0.000757890753, 0.0146143194, -0.0430316068, -0.105958819, -0.0228075683, -0.0752149299, -0.0152789466, 0.0252250638, 0.00773550943, 0.147780925, -0.0151827568, 0.0613514408, -0.0986682922, -0.0442262664, -0.0455808938, 0.0428584889, -0.0703783184, 0.0335962176, 0.022636719, 0.000310000032, -0.0391520672, -0.0628906041, -0.0938398689, -0.0734697208, -0.0291133802, 0.179060459, -0.0784291476, 0.0768223926, -0.0370093696, -0.0368609205, -0.0792517066, 0.0696835145, 0.0456825048, 0.0358340479, 0.0434729829, -0.0668236166, -0.0652068704, -0.183176398, -0.0633447096, 0.0550470129, 0.0324314684, -0.131186828, 0.00050502643, 0.0845886469, 0.0555002876, -0.0492061079, -0.201960742, -0.0906325206, -0.0749930367, 0.050311245, -0.0290989503, -0.0318274796, 0.0245478377, 0.0217907615, 0.0250097271, -0.0652556121, -0.0649409145, 0.0265176073, 0.0243124366, -0.0689618066, -0.107658178, -0.0692645833, -0.054567121, -0.0179806706, 0.0172811598, -0.13332127, 0.0765545368, -0.0310513452, -0.0622933619, 0.0652891845, -0.0139535349, -0.00840768591, -0.0719554275, -0.103346743, -0.205132723, 0.047608614, -0.00250128657, -0.000518750399, 0.0459744036, -0.108746588, -0.0344416574, -0.09308438, 0.0268362872, 0.0715449229, -0.059631139, -0.0216482393, -0.0235823784, -0.0962414742, 0.0395797528, 0.0250034407, 0.0147794839, 0.016083248, 0.0418951213, -0.0584590547, 0.0527435131, 0.0311591234, 0.130391851, 0.150298372, -0.0433518961, 0.0115818251, -0.103978656, -0.00348509476, -0.0824357718, -0.071391426, 0.00255766511, 0.0320981182, -0.22617498, -0.0560468659, -0.0822790861, -0.219181985, 0.00953684561, -0.0300233066, 0.111459889, 0.0274805464, -0.140019536, 0.0153040197, 0.0539604127, -0.0157690719, 0.0947029889, -0.070151329, 0.00172157213, 0.0609328263, -0.0234152079, 0.0360128805, -0.114299558, -0.0119139217, -0.0178148597, -0.0278276093, -0.0883894339, 0.064821586, -0.15142858, 0.0802713782, 0.0321872979, -0.0716421828, -0.122801922, -0.0259564184, 0.123508014, 0.0335269272, 0.0583531, 0.043163009, -0.0497357398, -0.0202746131, 0.0915562809, -0.0884398818, 0.00746741146, 0.0121395029, 0.0458049811, 0.0897039324, -0.0835799426, 0.00104040024, 0.0218561664, -0.0829297453, 0.0716589317, 0.00597879291, 0.00369991735, 0.0972465575, 0.0318837091, 0.0861498266, -0.125971302, -0.0046215672, 0.039220728, -0.0331700929, -0.0022045821, 0.0141417515, 0.00824223831, 0.100044392, -0.0323052891, -0.00785260275, 0.0707256421, 0.0591015667, -0.00800828263, -0.0836099014, 0.0224461854, -0.00758463563, -0.0430032499, -0.0993371308, 0.0381070673, -0.0292616654, -0.0305680539, -0.0527784973, 0.0147669194, -0.0452954806, 0.00313056516, -0.0710692182, 0.0366714299, 0.154665232, -0.132521346, -0.115051359, 0.0153902564, -0.0508783571, 0.0555030368, -0.0203189589, 0.0208809953, 0.0317924544, 0.0976715684, -0.163995042, -0.0313210711, 0.0696517229, -0.0985373706, 0.0176254176, -0.0817904994, -0.111890033, 0.0534250289, 0.0213724207, 0.0842697173, -0.0279486086, -0.00327455997, -0.0896307826, -0.00842390582, -0.0768062845, -0.106076509, -0.074272871, 0.0391257666, 0.0854253918, 0.0249287318, 0.00916362368, 0.0300335549, -0.0668060482, -0.100941926, -0.075986661, -0.00613939017, 0.0470039733, -0.0999038219, -0.0575053319, 0.019524131, 0.0361823663, 0.131882608, -0.0096709393, 0.0882648826, 0.041786477, 0.034654133, 0.0255509745, -0.0886439085, 0.00837724656, -0.0773778856, 0.0229398739, 0.0581588559, -0.0465174727, 0.0858686119, -0.0553110354, -0.0148559269, -0.0410864353, -0.00901198946, -0.00128553924, -0.0114130266, 0.0124721397, 0.0549827255, -0.007832665, -0.0482536331, -0.0951088592, -0.0759178251, 0.0608368292, -0.0407103449, -0.0283425767, 0.0321998298, 0.126301706, 0.067398712, 0.139780685, 0.0905814394, 0.00255679712, -0.00767655671, -0.00840915833, 0.088301219, -0.048137214, 0.0148405693, 0.00380565645, 0.0106215859, 0.089731425, 0.034143839, -0.0650838614, -0.0764127225, 0.13296175, -0.177675739, -0.0525807329, -0.104725361, 0.064101845, 0.10076917, -0.0463725515, -0.0662362948, -0.0379772894, -0.074941963, -0.141431734, 0.000464164652, 0.0287206192, -0.0947588235, -0.0683050156, -0.0300985053, 0.0466467403, 0.104172662, -0.134927958, 0.0471047983, -0.0949884206, -0.0951971039, 0.0283831507, 0.0657143593, 0.0462317839, 0.0435468554, 0.0596275926, -0.0388186611, -0.0583273657, -0.0233254395, 0.0902210325, -0.0985154659, -0.0384789072, 0.0537803955, 0.104289338, -0.0677582994, 0.0276348703, 0.0171381459, -0.0307430662, -0.0552040786, -0.0401273668, 0.00251147803, -0.0259028301, -0.128685653, 0.0270089079, -0.0281825364, 0.0558626354, -0.0426816903, -0.0650866926, 0.0326622389, -0.0483125076, -0.055412095, -0.0244423784, 0.0109835584, 0.0196121559, 0.0430874974, 0.0266159214, 0.00617672317, -0.107649848, 0.0332261026, 0.123890027, 0.067306675, -0.0808168426, 0.101745799, -0.0675554276, -0.0669053793, 0.0962668732, -0.104982689, 0.0697224736, 0.0392863825, 0.0293577798, 0.0433183499, 0.0401539989, -0.0264592841, -0.124858037, -0.0245554093, -0.071433872, 0.0490507632, -0.0315658227, 0.0505969934, 0.040864408, -0.000168052502, -0.0109752379, 0.0373206735, -0.145048499, -0.0239026174, -0.0684744939, -0.0636875778, -0.0114831738, 0.139179409, -0.00155177619, -0.15342024, -0.033083193, 0.000420395285, -0.117142901, 0.00887246989, 0.122661121, 0.113508984, 0.0204033777, 0.00637237635, 0.0819063187, 0.00776152499, -0.106520936, 0.0975836441, 0.0585022047, 0.0782554224, 0.046391435, -0.022785807, -0.0304160044, -0.0622793511, -0.0942288488, -0.0606903024, -0.00904364698, 0.0629969984, 0.0954230279, -0.12778683, -0.0284533855, -0.0272438936, 0.0757961869, 0.028047964, 0.0972610638, 0.0580233596, -0.0828812718, 0.119468622, 0.0710946023, 0.0221559331, -0.0590557754, -0.0555966273, -0.0606284887, -0.0115851667, -0.0940932408, 0.0262915269, 0.0135664009, -0.00717134774, -0.0664277151, -0.0882107168, 0.0916490331, 0.0246482864, 0.103041373, -0.123946175, -0.0915629715, 0.00223686872, -0.073600322, -0.0802451596, 0.108621851, 0.0714537129, 0.0417542085, 0.134732231, 0.0369990319, -0.082304731, 0.052722007, -0.0231204405, -0.00113231316, -0.0775985718, -0.0870465413, -0.0127883479, 0.0597468019, 0.0681404546, -0.0372708365, -0.00268130354, 0.0848922282, -0.0623495802, -0.00645769248, -0.117754631, 0.0372559428, -0.0158301927, 0.0494583473, -0.0121700251, 0.0199690834, -0.0330053344, 0.0689561367, -0.0206274483, -0.0206134468, 0.0432984717, -0.0370494798, -0.0341483019, 0.0488845222, -0.0686890259, 0.179095566, 0.0062625967, -0.0568772294, -0.091103442, 0.0186275057, 0.0290343128, 0.115588844, -0.0852092206, 0.0256224014, 0.0983831733, -0.00113785639, 1.40275806e-05, 0.0457989648, 0.0426610336, 0.152750835, -0.0321622267, 0.138436332, 0.0073488988, 0.0764992163, -0.0264629424, -0.0250669904, -0.00355184451, -0.0162453055, 0.0607386976, -0.125566661, -0.0264021866, -0.0892097577, 0.0325158015, -0.0342464149, -0.108295441, 0.0783299357, -0.0384992883, -0.045980528, -0.0264427215, -0.0641009584, 0.0916307718, -0.160485119, 0.101107836, -0.124456659, -0.0714205652, -0.0165864844, -0.0105503872, -0.0963487178, -0.00333322771, 0.0448205657, -0.0510514453, -0.0136782899, -0.096345827, 0.0154198436, 0.0299618877, -0.0672173873, -0.102037974, 0.0483165756, -0.0276720915, 0.130227983, 0.0581221469, -0.072762236, 0.047728993, -0.0352324732, -0.0594642349, -0.002675422, 0.139455602, 0.00566758122, -0.0134287253, -0.0688176528, 0.0625232831, 0.140319631, 0.0563304573, 0.0567270331, 0.0983596072, 0.150661379, -0.0800207555, -0.0853598565, 0.0336976275, 0.0131315533, -0.0819277465, 0.057536494, 0.00667545758, -0.0457928032, -0.038779866, -0.00723124668, 0.00690400228, 0.0680176616, -0.0253968798, -0.172183186, -0.0330998711, 0.0270697325, 0.0356532708, -0.0886402205, 0.0234502219, -0.0174542684, 0.0187187009, 0.00804674998, -0.0369820781, 0.00467156246, -0.0236953069, 0.104239531, -0.0260523707, -0.0250848345, 0.0440467596, -0.0172335394, 0.0141086634, 0.114409156, -0.0390056148, -0.143985286, -0.0538066439, 0.066485323, 0.0168812945, -0.0859410539, -0.00942959171, -0.0697698146, 0.15309763, -0.143645525, -0.191575617, -0.0842180029, 0.0131736286, -0.0419890843, -0.0355420783, 0.0517604202, 0.0332058445, -0.0892739147, 0.107086726, -0.047652822, 0.0188595317, 0.131176427, 0.0565858409, -0.021854572, -0.110475987, 0.0490295179, 0.118606359, 0.0701356754, -0.0754051432, 0.014309682, -0.00493702851, 0.00770587474, -0.00327124819, -0.00881879777, -0.0423447676, 0.010203043, 0.0713135451, -0.148224965, 0.00333502889, -0.0559453182, 0.0410412326, 0.0759655833, 0.0172477216, 0.0831833854, -0.0297368802, 0.111099362, 0.0883169025, -0.0722597763, 0.0131261591, 0.0140464399, 0.0175292101, -0.0339123756, -0.0285929143, 0.108016133, -0.0652214736, 0.0378189981, -0.05128555, 0.124187529, -0.0402831659, 0.0293531604, 0.00742054172, 0.00414653495, 0.0328657441, 0.00383558497, 0.0537207313, -0.0284183696, -0.0582612269, 0.0320823602, -0.0386008807, 0.0356729515, -0.0504770167, 0.0652536973, -0.098795183, 0.120945551, -0.0412323773, -0.113359623, -0.168529689, -0.044518292, 0.0557504669, 0.0932161137, 0.0808147937, 0.0658239126, 0.061269097, -0.0194292106, -0.0816457719, -0.122028135, 0.161170825, -0.0266123172, 0.000504847616, -0.10841462, 0.0521031097, -0.0749769509, 0.146326363, 0.085672766, 0.0806948692, -0.0364968404, 0.051602222, 0.00282965973, 0.015352767, -0.0605669692, -0.0158483312, 0.0319661647, 0.0238912627, 0.0661585629, 0.0638670698, 0.115828492, -0.15485394, -0.0117736533, 0.108005427, -0.0221562441, -0.0248847492, -0.00074852258, 0.0295029134, 0.0192475319, 0.0617187917, -0.0633570254, -0.0326333679, 0.109099194, -0.0391615331, 0.0408077464, 0.104218476, 0.0296367407, 0.141252548, -0.0425838605, 0.0149380863, -0.0466234013, 0.00988053158, 0.0613031909, -0.0232185572, -0.0452623069, 0.0944167376, -0.0354872383, -0.0408066846, -0.0227842871, 0.0703361928, 0.139385894, -0.095162794, -0.0230612122, -0.00723451842, 0.0986850411, -0.119977117, -0.00739560928, 0.112956479, 0.15224497, 0.0479522869, -0.0886996239, 0.105766222, -0.141112834, 0.028072454, 0.0646339506, -0.0836297721, 0.00408888934, 0.0167465769, -0.046307411, 0.0784704909, 0.103682615, -0.058488939, -0.0245305765, -0.180317387, 0.0136912018, -0.0455013961, 0.0150855631, 0.0137447789, -0.0616712347, -0.0202290341, -0.0954892188, -0.080296129, 0.0467284843, -0.0212473609, -0.0775994211, -0.00118725002, -0.0782555565, 0.0178641155, -0.0689989477, -0.0248651691, 0.0331919342, -0.0804729313, 0.147161454, -0.0213274248, 0.0495033935, 0.0764237717, 0.0679708943, 0.0652758181, -0.00163454004, 0.0484560132, -0.0121581219, -0.0294768251, -0.0991435349, 0.0434749015, 0.041380845, -0.0336263925, -0.00684622675, 0.00642223284, 0.113141291, 0.00063541159, 0.0797164962, 0.00572476164, 0.00803749915, 0.00497916713, 0.0753425732, 0.0550090857, 0.0912253633, 0.0515357107, -0.0963370577, 0.0212445389, 0.110619225, 0.0104701724, 0.038355682, 0.0566010661, -0.0528693311, -0.0188960116, -0.00828725286, 0.00950297341, 0.013510732, -0.00288709812, 0.036969047, 0.0287468154, -0.0306389034, -0.0461689308, 0.0143044386, 0.10684415, 0.0850169808, 0.0378084108, -0.0764039159, -0.11663378, 0.0441069901, 0.0465431176, -0.111619808, 0.161576584, 0.0282414705, 0.0527949333, -0.084071584, -0.0209491625, 0.0541457981, 0.0392391868, -0.0112208202, 0.131430283, 0.0981135964, -0.0509605333, 0.0122558931, 0.000687881373, 0.0265618041, -0.0195218176, 0.0836447179, 0.0750810206, 0.0458138585, 0.146810755, 0.112280034, -0.0652331486, -0.0341970846, 0.0334284902, 0.0540269427, 0.041710116, 0.00432903506, 0.00225922838, 0.0864569694, -0.0504702739, 0.0638329089, -0.103701279, -0.0741944537, 0.0245679785, -0.00566792488, -0.0840940848, -0.109055251, -0.092332907, 0.0407088175, 0.0101407645, 0.00827308837, 0.0545968898, 0.0400347561, -0.0566380098, 0.056541197, 0.17530027, -0.0367391258, -0.0958183855, -0.00934026763, -0.158351377, -0.155936778, 0.118473843, 0.0447239876, 0.0262825079, 0.0385334156, -0.109556459, -0.0255446192, -0.110488355, 0.00124787726, -0.0593225025, -0.00273051858, -0.119895019, 0.0221740324, 0.0167334601, -0.00351163605, -0.113927417, -0.0656535029, -0.0626883954, -0.104976065, 0.0191272385, -0.0353834517, -0.00768600404, 0.070701763, 0.0799218565, 0.0391910449, 0.00603917427, -0.059693262, -0.0492252111, 0.00577678531, 0.0442071334, -0.030128587, 0.066669561, 0.0311337113, -0.0896128789, -0.0929164663, -0.0267600212, -0.0353194922, -0.0334425792, 0.0913329497, 0.150555521, -0.028989261, 0.0309862904, -0.0615032986, -0.0679526925, 0.127847388, -0.050558269, 0.0688756928, -0.0219995752, -0.0388680398, -0.0246833228, 0.0794024989, 0.0578956082, -0.122922733, -0.00071552489, -0.0139164357, -0.030640576, 0.04551965, 0.0506845452, 0.0188603736, 0.0150425369, -0.0802400485, -0.154520959, 0.08918643, -0.0576012246, -0.0230565853, -0.0639366955, 0.0376155786, -0.00303743314, 0.0425109267, 0.0585362539, -0.0916770697, 0.0326580703, -0.0483011715, -0.0244255308, 0.00619422412, 0.0650111437, -0.0211275108, -0.0167442448, -0.0301489234, -0.0189132728, 0.0992666334, 0.099879846, -0.0303247832, -0.00238152314, 0.0860659778, 0.041869022, -0.0518088713, -0.116496213, 0.0370620675, -0.0484162308, 0.104685262, -0.10294643, -0.0191542041, 0.0183966011, 0.067674771, -0.0119359214, -0.0921194628, -0.0441772528, -0.0722718909, 0.0796230286, 0.0795891881, 0.061415635, 0.0472054407, 0.00711930217, -0.0801173747, 0.0219572019, 0.117652074, 0.0209528711, 0.0392731838, -0.0209772401, -0.14853999, 0.129064411, -0.0459602326, -0.0507139154, -0.0590851903, 0.0681848675, -0.0333252326, 0.0525169, 0.0554127023, 0.00368930586, 0.085702166, -0.0775162429, 0.00429337425, -0.0587444566, -0.113069221, 0.000643355772, 0.00562279858, 0.03658548, 0.052098155, 0.107099369, 0.0667936131, -0.0185411349, 0.054342512, -0.0529061705, 0.0734526962, -0.0151351551, -0.0273972377, -0.00876887143, 0.0737391412, -0.0285417158, -0.0303514209, 0.165578246, 0.0638718382, -0.117830209, 0.0496585406, 0.041049473, -0.041145876, 0.00240243599, -0.134060368, -0.0371007062, 0.156852558, -0.038457267, 0.117742702, -0.109646179, -0.0261033438, -0.0273322314, 0.0502961725, -0.00987560581, -0.176500574, 0.10560666, -0.0534770451, 0.0755180418, 0.073453106, -0.00855196454, 0.0408811681, 0.0972820148, 0.00222174916, -0.0196923241, 0.0295872837, 0.045618359, -0.0173810925, -0.0635485649, -0.05865952, 0.0125012361, -0.117654167, 0.0167404786, 0.00176727842, 0.0445348695, -0.110756509, -0.0411797725, 0.060854964, -0.0363162272, 0.0225862637, 0.148795485, -0.0943279639, -0.00545653328, 0.0138726663, -0.0828919411, -0.035351567, -0.0137856416, -0.0302281063, 0.00956151262, -0.000997079536, 0.0637324005, -0.124670953, -0.135817915, -0.0111148534, 0.0395183228, 0.0349599272, -0.0692137033, 0.0396531895, 0.0560348853, 0.0915048048, -0.0951796025, 0.104822598, 0.0226972662, -0.0891933069, 0.0428549908, 0.0416089669, -0.0720485374, 0.0193011872, -0.0514923371, 0.0840799958, -0.0275733396, -0.143871188, 0.0486096255, -0.120800242, -0.014725361, 0.0171756092, 0.0356361233, -0.0434459001, -0.0433174782, 0.0299344528, -0.0154602686, -0.0220428221, -0.0309799686, -0.0465802662, -0.00123932632, 0.01409504, 0.0529759042, 0.0602477156, -0.086191386, 0.0324929543, 0.128435671, -0.10888043, 0.000272087753, 0.0894615874, -0.0358649753, 0.166124359, -0.0133904777, 0.109172203, -0.0641209632, -0.107063599, -0.0110514136, 0.041730687, -0.0877945274, -0.142711118, -0.0765860453, -0.0497560874, 0.0428826585, 0.0574328303, -0.0130979903, 0.125451609, -0.0108842459, -0.0494310446, 0.109787889, 0.0778675824, 0.0823265761, -0.0133256987, -0.103071883, 0.0263200104, -0.0636986345, -0.0152745089, -0.0770010874, 0.0953732282, -0.0105203716, 0.0261606909, 0.027641397, 0.00574612617, 0.0131082274, 0.0553812869, -0.0236430056, 0.0110867014, -0.062127091, -0.0989792496, -0.0495412424, -0.0565992408, 0.0525233187, 0.0198662262, -0.179235637, 0.0898453221, 0.0248485431, 0.0347248986, -0.127199203, 0.0660550743, -0.0934803188, 0.00469446182, 0.00628458615, -0.015294848, 0.0112601621, 0.0915097445, 0.0121056205, -0.00299266726, -0.0751530081, -0.0402411073, -0.0411809869, -0.117185861, -0.0398585685, 0.083669208, -0.040651612, -0.0212481618, 0.0913396031, 0.0123984385, 0.0395914689, -0.0734995976, 0.0387141407, -0.0307631381, 0.0512015224, -0.0166006796, 0.0476839878, -0.00363002811, -0.044824414, -0.0565983057, 0.0472218171, -0.103720374, -0.0252437219, -0.0110661779, -0.0145094479, 0.0776091963, 0.132596031, 0.165300861, 0.105620116, -0.00800295733, 0.134556919, -0.0709809735, 0.0141896494, -0.0762698054, -0.0081240423, -0.0925129652, -0.0793496817, -0.0711927637, -0.0323574767, 0.0483066738, 0.0424038321, -0.0841650516, -0.0245392136, 0.0438334122, 0.0510460362, -0.0362881906, 0.0453605168, 0.0559055582, -0.0746992081, -0.0399772748, 0.0465168618, -0.141152978, 0.00446203956, 0.108306855, -0.0510297939, -0.0421319678, -0.0211320929, 0.0714860559, 0.104075775, -0.0466121845, 0.0498371385, -0.0711495504, -0.0451222062, 0.0821564347, 0.0265221037, -0.0201894213, -0.0309638102, -0.0375229344, 0.108002588, 0.1360026, -0.041354008, 0.0148476101, -0.136250153, -0.111906879, -0.114485517, -0.0318824686, -0.0298597962, 0.083672829, 0.0479454696, 0.0930844545, -0.060877461, 0.0467161275, 0.0868022069, -0.134293407, 0.00406222977, -0.0133788846, 0.00992775895, 0.0371012837, 0.000178516842, 0.0635174811, 0.0686589777, -0.0874956846, 0.0660264939, 0.0604191311, 0.0928163305, 0.00827313028, -0.0172130056, -0.0890372694, 0.0775875002, 0.0471425802, 0.0283339173, 0.0665764511, 0.121209987, 0.00305609987, -0.0121471994, 0.0831000879, 0.0268709604, -0.0201124046, 0.138248697, 0.100675456, 0.0173395015, -0.0172923226, 0.123695709, 0.0999183804, -0.0625192374, 0.193295047, 0.0205619447, -0.0610130019, -0.0741292834, 0.00925136171, -0.0755780712, 0.0248802584, 0.0684561953, -0.0357257873, 0.0628755689, -0.0676857382, 0.149378628, 0.078054443, -0.017178461, 0.0729198828, 0.0285188742, -0.0298199169, -0.107661113, -0.000575106591, -0.0742195025, 0.0206028353, -0.015194552, 0.0513066649, 0.0439567007, 0.11916057, 0.0410906821, -0.101361863, 0.00873067416, 0.0579848811, -0.00293635204, 0.0556497499, -0.0703574941, -0.0211555995, -0.0211676806, 0.0805090666, 0.0674633011, -0.0395794064, 0.0116857458, 0.0380934738, 0.0536395274, -0.0107757486, 0.0702201724, -0.0111099351, -0.0208020341, 0.0421061739, 0.015531511, 0.0450606272, 0.139781103, -0.0504179224, -0.151396498, 0.104282871, 0.168288693, 0.0592916235, -0.104686722, 0.077467382, 0.0554249324, 0.168543816, -0.0889628679, 0.0860685781, -0.075816907, -0.00723795965, -0.0432170518, 0.0212600082, 0.049996458, -0.0394047275, -0.0971770585, 0.0513941944, 0.0137694366, -0.0819444507, -0.0508803576, -0.09034881, 0.0181277636, -0.0112295821, -0.0214229617, -0.0297272354, -0.0584390461, 0.0124653149, 0.0346170813, -0.0422079898, 0.124681838, -0.126552731, -0.0979950204, -0.0617791265, -0.0607632399, 0.0271472353, 0.0653879493, 0.0878731906, 0.0700205639, -0.0435249135, -0.056338612, 0.0412846953, 0.0253047347, 0.027021125, 0.105870433, -0.0201928541, 0.0810924619, 0.0396603718, 0.0434814692, -0.0732205659, 0.152788639, -0.0767242163, -0.057194937, 0.0340616703, 0.0693667531, -0.0196612254, -0.0826099664, 0.0341789797, -0.0540570468, 0.0862257481, 0.155302301, 0.0740946457, -0.0832137838, -0.0889928043, -0.0929092243, 0.105825774, 0.110529013, -0.0169815123, 0.0412914976, -0.120870762, 0.0653953329, 0.0719392151, 0.0856548399, -0.0752637684, -0.0918144956, -0.0356733054, 0.0593351759, 0.0192785952, 0.134731516, 0.0298854578, -0.22963056, -0.089094311, 0.0390513539, 0.0759049505, -0.0633867681, -0.0268667713, -0.00343836844, -0.0256426632, 0.0398066193, 0.022945866, 0.0420098975, -0.00350727141, -0.014944654, 0.101577669, -0.108422257, -0.200207785, -0.00578112528, -0.139163405, -0.08182697, 0.0119988667, -0.0297275037, 0.0233182143, -0.103024743, -0.00383697683, -0.0522182137, -0.0818012059, 0.181222022, 0.0674812645, -0.0762788802, 0.0478710756, 0.0257269125, 0.0580434762, 0.00955753028, 0.0505937375, 0.0182330348, 0.0231178608, 0.0381997339, 0.0372849107, 0.0418353304, 0.0989421234, 0.0434807688, 0.0115981149, 0.0344024263, -0.0854934603, -0.00655464642, -0.0535590649, 0.11046946, -0.0398580283, 0.0241416339, 0.0115565509, -0.0263186991, 0.021106042, -0.00454965793, 0.00473457016, -0.0293057654, 0.00974595081, -0.153997883, 0.0386386216, -0.0189007111, -0.0384422429, -0.0820041448, -0.000343965366, -0.101367287, 0.158929065, -0.167421445, 0.0100682098, -0.0276947729, 0.127314717, 0.109571099, -0.0979896188, -0.00764027238, 0.0627418682, -0.062974833, 0.0021440573, 0.0187398717, -0.116322875, -0.0296423174, -0.0309300087, 0.0427315794, 0.0603606105, 0.0492910594, -0.0101312613, 0.0403695591, -0.122192383, -0.0596618354, -0.006468195, -0.00582188414, 0.0456683524, 0.08462248, -0.0642502531, 0.0695199221, 0.104578532, -0.0763068423, -0.0383230411, -0.115195557, 0.0805008113, 0.0371084101, 0.0499783009, -0.0620879009, 0.110976398, -0.0233650394, 0.178990453, 0.00924512744, -0.0522588454, -0.0252414644, -0.0995525867, 0.0605548769, 0.041917529, -0.0127279628, -0.0714572221, 0.0253617242, -0.113619633, 0.0571864396, 0.0421477221, -0.0455778614, -0.0354776122, 0.0346949771, -0.0156272464, 0.0213422589, 0.00892110169, -0.0124027561, -0.0183743574, -0.0407236591, -0.0177347586, 0.0878833383, -0.0695776194, 0.052132871, -0.0773894116, -0.144517958, 0.00482582301, -0.0226116925, 0.0160243455, -0.0286830291, -0.11305742, 0.101025783, -0.0856631398, -0.0672385097, -0.063888438, 0.134303913, 0.0549882837, -0.10768798, 0.0699498281, -0.00243488327, -0.0660401583, 0.0233532116, -0.0300203152, 0.0456442125, 0.101627544, 0.0769642889, 0.126996264, 0.000388812274, 0.0238995105, 0.0611703172, 0.161981046, 0.0104111126, -0.0210280977, 0.054599572, -0.163943604, -0.0888782218, 0.0246563032, -0.0952074975, 0.0669457465, -0.028490793, 0.124237835, -0.0327320583, 0.0467088819, 0.00436432566, 0.0165604576, 0.0425928347, 0.0523858219, 0.0352160819, -0.0192053169, -0.0619856268, 0.00652379543, 0.0649601892, -0.0250049718, -0.0268743802, -0.1220228, -0.04697432, -0.107010745, 0.0142582282, -0.1341566, 0.112670496, 0.0275352411, 0.0738019124, 0.0107060857, -0.132511884, -0.0193026438, -0.110272646, 0.0176010579, 0.0456731617, 0.0540217906, 0.101229809, -0.0176883563, -0.0548925437, 0.0111844558, 0.0977346152, -0.0939161479, -0.120759696, 0.00728588551, 0.0550565235, -0.029833205, 0.0463131741, 0.0199479777, 0.0799656361, 0.024923414, -0.0735116154, 0.133153856, 0.00860225316, -0.0625157654, -0.0283735283, 0.0827504992, 0.0140353963, 0.0028263703, 0.0391749628, -0.0747612491, 0.0264509879, 0.0634570345, -0.0968047306, 0.0735668764, -0.01932019, 0.0665857419, -0.0885678008, 0.0111907255, -0.0831329077, -0.0440419391, -0.0322117545, 0.0892609581, -0.0616574325, -0.0200462975, 0.0808087736, 0.0819935501, -0.0530164167, -0.0429007262, -0.00939739309, -0.0263765268, -0.137593597, -0.00815229025, 0.0761511475, -0.0534029752, 0.0863740742, 0.0341856666, 0.0761782378, 0.0798772946, -0.0981286988, -0.0827985257, 0.0168975629, 0.093077831, -0.168395638, -0.0431145653, 0.016699478, -0.00326111913, 0.015668232, 0.0981467217, -0.000121034682, -0.00150727481, 0.00911068171, -0.194074079, 0.14716652, -0.0177265238, -0.0327950604, -0.0578373149, 0.0473306887, -0.0268291067, 0.00913901348, 0.0758189857, 0.00338140503, 0.0992139801, 0.0170033798, 0.0540252551, 0.00315051153, 0.160677493, 0.0503151082, -0.0142692998, -0.0541427769, -0.0480790213, -0.141287893, -0.0236011781, 0.0220742133, 0.00780775771, 0.0283384491, 0.0634254366, 0.0844219178, 0.117850721, 0.0364065841, -0.00560771488, -0.0684203058, 0.0683472604, -0.0800958723, -0.024984628, 0.0593558885, 0.0699148774, 0.0657431185, -0.0415165834, 0.111496188, 0.0136796553, -0.00992874987, 0.0449885093, -0.0500408486, 0.00715490058, 0.0617081225, -0.0271681473, 0.0663627312, 0.0376835912, 0.00175093859, 0.0915442854, 0.105019227, 0.0400546379, -0.00614744518, 0.0322519839, -0.0272529051, 0.0788775086, 0.0287162662, -0.0435082987, 0.0217745118, 0.0680316836, -0.0822205916, -0.00315487385, -0.176027328, -0.121989861, 0.0802285671, 0.068146795, -0.168543041, -0.00805228017, 0.0575836152, 0.0659630448, 0.00027151301, -0.184287474, -0.077234745, 0.0259619169, -0.0104427869, 8.8326633e-06, -0.0462127365, -0.0143509647, 0.0386136211, -0.0137817906, -0.094456248, -0.159782857, 0.0176643096, 0.0408019051, -0.205906004, 0.0498316512, -0.0390802771, -0.00614602491, 0.0377606116, -0.0166628994, -0.0740462244, 0.0353523642, 0.180034012, -0.00229755789, -0.0284066554, 0.028490454, 0.0382132977, -0.0177712403, 0.00686036982, -0.030679781, -0.125406608, 0.0881356671, 0.0438567437, 0.117961451, -0.00673158048, -0.0559261478, 0.130192861, 0.189995065, 0.000300833955, -0.0918848291, -0.0665715709, -0.0063006077, 0.0395032689, 0.0745402798, -0.0587377436, -0.13368988, -0.180422559, 0.00515289791, 0.0346100554, -0.0216367804, -0.0543315858, -0.0574583523, 0.00970618054, -0.0398748443, 0.0254109539, 0.114461258, -0.121243052, -0.0534580722, 0.017572619, -0.0689000115, -0.0722096637, 0.0707206577, 0.0562217236, 0.0416003615, 0.110389158, -0.00586797949, 0.109078795, 0.0627859309, -0.0746139437, -0.178598255, -0.0356704518, -0.00472285412, 0.107308924, 0.0908543617, 0.0450132415, -0.0254008416, -0.00743856747, 0.0904664099, 0.0640947297, 0.0863719136, -0.0958629251, -0.0241381582, 0.0598428063, -0.0499173477, -0.0409107246, -0.0345571712, -0.0390259549, 0.0102475435, -0.0146067096, 0.0161825232, -0.150251925, -0.0792580172, -0.0553167947, -0.0292260703, -0.0188379996, 0.000643459149, 0.0435580686, -0.084482573, -0.0985249802, -0.0343088098, -0.0382055268, -0.0432224087, 0.0883175135, 0.0756114796, -0.107673466, -0.134927794, 0.156511784, -0.0245051514, -0.0353129432, 0.00829586387, -0.00211312249, -0.108969897, -0.00366004184, 0.0100791585, 0.0278191306, 0.0497515127, 0.0214323848, -0.178656191, -0.0619581416, -0.0192200616, -0.0922988132, -0.0254442655, -0.0353798307, -0.00773616694, -0.0958243981, -0.0667599365, -0.0184887256, 0.00128525868, -0.00953026954, -0.0225979239, -0.108141951, 0.0378866009, -0.00547851995, -0.0586479455, 0.0130515173, 0.0227658413, 0.0219786353, -0.202414721, -0.0952945799, 0.0276389942, -0.0366673917, 0.200630739, -0.0574049354, 0.219369635, -0.00560873933, -0.0660076439, -0.0390148684, -0.031058291, -0.0553637519, -0.0270704888, 0.0335120894, 0.0195704568, 0.150406182, 0.0333154984, 0.0506328456, -0.0182577893, 0.0639431775, -0.0194490161, -0.00723955827, 0.0276241396, 0.0438724533, 0.00639448036, 0.122798778, 0.143087864, -0.0388212763, -0.0141448826, 0.0388008952, -0.144713074, -0.0721375495, 0.0446854755, 0.109467804, 0.120496161, 0.00206460478, -0.0913183168, -0.0142692104, -0.0134913214, -0.0455319732, 0.0245725252, 0.0421691984, 0.0899413675, 0.102732658, -0.0451376662, 0.00271292776, -0.0701145157, -0.000515389256, -0.00187888183, 0.123769432, -0.0278835259, 0.000219712034, 0.0368434861, -0.0115500763, 0.0699552074, 0.0782960579, -0.00789592229, -0.0588972867, 0.015475966, -0.0345260911, 0.0453729257, -0.0503094792, 0.0914688855, -0.0559914261, 0.0229284205, -0.0123081263, -0.032612633, 0.0111059695, 0.0172873586, -0.0874353051, 0.0297923144, 0.0108721172, 0.0613508858, -0.00696083298, 0.0901359767, -0.0355426744, 0.0571047217, -0.0433449, -0.0547627285, 0.0374375358, -0.241334602, 0.00544045493, 0.0808352008, 0.0276897345, -0.0174633767, 0.071427986, 0.0266567338, 0.0054734163, 0.0435120538, -0.015824059, 0.123210691, -0.0259859301, 0.079398334, -0.0699486658, -0.0321526751, 0.0427672118, 0.107578516, 0.0229987837, 0.112871855, -0.0395532139, 0.00172494003, -0.129916966, -0.117473572, 0.118357927, -0.061017476, -0.0727849305, 0.0315671861, -0.0112778656, 0.00469734892, -0.106646806, -0.0425762646, -0.0328396969, 0.0200689025, -0.126754105, 0.0516137779, -0.00969748292, 0.0385525115, 0.0171331055, 0.0715736002, 0.0561930761, -0.0456623957, -0.0544602834, 0.0509038232, -0.0235189423, 0.0454678312, -0.0445984229, -0.0730791166, -0.0636863112, -0.0429399535, 0.0852165446, -0.00184737332, -0.0186565965, -0.0110966153, 0.162937522, -0.0437614545, 0.0861722082, -0.072525084, 0.0506918468, 0.0179148056, -0.0612825491, -0.0275459439, 0.0272253174, -0.0334783643, -0.0732806772, -0.0769508258, -0.0695436373, 0.0133161955, 0.0472069159, -0.0879593343, -0.0580082238, -0.0633575395, 0.0257822312, 0.030667264, -0.0600329526, 0.10595277, -0.0886051506, 0.092257075, 0.00813044235, 0.013223296, -0.0289506428, -0.00761445984, 0.107809797, 0.0216514673, 0.0489909947, 0.0685153082, -0.104536615, -0.154011056, -0.0122282058, -0.100846365, 0.00166160613, -0.00527038006, 0.0229451079, -0.169116393, 0.00357444584, 0.130249828, 0.0318445526, 0.0451219939, -0.0985371321, 0.077016972, -0.0675574839, -0.0485341214, 0.0892937258, -0.0119261499, 0.11686936, -0.0256366096, -0.064719893, -0.138646811, -0.0230368841, -0.0518703535, 0.0107466932, 0.0913660228, -0.0292170253, -0.00676173903, -0.161402151, 0.0616877712, -0.00999165885, -0.138042018, -0.0479046628, 0.109722525, -0.020709455, 0.00616726419, 0.0622854307, 0.0453955196, 0.0129737593, -0.0028758687, -0.0481419265, -0.0273242481, -0.0312653147, 0.0190724395, -0.102354854, 0.133722231, 0.0744988471, -0.0438664332, -0.118296951, -0.060179811, 0.0385666713, -0.0278032012, 0.0657609701, 0.0827093944, 0.0629360303, -0.0218015127, 0.0498604961, 0.0824899077, 0.00780756585, -0.121808678, -0.023255948, 0.018228665, 0.0122035956, -0.0136935897, 0.0258074179, 0.0411146283, 0.021556396, -0.0242421646, 0.0856881812, -0.0653296635, 0.0157615319, 0.0421842411, 0.0580450147, -0.00777962804, -0.0839014277, -0.151935533, 0.0329401083, -0.0699129552, 0.0765977055, 0.0439387038, -0.0685167909, -0.0831892118, -0.0514106527, -0.028607633, 0.061502032, 0.086351648, -0.00262156688, -0.0871760249, 0.12683478, -0.159808025, -0.163172737, 0.033106152, 0.00390011352, -0.0290324241, -0.0548253208, -0.0273482688, 0.11500749, 0.202738315, -0.00152360462, 0.0413755588, -0.00100732222, -8.979626e-05, -0.170355201, 0.06213855, 0.062782988, -0.062111754, -0.0467889421, -0.123734884, -0.0822224766, 0.0064563714, -0.0526950732, 0.0135611612, 0.00378175639, -0.0321302637, -0.00103278458, -0.0106755365, -0.0156611875, -0.0274015479, 0.066288501, -0.00762125198, 0.0554921851, -0.0248665251, 0.0889319927, -0.193257019, 0.00683034211, -0.00892718881, 0.0225240719, -0.0810979083, 0.0546551943, 0.0133333094, -0.00835020654, -0.0154363895, -0.0218534134, 0.0765927285, 0.0662077218, -0.0222853124, -0.0838636458, 0.0949314907, -0.0462717786, 0.0445657931, -0.0973079279, 0.00222689845, 0.052203007, -0.0551824458, -0.016072819, 0.157039225, 0.146399975, 0.214229614, -0.00472382829, -0.0298488569, -0.0895316973, 0.0459648371, -0.0893030912, 0.0142214783, 0.00727055222, 0.0673766881, 0.153079078, 0.0623493977, -0.0353417471, -0.0408567637, -0.0287689026, -0.164291218, -0.072588101, 0.122869678, -0.0809252784, -0.0744258314, -0.0263943821, 0.022311585, -0.0519490838, 0.0310675688, -0.0436468273, 0.023407463, -0.0411918163, 0.0230428837, 0.0311317667, -0.066521503, 0.0143625438, 0.0257104225, 0.055129271, 0.0788489655, 0.0219211429, 0.0075901784, 0.0655827448, -0.00681952946, 0.0695478916, -0.0999718606, 0.0466005281, 0.0790512338, 0.0724594891, -0.0388102382, -0.0497607887, 0.0118607767, -0.120786272, -0.0297009759, 0.0503409319, 0.0806155726, 0.0945888907, 0.0203324463, 0.1338211, 0.00627672672, -0.0638806894, -0.096447587, 0.0469171293, 0.134490743, 0.0629716888, -0.0161998235, 0.0417893231, -0.127393022, -0.0704433918, -0.00859997049, 0.0384261608, -0.00676104892, -0.0117424373, 0.00263016298, 0.0532458425, -0.0523997359, 0.0430650339, 0.0897080898, 0.0859533995, -0.037975464, 0.00416474417, -0.207259476, 0.0323172584, -0.0114803053, 0.0962532684, -0.0106872888, 0.0364580899, -0.16184397, 0.0418573469, -0.122858383, 0.0221215859, -0.121820882, -0.102466725, -0.089056842, 0.0367734917, -0.110163748, 0.0508830175, 0.0022703018, -0.0185247958, -0.0431330279, -0.0516164042, -0.0410573855, 0.0802833885, -0.0442520902, 0.00709324144, 0.0835353509, 0.0636074319, -0.01820039, -0.116703451, -0.0991834998, 0.0787881315, -0.00421014987, -0.0709599182, 0.0636661947, -0.0746797398, 0.0826184154, -0.0111790467, 0.0135124158, 0.0346965566, 0.0317447968, -0.0182662159, 0.0654354095, -0.0183947254, -0.0237028897, -0.112371206, -0.00207559043, 0.0984482542, 0.057263054, 0.145837754, -0.0390798263, 0.0178938676, 0.0160873868, 0.0243467428, -0.0410782658, -0.0260812677, -0.0531546474, -0.011475645, -0.0513886809, -0.0241638664, 0.00806893036, -0.0697995052, -0.16929169, 0.144684523, -0.0839521885, -0.0113528688, -0.133523107, 0.0680152699, -0.00267725252, -0.0366772451, -0.0540373474, 0.0585089996, 0.00522282999, -0.0195852555, -0.00349725457, -0.0399441458, -0.0847067609, -0.0519267805, 0.0270239264, 0.0249403715, -0.0854221731, -0.0345031247, -0.0426385999, -0.114951417, -0.11833813, 0.0797540545, -0.138187185, -0.200031623, 0.0208405778, -0.114357784, -0.0794100016, -0.0402523465, -0.0483966842, -0.055653058, 0.0419644527, -0.0422492661, -0.0022473936, -0.016253138, 0.103890084, 0.0317640528, -0.0461630151, 0.0666900128, -0.0453241915, -0.0304095335, 0.120142452, -0.0867946148, -0.0395014733, 0.0954977423, -0.0116896294, 0.0413545854, -0.0663651079, -0.0479582623, -0.0986374393, 0.01779503, -0.0141012948, -0.147269323, 0.043544963, 0.0628029183, 0.0814529136, 0.103698663, -0.0168878809, 0.0208992399, 0.127812594, 0.133393362, -0.0354451574, 0.0245596617, -0.0433239639, 0.116616994, -0.029590657, 0.0375297517, -0.0554959513, -0.00119716767, 0.044206921, 0.0155456532, 0.0627288669, -0.0212567691, 0.0345831551, -0.0273814127, 0.070053488, -0.0332821012, -0.0976672098, -0.0103713432, 0.112356469, -0.110892266, -0.115188025, 0.0184156187, 0.15654473, 0.105028741, 0.0263991877, -0.119852051, -0.124294557, 0.0738592073, 0.0314462334, 0.0596648566, 0.0754985213, -0.0108051253, 0.00271856412, -0.0948751941, 0.0416161828, 0.094782874, 0.0168600567, 0.100057401, 0.0786821395, 0.0506573021, 0.0367843024, 0.122363187, -0.0764172822, -0.0260445774, -0.0560432374, -0.137111887, -0.0604897812, 0.000700753182, 0.0843180567, 0.0795811936, 0.106576502, 0.0707424656, -0.00559558813, 0.186479449, 0.00338681787, -0.0375811607, -0.0175246857, -0.206482515, 0.0203088261, -0.00335052237, 0.00765392184, -0.0219054036, -0.092422016, 0.130213648, -0.00963715278, 0.0746578574, 0.0298792869, 0.0852276832, 0.0452477895, 0.00293635018, -0.0406028107, 0.0471775532, 0.00875167921, -0.103349723, -0.0448772684, -0.0290297251, -0.0449584275, 0.0139079317, 0.042584952, 0.0688365772, -0.0339850076, -0.0264592171, -0.029722875, -0.0137560796, 0.0814295486, 0.139631897, 0.0442709774, 0.0383184664, 0.00529657491, -0.0937576964, 0.0498953275, -0.0153518096, 0.109351449, -0.102684058, 0.0631108433, -0.0590194762, 0.00657091849, 0.0752271339, 0.0661112741, -0.0187464096, 0.075098075, -0.00506668538, -0.0846352205, 0.102858834, 0.0224678852, -0.12960352, 0.0128765544, -0.047212813, -0.0523117818, -0.0533741787, 0.0276528094, -0.0502135083, 0.0194695443, -0.0143132471, -0.108509399, 0.148433045, 0.0380441174, -0.00505725481, -0.00490636192, 0.00429776311, 0.0980975479, 0.0316283181, -0.0629595444, 0.0340179801, 0.0504700691, -0.0740982369, -0.0247772243, -0.00488639064, -0.0241223183, 0.0343791023, 0.0140596097, -0.11004588, -0.162041143, 0.160919592, 0.0192217976, 0.0153533816, -0.116443589, 0.0119418502, 0.0596936829, 0.0197722968, -0.0355095007, 0.0546094067, 0.0722641721, -0.14327307, -0.0360650346, -0.0379500166, 0.0014279075, -0.147924304, -0.020114379, 0.0699339956, -0.170718387, -0.0270746127, 0.00512433425, 0.092315577, 0.131550461, -0.00501552038, -0.0553552136, -0.082342945, 0.0269107912, -0.0393439606, 0.0932399482, -0.0991183147, -0.0281126946, 0.0545121729, 0.158625185, -0.151274264, -0.0417198464, 0.106845811, 0.0443828851, -0.0319172107, 0.106447905, 0.0355612896, 0.0712697878, 0.0547756553, 0.0446596593, -0.00519914692, -0.0135855507, -0.0165826976, -0.0246209577, 0.0719221979, -0.0314692408, 0.0288045667, 0.0762285292, -0.0109113827, -0.022664547, -0.0388147011, 0.0331881642, 0.0150379529, 0.0966883153, -0.0536429547, -0.00123625062, 0.0361921415, 0.0258746333, 0.00602638721, 0.0252074562, -0.0116876867, -0.0563903525, -0.0773122236, 0.0541616417, -0.0449338108, -0.0872624815, 0.0239573307, 0.044475887, 0.109698713, 0.00538090896, -0.110722005, -0.0317043215, -0.0926145539, 0.134996489, 0.0132420855, 0.0307217035, 0.129866838, 0.0446491763, 0.142542303, 0.0755499601, 0.0766458809, -0.0939057022, 0.0864705145, 0.0947403759, 0.0673735887, 0.0167821161, 0.081167236, 0.0321459137, 0.0442270897, -0.12323533, -0.00251188874, 0.128289878, 0.0102645457, 0.0948777199, -0.0265928544, -0.0382959172, 0.0444154963, 0.00423470698, 0.0442593768, 0.0491274074, 0.0461569838, -0.00353324227, -0.00449061394, -0.00850099511, -0.0989271998, -0.020404553, -0.0843655318, -0.0262944549, 0.0354807973, 0.0195747688, 0.111938857, 0.0576216951, -0.0198118836, 0.0159228332, -0.0617595017, 0.0832970738, 0.125676692, -0.0676809177, -0.044418402, 0.112666965, -0.139435753, 0.0150006581, 0.0409631506, 0.00353996176, -0.0138108842, 0.0315121263, -0.138240442, -0.0448639207, -0.0652330965, 0.168961555, -0.00368394144, 0.0176044479, -0.0080471728, 0.0863961801, -0.0953193232, -0.1276021, 0.00624971464, 0.0463307425, -0.104270786, -0.012664225, -0.143328652, -0.0620809272, -0.0988290012, -0.0149173979, -0.133307338, -0.0877726898, 0.0622825958, 0.0848572403, -0.0544980206, 0.0604782254, -0.0921068341, 0.136214122, -0.136167347, -0.0482977405, 0.0570528917, 0.00825358182, -0.0369862393, 0.000268530101, -0.128857091, 0.0113458, 0.201225728, -0.0113300551, 0.117818505, -0.0952969566, 0.0119970953, -0.096570082, 0.0346703082, -0.000416658819, -0.0108677037, 0.0852801204, -0.00154381618, 0.0486050583, -0.0845545381, -0.0183461979, -0.00870124996, -0.0703145713, 0.127825424, 0.0226284154, -0.108716726, 0.07842464, -0.0543230176, -0.000194082037, 0.119213894, -0.0854408368, -0.016298499, -0.0377904773, 0.0239778813, 0.0804838911, 0.159557447, 0.0241290852, -0.0569810495, -0.0283770934, 0.00125440955, -0.0842455029, -0.00941268913, 0.00669839699, -0.140971035, -0.121554032, 0.0335644558, -0.0518988892, 0.0265859105, 0.071242772, -0.0262365974, -0.0189802349, -0.0420945585, -0.0380737334, -0.0346987396, 0.104707107, -0.0260187313, -0.00708856294, 0.0157035533, 0.00604697037, 0.00217210129, -0.00494368188, 0.0197832491, 0.0417141728, -0.129215866, -0.0305279493, -0.0844836831, -0.0354751274, -0.0694699809, 0.0929484665, -0.0291762762, -0.188328281, -0.0487990417, 0.0315973833, 0.0206779912, 0.128925368, 0.030309651, -0.118210331, 0.057885319, 0.0857507288, 0.213871256, -0.0757404938, -0.0637934059, -0.0889232978, -0.070100069, -0.125684023, 0.0101588191, 0.0788855776, -0.0299824625, -0.096968323, -0.00361710414, 0.0302541051, 0.060895294, 0.117318891, 0.00945788436, 0.00684899278, -0.0141613223, 0.0400242209, 0.0520439968, 0.0600204505, -0.0246140398, -0.0945139974, -0.0242358223, 0.0106533356, 0.00207729638, 0.138632506, 0.0240307096, -0.205044702, 0.099337101, -0.105229884, -0.0547111779, 0.0454545133, 0.0346658826, 0.0309550203, 0.105702542, -0.0286708586, -0.0798922405, -0.0711463839, 0.0419986509, 0.0664751306, -0.0887834206, 0.115568608, 0.106128082, -0.0161237307, 0.0741705745, -0.0297651812, -0.10414964, 0.0249607414, 0.0709991083, 0.0542765446, 0.0252491813, -0.153204277, 0.114114977, -0.103163362, 0.0376967713, -0.0982381552, 0.0341025777, 0.0852912813, 0.0688287467, -0.00458452106, -0.0439122654, 0.0618342012, -0.0331042111, -0.0731438547, -0.00486975163, -0.134314567, 0.043294467, 0.0666260123, -0.135846078, -0.0551270843, 0.087324217, 0.0839074999, 0.0684562847, -0.0524627268, -0.0236464273, -0.0132759549, -0.0257256441, 0.0554094352, 0.0464685708, -0.0353934243, 0.0220088363, 0.0119866524, -0.0649880096, 0.0026059635, 0.0198674537, -0.0815643817, -0.154027954, 0.0209241249, 0.102914758, 0.104896873, 0.0796399266, -0.00783735327, 0.0127343731, 0.00208612438, -0.0909104943, 0.00549368933, 0.165070027, 0.0412174463, 0.0781062245, 0.0734480992, 0.12345285, -0.123697817, -0.0625981539, 0.092018649, 0.161089271, 0.0978915393, 0.0666619316, 0.0156493112, 0.0594945885, 0.112634279, 0.0463874377, -0.123239174, -0.188735694, -0.0156784058, 0.012096677, -0.0238690488, 0.0179750621, -0.078954801, -0.00978407636, 0.0626665205, -0.0990869999, -0.0145246116, 0.00753659382, -0.00861090422, -0.0665304884, -0.151779816, -0.029356245, 0.0170859136, -0.0718050748, -0.0878710374, 0.0907980502, 0.0137243588, 0.0385664813, -0.0811820328, 0.110349387, 0.0768834054, 0.00795546919, -0.0456569828, 0.0282176752, 0.0154700279, -0.0885322466, 0.0165600739, 0.0242743976, -0.0512486175, 0.134710655, -0.0499701425, -0.0583954751, -0.00552345859, 0.154104307, -0.0116950572, -0.0820651501, -0.0163469426, -0.0135069452, 0.0772170275, 0.164869577, -0.038731534, 0.0343382843, 0.038465336, -0.136547878, 0.165900111, 0.0708707944, -0.0871039405, 0.0610905364, -0.0182755925, 0.0436922237, 0.050334923, 0.10117881, -0.120075844, -0.0543433391, 0.0410908833, 0.00921290368, -0.185134232, 0.188845456, -0.0383938029, 0.0805517957, -0.0509419739, -0.0603957325, -0.0172433928, -0.130541846, -0.0454375632, -0.0793359652, -0.211888015, 0.124995843, 0.0437471159, -0.0308959447, 0.0279041976, -0.118342206, 0.105505772, 0.0511259995, 0.0539516434, -0.0503093079, 0.0535409003, 0.0130187161, 0.0835435614, -0.0394603834, 0.00284699211, -0.0404362157, 0.0310821142, 0.100886263, 0.0214795284, -0.0352247208, -0.0306135565, -0.00715743657, -0.0303195789, 0.0534922257, -0.0375283137, -0.0457643941, -0.000629881397, -0.131434873, -0.0565093048, 0.0461451709, 0.0843777359, 0.00991098676, -0.024788959, 0.0906525478, 0.0581897125, 0.0328901224, 0.0550921038, -0.0313090384, 0.100491121, 0.0201333854, 0.062505886, 0.00610055029, 0.0380043164, 0.123201445, 0.000253286678, 0.0919304714, 0.0447422415, -0.026506843, 0.0406525247, -0.031096993, 0.0363907889, 0.00152044883, 0.080487363, 0.0627110079, 0.0874619409, -0.0519537963, -0.127790511, 0.00459417142, 0.00682846317, -0.0457928702, 0.0522196144, 0.0924303308, -0.038464509, -0.086849615, -0.160356224, 0.0408706851, 0.095490247, 0.0122903381, 0.0136974026, 0.0707636774, 0.12187013, 0.0146573596, 0.082080096, -0.0131755602, 0.0621735193, 0.0556824245, -0.108569272, -0.076609239, -0.0237353258, -0.00559871644, 0.115258977, 0.191743419, -0.0252263285, 0.0221248195, 0.0200040527, -0.0291588716, 0.0777552426, 0.0164593514, -0.0550806075, 0.0520639569, 0.0552635677, 0.0685346872, -0.0388821326, 0.0650468916, 0.0153346471, -0.0405179337, 0.0162673183, 0.173001856, -0.0572070144, -0.158739433, 0.0474437848, 0.0186247621, -0.0384489819, -0.025185056, 0.0661928505, -0.0579020381, -0.00272467011, -0.0764068663, 0.0295968316, 0.0987232104, -0.0359727219, -0.0147707537, 0.066143699, -0.0598340631, -0.0150769847, -0.119023167, 0.149456948, -0.00938773807, -0.00291891396, 0.0483479574, -0.00588743994, -0.0343669839, -0.00993183814, 0.0173940733, 0.0307970271, 0.0672329217, 0.101019584, 0.0220003892, 0.0636140481, -0.0627934486, -0.0827511996, 0.154713675, -0.0319037884, 0.0897481441, 0.00334194303, 0.0564720593, -0.141668037, 0.0508314818, -0.124435812, 0.0426802114, -0.0346642956, -0.038462922, 0.0804857686, -0.0440798588, 0.025364805, -0.0434191748, 0.11817079, 0.0416435152, -0.0273104757, 0.157931626, -0.0276355185, 0.123778537, -0.0851543918, -0.0501176491, -0.0156346746, 0.0620692186, 0.0481165498, -0.160365403, -0.0612192973, -0.0219055358, 0.0891804919, 0.102926239, -0.0611294955, 0.0267112441, -0.00692081638, -0.0512603037, 0.0842123702, 0.0915205926, -0.080886066, 0.0240275264, -0.138876632, 0.0464169867, -0.0722726956, -0.00494793104, 0.0103371255, 0.053213045, -0.0334090777, 0.128605515, -0.012526406, 0.106924511, -0.0166248754, 0.0593191124, 0.036283195, -0.0135625023, -0.146235406, 0.0251276847, -0.126170442, 0.044441469, -0.0732398182, 0.0177746881, -0.00336868223, 0.0126545895, -0.125758231, -0.0463296212, 0.000760551542, 0.0746849254, -0.0746463388, -0.103783503, -0.21176663, -0.00526075624, -0.196705297, -0.0411077552, 0.0015835464, -0.0345042162, 0.0313511938, -0.0428696312, -0.00496423617, -0.0575777479, -0.040053606, 0.100102738, 0.189796567, -0.0651216954, -0.00988450833, 0.00966881588, 0.00536490232, -0.0826966986, 0.0192021336, -0.0573377647, -0.057390485, -0.00228849798, 0.102888875, 0.0277957432, -0.0254602786, 0.0783777982, 0.0107650012, -0.016606804, 0.0569796078, -0.0925672203, -0.0503984913, -0.0248753857, 0.0985915661, -0.0352421179, -0.119261652, -0.0386371911, 0.0383000784, 0.00993614178, -0.0306219943, 0.0372465104, -0.0314411968, -0.0700695142, 0.0865592733, -0.110574499, 0.0532203689, 0.040152695, -0.11676003, -0.0943935215, -0.0335536599, 0.0619540289, 0.0414873697, 0.0805522352, -0.0169619527, 0.0864372402, -0.0705546364, 0.0452733934, -0.00907016173, -0.064847514, 0.0581720583, -0.114057466, -0.0363059863, 0.0896648243, 0.0615061969, -0.111177891, -0.00641831011, 0.0757474527, 0.0730857551, -0.0960297883, -0.121426262, 0.179821208, -0.0260676071, -0.112282872, -0.0372998379, -0.161543563, 0.0876609832, -0.0419862084, 0.0595651567, 0.047704272, -0.0540253408, -0.246272579, -0.114966534, 0.0210301299, 0.0170566794, -0.058123529, -0.00903307181, 0.108617522, 0.123143926, -0.106013909, 0.140455604, -0.00474341772, 0.0790526718, 0.0832593143, 0.0311025977, -0.0661242753, 0.0702918619, 0.033441782];
    CONSTANT bias_w_0_h : ARRAY[0..63] OF REAL := [-0.0328608565, 0.0353249349, 0.0676618442, 0.0616552494, -0.0419506915, 0.0316758305, -0.0423809998, 0.206494898, 0.050283879, -0.110759951, -0.186538026, -0.0580092184, -0.00209416403, 0.00920274295, 0.0975962356, -0.0612216219, 0.0531282201, -0.1364595, -0.0861791223, 0.0857749358, -0.0629618913, -0.140043736, 0.0230254605, 0.0186893195, 0.274617553, -0.143400162, -0.0180932954, 0.0126953581, 0.00789607875, -0.102969147, -0.00854359195, 0.110707261, 0.101612948, 0.104877286, 0.155045539, 0.120350428, -0.0493059158, -0.109052174, 0.0994426012, 0.120997518, 0.0253830422, 0.0221965443, 0.0652017593, 0.127511516, 0.0405574776, -0.223452628, -0.106970645, -0.184132561, 0.130376682, -0.000101010766, 0.0180109702, 0.0785107389, -0.0454430841, 0.00758665288, -0.0226881728, 0.0657565445, 0.175357804, -0.0399201475, 0.0946480408, -0.0675376579, -0.0944304764, 0.0255580787, 0.114538141, -0.0542288534];
    CONSTANT bias_r_0_h : ARRAY[0..63] OF REAL := [-0.02572597, 0.0358566716, 0.0725965649, 0.0658897385, -0.0349466167, 0.0312440004, -0.0520541295, 0.229264349, 0.053602159, -0.114199713, -0.188671976, -0.0562148206, -0.00815096032, 0.042876251, 0.128237545, -0.0830967203, 0.0521300212, -0.172336012, -0.0845128968, 0.120621495, -0.0981689841, -0.171339214, 0.0380116738, -0.00155168783, 0.27826634, -0.166642264, -0.0124149593, 0.00777016627, 0.0202645063, -0.110686347, -0.00758656999, 0.116100229, 0.137906507, 0.108378269, 0.189799592, 0.156204492, -0.0414909273, -0.111529253, 0.11403127, 0.138321266, 0.0324263275, 0.0199548732, 0.0663017482, 0.155816868, 0.0454924814, -0.249957547, -0.124289908, -0.17978096, 0.148145601, 0.0183632877, 0.0141077479, 0.0873264968, -0.0591249838, 0.00012417727, -0.0334720835, 0.0621513799, 0.192247525, -0.0562552325, 0.11991331, -0.0805595443, -0.108275652, 0.0187377501, 0.144540057, -0.0489126071];
    CONSTANT weights_3_u : ARRAY[0..4095] OF REAL := [-0.726234972, -0.82971102, 0.359873623, 0.467501462, -0.795098782, 0.642522633, -0.834418893, -0.800529778, 0.752689779, 0.406455636, 0.616274774, 0.617786705, -0.741933465, 0.632032633, -0.739187837, -0.503853142, 0.545782745, 0.567466497, -0.337621212, -0.339030087, -0.389321893, 0.674896181, 0.789721549, -0.746486127, -0.669301271, 0.820195556, 0.72258997, -0.971024632, -0.772712708, 0.568969786, 0.828069806, -0.664833724, -0.332123041, -0.638633251, -0.857070208, -0.492956102, -0.802621424, 0.136594638, -0.361942023, -0.667052031, 0.616791487, 0.744978189, -0.954466581, -0.57189548, 0.74708873, 0.656679034, 0.282293171, 0.660095751, -0.696134508, 0.818064272, 0.902193606, -0.636808872, -0.692610443, 0.638984621, -0.867889166, 0.462693274, -0.667061865, -0.625101268, -0.593671858, -0.351741135, 0.234290212, -0.588220656, -0.595141947, -0.701019764, -0.372747988, -0.607375026, 0.464761764, 0.530245066, -0.573789001, 0.530546367, -0.433061302, -0.461016506, 0.59694773, 0.0462750606, 0.332048684, 0.404971868, -0.498975754, 0.562286198, -0.327837288, -0.52094245, 0.35660404, 0.363930374, -0.340805382, -0.0284396466, -0.445062369, 0.1347083, 0.55759269, -0.618813932, -0.599301457, 0.350034744, 0.372941881, -0.528004527, -0.534632623, 0.234335199, 0.397439361, -0.0195646528, -0.0915857852, -0.0818935558, -0.397882402, -0.0978519842, -0.491226345, -0.166510537, -0.00829036627, -0.282786936, 0.626897216, 0.404613793, -0.491245329, -0.337422758, 0.430924863, 0.278444827, 0.0179173294, 0.231050387, -0.347322822, 0.3725501, 0.48292917, -0.507511616, -0.393044561, 0.602047801, -0.562717617, 0.321077079, -0.230540395, -0.587909281, -0.0499534346, -0.369197726, -0.169617653, -0.41201207, -0.260386378, -0.412834316, -0.803556919, -0.740769684, 0.440442294, 0.568141937, -0.475784481, 0.644459307, -0.596662343, -0.940275252, 0.656770587, 0.322523296, 0.875917017, 0.875438809, -0.816106558, 0.825712204, -0.592998028, -0.347098321, 0.495246083, 0.658055961, -0.403978735, -0.0876639634, -0.502450585, 0.64121145, 0.575357795, -0.643270314, -0.996893167, 0.557650566, 0.867267251, -0.850942194, -0.756620347, 0.329067886, 0.669194162, -0.383174628, -0.0802536532, -0.551262677, -0.718719363, -0.598996222, -0.631955266, -0.0989504158, -0.0885992125, -0.713463306, 0.518353522, 0.730688989, -0.800943017, -0.605422258, 0.701749504, 0.95046109, -0.0751864091, 0.87148875, -0.567332923, 0.663198709, 0.649199545, -0.935164213, -0.753644347, 0.803934813, -0.580185413, 0.378011674, -0.636774302, -0.702305377, -0.344566911, -0.367477775, 0.00891227275, -0.607614458, -0.661959112, -0.687778234, -0.625213504, -0.534323871, 0.356132567, 0.448352844, -0.662155986, 0.502999783, -0.572085738, -0.688427746, 0.490987062, 0.707427204, 0.605727017, 0.829243064, -0.728774309, 0.576677978, -0.878341854, -0.301144749, 0.548745811, 0.666547835, -0.0080199372, -0.474185884, -0.431044191, 0.850138128, 0.552011251, -0.779790699, -0.770057082, 0.645845652, 0.763373435, -0.612323225, -0.813291967, 0.79515928, 0.696035445, -0.785743177, -0.688787401, -0.600066721, -0.71572578, -0.727747619, -0.471354902, 0.656914413, -0.512712061, -0.605490208, 0.525177181, 0.528167665, -0.758861125, -0.702212036, 0.415254414, 0.783526659, 0.741826832, 0.719366014, -0.687756479, 0.683343053, 0.737960219, -0.525721431, -0.455234349, 0.570235014, -0.521014452, 0.321572721, -0.731491745, -0.51282382, -0.718585134, -0.164967939, 0.67603749, -0.509025753, -0.7481004, -0.456257671, -0.669510841, -0.814430475, 0.570815623, 0.526050806, -0.529686749, 0.621858954, -0.670453012, -0.304120302, 0.726401627, -0.0356775187, 0.260329664, 0.624240518, -0.748086572, 0.772515833, -0.125408188, -0.57220155, 0.498111188, 0.0558861159, -0.435518563, 0.303609818, -0.723968267, 0.32118696, 0.692383528, -0.775559604, -0.599537134, 0.294759721, 0.716790199, -0.824359059, -0.780710399, 0.106178224, 0.59846735, -0.206296533, 0.128306508, -0.146541059, -0.224539533, -0.0289100092, -0.765631378, -0.220809624, 0.142412528, -0.384071648, 0.592445076, 0.540259898, -0.638875484, -0.205305457, 0.619496822, 0.442066103, -0.0485938378, 0.466518402, -0.158942863, 0.672467291, 0.807129443, -0.740897119, -0.669203401, 0.666509151, -0.744766951, 0.648471951, -0.381909788, -0.573550165, 0.188253239, -0.540039003, -0.318327606, -0.523213089, -0.323695183, -0.519757688, -0.785824299, -0.818390846, 0.508213222, 0.483413875, -0.783533275, 0.773789883, -0.734820127, -0.79764092, 0.595962107, 0.348774403, 0.728198171, 0.80280596, -0.905285239, 0.696726441, -0.556371629, -0.303590208, 0.505447924, 0.654682875, -0.246009961, -0.223182008, -0.24971877, 0.70417136, 0.801208556, -0.83401686, -0.837068319, 0.727295339, 0.710075676, -0.732324839, -0.919261158, 0.631765366, 0.908012867, -0.489900053, -0.275408089, -0.695942461, -0.762747347, -0.440948963, -0.733398139, 0.183654517, -0.027274197, -0.62028116, 0.811902761, 0.743571997, -1.0051589, -0.525409877, 0.59080416, 0.890070081, 0.162616029, 0.72517395, -0.71613127, 0.769188046, 0.83349818, -0.766713858, -0.669896007, 0.711548209, -0.647645533, 0.33983916, -0.509689867, -0.800435543, -0.344411999, -0.346289754, 0.314366817, -0.663431704, -0.645073771, -0.560695171, -0.580787599, -0.820379198, 0.494530648, 0.398333371, -0.511259377, 0.692627907, -0.654955804, -0.870129108, 0.622329593, 0.41138804, 0.681844473, 0.7009812, -0.699940562, 0.538193107, -0.626960039, -0.446550846, 0.611533403, 0.669651389, -0.173716933, -0.318383664, -0.307127029, 0.626539707, 0.756940067, -0.76652962, -0.840944767, 0.790242732, 0.646067619, -0.767073929, -0.862344623, 0.598574519, 0.593686044, -0.577582955, -0.0423634201, -0.574055374, -0.77169019, -0.707057357, -0.778539598, 0.205691278, -0.00679121865, -0.854793429, 0.703709006, 0.763270438, -1.00914109, -0.775699973, 0.657759905, 0.725754857, 0.0530802906, 0.774340749, -0.833031714, 0.78519094, 0.71297121, -0.876600504, -0.740658998, 0.718503237, -0.687330544, 0.385003448, -0.725991547, -0.754310906, -0.279794812, -0.459310025, 0.188008204, -0.733313024, -0.775156617, -0.419203967, -0.273565292, -0.338725805, 0.221741572, 0.281494081, -0.342794389, 0.295483947, -0.291649103, -0.420268297, 0.387898266, 0.168785974, 0.339827657, 0.513234437, -0.494564533, 0.233384728, -0.230191156, -0.308273941, 0.325547248, 0.405156314, -0.0751813129, -0.066444248, -0.128334582, 0.244734526, 0.429480523, -0.436590225, -0.505181551, 0.468694657, 0.35836184, -0.543859482, -0.418227315, 0.220673606, 0.348470032, -0.428927124, -0.277986884, -0.291793585, -0.206854329, -0.250032306, -0.438212544, 0.218785331, 0.0412712507, -0.282670617, 0.316561878, 0.467533499, -0.459543943, -0.365904897, 0.383837134, 0.291643828, 0.1889994, 0.21689266, -0.294608653, 0.276400536, 0.293337226, -0.420555532, -0.405189395, 0.228911266, -0.250243455, 0.240290195, -0.447692513, -0.475426018, -0.201851323, -0.297056526, 0.137493655, -0.48626101, -0.345898688, -0.396780074, -0.780549526, -0.823537588, 0.542945087, 0.354397655, -0.507387161, 0.698669791, -0.818379283, -0.727007926, 0.678681433, 0.212808281, 0.604210854, 0.803043723, -0.779703319, 0.685046077, -0.663781881, -0.521312237, 0.596160948, 0.652478755, -0.35376817, -0.15544413, -0.422452629, 0.534026861, 0.805908442, -0.847195268, -0.851938188, 0.799646616, 0.857016563, -0.839247882, -0.884811521, 0.510792196, 0.88849473, -0.392984003, -0.261963129, -0.586921692, -0.646880448, -0.462142944, -0.818890929, 0.035946276, -0.281571209, -0.74871695, 0.613813758, 0.680141926, -0.949269414, -0.684969604, 0.565539658, 1.00042653, 0.150313571, 0.684495986, -0.722136557, 0.778911769, 0.782094896, -0.730289161, -0.794239044, 0.885579526, -0.69606334, 0.444901079, -0.845269442, -0.598321259, -0.542192876, -0.288296878, 0.215937302, -0.722411454, -0.702072799, -0.705431938, -0.71226716, -0.786647379, 0.531604886, 0.609665036, -0.597535908, 0.666882694, -0.793303609, -0.787642837, 0.698806942, 0.348492414, 0.540394783, 0.626096666, -0.706491232, 0.829213083, -0.538429081, -0.65759629, 0.687242925, 0.430694371, -0.264121145, -0.216645733, -0.692179024, 0.672817349, 0.805104256, -0.622378051, -0.844789565, 0.451787233, 0.719521761, -0.836445928, -0.842959404, 0.355159968, 0.653186679, -0.37796697, -0.291634262, -0.63452822, -0.671194732, -0.504214764, -0.844722986, 0.306022525, -0.0711536258, -0.702196002, 0.737235725, 0.809727132, -0.613162577, -0.383354962, 0.606713057, 0.591403484, 0.339256108, 0.54715246, -0.473906338, 0.783900678, 0.663366318, -0.75187254, -0.493442833, 0.800020874, -0.789069772, 0.564043283, -0.611755073, -0.86263907, -0.336834759, -0.462656617, 0.237991378, -0.707368851, -0.405766249, -0.630902052, -0.821267247, -0.829749942, 0.509847701, 0.460671842, -0.807606995, 0.74302882, -0.736985207, -0.782585621, 0.754141986, 0.416912496, 0.794934273, 0.86178571, -0.872833729, 0.614410043, -0.788762808, -0.349991858, 0.646541595, 0.541881561, -0.174803972, -0.426443964, -0.381490558, 0.821741939, 0.750299513, -0.836915433, -0.74960041, 0.727819622, 0.92942059, -0.863370955, -0.941732585, 0.573167384, 0.670918107, -0.577338278, -0.318402857, -0.76259917, -0.771713018, -0.665239751, -0.721295357, 0.246406525, -0.497510284, -0.683297992, 0.660865605, 0.732286155, -0.704380989, -0.739708781, 0.889108539, 0.684882641, 0.533998311, 0.649343133, -0.691442072, 0.747027636, 0.723184109, -0.669957519, -0.683325231, 0.681482494, -0.914686978, 0.17408444, -0.640013218, -0.716807425, -0.482498884, -0.154035002, 0.310868859, -0.874958694, -0.748723865, -0.56742239, -0.887781858, -0.652014136, 0.452641785, 0.549586773, -0.645061731, 0.63546443, -0.579267085, -0.748191714, 0.554392397, 0.467173159, 0.758127451, 0.917132854, -0.757915795, 0.769090831, -0.851054728, -0.255667329, 0.637966394, 0.573545754, -0.222050503, -0.438768119, -0.314697772, 0.606786788, 0.856207848, -0.851828158, -0.720914125, 0.806266189, 0.729975462, -0.809783995, -0.858449399, 0.63611263, 0.791059971, -0.416043282, -0.307958245, -0.517980218, -0.714065015, -0.545959234, -0.723166049, 0.29447791, -0.254560858, -0.749505579, 0.825292349, 0.793439567, -0.854955912, -0.56521672, 0.660036385, 0.849229217, 0.315747947, 0.638653874, -0.577628732, 0.616680264, 0.968390405, -0.862338424, -0.541128039, 0.630861163, -0.679648817, 0.262172341, -0.719775438, -0.644159377, -0.345081747, -0.21565415, 0.271060109, -0.728009224, -0.683839321, -0.481576353, -0.570552051, -0.777552724, 0.622478604, 0.579048872, -0.596874118, 0.700840712, -0.657557487, -0.895704746, 0.521527052, 0.291102052, 0.669102132, 0.621534884, -0.792802751, 0.641864598, -0.615286052, -0.564382076, 0.658665776, 0.569696784, -0.29823938, -0.0890338346, -0.522620618, 0.498231977, 0.794570863, -0.825930715, -0.709672213, 0.49634099, 0.715287268, -0.878186584, -0.740223408, 0.342125803, 0.71430409, -0.333702475, -0.176821321, -0.435841233, -0.795084834, -0.508588672, -0.649351716, -0.0135515844, -0.00657207659, -0.628678024, 0.758297741, 0.722372234, -0.989041865, -0.492844343, 0.558204472, 0.986102402, 0.104362853, 0.769734919, -0.783679724, 0.814909697, 0.65221858, -0.909674704, -0.94838649, 0.790295839, -0.832857609, 0.358761221, -0.695959747, -0.763435304, -0.301868916, -0.560335457, -0.073698774, -0.803123415, -0.589908421, -0.699640691, -0.89512831, -0.89859134, 0.456811368, 0.526388049, -0.883316159, 0.668905437, -0.864467144, -0.77936691, 0.668658853, 0.686980963, 0.708051503, 0.897727907, -0.782424867, 0.870139658, -0.710069895, -0.290644497, 0.861719429, 0.686867714, -0.0812829584, -0.515805244, -0.619343758, 0.87452513, 0.647835255, -0.735748649, -0.724878669, 0.730390191, 0.706322849, -0.945946515, -0.875465572, 0.565879285, 0.718600035, -0.742332637, -0.467122614, -0.813044608, -0.77358681, -0.570550144, -0.745883226, 0.471848935, -0.442510426, -0.769583106, 0.646922112, 0.724060833, -1.03937078, -0.738261163, 0.878113747, 0.91464299, 0.451797158, 0.864410758, -0.641917169, 0.683274686, 0.916965365, -0.788966, -0.736622751, 0.830067337, -0.689770639, 0.21498701, -0.684152961, -0.942618608, -0.576527417, -0.366254419, 0.413313627, -0.873114645, -0.718489408, -0.583863616, -0.729837894, -0.627582729, 0.446807176, 0.410488844, -0.707820356, 0.574976921, -0.890346527, -0.6144858, 0.741384029, 0.301623613, 0.731503785, 0.6993469, -0.782861829, 0.707979858, -0.698563576, -0.491824239, 0.807846844, 0.705500066, -0.118933909, -0.514284432, -0.541995108, 0.544251263, 0.638027668, -0.623156488, -0.679441869, 0.760259151, 0.714749157, -0.856507719, -0.740746558, 0.407242507, 0.653954327, -0.48238948, -0.237410322, -0.433872312, -0.78880173, -0.499718726, -0.948717713, 0.38727656, -0.382465541, -0.525140166, 0.694271028, 0.800766528, -0.854491174, -0.519459486, 0.69115299, 0.829451561, 0.367598891, 0.702863634, -0.566851914, 0.780456722, 0.797254324, -0.647499442, -0.79959631, 0.792972267, -0.824902415, 0.502618432, -0.768850267, -0.846130311, -0.492772669, -0.54319489, 0.261164606, -0.788439989, -0.598921239, -0.816673398, -0.778527617, -0.844715834, 0.340323418, 0.428646266, -0.54244858, 0.792509854, -0.643731296, -0.842107594, 0.733490527, 0.408700466, 0.724223852, 0.683781266, -0.885363996, 0.572960675, -0.702454209, -0.350052059, 0.623003006, 0.453214765, -0.112270817, -0.282705426, -0.403194994, 0.685073912, 0.766042054, -0.868627787, -0.765646458, 0.69943887, 0.751629233, -0.739947796, -0.768767118, 0.463029802, 0.651656747, -0.593756258, -0.41636619, -0.488620043, -0.625012338, -0.534433126, -0.712874651, 0.208950907, -0.133826539, -0.598224044, 0.815514505, 0.730447471, -0.830714822, -0.623293459, 0.772215545, 0.647283673, 0.318770945, 0.789138079, -0.700474203, 0.864484668, 0.667024732, -0.678884387, -0.587849855, 0.697911382, -0.829990804, 0.179155171, -0.727644086, -0.696924448, -0.538560808, -0.416034847, 0.502129376, -0.694367468, -0.645184517, -0.723423243, -0.49315697, -0.625419617, 0.38362208, 0.653656721, -0.661024809, 0.622956514, -0.517229497, -0.238649622, 0.600716591, -0.0996971205, 0.362163216, 0.714113176, -0.630294204, 0.537375927, 0.00633827038, -0.446282089, 0.578546643, 0.0746347681, -0.4034895, 0.143355817, -0.42931506, 0.271517873, 0.443827868, -0.597008765, -0.408510149, 0.279152721, 0.637251139, -0.680869997, -0.600134134, 0.105825603, 0.446815252, -0.0732483864, 0.131000474, -0.18368794, -0.113074012, -0.129835978, -0.52116704, -0.341600209, 0.373502314, -0.0196969714, 0.633913875, 0.636404634, -0.549856961, -0.143283263, 0.693931937, 0.384506464, -0.140485421, 0.332994014, -0.210686848, 0.494369686, 0.509069741, -0.465097696, -0.556577265, 0.584524512, -0.634896696, 0.527375817, -0.277327806, -0.727154315, 0.244570479, -0.380336553, -0.229002371, -0.681452513, -0.141134918, -0.518900514, -0.655364513, -0.729059339, 0.458059072, 0.374501973, -0.576015532, 0.421382129, -0.445639879, -0.613623679, 0.323306084, 0.220022663, 0.765763342, 0.710305631, -0.466584563, 0.642416716, -0.566652477, -0.159625024, 0.368171424, 0.560183525, -0.0803456977, -0.244403571, -0.230083123, 0.565429151, 0.444226772, -0.678660274, -0.834407389, 0.453305334, 0.794850767, -0.623285592, -0.748075902, 0.327078044, 0.546659946, -0.332765788, -0.0947347432, -0.348671585, -0.549773335, -0.498938233, -0.791302204, -0.0774794742, -0.111681581, -0.462142825, 0.601308405, 0.524632215, -0.952877581, -0.464764923, 0.449773759, 0.883271515, 0.108514138, 0.694043458, -0.71735549, 0.57161361, 0.592660844, -0.839791715, -0.60587889, 0.749918222, -0.508633018, 0.236129105, -0.743721902, -0.476489544, -0.195013925, -0.282672107, 0.0493622757, -0.517781019, -0.535562217, -0.329918176, -0.847776532, -0.732566774, 0.510883033, 0.623402357, -0.765968084, 0.828452766, -0.703445256, -0.628907382, 0.866131842, 0.509048045, 0.585640192, 0.649587214, -0.69290334, 0.82051605, -0.58204633, -0.753176332, 0.677423954, 0.538980126, -0.343862832, -0.418356091, -0.545816958, 0.605414629, 0.631203949, -0.595712364, -0.771879792, 0.87947458, 0.71730864, -0.630509079, -0.781133711, 0.537814319, 0.850713968, -0.634746552, -0.460097373, -0.737617075, -0.642009556, -0.758920729, -0.581466377, 0.621308506, -0.58778739, -0.690724969, 0.78928262, 0.867532611, -0.669017315, -0.833978355, 0.562109888, 0.721790433, 0.676322162, 0.621345937, -0.854133487, 0.876233518, 0.645316303, -0.745479703, -0.547867, 0.74179703, -0.88884449, 0.478366524, -0.884673536, -0.711467445, -0.470088303, -0.41912964, 0.452502936, -0.781383872, -0.814150214, -0.541235626, -0.710442781, -0.681503534, 0.536275685, 0.384036362, -0.749922991, 0.711969078, -0.740409434, -0.725102127, 0.727339864, 0.341918498, 0.818270028, 0.627205968, -0.632465899, 0.722316206, -0.669062614, -0.375851154, 0.657044291, 0.446246296, -0.219635457, -0.43148765, -0.558377326, 0.569771409, 0.593329668, -0.695811629, -0.849102795, 0.527087867, 0.578450203, -0.888826013, -0.785208881, 0.582609951, 0.618132293, -0.591299593, -0.327320755, -0.447967768, -0.604386806, -0.402412832, -0.758327961, 0.391073734, -0.389803439, -0.66774869, 0.692318916, 0.817701697, -0.829085171, -0.63115406, 0.610895157, 0.692555726, 0.369530261, 0.619796872, -0.578089237, 0.65516305, 0.839975417, -0.714050353, -0.745283663, 0.742054462, -0.830090344, 0.18377535, -0.664344668, -0.776352465, -0.420603633, -0.384506494, 0.312064558, -0.62918669, -0.657724321, -0.738200486, -0.94836539, -0.778746307, 0.483145922, 0.703871608, -0.854615748, 0.926780462, -0.809766114, -0.760736287, 0.686831355, 0.42373687, 0.84679538, 0.906513274, -0.940874815, 0.677461803, -0.703147888, -0.676685631, 0.776708007, 0.517841399, -0.369472772, -0.478993565, -0.632530391, 0.686751187, 0.770708263, -0.658292234, -0.901899755, 0.63416034, 0.723803461, -0.916967928, -0.851831198, 0.582687438, 0.92195642, -0.693708897, -0.417580545, -0.636184752, -0.802806199, -0.494223386, -0.753114402, 0.482324481, -0.390217453, -0.83683461, 0.722103834, 0.941145539, -0.733774066, -0.697950721, 0.84744823, 0.903916419, 0.276334882, 0.747675598, -0.871818721, 0.641804755, 0.958486736, -0.652596593, -0.662544787, 0.954618335, -0.931458354, 0.38261348, -0.618713975, -0.795758426, -0.476883709, -0.321306169, 0.372669131, -0.628606498, -0.773585498, -0.705211937, -0.513652921, -0.564952254, 0.429203838, 0.631790817, -0.424225926, 0.703489482, -0.739444435, -0.327212363, 0.65977639, -0.0436902121, 0.294750094, 0.699085772, -0.498512357, 0.707677662, -0.0511214808, -0.666952133, 0.649589896, 0.0616720095, -0.373967946, 0.316006213, -0.487739474, 0.341629297, 0.508030772, -0.795359671, -0.532108784, 0.133212075, 0.792977333, -0.843702078, -0.695294678, -0.0300426763, 0.527421176, 0.148822859, 0.274006784, 0.132002801, -0.177068904, -0.123832136, -0.813948452, -0.385466427, 0.25638929, -0.201113567, 0.684263825, 0.479077369, -0.674763739, -0.0226189308, 0.537450373, 0.612549424, -0.166918933, 0.320700228, -0.0951954722, 0.679965496, 0.61227119, -0.840546191, -0.634014845, 0.692002535, -0.720923662, 0.471729636, -0.273466438, -0.487667233, 0.221207723, -0.483702719, -0.364673913, -0.528105438, -0.20860064, -0.63447243, -0.864778221, -0.824272394, 0.263325602, 0.499057829, -0.529165149, 0.692652166, -0.723354042, -0.789388597, 0.558536112, 0.540036798, 0.613343656, 0.787046909, -0.741134465, 0.784529388, -0.635947287, -0.409773231, 0.533056259, 0.652541399, -0.0424025841, -0.277122438, -0.57015878, 0.5594275, 0.703241646, -0.675032914, -0.726343215, 0.618670523, 0.695467234, -0.891808033, -0.895254016, 0.585447133, 0.828479052, -0.423756212, -0.361082226, -0.632846653, -0.778389513, -0.574056745, -0.610268235, 0.310293734, -0.219143718, -0.781860769, 0.745597601, 0.836865366, -0.806676924, -0.710307598, 0.765738964, 0.700198293, 0.134091407, 0.606047928, -0.828570783, 0.783700168, 0.885118484, -0.847240925, -0.601313412, 0.667737484, -0.857893348, 0.206913203, -0.656649649, -0.590756834, -0.591427386, -0.167132616, 0.210622162, -0.674396753, -0.735662997, -0.550461888, -0.438653499, -0.484567106, 0.0423764028, 0.402782738, -0.39615652, 0.527801216, -0.405160308, -0.540103197, 0.317408293, 0.758783579, 0.668566465, 0.7315467, -0.478771001, 0.391726941, -0.548839748, -0.151168957, 0.532397807, 0.801022947, 0.0191140678, -0.552368999, -0.369526327, 0.842350483, 0.593827605, -0.494756907, -0.704736352, 0.812934518, 0.552430868, -0.62915194, -0.752106965, 0.56200552, 0.59557122, -0.596497178, -0.491576523, -0.77894181, -0.697859466, -0.540353298, -0.392811835, 0.589950562, -0.50101465, -0.765250444, 0.439478427, 0.486397952, -0.583910704, -0.842351794, 0.298052102, 0.800410271, 0.721171498, 0.577043176, -0.711164594, 0.529448986, 0.579870582, -0.761946082, -0.334211707, 0.426836669, -0.544145286, -0.0236858372, -0.72631222, -0.269898385, -0.546507418, 0.150488898, 0.486382157, -0.541724324, -0.581802309, -0.334866315, -0.60239023, -0.679095268, 0.433860898, 0.470565766, -0.718216181, 0.62314868, -0.704164386, -0.857846975, 0.596488595, 0.312603414, 0.859928668, 0.779130697, -0.86165446, 0.697177708, -0.553644001, -0.406514913, 0.730294526, 0.61478579, -0.251439095, -0.25065136, -0.441192597, 0.799790978, 0.852701426, -0.738498449, -0.6936149, 0.683245599, 0.889102221, -0.760666132, -0.890614629, 0.408153266, 0.693063498, -0.6267699, -0.428469628, -0.436086804, -0.851893008, -0.408915699, -0.692253232, 0.288505495, -0.284870684, -0.728752315, 0.845336199, 0.715213299, -0.94300127, -0.678461432, 0.612001181, 0.698265493, 0.415461838, 0.657033384, -0.831675112, 0.581083179, 0.632179201, -0.819402874, -0.801949084, 0.665694177, -0.723644853, 0.517686546, -0.691868901, -0.683371305, -0.526625633, -0.533140421, 0.305379122, -0.800289869, -0.615729034, -0.727103829, -0.730080843, -0.748888373, 0.515534759, 0.503465474, -0.710360944, 0.838060856, -0.988474727, -0.781527102, 0.7566365, 0.654545665, 0.769656599, 0.813188851, -0.902251959, 0.723203838, -0.624532938, -0.469336659, 0.796414196, 0.521895111, -0.162911385, -0.668885231, -0.52628547, 0.751163602, 0.890729189, -0.839278996, -0.962187886, 0.834596097, 0.762223721, -0.883046627, -1.05751264, 0.684665084, 0.961484551, -0.749053955, -0.341711491, -0.637594283, -0.957236946, -0.551831722, -0.882907093, 0.296203643, -0.431090772, -0.767115414, 0.733907461, 0.938528359, -0.9906919, -0.751880229, 0.84377557, 0.96890384, 0.506706834, 0.656855583, -0.781019568, 0.857784092, 0.918415487, -0.857643902, -0.841950774, 0.787070394, -0.750242233, 0.40217787, -0.849638402, -0.753489494, -0.758095026, -0.606765985, 0.335884303, -0.65856272, -0.808486819, -0.885119617, -0.671191096, -0.675404072, 0.322195232, 0.439209133, -0.442668408, 0.53856045, -0.609920025, -0.924227893, 0.699789643, 0.167366132, 0.90906626, 0.814170897, -0.704245687, 0.716417432, -0.437005758, -0.315517783, 0.643189311, 0.343112886, -0.193849027, 0.0624860041, -0.579222381, 0.521086574, 0.524299681, -0.84888345, -0.956672847, 0.606286645, 0.658358991, -0.964612246, -0.787381589, 0.4372302, 0.825733185, -0.355769753, -0.0480801389, -0.540993035, -0.848746598, -0.410088539, -0.820118845, -0.0829904303, -0.0389961936, -0.661750019, 0.672849178, 0.670697868, -1.06788826, -0.460059553, 0.770552814, 0.940687656, -0.152831227, 0.7278862, -0.698670506, 0.82937777, 0.663784087, -0.84242171, -0.728216648, 0.728243887, -0.673153818, 0.513519049, -0.753371477, -0.562419951, -0.0328404419, -0.560846388, -0.160596967, -0.750968993, -0.493129641, -0.480887413, -0.471878946, -0.570706725, 0.190867126, 0.619297624, -0.657996356, 0.641835988, -0.615748346, -0.727557659, 0.42367655, 0.645834148, 0.564158618, 0.677742243, -0.760552824, 0.562094748, -0.760540366, -0.518487215, 0.581878543, 0.531943381, 0.139630035, -0.56694454, -0.510860264, 0.56850177, 0.45130375, -0.611318827, -0.780234337, 0.677732229, 0.788224757, -0.521191955, -0.696267605, 0.604700446, 0.697250664, -0.558842182, -0.64243567, -0.664067626, -0.567382276, -0.541549802, -0.474666208, 0.383841902, -0.483801514, -0.742288053, 0.706105828, 0.699141741, -0.677887678, -0.724218667, 0.462450176, 0.588963926, 0.647865117, 0.79887259, -0.558031619, 0.72386378, 0.548757076, -0.627694726, -0.449682295, 0.678358495, -0.781508863, 0.34308818, -0.572469234, -0.358995378, -0.657875001, -0.091854915, 0.417881787, -0.64309746, -0.650072634, -0.474960387, -0.807871401, -0.87663269, 0.600731075, 0.540997148, -0.502753854, 0.50888139, -0.656033993, -0.746612072, 0.48891297, 0.265826792, 0.717237949, 0.908482969, -0.633575022, 0.726195335, -0.622035325, -0.438288063, 0.762185693, 0.634955287, -0.34310177, 0.0347639322, -0.351194203, 0.716493368, 0.632564485, -0.630600393, -0.802460313, 0.60208261, 0.898235619, -0.893882751, -0.721909344, 0.53441304, 0.595046163, -0.477534801, -0.00178506097, -0.564549625, -0.836093783, -0.445003271, -0.642233789, -0.102366239, -0.127859131, -0.575787961, 0.552174449, 0.811557174, -0.839536726, -0.513024151, 0.73071909, 1.03467178, 0.0279106591, 0.767786324, -0.663220465, 0.635928929, 0.696484566, -0.909432828, -0.634868801, 0.831269205, -0.811127245, 0.419034213, -0.797002971, -0.720269203, -0.443168491, -0.527125359, 0.078103736, -0.729779184, -0.62820518, -0.514111221, -0.945336878, -0.896292031, 0.628046334, 0.775375545, -0.839837193, 0.991284788, -0.87743324, -0.702488542, 0.801653445, 0.591093957, 0.845495939, 0.995687902, -0.867820919, 1.01508343, -0.592688203, -0.701304674, 0.719586432, 0.5491395, -0.42802316, -0.381718159, -0.723167658, 0.615308344, 0.778011024, -0.982355416, -0.971625388, 0.562777638, 1.04408884, -0.874234378, -0.8119753, 0.475267857, 0.857940078, -0.537086546, -0.357432067, -0.619285464, -0.798609316, -0.472768217, -0.919322491, 0.0175475124, -0.268886387, -0.639463007, 0.971882164, 0.976396561, -0.829320788, -0.662895501, 0.989574671, 0.921676993, 0.285999775, 0.725146711, -0.858463764, 0.864225805, 0.83296448, -0.995106757, -0.909235537, 0.770166218, -1.03288674, 0.830250442, -0.810505748, -0.901980817, -0.35455966, -0.747324765, 0.103498332, -1.01383245, -0.698522568, -0.989441216, -0.875591397, -0.758631289, 0.534163296, 0.593221068, -0.766667783, 0.581122577, -0.680642247, -0.748880625, 0.813236117, 0.420501381, 0.509810269, 0.633358181, -0.721417844, 0.870527506, -0.716211557, -0.643129826, 0.594161093, 0.48839438, -0.380239099, -0.440621912, -0.62062639, 0.536787987, 0.760927856, -0.586608708, -0.759728014, 0.663005352, 0.621978164, -0.739436448, -0.795778632, 0.38639766, 0.865861237, -0.483696818, -0.289453, -0.495639235, -0.718874395, -0.537962198, -0.53384608, 0.151461318, -0.205503523, -0.568728864, 0.866042733, 0.695957661, -0.820673227, -0.581232011, 0.865490794, 0.787113965, 0.371780962, 0.685358405, -0.609164536, 0.741983473, 0.676958382, -0.71614629, -0.689819038, 0.870664418, -0.796582878, 0.421531945, -0.676896632, -0.780096352, -0.479086488, -0.28850174, 0.189821914, -0.569561064, -0.613025904, -0.847247124, -0.753034234, -0.821277082, 0.352717817, 0.437189221, -0.591018021, 0.58764863, -0.836360037, -0.888586044, 0.62162894, 0.591918111, 0.696287513, 0.847621679, -0.901061475, 0.817827344, -0.919304192, -0.302406639, 0.495800436, 0.577167511, -0.294019133, -0.506304026, -0.355751038, 0.810717702, 0.767890096, -0.919171154, -0.83949095, 0.7900666, 0.805035353, -0.773693919, -0.883592606, 0.62864089, 0.692126155, -0.61671406, -0.191977829, -0.642546952, -0.862159908, -0.621910453, -0.652162194, 0.276267111, -0.120133847, -0.741554439, 0.571325481, 0.715305507, -0.94157517, -0.67414248, 0.568462908, 0.840916693, 0.100790963, 0.655533969, -0.888875723, 0.739804924, 0.701006174, -0.979101002, -0.886520743, 0.66766119, -0.816392601, 0.455491394, -0.83178401, -0.57834661, -0.482791305, -0.331682682, 0.252267569, -0.64348048, -0.603320003, -0.503108501, -0.673919201, -0.674786091, 0.321125358, 0.282516241, -0.41301924, 0.49846524, -0.644164741, -0.556176603, 0.414570183, 0.0295571964, 0.532456696, 0.744642496, -0.728139222, 0.638748229, -0.241313726, -0.446577042, 0.373588115, 0.214588135, -0.42782855, 0.23797965, -0.436457992, 0.29760024, 0.471895516, -0.613751709, -0.756712735, 0.247900277, 0.544378281, -0.757288158, -0.742842615, -0.00422132853, 0.727512598, 0.127632841, 0.216005534, 0.00528804818, -0.24746415, -0.042836979, -0.481200725, -0.232504398, 0.312444508, -0.129482701, 0.689032257, 0.538662612, -0.663054168, -0.346863031, 0.631804407, 0.696779668, -0.141457081, 0.54328084, -0.213508695, 0.721033394, 0.469021231, -0.680828452, -0.671968102, 0.426979959, -0.451262534, 0.405148834, -0.477650434, -0.577977121, -0.0180714726, -0.595816553, -0.234744281, -0.677820146, -0.210872546, -0.35164547, -0.752111197, -0.592380166, 0.384332597, 0.38259539, -0.623815179, 0.696658492, -0.568687916, -0.668709636, 0.438631833, 0.0161281209, 0.541475534, 0.812331438, -0.739946544, 0.670636892, -0.569358468, -0.539536774, 0.564501464, 0.410508871, -0.434464753, -0.06972415, -0.520966589, 0.541325152, 0.586624146, -0.600775838, -0.951261282, 0.725977182, 0.881927729, -0.653428972, -0.739407599, 0.505920291, 0.819680393, -0.280781657, 0.0477778353, -0.529438376, -0.519729137, -0.478428662, -0.771895468, -0.115888581, 0.041262541, -0.501470804, 0.754126072, 0.655037463, -0.79851985, -0.617849946, 0.508627951, 0.937227786, 0.0741532892, 0.752697289, -0.638364196, 0.679024935, 0.573970377, -0.784812629, -0.628459752, 0.786691964, -0.724843383, 0.5313223, -0.691406608, -0.75389111, 0.0104060043, -0.52564913, -0.188856304, -0.619440973, -0.435179591, -0.541983306, -0.690828145, -0.742705524, 0.616703749, 0.559063494, -0.721412361, 0.819967091, -0.772261322, -0.781257987, 0.631072998, 0.380338579, 0.878968239, 0.641927123, -0.675080061, 0.797613561, -0.481859565, -0.588425994, 0.635215223, 0.529319406, -0.18409355, -0.104161449, -0.584507048, 0.729360759, 0.677086115, -0.91838634, -0.699541748, 0.733176768, 0.760962009, -0.877713263, -0.714370131, 0.56864804, 0.716714859, -0.351008207, -0.0716526881, -0.416153759, -0.674840271, -0.38810128, -0.85689503, 0.106242314, -0.125452623, -0.578308284, 0.581332147, 0.908393562, -0.947099328, -0.463029057, 0.596999586, 0.669750869, 0.124098182, 0.834454834, -0.625547647, 0.756004095, 0.855139315, -0.944711149, -0.826468945, 0.742309391, -0.644201279, 0.416745484, -0.830237687, -0.879375517, -0.241261527, -0.518852293, 0.208572835, -0.896292627, -0.489128619, -0.791282713, -0.693568945, -0.740639925, 0.372672617, 0.433634013, -0.574363589, 0.647077322, -0.755927563, -0.905629396, 0.704541504, 0.472369015, 0.741631627, 0.888307929, -0.764778197, 0.816288471, -0.639776289, -0.400392085, 0.648703933, 0.462509871, -0.321077108, -0.397640973, -0.265255511, 0.60962826, 0.817197382, -0.608798206, -0.813515663, 0.745844901, 0.767741144, -0.782118082, -0.976574183, 0.521064103, 0.811404645, -0.550130546, -0.200923726, -0.801614046, -0.7105757, -0.534501076, -0.834816158, 0.108991764, -0.284213603, -0.598311722, 0.634516656, 0.662789702, -0.961711645, -0.55547899, 0.689463377, 0.925820708, 0.321004957, 0.651610434, -0.788481355, 0.839279532, 0.896962583, -0.826938093, -0.625647545, 0.783975482, -0.765987933, 0.290778339, -0.697226048, -0.772948563, -0.520532966, -0.302889884, 0.307582259, -0.853788257, -0.661415219, -0.415231556, -0.766534269, -0.880717814, 0.779176176, 0.573440909, -0.80526334, 0.675502658, -0.7605474, -0.908923686, 0.559892893, 0.478005707, 0.702541709, 0.698307514, -0.663857162, 0.71693635, -0.757445753, -0.617220759, 0.647994876, 0.76613915, -0.380599052, -0.476907998, -0.581870794, 0.834186792, 0.627154231, -0.657073915, -0.671102643, 0.841464877, 0.697518826, -0.738666475, -0.81698674, 0.449527919, 0.859983444, -0.57618016, -0.373709887, -0.46734497, -0.819586575, -0.523836017, -0.880162895, 0.242388174, -0.180107474, -0.741554737, 0.631468177, 0.889757693, -0.787249923, -0.486703157, 0.765184164, 0.743254244, 0.429390669, 0.710775793, -0.826795936, 0.700413525, 0.743750095, -0.841565013, -0.796144485, 0.741605341, -0.869812429, 0.636555493, -0.769874454, -0.753798962, -0.390066355, -0.462443918, 0.316380143, -0.839541554, -0.594413042, -0.820055544, -0.386250556, -0.766966522, 0.356104404, 0.458123624, -0.598576725, 0.611094415, -0.385008574, -0.720398903, 0.598801851, 0.609170914, 0.564221084, 0.761261463, -0.569838047, 0.671205938, -0.59444052, -0.273799837, 0.431002319, 0.572460234, 0.0684290826, -0.524966538, -0.33802247, 0.701965511, 0.488980323, -0.526777029, -0.605396628, 0.653136611, 0.723090231, -0.658642232, -0.569547355, 0.67019093, 0.650734484, -0.830076218, -0.439730167, -0.690865159, -0.595351458, -0.777168036, -0.59454143, 0.50659126, -0.472202897, -0.82173121, 0.476545066, 0.708236814, -0.645752132, -0.83805418, 0.645649672, 0.63295567, 0.571810722, 0.601033151, -0.722490191, 0.507057011, 0.666704178, -0.780126572, -0.54492557, 0.49361372, -0.570636034, 0.139321253, -0.648267686, -0.601916194, -0.568152547, 0.00459315116, 0.585618138, -0.604337692, -0.612028778, -0.489147723, -0.673163533, -0.82612592, 0.331939816, 0.503432572, -0.595406413, 0.775024772, -0.601431549, -0.774770617, 0.696077585, 0.491742283, 0.826150775, 0.60972935, -0.617925227, 0.681661546, -0.496898532, -0.407171398, 0.738607049, 0.521275997, -0.164188981, -0.427779019, -0.57765162, 0.497248143, 0.58968693, -0.774330497, -0.724048913, 0.561790466, 0.901737273, -0.811422408, -0.920115411, 0.60594362, 0.844089687, -0.510447741, -0.0845303088, -0.505962789, -0.722236633, -0.588820279, -0.905805886, 0.161147177, -0.0675906166, -0.613443792, 0.805045784, 0.740983009, -0.795017958, -0.657744527, 0.771991968, 0.768809021, 0.0715370178, 0.730388463, -0.757172644, 0.610588789, 0.921177149, -0.660802126, -0.704743028, 0.894296169, -0.776598215, 0.40083468, -0.766098022, -0.631082892, -0.482050449, -0.456523091, 0.204471916, -0.742328823, -0.618026674, -0.582585573, -0.582920492, -0.821842253, 0.319727004, 0.406875104, -0.6655913, 0.455741823, -0.710364878, -0.664153576, 0.508424401, 0.288870007, 0.550063491, 0.808270574, -0.626519382, 0.581452131, -0.569593787, -0.476818293, 0.457556635, 0.445561707, -0.0485610664, -0.24738045, -0.444985181, 0.649168253, 0.600435913, -0.82338953, -0.819419324, 0.621534169, 0.59906435, -0.827731371, -0.725520134, 0.373910338, 0.621072352, -0.55123657, -0.122939125, -0.528970182, -0.661496878, -0.421430945, -0.704984426, 0.136317551, -0.129085422, -0.465678006, 0.711385965, 0.720281601, -0.808288276, -0.476439506, 0.492560297, 0.800636828, 0.0788417608, 0.539779246, -0.795838237, 0.750571787, 0.759191751, -0.687685132, -0.687194109, 0.655379653, -0.739059687, 0.418908745, -0.578194499, -0.621934414, -0.250479013, -0.307500094, 0.276355982, -0.756483793, -0.476955831, -0.580926478, -0.880090296, -0.903894961, 0.526468813, 0.438662648, -0.586907506, 0.774678111, -0.848770678, -0.704209864, 0.764953375, 0.166147113, 0.688481331, 0.632664442, -0.728086412, 0.752528667, -0.55796206, -0.527783811, 0.602526486, 0.365419745, -0.382094741, -0.275969684, -0.543003142, 0.763042033, 0.673357308, -0.731986105, -0.954332829, 0.553861737, 0.776516736, -0.868581176, -0.702298999, 0.566449225, 0.738316536, -0.300097197, -0.0250236187, -0.584532082, -0.83366096, -0.365447819, -0.682086706, 0.0813199356, -0.108937353, -0.510033131, 0.831014156, 0.854750335, -1.01503098, -0.408001602, 0.596535981, 0.956232905, 0.0837642699, 0.824545801, -0.576045811, 0.599528611, 0.737659991, -0.831438065, -0.805607975, 0.676522672, -0.821888208, 0.54248637, -0.770706773, -0.587351501, -0.341309696, -0.550333679, 0.254630625, -0.784025252, -0.434925675, -0.583545804, -0.700247288, -0.623690605, 0.747710407, 0.651148736, -0.629630804, 0.811769664, -0.966323435, -0.811420202, 0.80123955, 0.470187068, 0.941537738, 0.727977037, -0.844709992, 0.78723067, -0.710786164, -0.578857183, 0.682575226, 0.577266693, -0.361889452, -0.41349709, -0.478509456, 0.63676703, 0.808829844, -0.806750596, -0.78288722, 0.738270819, 0.718547761, -0.728419125, -0.906690955, 0.564367294, 0.700948358, -0.680756569, -0.20343551, -0.651196122, -0.70710212, -0.679091752, -0.882806182, 0.201177254, -0.296743393, -0.753044188, 0.663322151, 0.83742255, -0.941375911, -0.575195432, 0.874027967, 0.684853911, 0.138523683, 0.814414501, -0.620623648, 0.827720344, 0.946218967, -0.781000137, -1.07697952, 0.815017819, -0.788599968, 0.502321661, -0.839025795, -0.750845373, -0.573712826, -0.620826781, 0.376246095, -0.650368869, -0.546986699, -0.63691777, -0.535458803, -0.661363959, 0.64222914, 0.445760667, -0.650036573, 0.552645326, -0.524723887, -0.470716357, 0.408812314, -0.0521448217, 0.302379608, 0.754069269, -0.734246969, 0.649500787, -0.14728868, -0.611519575, 0.548350036, 0.180664763, -0.329953641, 0.404439777, -0.46179083, 0.233125389, 0.667019188, -0.667292356, -0.578000605, 0.143258646, 0.561079979, -0.572558224, -0.53526473, -0.0906038955, 0.554567277, 0.0830396116, 0.345211923, 0.0422255769, -0.379443973, -0.0188870002, -0.753450751, -0.27103126, 0.269124418, -0.0796215534, 0.622003257, 0.532311082, -0.766920328, -0.0959044099, 0.416122735, 0.438820273, -0.333582342, 0.313035697, -0.136017337, 0.698964596, 0.491872907, -0.490498453, -0.610670626, 0.61041522, -0.681962848, 0.608779311, -0.297278106, -0.602056086, 0.0237780996, -0.524540901, -0.168225974, -0.601503134, -0.0488869548, -0.614751041, -0.709879696, -0.81053257, 0.618391991, 0.481366783, -0.586239636, 0.48582685, -0.760471582, -0.698308468, 0.743673205, 0.227188304, 0.817469895, 0.748536706, -0.744036376, 0.707273901, -0.468130052, -0.512849033, 0.601515889, 0.481829971, -0.287206113, -0.275168508, -0.35080409, 0.626506507, 0.646277785, -0.783339739, -0.864806712, 0.626492918, 0.712349594, -0.698523939, -0.916393638, 0.532894731, 0.861266494, -0.355742395, -0.180526912, -0.492354751, -0.73325032, -0.52450633, -0.812147796, 0.287403464, -0.0731531456, -0.694485307, 0.76377815, 0.586709619, -0.750046194, -0.631363273, 0.649213135, 0.623009562, 0.316970795, 0.730307519, -0.562623203, 0.680675983, 0.778665662, -0.632263839, -0.766701758, 0.748266935, -0.644944012, 0.483556539, -0.655284286, -0.631178498, -0.288947672, -0.524350405, 0.161109626, -0.751300216, -0.568219364, -0.631061614, -0.459654063, -0.453424454, 0.4379327, 0.246354833, -0.393866688, 0.473403245, -0.224508211, -0.136230782, 0.454040915, 0.0736969262, 0.0650235489, 0.224952474, -0.245984912, 0.263276607, -0.10896042, -0.407990217, 0.373538494, 0.0658154264, -0.202472121, -0.0177803878, -0.376174629, 0.212074891, 0.204538375, -0.389253467, -0.273314506, 0.14198412, 0.442196608, -0.42727685, -0.368806392, 0.0250752289, 0.319224954, -0.0275438055, 0.153941676, -0.128593057, -0.0405203588, -0.00136987807, -0.258995146, -0.129632786, 0.0687909126, -0.178865761, 0.272538632, 0.291231513, -0.438901156, 0.0344174653, 0.234318942, 0.240363508, -0.0146555128, -0.0116621116, -0.152764007, 0.43221733, 0.293311298, -0.371143252, -0.293728679, 0.235918984, -0.391553432, 0.233665392, -0.0871992037, -0.456803441, 0.10449788, -0.356044739, 0.00685795257, -0.384432673, 0.0964239314, -0.377044171, -0.885274708, -0.881318748, 0.253104359, 0.446624637, -0.68234092, 0.765807927, -0.643134177, -0.718705595, 0.599717915, 0.561697781, 0.792307496, 0.936580896, -0.690402985, 0.773174942, -0.745944798, -0.402243197, 0.582286894, 0.654970646, -0.142961577, -0.536586404, -0.349747986, 0.59360075, 0.916892231, -0.862155676, -0.807970583, 0.872830153, 0.995110512, -0.833628416, -0.78662163, 0.503455997, 0.867108881, -0.557180941, -0.245067909, -0.628006876, -0.778172553, -0.509984016, -0.902629256, 0.221031204, -0.410905778, -0.60523653, 0.781412959, 0.710905313, -0.821959317, -0.540201783, 0.886811733, 0.900645852, 0.404937506, 0.868565142, -0.854416847, 0.824203849, 0.960867167, -0.978561938, -0.785064995, 0.911447525, -0.702819347, 0.223130912, -0.829280257, -0.814641654, -0.484858781, -0.269801229, 0.268610418, -0.649877191, -0.747808099, -0.815822065, -0.656320214, -0.815543652, 0.276486754, 0.287251383, -0.579886198, 0.543531537, -0.69070071, -0.550088942, 0.576355577, 0.166552976, 0.545751989, 0.793423891, -0.554714322, 0.671759546, -0.616303027, -0.177101985, 0.416990668, 0.419458419, -0.263717473, -0.386263788, -0.426950902, 0.729058325, 0.717306614, -0.584142983, -0.870174706, 0.662294269, 0.703803718, -0.8443048, -0.807497203, 0.302130997, 0.640786469, -0.328456789, -0.208200663, -0.435652047, -0.798655868, -0.473939508, -0.58023721, 0.108643815, -0.151288792, -0.425067931, 0.54358995, 0.489806861, -0.955569923, -0.523314834, 0.548543096, 0.705176771, 0.269364238, 0.721559882, -0.485653043, 0.738701642, 0.556263268, -0.65787977, -0.59525764, 0.704077065, -0.578215659, 0.406451851, -0.627702355, -0.429527014, -0.364257008, -0.394973516, 0.261529177, -0.649741352, -0.676808894, -0.584805846, -0.629884362, -0.771311998, 0.469886601, 0.661175489, -0.873140037, 0.717514813, -0.739519358, -0.585066617, 0.757585883, 0.374872744, 0.537243068, 0.78802067, -0.637313068, 0.84425354, -0.633909047, -0.645332694, 0.598048151, 0.486647695, -0.390491188, -0.397720188, -0.545434415, 0.514657676, 0.814876378, -0.687656522, -0.646742165, 0.669502914, 0.751603901, -0.918543041, -0.719638765, 0.509990275, 0.652769685, -0.355132073, -0.333902717, -0.650711894, -0.57162106, -0.634329498, -0.857199669, 0.319073766, -0.193643615, -0.664176762, 0.715555668, 0.724739909, -0.88206625, -0.446540654, 0.897243142, 0.653189182, 0.292568058, 0.775917113, -0.535787761, 0.790724456, 0.658093572, -0.880992055, -0.838543773, 0.637600482, -0.809378326, 0.59145391, -0.600317597, -0.659047484, -0.531531334, -0.40995428, 0.377802968, -0.835502625, -0.444133312, -0.715831339, -0.659778833, -0.909406066, 0.34459123, 0.36241433, -0.573488176, 0.676793218, -0.925030172, -0.666074097, 0.750683963, 0.34170568, 0.745981514, 0.661837518, -0.658390462, 0.661465526, -0.844284654, -0.362855017, 0.820108414, 0.573328674, -0.245461404, -0.388630271, -0.492695957, 0.665697277, 0.839606345, -0.945376277, -0.834185362, 0.704771042, 0.984751403, -0.802317083, -0.847898126, 0.512270451, 0.934234083, -0.548366427, -0.196056202, -0.769618511, -0.91448462, -0.586469769, -0.686836421, 0.324442148, -0.226726711, -0.699259937, 0.787815928, 0.77986908, -0.906870186, -0.622646213, 0.664633512, 0.965379953, 0.261142105, 0.739521444, -0.882350028, 0.77965039, 0.866730452, -0.685767531, -0.897825956, 0.885700345, -0.851926386, 0.341880292, -0.788809717, -0.90377146, -0.634577394, -0.18189238, 0.202429622, -0.838257372, -0.587727785, -0.792346656, -0.633845747, -0.631282032, 0.230794728, 0.35575673, -0.635922968, 0.522366881, -0.589991629, -0.824365258, 0.563995719, 0.270632148, 0.520304382, 0.719724059, -0.703722715, 0.76465863, -0.446904123, -0.332921058, 0.617324591, 0.460172296, -0.0889797881, -0.414205134, -0.221735567, 0.722010136, 0.666653395, -0.727845311, -0.6857512, 0.691950381, 0.679212689, -0.729128301, -0.873222232, 0.429747105, 0.632395744, -0.502513945, -0.101058438, -0.613713026, -0.658724427, -0.465612978, -0.710263848, 0.206008941, -0.206594348, -0.643254042, 0.460749328, 0.692132831, -0.723083198, -0.489309937, 0.447513372, 0.885030866, 0.076142408, 0.641402721, -0.516031563, 0.681621075, 0.613610268, -0.655405343, -0.622511804, 0.722302198, -0.58512634, 0.152508721, -0.619448543, -0.672749519, -0.371426702, -0.178846836, 0.37492907, -0.680418432, -0.441070706, -0.510757267, -0.880476117, -0.724268019, 0.34619385, 0.431624055, -0.714189768, 0.486258388, -0.851258337, -0.823630869, 0.649866939, 0.534181118, 0.621223152, 0.763567924, -0.879760146, 0.846098661, -0.704669833, -0.378155023, 0.670836568, 0.726910651, -0.0993666723, -0.348512292, -0.376732111, 0.773108244, 0.582655966, -0.71459043, -1.00996244, 0.590018034, 0.840767682, -0.798443496, -0.759210229, 0.501235783, 0.751499772, -0.490923017, -0.199188262, -0.675305605, -0.689773262, -0.431640506, -0.647069097, 0.341923743, -0.18180503, -0.608682752, 0.557936788, 0.64294225, -1.08424616, -0.781532526, 0.771675706, 0.852573812, 0.121008001, 0.86827153, -0.730012476, 0.685991526, 0.905628443, -0.957201123, -0.886822999, 0.832894027, -0.599573195, 0.327064723, -0.733655334, -0.730279922, -0.53496325, -0.240384325, 0.448531389, -0.614097893, -0.794672966, -0.706376314, -0.74544096, -0.773173034, 0.570546448, 0.427514106, -0.444615722, 0.438615471, -0.742748201, -0.663514256, 0.441997886, 0.223081052, 0.768652141, 0.767352939, -0.82819891, 0.591905892, -0.502386332, -0.232138827, 0.458612621, 0.483412117, -0.339043438, -0.297307998, -0.31513688, 0.685150385, 0.517466128, -0.757387996, -0.79981643, 0.646684349, 0.64423269, -0.863603234, -0.77957648, 0.457524031, 0.581705213, -0.500070035, -2.3287168e-05, -0.416274309, -0.822454572, -0.494968981, -0.724004745, 0.151759654, -0.0470242016, -0.458320737, 0.487453431, 0.58742553, -0.985899448, -0.524392545, 0.619049549, 0.672451138, 0.015001921, 0.548505127, -0.609336197, 0.618811011, 0.609387755, -0.616203606, -0.868938386, 0.648502886, -0.706217647, 0.422117949, -0.607814133, -0.69769448, -0.282395065, -0.329915673, 0.270893067, -0.620717227, -0.434449941, -0.541051507, -0.624369562, -0.558936834, 0.36058712, 0.244339034, -0.509721339, 0.602007687, -0.488616526, -0.82423687, 0.558339775, 0.303887308, 0.681071222, 0.791698992, -0.639396489, 0.540880263, -0.672880232, -0.230734691, 0.612652302, 0.298571467, -0.315639675, -0.207863599, -0.476127803, 0.528039217, 0.636137307, -0.730558574, -0.918804824, 0.500870228, 0.709573925, -0.729761302, -0.659218788, 0.32433477, 0.783052802, -0.398996264, -0.198050335, -0.539138496, -0.606561542, -0.257705718, -0.749406338, -0.010693701, -0.0518695638, -0.626358807, 0.694365501, 0.568448782, -0.773178041, -0.513458908, 0.596947312, 0.637067676, 0.0874893591, 0.553110361, -0.563885927, 0.559856832, 0.688722372, -0.619764328, -0.72137177, 0.548958659, -0.621736526, 0.505205154, -0.535925269, -0.674300134, -0.40449509, -0.399067283, 0.189447448, -0.615793705, -0.604717553, -0.589698255, -0.838647723, -0.752080619, 0.788835049, 0.69460237, -0.737440825, 0.753825486, -0.866874754, -0.553911388, 0.60568279, 0.381400913, 0.799542606, 0.658922553, -0.826175392, 0.763886094, -0.750403881, -0.513383687, 0.743360698, 0.473003924, -0.250108391, -0.416798174, -0.682477057, 0.493673325, 0.894135594, -0.72825706, -0.762408912, 0.562559485, 0.661762416, -0.776120186, -0.684534967, 0.593696475, 0.69683367, -0.48964873, -0.251934528, -0.473286778, -0.553586721, -0.571152627, -0.764987946, 0.285947382, -0.152190328, -0.743868053, 0.636850536, 0.654663205, -0.828935623, -0.457564354, 0.71596992, 0.879196167, 0.17749086, 0.76696682, -0.50241363, 0.749014556, 0.827994943, -0.729129791, -0.730309308, 0.760133088, -0.803988159, 0.462360501, -0.660810411, -0.764885366, -0.571637869, -0.578510582, 0.438658893, -0.750849068, -0.506327748, -0.822021663, -0.714650154, -0.825934231, 0.539240301, 0.631770253, -0.681773484, 0.768352687, -0.684669495, -0.826654851, 0.555521011, 0.298306823, 0.615761995, 0.853095591, -0.768198848, 0.748523414, -0.433759421, -0.60152334, 0.576286256, 0.399834365, -0.356214404, -0.0477745645, -0.466592401, 0.760694146, 0.791846514, -0.755647898, -0.994643748, 0.675257623, 0.823906958, -0.849487364, -1.06035781, 0.467603236, 0.874277651, -0.267676383, -0.0789039806, -0.523667037, -0.837654352, -0.370442241, -0.746147215, -0.193121627, 0.109492853, -0.508127868, 0.706793606, 0.760867774, -0.912249506, -0.614453435, 0.621820748, 1.05616903, 0.0724092796, 0.778449535, -0.600701749, 0.685213864, 0.713173747, -0.947834909, -0.92477721, 0.782118082, -0.910845876, 0.557262957, -0.642096281, -0.901124358, -0.165086895, -0.645973027, 0.0933399722, -0.692308605, -0.448648006, -0.55952388, -0.670140684, -0.905963659, 0.306854993, 0.531633437, -0.750165701, 0.758622468, -0.742368817, -0.650009394, 0.735341311, 0.507363021, 0.553088129, 0.789965332, -0.782577038, 0.722765386, -0.613248527, -0.515472889, 0.760704994, 0.620433271, -0.181457773, -0.292714357, -0.51450026, 0.712335289, 0.832214117, -0.617399156, -0.663556159, 0.709122777, 0.762562096, -0.86058712, -0.972798586, 0.637008429, 0.631769896, -0.386212826, -0.238182008, -0.503032207, -0.731764913, -0.542757154, -0.684528172, 0.145795241, -0.26232785, -0.694706678, 0.654279888, 0.848053336, -0.869346499, -0.627607524, 0.800941706, 0.792691588, 0.164885432, 0.642134964, -0.732307255, 0.851825595, 0.661572695, -0.66988337, -0.766816974, 0.838316202, -0.917763174, 0.210481569, -0.714864135, -0.621068001, -0.369671047, -0.29421562, 0.194236115, -0.648427188, -0.541722834, -0.700538337, -0.609870732, -0.713482261, 0.533526957, 0.505420506, -0.761462092, 0.605680764, -0.736602604, -0.675286412, 0.51925087, 0.31862694, 0.556803346, 0.868467152, -0.661071837, 0.84828496, -0.618372321, -0.331619322, 0.755493104, 0.53644377, -0.376695037, -0.236938447, -0.668599784, 0.671508372, 0.717017174, -0.700174928, -0.876824677, 0.544158936, 0.644148827, -0.691998482, -0.885807157, 0.352006167, 0.70680356, -0.399598837, -0.373940706, -0.555352867, -0.686695516, -0.39205569, -0.804119766, 0.0855121389, -0.205437869, -0.432054162, 0.737186611, 0.873384297, -0.78546083, -0.479268819, 0.852739275, 0.745189786, 0.145215303, 0.592113376, -0.56983906, 0.796408176, 0.626489222, -0.890051663, -0.761890113, 0.804768026, -0.804488063, 0.562567174, -0.607810378, -0.657597065, -0.401996285, -0.353776366, 0.306756914, -0.631820917, -0.519993901, -0.519025266, -0.517664015, -0.691131711, 0.36419484, 0.609319508, -0.437314779, 0.45794186, -0.695542932, -0.202282354, 0.521171153, 0.0124146258, 0.248000398, 0.515286684, -0.462535262, 0.584330499, -0.0601333044, -0.483984798, 0.579564869, -0.00630701752, -0.440996796, 0.221724525, -0.497643888, 0.241753414, 0.429231167, -0.594967127, -0.696366668, 0.21122545, 0.76387006, -0.725295663, -0.682499707, 0.136870936, 0.640352666, 0.0971844271, 0.181079447, -0.093014814, -0.118214674, -0.0885042697, -0.630984008, -0.38630563, 0.343149573, -0.0148162777, 0.457977355, 0.722049475, -0.770289063, -0.171033204, 0.526406705, 0.489453018, -0.127697423, 0.378924906, -0.278416127, 0.67813158, 0.445674479, -0.490538061, -0.587413192, 0.50061655, -0.601593077, 0.658657491, -0.124319792, -0.475965083, 0.11623431, -0.622034311, -0.248465717, -0.683995664, -0.246266603, -0.596609175, -0.596734047, -0.608198345, 0.417361289, 0.346513689, -0.668772399, 0.571508229, -0.553525627, -0.786572993, 0.699519455, 0.47918123, 0.805457294, 0.825717449, -0.587299824, 0.721440732, -0.770340621, -0.458128452, 0.456814826, 0.534690917, -0.0717943162, -0.355185479, -0.490397304, 0.768769026, 0.620793104, -0.702713192, -0.69406867, 0.731720805, 0.685039222, -0.709784985, -0.866937339, 0.600554228, 0.894621968, -0.39824304, -0.373409122, -0.528678238, -0.57516098, -0.451306015, -0.687205434, 0.157774508, -0.212319404, -0.774072707, 0.5095281, 0.78033942, -0.855686426, -0.435578614, 0.479955196, 0.731096566, 0.0855724514, 0.790767193, -0.728350103, 0.576205313, 0.839295089, -0.918894947, -0.518834651, 0.634736121, -0.622217238, 0.191857859, -0.624470174, -0.80250901, -0.496632963, -0.225754946, 0.297484487, -0.741780341, -0.711499035, -0.498131931, -0.770092607, -0.841350377, 0.710871935, 0.60860157, -0.634379983, 0.62338388, -0.786254048, -0.743752658, 0.778513968, 0.380605906, 0.741564929, 0.70950824, -0.632787704, 0.81374234, -0.680804193, -0.592398763, 0.656908572, 0.738384008, -0.337080717, -0.0387269668, -0.671773136, 0.562348604, 0.677132905, -0.871127427, -0.902743757, 0.662843525, 0.642007768, -0.722330868, -0.686625183, 0.543022215, 0.852080941, -0.396655589, -0.234145701, -0.704787552, -0.892564118, -0.563664794, -0.700944304, -0.0499284975, -0.100071982, -0.824975193, 0.785685837, 0.733327806, -0.985789955, -0.494533747, 0.569079041, 0.995475829, 0.0173491687, 0.716639459, -0.597337127, 0.716359913, 0.881419241, -0.705274582, -0.763357162, 0.788009644, -0.671955466, 0.600070059, -0.857818961, -0.832677364, -0.356224716, -0.592254996, 0.16872856, -0.698387325, -0.623712182, -0.604543328, -0.763082504, -0.834628224, 0.306040227, 0.354302883, -0.690976858, 0.498179018, -0.558686435, -0.842178226, 0.438858449, 0.357613653, 0.620885849, 0.764080763, -0.636522174, 0.613910079, -0.523531854, -0.403488576, 0.608101547, 0.396393418, -0.371086329, -0.102414593, -0.344746709, 0.537199318, 0.770033062, -0.823680878, -0.7562536, 0.477918386, 0.816444635, -0.855723262, -0.935863197, 0.25004217, 0.567221284, -0.451333195, -0.189253494, -0.313493073, -0.591894507, -0.536549568, -0.795074642, -0.0487271845, -0.081170328, -0.453078747, 0.655549645, 0.607715666, -0.960428238, -0.330212355, 0.587273061, 0.872655749, -0.066790849, 0.751874685, -0.540155113, 0.666716278, 0.634060979, -0.762022197, -0.850647628, 0.606674075, -0.552743554, 0.432056487, -0.705360293, -0.635362208, -0.265966207, -0.312942952, 0.163740516, -0.781231821, -0.646184325, -0.497765034, -0.594749868, -0.651977241, 0.510962903, 0.48331815, -0.711388707, 0.794482172, -0.634144604, -0.600354552, 0.771782517, 0.279378742, 0.664090395, 0.772180378, -0.86859268, 0.664606512, -0.463581741, -0.459145635, 0.745127141, 0.625650525, -0.388047993, -0.26752314, -0.356980205, 0.603207767, 0.558677435, -0.837008119, -0.860293925, 0.733782053, 0.654158711, -0.948712885, -0.706182182, 0.542136014, 0.795793593, -0.578172207, -0.244856983, -0.551398873, -0.859765828, -0.471795768, -0.957506418, 0.00114870397, -0.14141044, -0.672573149, 0.543505609, 0.854262054, -0.974989355, -0.570677876, 0.592236638, 0.753340125, 0.258676648, 0.774816573, -0.561520278, 0.720794737, 0.861506224, -0.818280399, -0.816248298, 0.660308182, -0.783487797, 0.472559541, -0.567909062, -0.769841135, -0.36992982, -0.44512248, 0.211672798, -0.85831058, -0.564784288, -0.736187398, -0.856575489, -0.688995361, 0.528019369, 0.580864489, -0.717701197, 0.575223446, -0.840357184, -0.644141495, 0.560073078, 0.418458194, 0.813837826, 0.743292391, -0.85651195, 0.694204092, -0.666799128, -0.335520416, 0.796116233, 0.490970165, -0.245439738, -0.314309359, -0.502725542, 0.765975296, 0.652717173, -0.740998805, -0.803605855, 0.834221482, 0.872561216, -0.75937748, -0.92128849, 0.614450514, 0.732889235, -0.589897335, -0.390999287, -0.749984324, -0.617868781, -0.692896664, -0.862923086, 0.263996333, -0.164384902, -0.605936825, 0.638017118, 0.914242387, -0.919540823, -0.641202629, 0.672807336, 0.821525395, 0.146091089, 0.731206298, -0.78296268, 0.688082337, 0.840435922, -0.965001762, -0.908083916, 0.851012588, -0.926303267, 0.385692447, -0.648626029, -0.831952035, -0.507010758, -0.316051006, 0.214994669, -0.90746206, -0.628715456, -0.815836489, -0.741105139, -0.597110569, 0.524019599, 0.573146105, -0.56936115, 0.471742421, -0.512584746, -0.495997608, 0.447572201, -0.0882092565, 0.514143169, 0.578645289, -0.544580996, 0.523378611, -0.346962571, -0.357619643, 0.54893893, 0.158550799, -0.386341751, 0.198253721, -0.508448303, 0.405493885, 0.60287261, -0.553333104, -0.846876681, 0.306857377, 0.784080625, -0.839027166, -0.768278539, 0.38080126, 0.679028571, -0.257493436, 0.00781017542, -0.178098157, -0.550591588, -0.229759976, -0.516107321, -0.101500362, 0.332074463, -0.374716163, 0.481380939, 0.503152072, -0.742745996, -0.411417663, 0.519585848, 0.61863476, -0.272574306, 0.530502439, -0.326629937, 0.633793116, 0.552621722, -0.820581615, -0.661003768, 0.581622362, -0.710823774, 0.636210501, -0.430048436, -0.610860944, 0.161980703, -0.536463141, -0.158715799, -0.59583956, -0.228576854, -0.652957439];
    CONSTANT recurrent_3_u : ARRAY[0..4095] OF REAL := [0.0300211906, -0.0726404935, -0.0737517402, 0.158155724, 0.101881593, 0.0459016934, 0.106127605, 0.0329704545, -0.0344988927, -0.0758979842, -0.0294167735, 0.0405295789, 0.0192210935, 0.113318145, 0.0260757133, -0.0657523498, -0.0224163197, -0.134512767, 0.00873535872, 0.0424721651, 0.103415355, -0.0688372254, 0.084060438, 0.0470905825, 0.0343437381, -0.0326196477, 0.0298775509, -0.0407948419, 0.101322442, 0.0656937957, -0.142149746, 0.015102867, -0.0493602864, -0.0175211914, -0.0303692408, -0.197288126, 0.14125213, 0.0856058896, 0.0221487749, 0.0296264663, -0.0948507115, -0.0278902445, -0.0167066362, -0.0772125348, 0.0345653631, 0.113668807, 0.119799644, 0.109393142, 0.0327464528, -0.112259045, -0.132422939, 0.116845936, -0.0464105122, -0.0504373275, 0.148030668, 0.12590833, 0.0312110968, -0.0305655356, -0.00114641618, -0.00481387228, -0.00148997642, -0.0140454788, -0.043380253, -0.0010807598, -0.014458037, 0.0159579515, -0.0403428823, -0.014772784, 0.0942004994, -0.082610406, -0.0322015435, -0.00887908973, -0.0458164886, 0.0110293124, -0.0739976466, -0.0362581946, 0.0755177662, 0.10764505, -0.100206763, -0.0479895957, -0.111544885, 0.11783307, -0.0622494444, -0.0618790276, -0.126783609, -0.111381091, -0.0407576784, -0.130454913, 0.0215890706, -0.0911371484, -0.0917792618, -0.130048037, -0.0297309868, 0.0877916068, -0.000393094262, -0.0588469468, -0.0297936685, -0.0971366912, 0.0301536247, -0.0722011104, -0.0837551877, -0.0260783099, -0.0586579666, 0.108883359, 0.0492240526, -0.16584681, -0.00450916216, -0.0253114011, -0.142470971, 0.0402365401, 0.0252783075, 0.0431143455, 0.0667134449, -0.10590326, -0.0664104894, 0.019558616, -0.0875182301, 0.033093445, 0.0697155371, 0.137690231, 0.0145864999, 0.0742130131, 0.150406629, -0.048722323, -0.0507028066, -0.0139164925, 0.0272116177, 0.0848037228, 0.103041291, 0.133840501, 0.128629327, 0.114150807, -0.0149933994, 0.136328578, -0.00714633893, 0.0632263646, -0.00389948674, -0.0373136587, -0.0361660421, -0.0706003681, -0.0132233119, 0.102651268, 0.0970900208, 0.0556763969, -0.0266075041, 0.16801855, 0.122122914, -0.0653990805, 0.0837429464, -0.0436800718, -0.0256232154, 0.102124937, 0.0752657056, 0.154713422, 0.0260666274, -0.0506237373, -0.0284463856, 0.0192195773, -0.00573915523, 0.0273115728, -0.00244970806, -0.138179153, -0.151856139, -0.0549204648, 0.0667010546, 0.0133919455, 0.0681342036, 0.083140105, 0.0790066496, 0.101608828, -0.0148200337, -0.0527088344, 0.0216680504, -0.126744986, 0.0727042332, -0.0177761577, -0.0781563297, -0.0114615867, -0.101109624, -0.134685636, 0.0576641485, -0.147509247, -0.0655705184, -0.0140403695, 0.099234961, 0.00335595477, 0.0481827967, 0.00108642969, 0.0677736476, -0.0509829633, -0.0663982257, 0.0251895357, 0.0575018488, 0.0351390764, 0.0143772382, 0.0510687828, 0.128724203, -0.0524879545, 0.0846009701, 0.0215634666, 0.0215874463, -0.0228919853, 0.136334121, -0.0845987946, 0.0723666176, 0.0102376565, 0.00383732724, 0.0103866477, -0.0431142226, 0.124460228, 0.200107276, 0.0479671881, -0.0755812079, 0.0902619064, -0.142843604, -0.0545342304, 0.0527493209, -0.0541797392, -0.0768503621, 0.0616208948, 0.0837951601, 0.00714502344, 0.0858522058, -0.0840131864, 0.0268256329, -0.0438843518, 0.0573481992, 0.0930459574, 0.0372035205, -0.143966675, 0.00481981924, 0.0248197056, 0.0165912248, -0.0476145633, -0.0617588572, -0.0879868492, 0.0660810098, 0.100188769, 0.0131307421, 0.0687118918, 0.02752617, 0.0834473521, -0.0857155919, -0.0603220463, 0.0110164033, -0.0817635432, -0.0143848229, -0.0562525913, 0.104724899, 0.0878890306, -0.0319999419, 0.123851545, 0.089456372, 0.028816184, -0.0516834185, -0.0678242892, -0.000487238081, -0.0662352368, 0.0014590444, -0.0246563964, 0.0686305761, 0.00554418843, 0.0282515567, -0.0481138304, 0.109705061, -0.106394254, -0.0443215072, 0.0999002159, -0.139139235, -0.00928665511, -0.0397253111, 0.0938298702, -0.0839995667, 0.0965257809, 0.0854988843, -0.00975783449, 0.0243535042, 0.0170450639, 0.0159549676, -0.100652389, -0.0341138393, 0.109760039, 0.0544666052, -0.118620828, -0.129411712, 0.125624835, -0.00942844898, 0.0457218885, -0.0322152488, 0.154747665, -0.0719875544, 0.0825248212, 0.0222184435, -0.107487805, 0.0240580626, 0.0342749134, 0.0545804426, 0.118475847, -0.0381727219, -0.0196922328, -0.0122831464, 0.0579704605, -0.102477662, 0.0445675552, -0.0130214822, -0.127181083, 0.0127406744, -0.0519533753, 0.0756189078, -0.0517086349, 0.0865597799, 0.108242944, -0.026486462, 0.0976301357, 0.0297792871, 0.089461118, 0.111656331, 0.11560344, 0.0867624208, -0.100683779, -0.0620547384, -0.00687698228, 0.0556412488, 0.0257217046, -0.12562339, 0.0703864098, 0.00830022153, 0.0186630096, 0.0221271738, 0.00233624596, -0.0128272325, -0.107483052, 0.115353957, 0.0140514653, 0.00380971842, -0.0164475031, 0.0248292983, -0.0229293928, -0.0233162344, -0.0321218781, -0.038253095, -0.0523340404, -0.0502889566, -0.0859642029, -0.0186352953, 0.0504419096, 0.212066144, 0.030847637, -0.0039832443, 0.20387359, 0.0830581039, -0.0162938889, -0.052821219, -0.0775873214, 0.0432782136, 0.00630828878, -0.0598597825, -0.0590133592, -0.0160276555, 0.0762145072, 0.0913062766, -0.0763732195, 0.0536984429, 0.126260594, 0.166124925, 0.0996124595, -0.0353368782, 0.0919128805, -0.0817618892, -0.13060537, -0.0492496602, 0.0797692761, -0.0509658232, 0.0341931991, -0.0244456176, -0.144371673, 0.016945241, 0.0437188074, 0.17513822, 0.161979482, 0.0447574817, 0.0721322522, 0.0259358902, 0.0513263829, -0.00340208528, -0.0856347457, 0.0574826561, -0.0435986854, -0.0393212289, 0.0103515256, 0.0027629137, 0.0590720773, 0.161202669, 0.0285558328, 0.042487599, -0.0245804042, 0.0756384581, -0.0490016155, -0.0437188633, -0.0879897624, 0.0908604413, 0.132594928, -0.0411755107, 0.0144351618, -0.0396872498, -0.0632711202, -0.0996934697, 0.079484418, 0.0767583698, -0.0284296796, -0.0203310624, 0.0465131924, -0.0777078941, 0.0394401476, -0.110213131, -0.0243016966, -0.0619608201, -0.00736968173, 0.0807653293, 0.0781108961, 0.0670029446, 0.0359667651, -0.17489022, 0.106508911, -0.0314920023, -0.0596255064, 0.0357943326, -0.0147969089, -0.0322091728, 0.121625692, 0.0630649924, 0.0156011377, -0.154010162, 0.156323478, 0.0521048158, -0.0744174048, -0.0438708104, -0.0274148509, -0.0384579822, -0.0622124374, -0.0403489545, 0.0828858912, 0.0269311965, 0.0437574945, -0.0243850574, 0.0194006916, 0.0877681375, -0.00616865419, -0.0443016589, -0.151599303, 0.0342801288, 0.1373882, -0.118570536, 0.0311327502, -0.0471654721, 0.0557361841, 0.0510144457, 0.167004779, 0.0370514207, -0.176691324, 0.10364899, 0.175244823, -0.0285309106, 0.0586183444, -0.137841046, -0.0251355357, 0.0926762149, -0.00946547836, 0.0714036003, 0.0133831464, -0.0166843832, 0.104796365, 0.0341226198, 0.0298807379, 0.0892409384, 0.0160754696, -0.0776526034, 0.0406826064, 0.00695893914, 0.00179352146, -0.0359312594, -0.0307491533, 0.0842620283, 0.0597327799, -0.058489684, 0.0652802438, 0.120634273, 0.00839943811, 0.0148034543, 0.0289159715, -0.181493834, -0.0612624437, 0.0701209456, 0.124627896, 0.0699967667, -0.0332627669, -0.00146601256, 0.0155480355, 0.0124639738, 0.101679124, 0.0661147386, 0.0655676425, 0.032507211, -0.00537183508, -0.116009071, -0.0426227786, 0.0338342711, -0.133613735, 0.103789069, 0.0237721466, -0.0146712111, 0.00209892727, 0.0812517703, -0.0960010216, -0.0398812182, 0.0841294602, 0.171301529, -0.0616740137, 0.0314620994, 0.0257012378, 0.138789892, 0.07173419, -0.0192908831, 0.0400421247, -0.0696838275, 0.00150038349, 0.0377930924, -0.113104664, -0.134451911, 0.0513372198, 0.00518697686, -0.00657348242, 0.131591082, 0.142681986, -0.166281387, 0.0281995982, 0.0722631142, 0.0553090014, -0.118525259, 0.0537127964, -0.0449562706, -0.0177839696, 0.0959131941, -0.0462499596, -0.0772643313, 0.235673472, -0.0921119079, -0.0824815929, -0.128127351, 0.0130128087, 0.0265209489, 0.00377602875, 0.133012831, 0.019820774, -0.065849863, 0.0459060445, -0.0681104958, 0.176234603, 0.0335450768, 0.000476682559, -0.134560227, -0.068593353, 0.059597306, 0.061161451, 0.089002952, 0.0547687411, 0.0282784533, -0.0931563526, 0.0148324687, 0.0850364491, -0.0328171328, -0.0634967685, 0.0538393185, -0.097870335, 0.0359249488, -0.0242960434, -0.0517275594, 0.0977952927, 0.0730445832, -0.0189512577, -0.030794397, -0.0424824655, 0.084905915, -0.0634760335, -0.0200301968, -0.0350165367, -0.0351203829, -0.0237792451, -0.0402107127, -0.0557167828, -0.0084409751, -0.015320668, -0.0336955488, 0.0718489289, 0.0624024086, -0.0760541111, -0.0849370658, -0.0865568519, -0.022664452, 0.045539435, 0.019727692, -0.00562720094, 0.00124942325, 0.128961012, 0.0534549765, 0.0855579302, 0.135221332, 0.0438616425, 0.0642335489, 0.0753047913, 0.0217456222, 0.0435579643, 0.0114335567, 0.00198130636, -0.0206198171, 0.0332672745, -0.0287975669, -0.0422020666, -0.0687767342, -0.0427560359, -0.136115283, -0.035427317, -0.0615837239, -0.107946299, -0.0263088681, -0.0157322623, -0.148495913, -0.0870623365, -0.0430138223, -0.0760763884, 0.012971051, -0.0292470958, 0.100048348, -0.019314222, 0.043334052, -0.0361490287, -0.125617921, -0.00180942146, -0.0627233908, 0.0159676187, 0.06812042, 0.115724817, 0.0870643035, 0.089640528, 0.0293276422, -0.0362524278, -0.0057851607, 0.079749383, 0.0676407516, -0.0731888264, -0.0598182678, -0.0336906984, 0.134522706, -0.0538420193, -0.0105081927, -0.0904522911, -0.0529807955, -0.115023464, -0.038046483, 0.0693064481, 0.0703464672, -0.101286009, -0.0829353929, 0.0810176209, 0.0267352816, -0.101998039, -0.0210474525, 0.0896722525, 0.0948957875, 0.0764785707, 0.0969453454, -0.044386968, 0.0178281143, -0.0157930516, 0.0637591705, 0.0534478016, -0.081791535, 0.0674777701, -0.0889050141, -0.0679636002, 0.227865309, 0.0386979356, 0.0846257955, -0.0238306765, 0.06915465, -0.0421275944, -0.0846743137, -0.0721803308, 0.0645987764, 0.0114659499, -0.0156908818, -0.0076075457, -0.0451015644, 0.0247296635, 0.0169328228, 0.101324432, -0.0569279343, 0.0550814345, 0.0642896295, 0.0399167463, -0.112161696, 0.000747356564, 0.0287158061, 0.00583758857, -0.0576586165, -0.177706122, -0.0233383477, 0.0158482641, 0.0426830277, 0.0378117561, -0.0384511724, 0.096626699, -0.0304281991, -0.0344576202, -0.068981126, -0.00999236107, -0.145686835, -0.018794328, 0.0549363159, 0.124868475, -0.0528515503, 0.00542497449, -0.00926763751, 0.00520887785, -0.0385200195, 0.105377898, -0.0153157115, 0.0096886605, 0.00409470033, 0.0240849257, 0.0299824476, 0.160701066, -0.00693662558, 0.110601895, 0.00107865594, -0.0841737986, 0.136813968, -0.0556525066, 0.0395123363, -0.0475255772, -0.00245102565, -0.0300234612, -0.0887759477, 0.0292069353, 0.0324145108, -0.0729678869, -0.144896433, 0.0627085492, 0.121023059, 0.101523846, 0.0460572615, -0.0130476011, -0.00442671869, 0.0776944309, -0.0256401189, -0.0258534029, -0.0875134617, 0.0316531472, 0.0134338001, 0.0183724258, 0.0910221785, -0.0448424555, -0.0671966597, 0.0819778144, -0.0927601233, 0.00420876965, 0.158277199, 0.0418164693, 0.029462399, 0.00131501374, -0.0552261472, -0.0408456959, -0.0457095131, -0.0668665469, 0.0422913805, 0.0386807621, 0.0470974259, -0.0555757433, -0.0114802998, -0.0459007248, 0.074424386, 0.0140240137, 0.0515092053, 0.109739125, -0.0375749506, 0.0098653771, 0.0736354217, -0.122812606, 0.0480498485, -0.0437185392, 0.0702512339, -0.0894126296, -0.0827951878, 0.0436093435, -0.0645922944, 0.0789797977, 0.0291797891, -0.0355316103, 0.101332135, -0.198943242, -0.104029313, -0.0112727433, -0.0789091587, 0.0118773729, -0.000342540676, 0.00273814611, -0.0632523596, -0.0654634759, -0.14086774, 0.136601105, -0.00821176264, -0.05583781, -0.0290638618, -0.0186112896, 0.106708393, -0.00524609815, 0.111985132, 0.0159759019, -0.0196489394, -0.0310848951, 0.0919062495, 0.00128706126, -0.0524096899, -0.0410058796, 0.0994544774, 0.0383059569, 0.001709793, 0.0270505175, -0.0850914195, -0.0341122113, 0.0382801443, 0.0187875647, 0.03861361, -0.0111816321, 0.0419666916, -0.00145811588, -0.0587432943, 0.0371218286, -0.00978743471, -0.0155214313, 0.0722185299, -0.0625950396, -0.051668454, 0.00635217084, -1.98557973e-06, 0.0266079903, 0.0965104178, 0.0593874231, 0.0157394018, 0.0291254073, 0.0470053293, 0.0284078233, 0.0667273998, 0.0530054197, 0.0479614139, -0.0406582095, -0.0848233402, -0.00881057326, -0.0390305854, 0.0470714867, 0.0330141634, 0.00621182565, -0.0400558338, -0.0110622616, 0.0188171957, 0.0332569443, -0.0973213315, 0.0514376462, 0.020230297, 0.00126702804, -0.109365977, -0.0354114696, 0.00999673083, -0.0252558291, -0.0149314767, 0.00663108286, -0.0941324905, 0.0610380322, -0.0831719339, 0.140592024, 0.0717088357, 0.0179549288, 0.0568820946, 0.0589482784, -0.00344366487, 0.0709155127, 0.0246975198, 0.0629138201, 0.0472637042, -0.0260836314, 0.0358886868, -0.0351610072, 0.0206064209, -0.0899197832, 0.0360539705, -0.0156198898, -0.0287199263, -0.0237169545, 0.140227064, -0.0215220582, -0.0155000035, 0.0248110592, -0.0333273523, 0.0362003744, 0.120821871, -0.0120896529, 0.0651367903, -0.104569778, -0.0685840696, -0.0592691414, 0.0800046921, 0.0394370072, 0.0483403578, 0.0630822927, -0.0838180184, 0.0636225641, 0.0329086259, 0.0978200436, 0.0213489477, -0.0855389982, -0.0740655288, 0.0161811933, 0.151725888, -0.0902655944, -0.0280115698, -0.0420006812, -0.0466880724, -0.0898003578, -0.141560018, 0.0149214026, 0.039345447, 0.0207163505, -0.0258197337, 0.0121819992, 0.0104798116, -0.019134406, -0.0742832571, -0.0608402789, 0.00371132605, -0.0716577843, -0.0102680735, -0.0282074492, -0.013085071, 0.00696290471, 0.00381721556, 0.052351106, -0.104948543, -0.00349350553, 0.0223676227, 0.00554437935, 0.0151917338, -0.0154319704, 0.0451491438, -0.0366223976, 0.0613482259, 0.00938831456, 0.12777096, -0.111735135, -0.0348628685, 0.0266387966, -0.0848575756, 0.0460705794, 0.00341442367, 0.0079893088, 0.00728575746, 0.0120959003, -0.103442483, -0.0214767233, -0.0122043844, -0.104347214, 0.0350893177, 0.113822937, -0.00995320454, 0.0689455718, -0.0145815704, -0.0428336859, -0.0286409333, -0.0811021999, 0.125193283, -0.0192737803, 0.0276477393, -0.00993182324, 0.0471581817, 0.0231339596, -0.109355502, -0.117305204, 0.144997433, 0.0151157714, 0.0844534338, -0.0343651734, 0.0428620316, -0.00809036475, -0.0672432184, 0.0611731224, -0.0845748857, 0.0148144085, 0.0099927634, -0.109748997, -0.0800439194, 0.0179431085, 0.0386479609, -0.0328162126, 0.0233447067, 0.000507566147, -0.0540861897, -0.0436197668, 0.136744231, -0.0723383427, 0.120576993, 0.0313198715, 0.0151343495, 0.00956058688, 0.0441376679, -0.0929630175, 0.0826271847, -0.0876522288, 0.0497241579, -0.0532637313, 0.0360197909, -0.120650068, 0.0634097308, -0.0932886973, -0.152571946, 0.0495552868, 0.0512149744, -0.0588000938, 0.00934654661, 0.00886407867, 0.120594025, 0.0621935613, -0.0745492056, -0.00351090031, -0.0503250659, 0.0951018482, 0.0218997821, 0.0429161862, 0.00255380943, -0.192196816, 0.00421994459, 0.0331431404, 0.0209429264, -0.0102446675, 0.065385744, -0.00934347603, -0.0778645501, -0.0742510259, 0.0279874597, 0.00824572891, 0.022834558, 0.0787923485, 0.068176806, -0.142575294, -0.0214019455, 0.0431722999, -0.00839523599, 0.0336834826, -0.0530726165, -0.0890816003, 0.0272959881, -0.0813687444, 0.0251530595, -0.0454012901, -0.0119484328, 0.0687285289, 0.0111977039, 0.042694129, -0.0184652433, 0.0290676206, 0.120775983, 0.0462502204, 0.0458604582, 0.0991594046, -0.0471682623, 0.0169123765, -0.0223320536, 0.0584361143, 0.0313238092, 0.0598582178, 0.0452558696, -0.0473417453, -0.0160958096, -0.0382179171, -0.113199547, 0.0429387018, 0.0126064243, -0.141708672, 0.0561275259, -0.0514974706, 0.0028870441, -0.00186583144, 0.0542809814, -0.133144855, 0.13110131, -0.0619775467, 0.0667550638, 0.00407430343, 0.0933402628, -0.0220654439, -0.0276085194, 0.0261877533, 0.0389356427, 0.0085213501, -0.119906865, 0.0741268024, -0.0328141563, 0.0718610287, 0.0872857198, -0.0447113216, -0.110671438, -0.0578399003, 0.0857168809, -0.03271107, 0.0738816559, 0.108883522, -0.0343707502, -0.00753945531, 0.0515688322, -0.0147661353, -0.0524580479, 0.0608402789, 0.0445684753, 0.0285523068, -0.109277993, 0.070337534, 0.0272401553, 0.0353941433, 0.0222975779, 0.0128672598, -0.00301552005, -0.0973205864, 0.10792546, 0.018098237, 0.104823112, -0.0538132042, 0.141909778, 0.0314420238, -0.0277270172, -0.0402160212, -0.015063649, -0.0499392673, 0.090666987, 0.10393694, -0.0378711149, -0.0596093759, 0.0535159633, -0.130450368, 0.0946984887, -0.0148644941, -0.0580188856, -0.0506390184, 0.0958756357, -0.00710751256, 0.04835172, -0.00110983336, 0.0637535378, -0.0741288438, -0.0353915319, -0.0536486879, 0.0236730259, -0.01360323, -0.0201059133, -0.197702736, 0.0104328562, 0.0219679624, 0.0193600822, -0.0580621734, 0.000722768717, 0.020218214, -0.0416449681, -0.0252169892, 0.0284183025, -0.0408081897, 0.0971229225, -0.0989613086, 0.0676739514, -4.57838178e-05, -0.0325548425, 0.124891654, -0.0249339845, -0.0448648669, -0.0860858411, 0.135519788, -0.0126024559, -0.00650942046, -0.0178682227, 0.0157775246, 0.0321179777, 0.0359329842, -0.154746488, -0.0417040624, 0.0106083816, -0.0687999204, -0.04342594, -0.00977691263, -0.114951603, -0.167931125, 0.130631298, 0.180089399, 0.0460239872, 0.00140842423, -0.0103462273, -0.0837078989, 0.203594267, -0.139691621, -0.0553071611, 0.0519921556, 0.0752987489, -0.02307266, 0.0217926558, 0.0384444743, -0.0378084481, -0.00622680411, -0.0154887512, 0.0137523329, 0.02744684, 0.0529851243, 0.00022099771, -0.0210061241, -0.0213450324, -0.00144641288, -0.0338753499, 0.0976678208, 0.0839371234, 0.00644144183, -0.0212083384, -0.00823141076, 0.00303189107, -0.0606096461, 0.0214796457, -0.0091151977, -0.149327904, -0.0816511363, -0.00109600648, 0.160985664, -0.0915080979, -0.0764324665, -0.0513857156, 0.0188563056, -0.0482605658, 0.0110944454, 0.00537128374, 0.00916528888, 0.111269832, 0.0517503619, -0.00489495322, -0.0374845117, -0.00212028786, -0.0960891694, -0.0880883113, -0.0025981334, 0.0541328788, 0.0289277323, -0.0322767906, -0.0763743296, -0.124166809, 0.0541787446, 0.0224841125, 0.10735859, -0.112267554, 0.0613304041, -0.0375550166, 0.0711611584, 0.0157942362, 0.0914436802, -0.0144078666, -0.0181604102, 0.0121784825, 0.00565243559, -0.0955590308, 0.0696517527, 0.0795066208, -0.00259897113, -0.0420458987, 0.0728832036, -0.0184523873, -0.202795371, -0.0350662023, -0.0611995086, -0.0217991471, 0.0101415236, 0.0153950425, -0.0374389775, 0.0952190459, -0.0143837286, -0.0147394054, 0.0437798947, -0.140954733, -0.0967265069, -0.00696234219, 0.00492353737, -0.0288501102, 0.0016134372, 0.00987270288, 0.0545649603, 0.183393598, 0.0611884519, 0.0782967359, 0.0560247451, 0.0338543355, 0.00486933626, -0.0185989141, -0.127538711, -0.112394586, 0.0266220234, 0.0501661748, -0.238818854, 0.075178951, -0.0953118056, -0.0361153409, 0.0358236432, -0.192152649, -0.091668129, -0.0130089419, -0.00927320961, -0.0107419714, 0.0461085662, 0.0165692661, -0.0513927191, 0.00370220933, 0.0259465929, -0.100428723, 0.0388426632, -0.0524522066, -0.025584789, 0.0589909889, -0.00583225675, 0.0193980969, -0.0032009799, -0.0188045986, 0.0178497285, -0.0385144688, 0.081183672, 0.061315082, 0.0825035498, -0.0108325351, 0.0939969048, 0.118712887, -0.110002652, 0.0159510095, -0.0272368379, 0.0272152591, 0.075575456, 0.0401944853, -0.139272094, 0.0121700456, 0.0693234056, 0.067877762, -0.0503801927, -0.0100093447, -0.0268891584, 0.0517582633, -0.0206706841, -0.035483554, -0.0586260855, -0.0300630294, -0.119854912, -0.0620919578, 0.100395717, 0.113561206, -0.0681952164, -0.112974942, -0.0581537336, -0.00899193622, 0.0414297767, -0.0132136792, -0.027603507, -0.022939615, 0.134260103, 0.134957984, 0.020267915, -0.0543925762, 0.00606182963, -0.0194226392, 0.00143498369, -0.180657759, -0.010997694, -0.0365972891, -0.0676313266, -0.137266397, 0.0148993051, -0.133080408, 0.0260280091, -0.00607299339, -0.0297786333, 0.0242825039, -0.0418978855, 0.0773347393, -0.000944940373, -0.0122882165, 0.134246141, -0.181817785, -0.00448207185, -0.0666503161, -0.000194192515, 0.0506850034, -0.182508036, -0.0106826015, 0.0565887913, -0.163172677, -0.000436317176, 9.17259604e-06, 0.00623785146, -0.213638961, -0.11311245, 0.114885837, 0.136188999, -0.0547634289, -0.0319928341, 0.063556686, -0.0383523665, 0.0233660601, 0.0244582798, 0.0156256612, 0.0102286264, 0.110123917, 0.0108919647, -0.00318586268, -0.0345591418, 0.02237924, 0.0220686905, -0.100356959, -0.0868106857, 0.0951698795, 0.0631417334, 0.0195696782, 0.0197948851, 0.046977967, 0.111540154, -0.0389526747, -0.124880537, 0.0932635069, -0.0240721647, 0.0736240447, -0.0713330284, -0.100934051, -0.0332081206, -0.056899704, 0.0142954942, -0.00425576791, 0.0407140888, 0.0232541263, 0.0660687611, 0.055978965, 0.205581218, -0.0522601232, -0.0177105553, -0.0709572136, 0.042501092, 0.136781737, -0.0591489449, 0.10280785, -0.0286009647, 0.0203699283, 0.0684441179, 0.0151023567, 0.00649720803, -0.011614088, -0.0292001143, -0.145675272, 0.0745430589, -0.0365434624, 0.0497663878, 0.0714009777, 0.0432593264, 0.000566895586, -0.0398042239, 0.0387506709, -0.01325492, 0.00306883641, -0.00806504115, -0.0631631538, -0.0358932018, 0.00865605939, -0.00388304912, 0.0228559636, -0.0118870949, -0.0144958608, 0.173925027, 0.0152818449, 0.0460042655, 0.0929632485, -0.11597693, -0.0457302704, -0.00481079146, 0.00812531728, -0.0175451841, -0.0146273216, -0.0324932411, 0.0914042816, 0.0152572189, -0.0973307192, 0.0300447084, -0.0236581732, -0.00614617858, -0.0062218681, 0.0844372511, -0.0257651359, 0.0486652851, 0.0117939711, 0.0269584842, -0.130671054, -0.0907182097, 0.0558942333, 0.0269881673, 0.0672956035, -0.0295029841, 0.0920254141, 0.00585082732, 0.00767091569, 0.0626625121, -0.0814452693, 0.062444672, -0.064830482, -0.153269723, -0.0444657467, 0.004085619, 0.0561959743, -0.0803028196, 0.0606159419, -0.0403594561, 0.0761666894, 0.0986458734, 0.0105678514, -0.0817268714, -0.0271067526, 0.123596549, 0.00231281528, 0.0176865272, -0.0248383991, 0.115191989, -0.0942414999, -0.0389549807, 0.059627112, -0.0159614347, -0.0179036092, -0.132311836, 0.0365776531, -0.00939529575, 0.0188696757, -0.0315882787, -0.138933256, -0.0103765316, -0.00589833222, -0.0435589291, -0.0838890523, -0.0195166953, -0.00982258283, 0.0193074346, -0.0212550163, 0.0524057858, -0.0268558655, -0.0110593773, -0.0858485326, 0.136565596, -0.0338770412, 0.0230880268, -0.0766331553, 0.0936120376, 0.0894639641, -0.00722966157, 0.0693049431, -0.0281773955, 0.0802517757, 0.0316463821, 0.0451297984, -0.117503449, 0.0870215446, -0.00771393441, 0.109934144, -0.0832953006, 0.058644902, -0.0155102331, 0.131189704, 0.0246528871, 0.0168847498, 0.0417052768, 0.0578640252, 0.12534298, 0.00086741522, 0.0603443943, -0.0755436271, 0.018010933, -0.0159134269, 0.0909223482, 0.105587371, -0.0225883648, -0.018136058, -0.00429809093, 0.0648536384, 0.00792603102, 0.100273214, 0.0426818356, 0.0358592942, -0.019300919, -0.099387452, -0.0207134746, 0.0274422728, -0.106460415, 0.0799673796, 0.00366885494, 0.0256798808, 0.0333483554, 0.0427413732, -0.000553729013, -0.0421616882, -0.0394642055, -0.0127464496, -0.00283724372, -0.0142694162, -0.00163088657, -0.105811559, 0.038578026, -0.111376107, -0.0123410979, 0.000582673354, 0.0306444187, -0.0510375798, -0.0955996513, -0.0337491222, -0.0427375436, 0.0668885112, 0.0387860388, 0.0303316265, 0.0527413785, 0.0891910344, 0.0156252384, -0.0414381102, -0.0514662415, 0.0876697078, 0.143676057, -0.00428622402, 0.131740123, 0.0262013078, -0.0214228537, 0.0162912421, 0.0362434909, 0.0137105649, -0.0189073104, 0.0995535105, -0.0660979897, -0.102600813, 0.0476988591, -0.0180132743, 0.0930725336, 0.0458689667, -0.0532454103, -0.000116987154, 0.0197553188, -0.0316911414, -0.0152121885, -0.0904175863, 0.0844524279, -0.165547609, -0.0619317517, 0.12770927, 0.0103618838, 0.066581279, -0.00753936358, 0.0160168111, -0.082596615, -0.0370407775, -0.0138111124, 0.0578644872, 0.0567265712, -0.00937330443, -0.0208524279, 0.00568321673, 0.0352295525, 0.0316374637, 0.0383372568, -0.00410140678, -0.0159495249, -0.119643256, -0.0967994928, -0.00457899366, -0.0840825886, -0.00609358307, 0.189631119, -0.00772488676, -0.0562163219, 0.116063178, -0.0523985811, -0.00439142808, -0.0318450294, -0.0286335051, -0.102702357, -0.0878510252, -0.0354822725, 0.113764897, -0.03534621, -0.104682565, -0.067143932, -0.018403139, 0.0943159834, -0.0787311271, -0.00701456051, -0.0965824127, 0.119348221, -0.0734687448, 0.0549593791, -0.06867522, 0.0889204815, -0.121300004, 0.0857042074, 0.0114896242, 0.125987515, 0.131136298, 0.0701710731, 0.0439608805, -0.047840327, 0.0277401656, 0.0564279035, 0.0779915899, 0.136212945, 0.00460846862, -0.0677497759, -0.0715289786, 0.0150211751, -0.0407311581, -0.0127222119, -0.042455323, 0.0607895777, 0.173657656, 0.104650997, 0.00195117109, -0.0108929705, 0.00134520046, 0.0316501334, -0.0480045862, 0.0740273222, 0.107059404, -0.0139094181, 0.0933045521, 0.0341952369, -0.110332601, -0.0287618712, -0.0501488298, -0.0959062278, 0.0929894671, 0.0538922958, 0.0178117007, -0.072513625, -0.0560367592, 0.0946408361, -0.0176601652, -0.0623949431, 0.11369361, 0.0758318007, 0.00737708248, -0.0665262491, -0.0557445325, -0.108372115, 0.00145903183, 0.124586642, 0.0352536514, -0.0335065126, -0.0505453572, 0.15350382, 0.102788538, -0.0545426793, -0.0371701829, -0.117617652, -0.0163915269, -0.0635081977, -0.0985327736, -0.0312759466, -0.0946389213, -0.101049721, 0.0435979217, -0.00786320865, 0.0426449627, 0.0169741418, 0.0111421272, 0.0265836753, -0.17795454, 0.0141290557, 0.0903434753, 0.0691457242, -0.0120085133, -0.0327966586, 0.00159727596, 0.0406891368, 0.0370729789, 0.0657485276, 0.10091044, -0.0109258816, 0.0501286685, 0.00371955708, -0.0208817869, -0.0126140974, 0.0867753923, -0.0718555823, -0.0448352732, -0.0100010429, 0.0135794897, 0.0442451313, -0.0854981244, -0.0428287387, 0.0145759936, -0.122173212, 0.0869320706, -0.025685735, -0.056249842, -0.039507661, 0.0238149613, -0.14451392, -0.0123944217, -0.0103876553, -0.0339916646, 0.046212513, -0.0512748808, -0.0487293378, -0.0314902849, -0.0570745468, 0.0528965704, 0.0513674095, 0.0355832055, -0.156722128, -0.0745223165, -0.054123722, 0.07634902, 0.0399962068, 0.0753087252, -0.0408569351, -0.0402079448, 0.0424394347, -0.180192992, 0.0247934405, 0.00698059797, 0.0393613018, -0.0503891483, -0.00118991546, 0.00325610489, 0.0749366581, 0.0247755647, 0.0585099757, 0.0318140201, -0.0235114805, 0.0815698281, -0.00935976766, -0.153780609, 0.143829837, -0.000695410185, -0.0505319089, -0.0805246457, 0.0407051295, -0.0339464992, 0.0287359748, 0.0735844597, 0.0347057283, -0.0256676152, 0.0358682089, 0.0351833589, 0.0243087821, -0.0101794899, -0.070938468, 0.0585412085, 0.0242326297, -0.0373695157, 0.0499537587, 0.0148751428, -0.0247470364, 0.0399893373, 0.00381147163, 0.0228822287, 0.0986248404, -0.0894921198, 0.106893569, -0.119953528, 0.0489409491, -0.0408462174, -0.05191724, -0.0571553521, 0.0414567068, -0.047445152, -0.0349077731, -0.0283654295, 0.0597603917, -0.0224978384, 0.030724559, 0.0843390897, 0.0264454894, 0.0966515765, 0.167522177, -0.111903526, 0.00882041454, 0.113430358, 0.0291332863, -0.0260825232, -0.0793373361, -0.0346951112, 0.0396763645, -0.0837606937, 0.00599098578, -0.0700120628, 0.0362895653, -0.201220602, -0.0652408451, 0.0983557552, -0.0305539519, -0.0905546769, 0.0781318843, -0.092222698, -0.103067264, 0.0987830758, 0.045919463, 0.0908412114, 0.00743933767, -0.000903667882, 0.0673883334, -0.00918021053, -0.0279686786, 0.0120513588, -0.0784084052, 0.0919407234, -0.000809054822, -0.0930619985, 0.00232095132, -0.0435902402, -0.066131644, 0.00156507734, 0.00279734842, -0.00235813973, 0.0383707695, -0.0504254848, 0.00257976586, 0.0383168086, -0.0559064522, -0.0534450486, -0.0758779496, 0.0953854695, 0.132303834, -0.0230809674, -0.0412184075, -0.017347794, -0.0476713926, -0.0258203596, 0.167052031, -0.0768064409, 0.0581221543, 0.0832431465, -0.0756253675, 0.073915869, -0.0277787428, 0.0670492351, -0.126199961, -0.0692963228, 0.0618876591, 0.061215423, 0.0948523879, 0.102515221, 0.0105340537, -0.0490158424, -0.066204682, -0.0114222281, -0.0259333961, 0.0268512424, -0.0240285192, 0.0975229889, 0.0199942347, 0.00509725977, 0.0178026408, -0.110453472, -0.145900846, 0.0381931141, 0.0195362102, -0.0643835962, -0.0124122482, -0.0106626721, 0.0120995101, -0.0803319365, -0.0431276858, -0.0610677041, 0.0589038916, 0.00969081745, -0.0979269892, -0.160353616, 0.00215788186, 0.0276951697, -0.00386547297, -0.0402911752, -0.0883995518, 0.0351082012, 0.00981349126, 0.0510662273, -0.0526945964, -0.0314154886, -0.125641719, -0.0229007266, -0.0723547637, -0.0714586675, -0.218625143, 0.0324526206, -0.00133723952, 0.0972320512, -0.0218060166, -0.0243024211, 0.068929255, -0.0148029383, -0.0295722019, 0.00892486051, 0.0101208016, 0.0139173307, 0.00760096917, -0.0666164532, -0.0561370701, 0.0248976778, 0.0537908785, 0.0947454348, -0.0378669389, -0.129367724, -0.171187624, -0.0988218933, -0.0418063924, 0.117174529, -0.08213377, 0.101846017, -0.0128666349, 0.0666807964, -0.0470159426, 0.000867781462, 0.130794257, 0.0302610211, -0.0359856896, 0.0312333647, -0.0520480908, -0.0232087225, 0.126273811, 0.0212589353, 0.00844010152, 0.0702419132, 0.069330968, 0.140420675, -0.0790618658, 0.0982266888, 0.0279324092, -0.021764446, 0.0403622873, 0.0360463038, 0.0522308312, 0.0263859164, -0.0660897195, -0.0260122716, 0.0587906465, -0.0165068898, 0.0118215568, 0.116144128, 0.0262203328, -0.129264325, 0.0846690685, -0.082121931, -0.0407930762, 0.110639967, -0.0203457363, 0.0497394279, -0.076648578, -0.109537818, -0.0968411043, 0.0174954198, -0.0489697829, -0.000839303248, 0.00780601799, -0.0506865941, -0.0235634819, 0.0124392062, 0.0553957298, -0.0309087858, -0.0106674321, -0.0123102777, 0.0587912202, 0.0771834254, 0.0601142459, -0.0440628566, -0.105514377, -0.0222603045, -0.0444181077, -0.118177205, 0.0587717034, -0.0497949123, 0.057883665, -0.0269314721, -5.55440784e-06, -0.0486246347, -0.0606392771, -0.0122536812, -0.180696011, -0.0932258815, 0.0564828068, 0.0683011413, 0.0668136999, -0.106748983, -0.034203209, 0.0697825253, 0.0776619911, 0.0430945531, -0.0202588513, 0.0135798603, 0.0685243011, 0.0470924824, 0.050038483, 0.0260951351, -0.0188981667, -0.05626598, -0.0308555029, 0.00269413646, 0.0321046747, 0.0673542842, 0.0152772674, 0.000534251332, -0.0957631543, -0.0416444466, -0.0481545255, -0.00117808534, 0.0869539008, 0.00363457063, -0.0844588056, 0.146690086, 0.00341843953, -0.0287580416, -0.131334633, 0.128242806, 0.0793444216, 0.0350410119, -0.122858815, -0.0029347213, 0.0196148157, -0.0958061218, 0.139851466, 0.178974509, 0.0849440545, 0.0649157688, 0.161671922, 0.0135882776, 0.102754846, -0.0809206069, 0.0411005467, 0.00458120648, 0.0303182937, -0.00111264363, 0.0546225011, 0.116480209, 0.0340099819, 0.0191972926, -0.0349055603, 0.0488266423, 0.0599862598, 0.0659702495, -0.0212834459, 0.155259833, -0.0356789827, -0.0589237735, -0.012385048, -0.0444460176, 0.0270156488, -0.0360074714, -0.0231806543, 0.0205656234, -0.0253960565, 0.0225299336, -0.0817852765, -0.0741998404, -0.0744033605, 0.08136262, 0.0998105779, 0.0145104919, 0.13637574, -0.0184606779, 0.112999789, -0.0340401269, 0.0372141972, 0.128838018, -0.0560116619, -0.054176271, 0.0386753529, 0.0168194808, 0.106321022, 0.0782190487, 0.0210235976, -0.109597981, 0.114914745, -0.100452952, 0.00199358165, -0.119633958, 0.0552967116, -0.00784056261, 0.085729368, -0.0139441267, 0.0154473465, 0.0230699964, 0.0630311817, -0.0285764374, 0.0794003531, -0.0662526786, -0.0403759107, -0.0215331204, 0.0585868806, 0.0641366914, -0.0714779049, -0.0516804829, -0.115252681, 0.03934066, 0.0521539487, -0.0521697477, 0.0632954016, 0.0472986735, 0.0540311188, -0.079566434, 0.0109893093, -0.0508477949, 0.0969278961, -0.0280641764, -0.0909949988, -0.0146755213, -0.00297376886, -0.00317909941, 0.0654218569, -0.055034548, -0.0476058871, -0.114990205, 0.0453802086, 0.0516088717, 0.131197974, -0.13477245, 0.0250613429, 0.0154938037, 0.0192972422, -0.00781201199, -0.0932095498, -0.115033433, -0.0839962438, 0.118021339, 0.0362724736, 0.0669088662, -0.0141215641, -0.00995045155, 0.0379489101, -0.0162990056, 0.0602151752, 0.099577032, -0.067778185, 0.0149203511, -0.00255671958, -0.113436691, -0.0915586203, 0.0136897275, 0.0411932655, -0.00953338202, 0.0263220593, -0.0732731596, -0.118662558, 0.0749758258, -0.0214597844, -0.0393433496, 0.0138760433, 0.0184391588, -0.208835825, 0.125120178, 0.0977995098, 0.0527613461, -0.120004192, -0.000734303147, 0.00713940524, -0.0657053888, -0.0646293834, -0.0411789007, -0.0304559097, 0.0198378935, -0.0110937105, 0.0679421574, -0.00985591859, -0.00248605758, -0.043492876, -0.0291730724, -0.0291538015, -0.0849319026, 0.0157827307, 0.0133116934, 0.0607607402, -0.0812886655, -0.0553325936, -0.0242931135, 0.117785767, 0.0170826335, -0.0091655273, 0.0149460379, 0.123396315, -0.0602605939, -0.0471653678, -0.0144482926, -0.0235987809, 0.00425107218, 0.0347998813, -0.025054194, -0.0339833088, -0.0931314826, -0.0289532151, -0.100628607, 0.00409202278, -0.0470786206, 0.0112245418, 0.0831836164, -0.0807382613, 0.0457447581, 0.0371434726, -0.00157180824, 0.0330429412, 0.0785487518, 0.117080823, -0.00489734113, -0.0406062566, 0.0132249352, 0.0562938564, -0.127077758, 0.0887920111, -0.00685449317, 0.139241233, 0.0873695537, -0.100828312, -0.0187399201, 0.115055084, -0.0487159081, -0.0302133579, -0.0768338293, 0.109716788, 0.0370821282, -0.0287049375, 0.0339346826, -0.0768983513, 0.0506638214, -0.0337555222, 0.0354681201, 0.11514692, -0.124518529, 0.0959410667, -0.0218171068, 0.024832489, -0.0312339403, 0.129222929, -0.0300681666, 0.0334382914, -0.0897566751, -0.0120510366, 0.0624336302, 0.0457688347, -0.0506006442, 0.137060016, 0.0133634377, -0.0277635027, -0.0519386791, 0.138215795, -0.0255931355, 0.0637193248, 0.0782612711, 0.043704588, -0.0706363916, -0.0867473483, -0.0280122384, 0.0143328644, -0.185355306, 0.050373856, -0.0229333751, -0.066549696, 0.0259219687, -0.0110726804, -0.0339643508, 0.0199308693, -0.0870389342, 0.0375659764, -0.133983865, -0.0622325093, 0.131928563, 0.0606075227, 0.068603076, -0.150959507, 0.0186037701, 0.0163800921, 0.0321337283, 0.00117886369, 0.000826181844, 0.0113856308, -0.0348047912, -0.0119585209, -0.0290229712, 0.0411998257, 0.0409038179, 0.118324578, 0.0484670438, 0.131134927, -0.047241576, 0.0746052638, -0.0132506397, -0.00523084402, 0.0403868295, -0.0415815935, -0.000496421009, 0.0481602177, 0.02978421, 0.0564897209, -0.0941936523, -0.0705231503, 0.0620953739, 0.0165946558, -0.0201972723, 0.00739394873, 0.0693807825, 0.152135521, 0.0163156874, -0.07376571, -0.149465919, 0.0617062971, -0.0557777435, 0.140250653, 0.0829453617, -0.0322103314, -0.0854051635, 0.0221399292, 0.00541131804, -0.119276442, -0.0918929577, -0.0844398737, 0.0397989228, -0.063847065, -0.054408513, 0.0407775901, -0.0566180088, 0.0307342559, -0.0669313669, 0.0502063967, 0.0694551468, 0.0186264273, 0.141365051, 0.208998054, 0.0882838815, 0.0431206562, -0.106544271, -0.025726106, -0.124994293, -0.108791724, -0.00610821694, 0.0892394409, 0.0467048548, -0.0183123369, -0.0259367432, 0.0793271884, 0.0753387809, -0.01059209, 0.150667146, 0.0324033499, -0.0317094512, 0.0576882437, 0.0694558024, 0.109828189, 0.11538896, 0.085645929, 0.031709671, 0.000370375812, 0.112622947, -0.0891636685, -0.0968724787, -0.144358069, -0.0474674366, 0.00848028064, -0.0375958011, 0.0430304445, 0.00660038553, -0.0156454258, 0.056116946, -0.0557026677, -0.0476781391, 0.0235502943, -0.125562862, -0.0046607703, -0.000461176038, -0.00376228988, -0.00742668286, -0.0267891437, -0.0796516612, -0.0622754246, 0.0241216607, -0.00720124412, -0.0482311323, 0.0269438699, 0.0341051444, -0.00857788976, -0.0618463457, -0.0687971115, 0.0168338753, -0.0437239334, -0.0133013222, -0.126889855, -0.0678971708, -0.0325310044, -0.158968776, -0.0658790767, 0.137922496, 0.159343541, 0.0599740259, -0.0736397728, 0.115832753, 0.00552628655, -0.159536272, -0.108788006, 0.0292282421, 0.0619180948, 0.0232697465, 0.0114452057, 0.00564116426, -0.0352590159, -0.0244480371, 0.120290115, -0.173366487, -0.0393587053, 0.131349578, -0.0242320467, 0.0382967778, -0.0374716818, 0.131232351, 0.00148183596, -0.0862775669, -0.0387868658, 0.0471384004, 0.0219578557, 0.025387682, -0.014806807, -0.0119337738, 0.0113282539, -0.0756373405, 0.0581592396, -0.0075218454, -0.068835184, 0.0475200154, -0.0637260675, 0.193392813, -0.0613547042, -0.00515126996, -0.107052475, 0.11569576, -0.119802773, -0.111610524, 0.0550946966, -0.0737449825, -0.045266822, -0.0353542194, -0.105106704, -0.1943589, 0.0179066919, 0.11703974, -0.0468418822, -0.013253523, 0.0484630913, 0.0434607863, 0.0510577559, -0.0305536259, -0.148791358, 0.0887724161, -0.097481668, 0.0422660895, -0.0535485707, 0.00857671537, -0.0413352959, -0.0438640192, 0.0100388546, 0.0508824401, -0.0646590143, 0.057626307, -0.0195472836, -0.0699712262, 0.115772441, 0.0393819921, -0.0359452814, -0.0358799808, 0.067502439, 0.0392773449, 0.0120418202, -0.177543595, -0.0146268904, -0.0204802621, 0.0016590287, -0.0298607051, -0.0187359713, 0.100402273, 0.115794286, -0.0648050606, 0.138902277, 0.0666446462, 0.0184744634, 0.0240013637, -0.0266780537, 0.0688692182, 0.0461845919, 0.0567253493, -0.0309719369, 0.0898457766, 0.0817998946, -0.0356795192, 0.0649556443, 0.106682301, -0.166588888, -0.00919233076, 0.141001731, 0.0420306027, -0.0658727512, -0.00433288515, 0.0317629911, -0.0550467074, -0.00407661311, -0.0857384354, 0.0598526224, 0.00708718784, 0.0864894912, -0.0628462583, 0.0308408234, -0.000600259751, -0.120377198, -0.0287705027, 0.0112019461, -0.0801755488, 0.0116645917, -0.078481406, 0.0767025799, -0.075545013, -0.140401378, -0.0802578405, -0.120694712, -0.0216989685, -0.0317520089, 0.0420968048, 0.070038408, 0.00442051981, 0.0610248409, 0.139262721, -0.0418416671, 0.050451614, -0.0104785236, 0.0406922102, 0.110013396, -0.0490329191, 0.12251652, 0.00627331156, -0.0276043098, -0.0187224839, 0.0982051641, 0.0293273591, 0.0450135656, -0.0379322655, -0.0112920254, -0.107056648, -0.0681236461, 0.118041284, -0.0493883193, -0.00300544873, -0.0748077631, -0.0504209548, 0.0146083888, 0.0419397876, -0.00454512984, 0.0104878852, -0.187521726, -0.0824201331, 0.0579334982, 0.0474240631, -0.0432562158, -0.0197104309, -0.0446122512, -0.0378362015, -0.00945643149, -0.0539182052, -0.00146937557, -0.111218169, -0.0110235699, 0.0074978359, 0.161174268, -0.0650610924, 0.0904625505, 0.0807929561, 0.0915387943, -0.00764246192, -0.0486331359, 0.0369200967, 0.118042879, -0.00210989453, -0.0401251242, -0.12022458, 0.0929566175, -0.0149899637, 0.0888923258, -0.162864044, 0.098613888, 0.0444668122, 0.00797554664, 0.0253885258, 0.0782689527, -0.0126456572, -0.0217401646, 0.132580444, 0.059950754, -0.00834976509, -0.0496116169, -0.037995778, 0.132465795, 0.0355909914, 0.027968524, 0.0530179814, -0.0166351162, 0.0771531537, 0.0245379992, 0.057781186, 0.0145554598, 0.0339131877, 0.188989908, 0.063147679, -0.025067037, 0.0142894313, 0.0364510752, 0.0422343612, -0.00567561947, 0.0124436766, 0.00300999358, 0.00380477495, 0.0679786354, 0.051919803, -0.0499886312, -0.144870698, 0.139361382, 0.0195103325, -0.0856847316, 0.0278958902, -0.00421368703, 0.00291786436, 0.0304587819, 0.0217464864, -0.0125341946, 0.0506761521, -0.0362862945, -0.0923682898, 0.0533040985, -0.00371540152, 0.000961206853, 0.0589806214, 0.000787030905, -0.131475985, 0.054873541, 0.0949562043, 0.0810329914, -0.0336201787, 0.126859963, 0.15160881, -0.0486177132, 0.0335220993, 0.0558877923, 0.0428225473, -0.0423192233, -0.0434767045, -0.0189460516, -0.107544094, 0.000446313992, 0.00141296652, 0.0334832147, -0.204021677, 0.178792879, -0.0609032884, 0.0193695966, 0.0513797626, -0.0362374894, 0.047803212, 0.0560990237, 0.0023830561, 0.0802260116, -0.0867181197, -0.0223791339, -0.047827974, 0.0230495315, -0.0701122582, 0.183097705, -0.0689380169, 0.105148278, 0.0907316059, 0.0237972438, -0.0149131007, -0.0549703613, 0.137934983, -0.0971860141, 0.0100527536, -0.110943921, -0.0569062233, 0.0577629618, -0.0443707705, 0.175148338, 0.0470523536, 0.0229153782, -0.108078659, 0.0912545621, -0.0411299206, -0.0125831012, -0.014442116, 0.0116702914, 0.0116804931, 0.00841268525, 0.00972991809, -0.0457131639, -0.0640593246, -0.0764123499, -0.0467268825, 0.0948646963, -0.110118203, 0.104310952, -0.0200548321, -0.00133190304, 0.112414286, -0.00887494348, -0.0175741073, 0.0546413921, 0.0407879762, -0.137215406, -0.0960658342, -0.0782571658, -0.0324235559, 0.0907090008, -0.0478524938, 0.030605752, 0.0432760715, 0.0325544327, -0.0496563055, -0.034460105, -0.0536670089, 0.00116366334, 0.061855834, -0.0359185711, -0.114783369, -0.0068679899, 0.0400654972, 0.0265578609, 0.0767074376, -0.072686851, 0.132775396, -0.0462088808, -0.0183823705, 0.00448135519, -0.0202818383, -0.065671809, -0.0463726036, 0.0428554304, 0.0909213647, -0.0419094712, -0.106354974, 0.0316834077, -0.0306691602, -0.0556162484, 0.142710477, 0.0494344719, -0.103703126, -0.059927728, 0.0554858632, -0.120031625, 0.0450445749, 0.0475841835, -0.0595748462, -0.00376545638, 0.0586875342, -0.0307709053, 0.0238728747, 0.0150918737, -0.000204436481, -0.00262482837, -0.0332630686, 0.102440573, 0.0357867703, 0.125794888, -0.112869285, -0.0243463106, 0.101468235, -0.12973693, -0.0667174682, 0.00922841486, 0.0572887175, -0.0303817522, -0.0662079304, 0.066669099, -0.129647031, 0.0546359047, -0.128584623, 0.010580454, 0.0101046814, -0.0312611423, 0.0791293904, -0.0426313728, -0.0680926144, 0.0335913859, 0.0148151731, -0.00421966705, -0.0111462269, -0.0224630907, -0.000497120433, 0.0246174708, 0.0833309144, -0.129092276, 0.0678693354, -0.131356567, 0.0588797405, 0.00920473225, 0.0612161979, -0.0848389193, -0.0071021202, 0.080742918, 0.0552304089, -0.0345649272, -0.00250155292, 0.0574286059, -0.0959362164, -0.135212213, 0.00283145555, -0.0284595434, 0.0140521834, 0.0576984659, 0.0464126095, 0.063174352, 0.040335957, -0.118675485, 0.135154814, 0.0202042088, 0.0609128438, -0.135530487, -0.0496266671, 0.00842737779, 0.107638665, -0.0529136173, -0.065190509, 0.0396431759, 0.0686914623, -0.131918639, 0.103470311, -0.016866155, 0.0228836238, -0.180925727, 0.0224847198, 0.0532157496, 0.172246039, 0.0417397097, 0.00659351051, -0.00833398104, -0.027996242, 0.0823713541, -0.0462665185, 0.00943694916, 0.0314624496, -0.0479518138, 0.0495952778, 0.0898738652, 0.00436242763, 0.0604423732, -0.0349833779, 0.0444733836, 0.0104675815, 0.0487625673, 0.0547988042, 0.122417681, -0.103307828, 0.0407392383, -0.0402793512, -0.0260798652, 0.0149922073, 0.0195754189, -0.05040773, -0.0902734175, 0.00871187635, -0.00195848197, 0.0102583338, -0.0978202, -0.0685906112, -0.139993802, -0.0051469449, -0.100025199, 0.00589732686, -0.0337264985, 0.215451062, -0.0984086841, -0.00606664969, 0.0359480307, 0.0565156266, 0.105717048, 0.0267035998, -0.0242278166, -0.00569936121, -0.0918593109, -0.0523912534, -0.0822795704, 0.113297582, 0.014958689, 0.0333733894, 0.117265664, 0.0192012917, -0.0707047284, -0.105211809, -0.0132810213, -0.071634531, -0.0505304076, 0.0251308717, -0.11762315, 0.030193273, 0.00410067569, 0.0369552188, -0.031379018, -0.0473172627, -0.0846178234, -0.0176126845, 0.0762565881, -0.0263493359, 0.0386259109, 0.00295338058, -0.0766040608, -0.0461957157, 0.085407868, -0.0253898911, 0.0454309508, 0.0543058626, 0.15222469, -0.0694000125, -0.150859237, 0.0406388752, 0.0129035041, -0.0507414937, 0.0925635695, 0.0131557621, 0.00173948146, 0.0527211428, 0.0082938252, -0.0199036524, 0.0526379533, -0.0866013691, -0.0417134427, 0.040677879, -0.0628831312, 0.082594268, 0.0365447104, -0.0956738889, 0.014216762, 0.0195986778, -0.0878263563, -0.0386111587, -0.0719939172, -0.0631440058, 0.161196768, -0.0623713508, 0.0674361512, -0.0172760263, -0.117272392, 0.0254153721, -0.189543292, 0.0338623449, -0.0333566591, -0.0785432607, -0.0825426802, 0.0212335829, -0.00181452557, 0.0224282667, -0.0112977102, -0.0815744847, -0.078524895, -0.0774800107, -2.10814178e-05, 0.0677622408, 0.0377039611, 0.043813847, -0.0690885931, 0.0389433466, -0.209852159, -0.00648564193, 0.016548641, -0.0730931088, 0.0825504363, -0.0176654309, 0.0567998029, -0.051393047, 0.0608661249, 0.0974092633, -0.0341625921, 0.0777445063, 0.0798430741, 0.0532468259, -0.066051513, 0.0264353119, 0.163517594, -0.0298399553, -0.0835821703, 0.0212889966, 0.0603696071, -0.0551470481, -0.0349132493, -0.073651202, 0.0817477852, -0.0104334783, -0.0674619302, 0.0600917898, 0.0395211875, -0.0919675902, 0.0394610986, 0.0600610226, -0.0318777189, 0.124784738, 0.0569640696, -0.089247331, -0.0424785838, 0.0129063651, 0.0959335864, -0.105632305, -0.0349580944, 0.124290213, 0.00742910523, -0.0856474265, -0.0649904013, 0.0538651571, 0.102797888, -0.0986762345, 0.0703774765, -0.0206485633, 0.0402970538, 0.0192304533, -0.00283538736, -0.056690678, -0.0873244852, -0.055459749, -0.00415593386, -0.0918343961, -0.0803622529, 0.108468682, -0.157544032, 0.0120868664, 0.0939099938, 0.132997841, -0.00674599037, -0.0179110896, 0.129941925, -0.0587300844, 0.0247610286, 0.0774628744, 0.0160910618, -0.0476965532, -0.102211349, -0.0750115514, -0.00666426728, 0.0836928189, -0.0767372474, 0.00125703483, 0.0226993021, 0.0866479278, -0.0185180958, 0.0609958544, -0.00676918775, 0.00245276652, 0.104882963, -0.0618118271, 0.0347103737, 0.0706075057, 0.0598387346, -0.0084846206, -0.0362102054, -0.108916335, 0.0123542259, -0.0172353536, -0.0278785471, -0.163362816, -0.0573998764, -0.085427314, -0.11744605, -0.103283063, -0.0401511155, -0.0180830099, 0.0555042364, 0.115041502, -0.0738493353, -0.00529451668, -0.00972217508, -0.0345094875, -0.0759169757, 0.103236079, -0.00818775874, -0.067956008, 0.0146953929, 0.13305375, -0.0778180435, 0.0579100139, -0.00344126951, -0.119493879, -0.0432206392, -0.0199865401, 0.0835982263, -0.00647525303, -0.0163019374, -0.0838292018, -0.00633716583, -0.0312179942, -0.0265295058, 0.0268367082, 0.115729399, 0.0971110016, -0.00338013656, 0.0156162735, -0.0879468098, -0.0433894545, 0.0345592611, 0.0536117218, -0.0351378322, 0.0382302962, 0.0127161127, -0.00957513787, 0.11938367, -0.0673539117, -0.0369861275, 0.0134010594, 0.0141588133, 0.105023503, 0.0664163977, 0.029922653, -0.117293611, 0.039896138, -0.0773853213, -0.0897473469, -0.0697960109, 0.0581272244, -0.107994184, -0.0148722082, 0.0915718973, -0.0251923297, -0.0658146143, -0.000552773476, -0.0682300031, -0.144395769, 0.0585696325, 0.0236287657, -0.0936093181, 0.00539004151, 0.0615960807, 0.0584734455, 0.00777017325, 0.0802931711, -0.106316745, -0.0129972901, 0.0404598229, -0.0114201587, -0.0783428848, -0.100179978, -0.0737028867, -0.0314852335, 0.00265409378, 0.0352568403, 0.094788298, -0.0325277448, -0.0307070017, -0.068057254, -0.00465865992, -0.0122316107, -0.0948953703, 0.208852217, 0.0282319412, -0.0256948993, -0.0362353139, -0.00716653233, -0.0289362669, 0.168159798, -0.0553451665, 0.0347298011, -0.0679618493, -0.0605969317, -0.0318555869, -0.0855532736, 0.0666620955, -0.119269513, 0.0350951627, 0.142051041, 0.0425311662, -0.0091514783, 0.0184900872, -0.0630475134, 0.133693263, 0.00296160299, 0.0309478026, 0.0415407345, 0.170553029, -0.0490989387, -0.135096058, 0.126458749, 0.0118405139, -0.0247989483, 0.00372360437, -0.023267014, 0.0483793914, 0.0218263846, 0.00648327172, -0.104708791, -0.0632834136, -0.0144017916, 0.038995266, -0.0494858362, 0.118353747, -0.00793843158, 0.0208233427, -0.08309789, -0.0353376158, 0.0120601878, -0.161479384, -0.0884625912, 0.0657360554, -0.0234829895, -0.0697832555, -0.0651538819, -0.056885317, -0.109124765, 0.0493674688, -0.00817315932, 0.0100291241, -0.0481616072, 0.000424249098, 0.0191879421, 0.0442795306, 0.0166311134, -0.118633807, 0.0365566425, 0.0225939676, -0.00260969903, 0.114157684, 0.0262636915, -0.0418700352, -0.083099097, -0.0560676157, -0.119343206, 0.0361770205, -0.116154544, -0.13569513, -0.0284458604, -0.025453655, -0.0674404427, 0.017628219, -0.0759436861, -0.0249355529, 0.0292041786, -0.0493779406, -0.0167716984, 0.108655222, 0.0311130378, 0.0179302357, -0.135022163, -0.0417784788, -0.0570391379, -0.135354355, 0.0101753296, -0.00823653676, 0.118374012, -0.057753209, 0.0182850026, 0.0976908654, -0.0130774835, -0.0517067276, -0.0648995489, 0.0260742195, 0.0781308338, 0.0817104727, -0.00144365057, -0.00840477273, -0.0647739768, -0.0124128386, 0.123619005, 0.00500325579, 0.126719385, -0.0177009441, -0.0213475171, -0.0480079725, -0.0449275188, -0.0113018146, 0.00201481557, -0.139193699, -0.0132091753, -0.0924841762, -0.0141410977, 0.0912420899, 0.0638051257, 0.0620417744, -0.0886238888, 0.0261636358, -0.189361647, -0.077522859, -0.113367982, 0.19848153, 0.0629237592, -0.0115735661, 0.0534239337, 0.0523569807, 0.0614056997, 0.017402282, -0.0137614813, 0.128127381, -0.0507759713, -0.0122432224, -0.137505561, -0.0140329935, 0.175129205, -0.0474996269, -0.0126683433, 0.0954533815, 0.0182087515, 0.102476642, -0.00505503453, 0.0445043184, 0.0157436822, -0.000684835017, -0.0446982607, -0.0160516407, -0.0268566143, -0.034871392, -0.0723624006, 0.0276829042, -0.106894553, 0.0297245849, 0.148517668, 0.0306119043, 0.024480788, 0.057873264, -0.0542904139, -0.0187257193, -0.0268429592, 0.0347781479, 0.182711676, 0.0387707427, -0.0413666219, -0.0304399971, -0.0249730311, -0.0115301311, -0.0225001946, -0.0538630486, -0.0358827002, 0.153448954, -0.016551502, -0.0279785749, -0.0211092904, 0.0145989303, 0.114712067, -0.0959315822, -0.0200077035, -0.00496096537, 0.0531129092, -0.00461301208, -0.092136547, -0.019290518, -0.0976062939, 0.0286135897, 0.136693239, 0.0312552676, 0.117106304, -0.122289285, -0.0588494167, 0.0291798022, 0.0087381117, 0.0761296526, 0.0589485057, 0.161292061, -0.0534005016, -0.0545016713, -0.0542927757, 0.0473307259, -0.026263196, -0.0648127347, -0.0510592088, 0.122262836, 0.0621393174, -0.00620839931, 0.120539084, 0.143868059, 0.00991750322, -0.00703470968, -0.133466795, -0.0672097951, -0.0992771462, 0.0398608893, 0.0112410393, -0.0732283741, 0.0225866288, -0.0965754241, 0.0600055791, -0.0412300713, 0.0300039612, -0.147102296, 0.145886332, 0.0533294939, -0.087719366, -0.11787077, 0.122798428, -0.0632750094, -0.0133608114, 0.0397222638, -0.120839655, 0.0279717967, -0.0290077776, 0.0442973301, -0.0888298824, 0.0969517604, -0.0830697343, 0.0314744674, -0.0240058973, -0.0318419263, -0.0793337822, -0.145824462, -0.0259806756, -0.056130074, -0.00145428069, 0.0159080252, -0.0695925355, 0.0958659872, 0.067442283, 0.0224857777, -0.0833125859, 0.0308842678, -0.0480967164, 0.253588706, 0.00488279015, 0.00748084858, 0.010573877, 0.105883926, 0.0911075398, -0.0282798465, -0.0420237556, 0.0919920504, 0.0166334547, -0.0042803511, 0.0474388972, -0.0794579312, -0.12708059, 0.0714929402, -0.116839588, 0.0495442934, -0.115805045, -0.0915021449, 0.0321426913, 0.00533871911, -0.149284571, 0.105603233, -0.159845412, -0.0764946789, -0.0513117686, -0.0528372861, 0.0752885342, 0.155340552, 0.00743776234, 0.0421962626, -0.120706692, -0.0271855444, 0.0263345502, -0.0189696793, -0.0801173896, 0.03058137, 0.0575154275, -0.0212100595, 0.0674094707, -0.0577037409, 0.0451060459, 0.00919431448, -0.101748303, -0.127133489, 0.00121978298, -0.0936859027, 0.144394696, 0.0653232187, -0.0212536044, 0.16899395, -0.000152459368, -0.0977137461, 0.0033859238, -0.117419414, -0.0493396297, -0.035705924, -0.024119677, 0.0573134907, 0.0069703497, 0.0261702631, -0.116585165, 0.00808379799, -0.146062806, 0.0126314852, 0.0150787905, -0.132542253, 0.0098644346, -0.0288225487, -0.010356755, 0.0386339724, 0.0684816912, -0.0271345451, -0.0483281352, -0.0399376117, -0.0557099693, -0.100194566, -0.102490455, -0.0575878583, -0.0679349005, 0.0249807127, -0.0806581378, -0.00437785126, -0.0550510548, -0.0687842146, 0.0311038904, -0.00495552784, 0.00638894085, 0.0355049297, -0.0132802539, -0.0234391242, -0.0858439803, 0.0587111451, -0.0252123624, -0.0960020944, -0.0448848084, -0.0496538766, -0.00416004006, 0.016414592, 0.0572075024, 0.0184295736, -0.0296163149, -0.026117295, -0.039015539, -0.137685612, 0.0715054572, -0.0219773948, -0.0229666159, -0.0302200988, 0.0363391303, 0.109770469, -0.0656398833, 0.0457481146, 0.094116956, -0.0773075968, -0.0314593501, -0.159501195, -0.110025816, -0.0458520651, 0.0304925535, 0.0181574859, -0.0170991682, -0.146890998, 0.0161250383, -0.204725102, 0.0404614955, 0.00172442512, -0.0773060024, 0.0338327289, -0.111908913, 0.0843269378, 0.0417656079, 0.0236102529, -0.0767799839, -0.0120361708, -0.0634715706, 0.00617155805, 0.0768341199, 0.15493007, 0.00329212658, 0.029349409, 0.125606447, 0.0361124091, -0.0804133043, -0.137538493, -0.0659092069, 0.0318373069, -0.160256818, -0.0132932011, -0.11344295, 0.0680131912, -0.0408285931, 0.0277636871, 0.0435267016, 0.0119331479, -0.0301122367, -0.0860860273, -0.0477272347, 0.0555923842, 0.0643539429, 0.0257913917, 0.0240713283, 0.148189276, -0.0128130158, -0.120931864, 0.094560191, 0.0486292243, 0.0279901735, 0.0159090422, -0.109461352, -0.00390604138, -0.015810281, -0.0487371013, -0.0140297767, -0.000135540962, 0.0851485655, -0.0680190176, 0.118419319, 0.0645026565, 0.0795653462, -0.0313418992, -0.0489860103, 0.0370845869, 0.0840737447, 0.00726946816, -0.0644930378, -0.0160436202, -0.0734778047, -0.218570292, -0.136610791, -0.0216169842, 0.135029256, -0.00319907814, -0.0150682442, 0.117365927, 0.0704264194, -0.0719463676, 0.0415127277, -0.0872843713, -0.0254714675, -0.0133848153, 0.0679500997, 0.0415262394, 0.0900941938, 0.0285563879, -0.00156569388, -0.0411640517, -0.0303782597, 0.000205819029, 0.00295572542, 0.0670176148, -0.137253135, -0.00285264291, -0.021808045, 0.0313622952, 0.0469728671, -0.0205262154, 0.00927074254, -0.0372303762, -0.0103757288, -0.0714906454, -0.157990828, 0.0343606398, 0.0954145193, 0.123222455, 0.0823525265, 0.117442392, 0.0234946515, -0.00873712823, -0.00445685443, 0.0669916421, -0.0227660593, -0.0154639501, 0.0184325259, -0.0205302611, 0.135972634, -0.06449496, 0.00152645307, -0.0575076118, 0.0527576469, -0.105739474, -0.187588841, 0.0853657201, 0.0738194585, -0.18257232, 0.00380814308, 0.0113347061, -0.0144741945, 0.0401724204, 0.0282401312, -0.0107867429, -0.0162548311, 0.155527055, 0.0126220174, -0.0744252354, -0.0558582246, -0.180569381, -0.123541631, 0.126075476, -0.13872765, 0.0357238427, 0.0408113226, 0.0505880788, -0.00524656894, 0.121458866, 0.228833333, -0.0176178459, -0.0455273241, -0.13362968, 0.109332412, -0.0374373719, -0.00115054101, 0.0354806446, -0.0877593532, 0.139906853, -0.0553748682, -0.0612836853, -0.0690333545, -0.120751485, -0.0274280068, -0.134869367, 0.130242035, 0.109948143, 0.0753683746, 0.0777142346, -0.037511088, 0.0469326377, 0.00097156316, 0.0486398265, 0.00589081924, 0.0846952945, 0.206510618, -0.0853412375, 0.0449974313, -0.0534627996, -0.0558119938, 0.0255994126, -0.0422267132, 0.0211019013, -0.101064906, 0.0302758403, -0.00200177729, 0.0577369705, -0.0173249096, 0.0458261706, 0.116266757, -0.0139172692, -0.0195216723, 0.0236957557, -0.00261176378, 0.102870516, -0.0350448191, -0.0415064879, 0.161883056, 0.10469836, 0.0162769742, -0.126410037, 0.0825980902, 0.0385107286, -0.0513081625, -0.0198488347, 0.0984914452, -0.114959389, 0.115681939, 0.0209397022, -0.0462179631, 0.0214058869, 0.105201021, -0.0764848813, 0.0111919772, -0.0412613116, -0.0272944085, 0.0146023501, -0.0598362722, 0.0309797414, 0.0782676339, -0.00873469189, -0.0515040122, 0.0926494226, -0.0146439606, 0.122180969, 0.0172243491, 0.096255213, 0.0478411429, -0.00864358619, -0.043324858, 0.0806294382, 0.0385359637, -0.110801741, -0.0747344047, -0.0966870263, -0.0405380689, 0.0107716825, -0.138293356, 0.0552434511, 0.0178805068, 0.027309062, -0.046948716, -0.0610931665, 0.088001661, 0.0763297454, 0.104673654, 0.0307341795, -0.0418299511, 0.0517079681, -0.0207884647, 0.117879823, 0.120932519, 0.0588165745, 0.112198956, 0.0273296181, -0.152703375, 0.0917826146, 0.0574529879, -0.127207488, -0.034267921, 0.038627021, -0.109168932, 0.103566602, 0.144766361, 0.0263313949, -0.00911980867, 0.025112465, 0.00483409502, -0.0115482705, -0.144090742, -0.0522341058, -0.0890554339, 0.123037137, -0.14432092, 0.0566201583, -0.0978538245, -0.0754307657, 0.0577240288, 0.115228221, 0.0717470497, -0.169151589, -0.0289260317, 0.0186712164, -0.0132641988, -0.0773575976, -0.13275443, -0.00525302626, -0.0448894016, 0.0724294782, 0.0305841565, -0.105213851, 0.0965616778, 0.0152161764, 0.0214027092, 0.0398187488, -0.124009691, 0.0709653571, 0.128675655, 0.0161593743, -0.0553461984, -0.0716221556, -0.0192435756, 0.0274756961, -0.0260479618, 0.0247825366, -0.0331113636, -0.0272251852, 0.067591548, -0.103237525, 0.00457238592, -0.0378931724, -0.0647895262, 0.111099169, -0.0802518725, 0.0201167539, 0.0551374778, 0.0205719061, -0.0536681078, -0.0430784672, 0.00408056565, 0.125642642, 0.124837883, 0.0629464313, 0.0523719788, -0.0555003472, -0.0356114469, -0.0642954111, -0.0556642935, -0.0128267063, -0.112548143, -0.0343009867, -0.0197926443, 0.032527376, -0.027550457, -0.0483105481, -0.1111186, -0.0533099994, 0.0897685438, -0.176952422, -0.111487359, -1.16974115e-06, -0.0101449145, -0.101750091, -0.0680906251, -0.0606357791, -0.00741220964, 0.130814746, 0.00218121661, 0.00785925984, 0.0854899511, 0.0221307538, -0.0848427489, 0.0814598054, -0.0656011105, -0.00223445706, 0.0759817585, -0.04201537, 0.000538141001, 0.155041024, 0.00807041302, -0.0581379309, 0.0459022969, -0.041241359, 0.175478607, 0.0606626831, -0.152528405, -0.00659666769, 0.0296979882, -0.0253408607, -0.0210521482, -0.00938495249, -0.0788428262, -0.0433672257, -0.0670581684, -0.0472778715, -0.0580407344, -0.0635472536, 0.105501935, -0.025068542, -0.114852771, -0.078055203, 0.0648784712, 0.0575545654, -0.115270779, 0.0121703502, 0.0322844461, -0.0923805609, -0.144185811, -0.0330828764, -0.0184293706, 0.0116816945, -0.13204585, -0.00187658332, -0.0570808128, 0.0447487347, -0.0320288502, -0.00365327112, -0.0644106045, 0.0492683053, 0.107609272, 0.020459529, -0.0907351226, 0.0351800546, 0.0128706573, 0.0705500469, -0.0460589565, -0.055538062, 0.0625325516, -0.00942290761, -0.0372318514, 0.0181166455, 0.0596277937, -0.0327496566, -0.0815372467, -0.143072665, 0.117885664, 0.0493902341, 0.0260507278, -0.0880189314, 0.0991055444, -0.124405935, -0.032854408, -0.018674368, 0.0103320964, 0.095204711, 0.0335261337, -0.0324110873, 0.0762193576, -0.0107756723, 0.0228998549, 0.0467691422, 0.0496879257, -0.00409949198, -0.134445935, -0.048339799, -0.0293532889, -0.0458019264, 0.0628730804, 0.070340015, 0.128977701, -0.0638133585, -0.00630695, 0.0475100204, 0.0443713255, 0.0790372193, -0.0519603938, 0.188868493, -0.0768636093, -0.0245793685, -0.0350950733, -0.0824217573, -0.100060083, -0.0734033883, -0.126760826, 0.145379573, 0.00923496857, 0.0131270029, -0.151082799, -0.042517446, 0.0937817767, 0.0573463663, 0.0198057704, 0.0535882413, 0.130594969, 0.162333325, 0.17903626, -0.0330195092, -0.00909163989, -0.0369175971];
    CONSTANT bias_3_u : ARRAY[0..63] OF REAL := [-1.01581478, -0.887849212, -1.0505383, -1.15503514, -1.07520187, -0.916982114, -0.917284429, -0.731233597, -1.29561114, -0.978517473, -1.07225573, -0.933320463, -1.01116836, -1.08638, -1.18247354, -1.04536152, -0.969618022, -0.833687901, -1.11044276, -0.937979698, -1.06253076, -1.03395391, -1.0668242, -1.07883251, -1.06569052, -1.17800641, -1.06056368, -1.06715477, -1.12462008, -1.39895415, -0.985698521, -1.04860067, -0.951921403, -1.17121184, -1.14114308, -0.945074677, -0.979631424, -1.1202879, -0.966821134, -0.93666774, -1.21267986, -1.05218196, -0.937734425, -0.909563243, -0.509452641, -1.04473948, -0.886089802, -1.02757108, -1.03394639, -0.899240732, -1.0388056, -0.880722702, -0.876731336, -1.037606, -1.27209771, -0.938842952, -0.941654742, -0.963986933, -0.950356603, -1.25041759, -0.941537082, -1.0247581, -1.06483781, -1.16372526];
    CONSTANT weights_3_r : ARRAY[0..4095] OF REAL := [-0.32606411, -0.305181414, 0.853710055, 0.643296003, -0.507959902, 0.360487521, -0.395130873, 0.414017469, 0.52319634, -0.479849488, -0.219426215, 0.15654248, -0.266728312, 0.461980253, 0.425416172, -0.556642294, 0.567818284, -0.549158752, -0.975931108, 0.67720896, -0.512712419, -0.328124523, 0.426616818, -0.443059117, 0.207611114, -0.310299754, 0.239883587, -0.236781195, -0.359037995, -0.36396715, 0.353712529, 0.408867657, 0.591968954, 0.530881524, 0.290289044, 0.594232917, -0.553219259, -0.784148693, 0.648065209, 0.490015626, 0.40664199, 0.315410346, -0.130245835, 0.343178451, 0.620505393, -0.133835554, -0.542454004, -0.264066935, 0.462930053, 0.207760662, 0.291069508, -0.347996682, -0.453460783, 0.382044703, -0.468908966, 0.723257065, 0.391256899, -0.62128371, 0.708973348, -0.712345123, -0.631182015, -0.333737373, 0.533903599, -0.446012765, -0.0378672406, -0.0479045957, 0.586389065, 0.264671922, -0.315799654, 0.208430871, -0.279002279, 0.175511852, 0.18931058, -1.05650055, -0.255715102, -0.00363925798, -0.0582851283, 0.244597003, 0.621904135, -0.331989348, 0.22773771, -0.47247237, -0.619856715, 1.33818412, -0.277933121, -0.213242188, 0.212933451, 0.106559314, 0.170447171, -0.224164695, 0.0732215643, -0.171327472, -0.0792607442, -0.611715198, 0.186487168, 0.723508537, 1.28295064, 0.690890372, 0.263711125, 0.478959203, -0.203083411, -1.04438186, 1.11608183, 0.370813042, 0.261939019, 0.276761144, 0.0417740121, 0.317641348, 0.114977218, -0.247694671, -1.47137809, -0.247703269, 0.447909325, -0.0339002497, 0.260987759, 0.177349597, -0.402403384, 0.156143531, -0.135770425, 0.510051191, 0.266276211, -0.167485476, 0.913470268, -0.461754829, -1.2195636, 0.077979736, 0.337161303, -0.141935438, -0.265271962, -0.035638582, 0.655573785, 0.537032127, -0.366385311, 0.203982592, -0.307501882, 0.381213546, 0.349319398, -1.1813004, -0.298807174, 0.0479753166, -0.37418431, 0.278960109, 0.840693057, -0.64014262, 0.474891245, -0.556242645, -0.614137411, 1.7334156, -0.526385307, -0.572337627, 0.248649359, -0.140956938, 0.119385995, -0.29798314, 0.244529814, -0.295158684, -0.300115496, -0.580093205, 0.226594269, 0.918142796, 1.74169719, 0.820151925, 0.248385459, 0.692447603, -0.396430552, -1.54747987, 1.38017225, 0.565111041, 0.392608315, 0.422911912, -0.119393133, 0.676306248, 0.460222095, -0.212124556, -1.80655181, -0.505402863, 0.301489621, 0.412834406, 0.181648746, -0.250534654, -0.471679151, 0.314968139, -0.233505979, 0.52545321, 0.381838292, -0.353975505, 1.25488007, -0.596149445, -1.74091864, -0.217042983, 0.638933122, -0.469897091, 0.245818049, 0.290093303, -1.08427835, -0.664157927, 0.370533347, -0.185779259, 0.533736944, -0.0601371452, -0.527724266, 0.60000211, 0.149180949, -0.224620834, 0.200513855, -0.258397371, -0.456327915, 0.949554861, -0.421606094, 0.376373112, 1.6443671, -0.485285401, 0.816311598, 0.243153811, -0.471630067, 0.139453158, -0.144242361, 0.317050517, -0.232827887, 0.255592555, 0.15091145, 0.247503817, -0.286755443, -0.362139732, -0.461967707, -0.363402843, -0.109364457, -0.491291016, 0.351950824, 0.639383376, -0.539893091, -0.424525499, -0.2290764, -0.199569568, 0.0934817418, -0.173082545, -0.35091725, -0.0301282555, 0.594287872, 0.188275486, -0.270237386, -0.136253968, -0.155206367, 0.0628562197, 0.550562918, -0.107881248, 0.202634931, -1.20844626, -0.0330623388, 0.419759899, -0.539858162, 1.55076027, 0.473937124, 0.114922389, -0.359740287, 0.358791083, -0.238371491, 0.0309315939, 0.379086971, 0.413848668, -0.293242633, 0.332917243, -0.141442761, 0.232743874, 0.242201135, -1.23438561, -0.296759665, -0.115022659, -0.164160192, 0.163818792, 0.685197115, -0.330099732, 0.304970264, -0.346489012, -0.779386997, 1.42712438, -0.523679256, -0.276608735, 0.150926173, -0.12271972, 0.232150823, -0.36957562, -0.0389995165, -0.138426706, -0.0751603991, -0.493225664, 0.166680902, 0.683986783, 1.75461292, 0.551047027, 0.17739968, 0.486676127, -0.162812993, -1.4567163, 1.28828633, 0.419575125, 0.305336416, 0.287140518, -0.0665183365, 0.310240835, 0.230046228, -0.329168618, -1.68186617, -0.129506499, 0.230660826, 0.191573709, 0.167725205, 0.0199827328, -0.31258601, -0.00548750907, -0.322434396, 0.417515099, 0.352410108, -0.267527252, 1.1229645, -0.469884247, -1.70649111, 0.0533591323, 0.396650195, -0.213872373, -0.247390494, -0.308249265, 0.885731876, 0.648571968, -0.310095698, 0.268737406, -0.389113486, 0.0871751979, 0.343963742, -0.485504836, -0.115139328, 0.23760289, -0.424925536, 0.500883222, 0.316645622, -0.702252448, 0.555773854, -0.386323303, -1.48340034, 0.66543299, -0.705020845, -0.37072435, 0.363651961, -0.446105599, 0.149830148, -0.358513474, 0.396215469, -0.265176088, -0.253546655, -0.286184102, 0.458667219, 0.252435833, 0.38352707, 0.340764135, 0.106404178, 0.436587185, -0.641245365, -0.495529294, 0.632080793, 0.337052464, 0.518227041, 0.220586628, -0.318199962, 0.406555504, 0.530345023, -0.155054793, -0.621839464, -0.295333445, 0.212138698, 0.228294671, 0.316329509, -0.364110976, -0.440465301, 0.486016542, -0.278429061, 1.33248186, 0.18339245, -0.53936249, 0.29928565, -1.45049202, -0.368015051, -0.349973351, 0.438491136, -0.403809279, -0.477971882, -0.304249853, 0.466022611, 0.498331398, -0.467597336, 0.348668754, -0.510163784, 0.410904944, 0.498593748, -1.05407882, -0.255845338, 0.185745597, -0.367634088, 0.333585799, 0.853473485, -0.660563707, 0.329295546, -0.603268206, -0.667021155, 1.56817055, -0.494137198, -0.403352022, 0.44587186, -0.295524448, 0.238873377, -0.393918365, 0.317173779, -0.151768267, -0.37963894, -0.579922795, 0.234902322, 0.674435318, 1.45155692, 0.716528475, 0.271678597, 0.764275908, -0.332182556, -1.46324396, 1.45741057, 0.597791016, 0.335873425, 0.256497473, 0.030166598, 0.484657943, 0.466247529, -0.41871053, -1.51203668, -0.494381219, 0.329711199, 0.293426394, 0.439302534, -0.11895518, -0.503041506, 0.27442047, -0.2831963, 0.558458626, 0.304881573, -0.32383275, 1.03910983, -0.792959034, -1.5608331, -0.257430762, 0.664614916, -0.501426876, -0.281351089, 0.0414545909, 0.447095424, 0.343832135, -0.255541176, 0.0612748638, -0.280172408, 0.177165255, 0.36193496, -0.925673783, -0.16850391, 0.0128063755, -0.0942704827, 0.134742722, 0.680249214, -0.383725584, 0.369982153, -0.395214558, -0.586839259, 1.06134593, -0.446925581, -0.405082673, 0.0176686663, -0.0800010785, 0.340114951, -0.200141653, 0.0898567736, 0.01082341, -0.143583834, -0.3846412, 0.0610680543, 0.750910878, 1.13939989, 0.655028045, 0.41650939, 0.57746464, -0.235219672, -1.15468717, 0.96712774, 0.269759059, 0.0998954624, 0.116918571, -0.0196392536, 0.38387078, 0.117413625, -0.302846849, -1.33640993, -0.398219466, 0.394320697, 0.0167492945, -0.0259594377, 0.0365658924, -0.192624837, 0.0477550216, -0.140257016, 0.48980245, 0.242636696, -0.0990151837, 0.977481246, -0.521247506, -1.034536, -0.171559945, 0.293284655, -0.237343356, -0.313935697, -0.232274383, 0.778067112, 0.62355727, -0.57867223, 0.428997576, -0.640505195, 0.250204235, 0.661255181, -0.649872541, -0.122935608, 0.126976743, -0.333370656, 0.507789612, 0.593846679, -0.838342011, 0.664126933, -0.352723658, -0.909550726, 0.843601286, -0.8069399, -0.315561473, 0.478078306, -0.322076082, 0.273690939, -0.423558116, 0.177327543, -0.399279118, -0.173438579, -0.431111574, 0.160768285, 0.451122195, 0.598117471, 0.364526689, 0.266648859, 0.584997833, -0.595889211, -0.674656212, 0.733342409, 0.516002715, 0.433507383, 0.472957939, -0.183722794, 0.407700777, 0.417470217, -0.197818443, -0.78360039, -0.190586895, 0.252519101, 0.269995302, 0.320930928, -0.201623842, -0.679484725, 0.476249129, -0.337365001, 0.729481757, 0.393714428, -0.458076656, 0.610665083, -0.840719402, -0.656802475, -0.316481829, 0.264371485, -0.371127099, -0.252732307, -0.239085466, 0.266183496, 0.417861938, -0.438964844, 0.221316725, -0.455889136, -0.13639456, 0.258295447, -0.0555382408, 0.164990604, 0.154210657, -0.170295238, 0.262882829, 0.0899999365, -0.248038337, 0.436610639, 0.148447692, -0.615800679, 0.150086999, -0.390931129, 0.154123083, 0.145448953, -0.182117596, -0.20823136, -0.00837396272, 0.134367272, -0.222348854, -0.404675871, 0.174651444, 0.138303235, -0.0794249997, -0.0343393162, -0.130718768, 0.00081770902, -0.0382439457, -0.424111843, -0.119458333, 0.230674118, -0.028081717, 0.415239364, 0.156845033, -0.163451418, -0.121806018, 0.408577055, 0.241918802, -0.0300814416, -0.0074230493, 0.0646340176, 0.324945062, 0.306441814, -0.211217076, -0.170305654, 0.242016852, -0.278236717, 0.575324535, -0.113995463, -0.432759374, 0.114849724, -0.533126533, 0.0167393349, -0.38273707, -0.0428678691, -0.28884092, -0.471949935, -0.268262804, 0.698775351, 0.698765576, -0.415175825, 0.310324371, -0.465906799, 0.294130713, 0.402897477, -0.594575763, -0.276606709, 0.336049944, -0.483903408, 0.384283513, 0.581177354, -0.83756572, 0.441531897, -0.380635679, -1.11072242, 0.831285536, -0.794558227, -0.485136062, 0.480796397, -0.478292763, 0.204729795, -0.229210749, 0.30153206, -0.166791767, -0.234277368, -0.397676736, 0.398091793, 0.483754039, 0.766412258, 0.511118889, 0.171075433, 0.313571274, -0.557242393, -0.641509473, 0.633744478, 0.381214678, 0.45218268, 0.479226977, -0.355552763, 0.230504155, 0.50238204, -0.196017981, -0.771038353, -0.19761245, 0.31358242, 0.489434212, 0.411978036, -0.132157326, -0.518997371, 0.482037663, -0.459952474, 0.861239672, 0.258370727, -0.446846068, 0.452018321, -1.01126957, -0.603265166, -0.195862025, 0.351056933, -0.368395925, -0.504480958, -0.367227137, 0.939662576, 0.660247386, -0.365831763, 0.541688263, -0.460847795, 0.307414412, 0.624971688, -0.344881892, -0.129336655, 0.271847337, -0.217659026, 0.245232657, 0.36421901, -0.855669737, 0.592403769, -0.393725753, -1.20529306, 0.547492087, -0.729086757, -0.410979331, 0.346642703, -0.328289866, 0.237400368, -0.295209855, 0.197553545, -0.485058933, -0.189968109, -0.304942578, 0.487791836, 0.54598552, 0.630286992, 0.37855649, 0.137780443, 0.480451822, -0.39389208, -0.634016931, 0.647453427, 0.214886963, 0.531250536, 0.445005357, -0.208312169, 0.374261469, 0.578697205, -0.139688984, -0.697460771, -0.35923028, 0.434657186, 0.464936823, 0.450845182, -0.302823961, -0.736231744, 0.452758044, -0.506413817, 1.14236045, 0.248236433, -0.505619764, 0.633802891, -1.08701026, -0.525048733, -0.285771459, 0.441548675, -0.56051898, -0.31927681, -0.324115783, 0.643988669, 0.405917078, -0.330453306, 0.375912219, -0.34731546, 0.176775172, 0.385320067, -0.976352394, -0.39451161, 0.302981526, -0.331505746, 0.394162476, 0.700016201, -0.629214704, 0.529205024, -0.680885017, -0.727290213, 1.39126933, -0.598196208, -0.611907423, 0.453459501, -0.260176986, 0.173567802, -0.294734448, 0.349817783, -0.168323874, -0.219119057, -0.633465707, 0.165119141, 0.66164422, 1.34298229, 0.864157617, 0.481791258, 0.551117599, -0.453588724, -1.33108592, 1.32759583, 0.400511742, 0.416378945, 0.210791215, -0.0152973225, 0.598210633, 0.338426322, -0.389807463, -1.30942619, -0.491540879, 0.587278724, 0.2986525, 0.20118694, 0.00159147358, -0.630330503, 0.450823069, -0.408089966, 0.715183794, 0.22981061, -0.406616211, 1.01547182, -0.78458935, -1.39109886, -0.209403127, 0.513578713, -0.506427526, -0.29192251, -0.365352601, 0.821260273, 0.799699843, -0.551483572, 0.347243428, -0.618902028, 0.104906209, 0.384635627, -0.678108811, -0.1532446, 0.366201997, -0.224698484, 0.291296363, 0.267117858, -0.721745253, 0.407198012, -0.250949353, -1.48795342, 0.745735586, -0.698526442, -0.408564717, 0.319990903, -0.258586496, 0.218047649, -0.279926717, 0.209587425, -0.461742342, -0.232960254, -0.45649752, 0.39823553, 0.316946059, 0.499801308, 0.365775526, 0.285763681, 0.410254568, -0.585092723, -0.758430243, 0.793517828, 0.347428501, 0.463376641, 0.282039613, -0.137573525, 0.201987252, 0.574360251, -0.147843152, -0.551913857, -0.105053365, 0.239548668, 0.268206239, 0.277595073, -0.292813897, -0.627250075, 0.332713664, -0.36461249, 1.09503412, 0.278442115, -0.570906878, 0.575401843, -1.14452851, -0.503782451, -0.222146109, 0.25390774, -0.435958177, -0.346188098, -0.287907928, 0.577285111, 0.625171602, -0.485937923, 0.279984206, -0.580171645, 0.304609418, 0.382132024, -0.720344841, -0.334448129, 0.338395119, -0.253193289, 0.320167184, 0.369183391, -0.75026536, 0.365687907, -0.602306545, -0.862038493, 0.716569424, -0.626643598, -0.529524446, 0.27669844, -0.231221542, 0.19715257, -0.364062011, 0.272420794, -0.193196043, -0.26943177, -0.40359816, 0.175001666, 0.61060524, 0.733311117, 0.647010386, 0.300696403, 0.531074643, -0.427513987, -0.991258919, 0.965829194, 0.505575061, 0.464456826, 0.370266259, -0.180219814, 0.514823973, 0.547894955, -0.30526337, -0.775482357, -0.277872801, 0.304864079, 0.438526511, 0.442127705, -0.185165703, -0.408223033, 0.372900993, -0.307785809, 0.803971171, 0.247336209, -0.346430957, 0.561486781, -0.784184873, -0.775968432, -0.33393088, 0.414071649, -0.414346129, -0.424316555, -0.228602037, 0.798046768, 0.589726985, -0.471872777, 0.375852257, -0.523459375, 0.312538296, 0.64948523, -0.564522266, -0.39429161, 0.392420679, -0.331350297, 0.406572282, 0.498701811, -0.538559735, 0.37152037, -0.500432014, -0.88565588, 0.814511836, -0.65060389, -0.32671982, 0.443832159, -0.366107523, 0.323150456, -0.431577086, 0.31207934, -0.443811983, -0.453019857, -0.491461039, 0.260425597, 0.649067998, 0.623069763, 0.515208781, 0.29761672, 0.553334832, -0.419336051, -0.74229908, 0.618693173, 0.562187016, 0.327073514, 0.328121513, -0.152062252, 0.258443296, 0.38306722, -0.219228178, -0.824401379, -0.364127398, 0.281175613, 0.228253767, 0.505391181, -0.260356188, -0.714000762, 0.434605122, -0.283382773, 0.759392858, 0.418259323, -0.480381697, 0.658830822, -0.828426778, -0.594255626, -0.434398293, 0.434758842, -0.475796342, -0.253429919, -0.151888281, 0.464026541, 0.447059274, -0.23363854, 0.234164312, -0.228685543, 0.108610779, 0.417265028, -0.949152887, -0.376021415, 0.127703905, -0.180501074, 0.241112828, 0.734871805, -0.522570789, 0.398032188, -0.564164639, -0.479930878, 1.43935657, -0.37222895, -0.455183208, 0.266491622, -0.0408120714, 0.311739117, -0.388832271, 0.182095289, -0.118631139, -0.00731076393, -0.43673858, -0.0472857542, 0.855252743, 1.33718526, 0.790244818, 0.398922116, 0.565711081, -0.20525077, -1.10990274, 1.13496363, 0.480120897, 0.20322676, 0.107450388, -0.0908780992, 0.300021589, 0.119640276, -0.191865563, -1.46495235, -0.298560351, 0.488960505, 0.0581271686, 0.0770600885, -0.103614494, -0.303027779, 0.0364120677, -0.139285401, 0.683296263, 0.190768391, -0.226745963, 1.05477059, -0.473936111, -1.46578884, 0.078238152, 0.489368916, -0.337299317, -0.444000721, -0.174462199, 0.626759052, 0.392545253, -0.330222338, 0.246465355, -0.421768636, 0.284421295, 0.400160909, -0.558163941, -0.282744735, 0.106122591, -0.385983437, 0.504063666, 0.545476139, -0.622974038, 0.304397136, -0.36480096, -0.651256442, 0.750828683, -0.651343167, -0.32135278, 0.462911516, -0.208699137, 0.344162047, -0.337207288, 0.166761756, -0.157386944, -0.209506616, -0.315502286, 0.185891688, 0.636180043, 0.588617742, 0.512386203, 0.317265481, 0.474550545, -0.591336787, -0.675465286, 0.629930377, 0.497780949, 0.283470303, 0.278181314, -0.152107403, 0.323860735, 0.300083309, -0.237705827, -0.707360804, -0.233611494, 0.298213273, 0.327645987, 0.474210054, -0.220958605, -0.43902716, 0.405127794, -0.285075426, 0.677587867, 0.197221667, -0.526327968, 0.604875863, -0.556873083, -0.553813517, -0.32801944, 0.378549248, -0.587617636, 0.21427089, 0.21984911, -0.875384271, -0.620468438, 0.364588082, -0.312358916, 0.41226685, -0.139815196, -0.175383493, 0.280132443, 0.102841973, -0.131755173, 0.0816493407, -0.245622069, -0.476292968, 0.712404072, -0.346726954, 0.30152601, 1.45562994, -0.407604456, 0.471377373, 0.0670249537, -0.208978981, -0.00896921568, 0.00792890228, 0.160337701, -0.126184568, 0.109025173, 0.0403974764, 0.385903925, -0.0472378358, -0.234496132, -0.592926741, -0.370333821, -0.015724184, -0.372033179, 0.464167625, 0.449376225, -0.561121225, -0.294491768, -0.269805431, -0.23032254, 0.113178119, -0.374025494, -0.24987562, 0.154645085, 0.500742376, 0.0921915993, -0.187845826, 0.00581417372, -0.133517161, -0.0244534146, 0.424528837, -0.286528796, 0.305054575, -1.10627806, -0.224664286, 0.403331935, -0.541942596, 1.32796419, 0.379160345, 0.156610399, -0.148328111, 0.27849111, -0.479717582, -0.416316181, 0.728976667, 0.47371915, -0.340526283, 0.425530344, -0.493184388, 0.196874604, 0.422890276, -0.734140754, -0.428865492, 0.295673072, -0.347783983, 0.275349826, 0.647607803, -0.740972102, 0.359515399, -0.355478734, -0.89868927, 0.693098068, -0.565694273, -0.45446521, 0.521305144, -0.423126072, 0.343195379, -0.36296463, 0.182377294, -0.3046498, -0.230392531, -0.479535222, 0.292608529, 0.443596572, 0.750985682, 0.678646863, 0.341219902, 0.37737909, -0.480458766, -0.824370861, 0.720338881, 0.468586832, 0.401706249, 0.337754607, -0.288740158, 0.38029319, 0.319494545, -0.25374651, -0.610306621, -0.489055008, 0.301279873, 0.242298141, 0.469092429, -0.316974074, -0.482820809, 0.29542467, -0.279328406, 0.800565243, 0.219063267, -0.567258596, 0.586478591, -0.836146533, -0.598628998, -0.277637094, 0.35739249, -0.349981159, -0.212868378, -0.132515892, 0.582968831, 0.245836794, -0.21859476, 0.248592272, -0.436507136, -0.0525316447, 0.219017044, -0.078199558, -0.0697035566, 0.325711846, -0.220956966, 0.382013202, 0.151345342, -0.482834786, 0.230038151, 4.8701273e-05, -0.896882534, 0.167872235, -0.556771755, -0.0531435348, 0.277634442, -0.303767294, -0.0111572994, -0.0296421107, 0.21856828, -0.113810413, -0.360011727, -0.141940147, 0.157705769, 0.144350186, 0.290767372, 0.136084914, -0.179874763, -0.0301123243, -0.427401155, -0.297967046, 0.323375195, 0.045945961, 0.229860306, 0.399075538, -0.240118444, 0.0239243489, 0.305032372, 0.043214988, -0.0338462107, 0.12562266, -0.0240930375, 0.38718912, 0.217619404, -0.29890126, -0.19797644, 0.214872062, -0.149662852, 0.862906933, -0.158315763, -0.35901013, 0.207159743, -1.03316343, -0.0435992517, -0.371495306, 0.0122571802, -0.222766235, -0.335296631, 0.00614431966, 0.442041367, 0.511820197, -0.271431029, 0.251062542, -0.354020029, 0.26408121, 0.380686581, -1.19595873, -0.199459553, 0.0512621887, -0.230785102, 0.121044502, 0.563847125, -0.476866037, 0.282984555, -0.610335827, -0.750677407, 1.48484993, -0.396005511, -0.4459984, 0.15016526, -0.165891528, 0.175520033, -0.253411263, 0.0663821399, 0.0307248328, -0.027399281, -0.577981889, 0.187904432, 0.716747284, 1.71462762, 0.719156265, 0.457143158, 0.491087288, -0.243744597, -1.26668429, 1.36153471, 0.529155016, 0.0915734097, 0.329717249, 0.151948646, 0.425810426, 0.218522847, -0.193444088, -1.54156172, -0.419055372, 0.324922889, 0.101474956, 0.0678244159, 0.0475526936, -0.368958205, 0.0250567012, -0.249778137, 0.567493558, 0.285005659, -0.29450646, 1.22011006, -0.566066265, -1.52908516, -0.0332701094, 0.39348945, -0.435152113, -0.279379427, -0.252164513, 0.88293618, 0.603829801, -0.557003856, 0.4126091, -0.611310482, 0.262114704, 0.39541617, -0.657683015, -0.419031233, 0.334631443, -0.439445496, 0.239912346, 0.594620764, -0.710724235, 0.625857174, -0.281924397, -0.94848001, 0.766416132, -0.573693395, -0.507681251, 0.455642968, -0.344042838, 0.120637521, -0.196149305, 0.187891915, -0.33866787, -0.461829305, -0.431388974, 0.473234236, 0.376484066, 0.671459436, 0.532400489, 0.414870739, 0.612779319, -0.447367132, -0.736575902, 0.608187616, 0.457972795, 0.391607225, 0.391642749, -0.270501822, 0.473758906, 0.371922523, -0.248366505, -0.516390562, -0.178563148, 0.301155925, 0.488553792, 0.470395386, -0.259697437, -0.604833424, 0.439455271, -0.526135087, 0.754391849, 0.213179052, -0.635523617, 0.726304114, -0.92388463, -0.556524396, -0.369461954, 0.522346735, -0.548059225, 0.257865012, 0.0679476708, -0.755721331, -0.416924179, 0.183604792, -0.196284577, 0.381534636, -0.153743476, -0.434020489, 0.365814686, -0.0303360354, 0.00483766757, 0.234462872, -0.1011682, -0.343322188, 0.688691437, -0.311507314, 0.243866593, 1.36334038, -0.447809219, 0.745755851, 0.321573853, -0.16720055, 0.0732166767, -0.0399155952, 0.141015455, -0.313092411, 0.0137336878, 0.160370693, 0.317644477, -0.166301489, -0.494622916, -0.501563907, -0.429580897, -0.0300284959, -0.421272367, 0.521287918, 0.609171689, -0.657234728, -0.159242377, -0.208006412, -0.282181531, 0.0125726322, -0.109527849, -0.450762987, -0.0350307785, 0.4969396, -0.00262273988, -0.0696354359, -0.0597759075, -0.103529476, 0.0310744941, 0.573780298, -0.313798845, 0.202677295, -1.02902234, -0.0767832696, 0.405816942, -0.357142836, 1.42817438, 0.576379418, 0.041038733, -0.40113923, 0.450059474, -0.249666899, -0.324406743, 0.645155787, 0.651951373, -0.335311472, 0.318877369, -0.377464861, 0.278273344, 0.577528358, -0.707005084, -0.454609185, 0.346883327, -0.375036657, 0.408443093, 0.604526222, -0.738248646, 0.488500953, -0.574646294, -0.803916037, 0.758122504, -0.623487353, -0.300931603, 0.519699752, -0.21979551, 0.182568133, -0.535689473, 0.355320454, -0.335205972, -0.333302468, -0.528201103, 0.384286255, 0.590183973, 0.814082682, 0.453687638, 0.449585825, 0.441816151, -0.566304922, -0.855111718, 0.909155846, 0.491852105, 0.46307838, 0.467540711, -0.180398166, 0.49356845, 0.508661568, -0.372565985, -0.889092684, -0.290327221, 0.393947303, 0.43914488, 0.396424651, -0.0341150574, -0.504731894, 0.242020696, -0.3221201, 0.611044109, 0.406554967, -0.525439441, 0.852771521, -0.805656016, -0.788086474, -0.3786515, 0.528430641, -0.327401429, -0.405131936, -0.401135057, 1.03028727, 0.547111273, -0.511407316, 0.484279543, -0.37078923, 0.317534953, 0.497445107, -0.566063821, -0.192737415, 0.17343004, -0.437663138, 0.27078265, 0.370668411, -1.03059494, 0.679856479, -0.484099001, -2.04160094, 0.550596535, -0.936203003, -0.326845407, 0.458781779, -0.330802292, -0.0390953943, -0.148416176, 0.282826245, -0.339116395, -0.44140628, -0.354241639, 0.373801202, 0.561958194, 0.471544474, 0.338501513, 0.190972656, 0.560675621, -0.60877955, -0.806209028, 0.740752816, 0.403585136, 0.44382149, 0.310492158, -0.165237129, 0.467229635, 0.639951468, -0.250467837, -0.719496429, -0.342186749, 0.346429437, 0.472102076, 0.423257083, -0.113565609, -0.611903667, 0.502099693, -0.454853475, 1.47754538, 0.192447752, -0.623071432, 0.622491539, -1.70403862, -0.689736545, -0.311849207, 0.346993446, -0.61403209, -0.32030949, -0.260404497, 0.606727421, 0.378895342, -0.522973001, 0.242676035, -0.503748238, 0.400032282, 0.409070313, -1.04656887, -0.23251985, 0.0598524436, -0.160751864, 0.267909467, 0.585713267, -0.53919065, 0.41407761, -0.638192773, -0.853965998, 1.66303492, -0.484024048, -0.597094715, 0.202447027, -0.31045422, 0.41164431, -0.37736547, 0.236909643, -0.288764238, -0.323797226, -0.65210408, 0.277571082, 0.785428286, 1.53385842, 0.603273511, 0.27001673, 0.734697819, -0.316855073, -1.2592355, 1.29509652, 0.566119313, 0.451303422, 0.450500518, -0.118251942, 0.5555861, 0.517378032, -0.212427497, -1.65542746, -0.387000918, 0.551443279, 0.295913428, 0.357824534, -0.0474563763, -0.501777112, 0.346730024, -0.255087167, 0.65019232, 0.233359382, -0.399132252, 1.20495582, -0.788980126, -1.47384763, -0.298721731, 0.547602355, -0.400281519, 0.415391237, 0.11500933, -0.764448643, -0.526417255, 0.471959233, -0.303978741, 0.411469579, -0.215374574, -0.552919745, 0.464531958, 0.180658236, -0.228912786, 0.307991862, -0.389285654, -0.357774109, 0.677281499, -0.538697839, 0.266804308, 1.55649245, -0.543816209, 0.663670182, 0.205055431, -0.306369811, 0.314960301, -0.0812868699, 0.244915798, -0.0972369686, 0.118134655, 0.228851423, 0.33507967, -0.178763539, -0.542017519, -0.440441757, -0.505637646, -0.00129357539, -0.469659418, 0.369825453, 0.763003647, -0.471925408, -0.229464024, -0.215304658, -0.216859743, 0.120160319, -0.403819114, -0.454149246, 0.198572591, 0.695058703, 0.091226548, -0.0968206972, -0.355034381, -0.354152858, 0.0810929313, 0.477759898, -0.261985332, 0.248434946, -1.40007436, -0.115490466, 0.2606875, -0.557928205, 1.54712737, 0.568113387, 0.0240328442, -0.371635526, 0.468986988, -0.3890315, -0.227186203, 0.558743656, 0.638008714, -0.2325169, 0.325430512, -0.360332191, 0.387367666, 0.388153821, -1.04519343, -0.269344211, 0.165706381, -0.168712839, 0.402218312, 0.652806342, -0.674834907, 0.41147843, -0.499225646, -0.734338701, 1.82643378, -0.444065362, -0.588895082, 0.455570638, -0.21291098, 0.110225089, -0.332531989, 0.181953952, -0.294583291, -0.264316112, -0.515410423, 0.162889913, 0.868188739, 1.86032271, 0.700357616, 0.513032436, 0.765919447, -0.49682951, -1.62329006, 1.45719647, 0.545549512, 0.451227427, 0.28905201, -0.142598704, 0.610706568, 0.444595754, -0.141367614, -2.04516983, -0.381730109, 0.318353266, 0.207129255, 0.14816165, 0.0522552989, -0.550924182, 0.407493293, -0.41661644, 0.614094198, 0.354451597, -0.451580673, 1.33644974, -0.551402748, -1.78111506, -0.0356309898, 0.558322489, -0.308785051, -0.253635705, -0.0270095747, 0.46169883, 0.35802564, -0.205481261, 0.318101376, -0.502353311, 0.353082567, 0.418376744, -1.11887336, -0.111144789, 0.117297441, -0.257290363, 0.253319979, 0.7175529, -0.568437874, 0.234085515, -0.576971769, -0.753595471, 2.22766876, -0.63931638, -0.406852841, 0.176097482, -0.0419444628, 0.108799115, -0.454771698, 0.139979661, -0.00126432185, -0.175606206, -0.553412139, 0.166107267, 0.923081875, 2.3204813, 0.596822083, 0.273973882, 0.590377271, -0.273627281, -1.66828382, 1.68053067, 0.356793612, 0.158161953, 0.292190343, 0.0725176632, 0.514080942, 0.25470531, -0.336534709, -2.26764321, -0.27513203, 0.21084933, 0.238806561, 0.319567502, 0.00441332161, -0.470187545, 0.247312322, -0.301804394, 0.539537251, 0.40202406, -0.321202397, 1.35585296, -0.678141296, -2.18601513, -0.156690359, 0.644770503, -0.447970003, 0.184947133, 0.0586535335, -0.842697203, -0.476564407, 0.326289117, -0.175858513, 0.337102354, -0.150091827, -0.393082768, 0.342845351, 0.0555129908, -0.0486602783, 0.266736895, -0.220026106, -0.269021273, 0.608967543, -0.186941519, 0.279839188, 1.1750114, -0.559024274, 0.393088549, 0.141963348, -0.172769904, 0.121606402, -0.110438086, 0.119224839, -0.16923289, -0.0105624478, 0.0515540726, 0.399702787, 0.0513814129, -0.278160423, -0.349841654, -0.216284662, -0.0206595752, -0.322790265, 0.407239199, 0.418390363, -0.452856183, -0.365659744, -0.303342491, -0.235371232, 0.132295564, -0.27970612, -0.363894314, -0.0102149583, 0.503446877, 0.252181977, -0.201562554, -0.140030086, -0.212522104, -0.102482498, 0.521413445, -0.0599606782, 0.317379594, -0.91857636, -0.0796753466, 0.374061078, -0.407837212, 1.13819242, 0.538435876, 0.0274906904, -0.203527272, 0.221570566, -0.585137784, -0.22554791, 0.897851586, 0.794410348, -0.348831713, 0.427135259, -0.493484974, 0.113772824, 0.674505949, -0.469446868, -0.368993729, 0.295242786, -0.40725553, 0.337209344, 0.473266065, -0.80423677, 0.664289951, -0.449214637, -1.27750874, 0.742842019, -0.766273737, -0.467851818, 0.290394068, -0.465311527, 0.238281116, -0.425370961, 0.435574234, -0.291806579, -0.428470105, -0.44762519, 0.277623832, 0.619269311, 0.458167434, 0.591054261, 0.323538482, 0.396119237, -0.537716269, -0.799658716, 0.515515029, 0.291549206, 0.352653205, 0.560084641, -0.245590121, 0.225990862, 0.502214193, -0.276380807, -0.484679371, -0.15336445, 0.211182415, 0.427163899, 0.443517625, -0.239297152, -0.777251482, 0.447269887, -0.335349888, 1.21866739, 0.410942733, -0.667268157, 0.692402005, -1.24103224, -0.534754515, -0.281618685, 0.307847261, -0.592071176, -0.17489098, -0.057309825, 0.622739553, 0.33250168, -0.18130222, 0.214820161, -0.32339251, 0.378621399, 0.253713369, -1.22676325, -0.325474322, -0.0511168316, -0.237608954, 0.160359859, 0.682873309, -0.438781857, 0.374165386, -0.598473728, -0.586400807, 1.50517404, -0.531930804, -0.505696177, 0.188739181, -0.0759081692, 0.322496235, -0.534777462, 0.0866990909, -0.220319897, -0.220647246, -0.589855194, 0.136748701, 0.710161626, 1.55659211, 0.811731458, 0.392696917, 0.581875682, -0.286527216, -1.25108588, 1.18614066, 0.594158888, 0.238403395, 0.324100316, 0.0939783454, 0.568623304, 0.285499305, -0.149848759, -1.64757788, -0.389623255, 0.426757812, 0.339580208, 0.224090979, 0.0706543475, -0.387865424, 0.149145648, -0.13083519, 0.49459061, 0.21732384, -0.269787997, 1.21367657, -0.599125087, -1.48657, -0.0794282928, 0.483454108, -0.495730668, -0.149702519, -0.12196622, 0.518101096, 0.498079419, -0.440585136, 0.377816558, -0.44399941, 0.298395574, 0.526369333, -1.3361609, -0.184671834, 0.198181227, -0.213837981, 0.227365643, 0.69264257, -0.642421722, 0.253970891, -0.459746599, -0.721164227, 2.0608139, -0.410998136, -0.295992911, 0.381521583, -0.0209507495, 0.356352538, -0.274228454, -0.0050154482, -0.0101287942, -0.149391398, -0.546611249, 0.244803205, 0.957121789, 2.423383, 0.761666834, 0.449197382, 0.818116665, -0.290270865, -1.38992047, 1.68735409, 0.584730566, 0.209530428, 0.390848577, -0.0938457027, 0.381666511, 0.222843274, -0.335909754, -2.28804636, -0.407721847, 0.495959103, 0.0609779879, 0.377927572, -0.000324302353, -0.402243406, 0.0875439867, -0.308821261, 0.752283812, 0.330103457, -0.535354733, 1.26573205, -0.805240512, -1.81103754, -0.212165743, 0.49315542, -0.27250576, -0.26895386, -0.23040916, 0.642885923, 0.658500731, -0.37262395, 0.37434265, -0.349618167, 0.240233302, 0.563242972, -1.00378811, -0.382425368, 0.209850684, -0.395602703, 0.19864963, 0.598141253, -0.55917263, 0.327447176, -0.54477936, -0.677006662, 1.02608597, -0.622659922, -0.374311239, 0.454068393, -0.1352209, 0.139970779, -0.393903822, 0.311810255, -0.347855955, -0.183584973, -0.613458753, 0.294341862, 0.695668757, 0.97671634, 0.629432797, 0.222873241, 0.576654196, -0.576174319, -1.17176938, 1.21802914, 0.463727653, 0.323104858, 0.385295808, -0.0564640015, 0.495977908, 0.560169458, -0.402570993, -1.24606681, -0.30742529, 0.446491867, 0.206024915, 0.378804684, -0.0637932569, -0.548548579, 0.264957011, -0.435918182, 0.714320481, 0.503891647, -0.490187079, 0.92835933, -0.653939903, -0.998602509, -0.234939784, 0.519885242, -0.345346838, -0.438330591, -0.199805692, 0.791778803, 0.772088349, -0.334469944, 0.533462465, -0.613139749, 0.273976594, 0.438189596, -0.5514853, -0.35970071, 0.340049952, -0.453285843, 0.468381822, 0.559531033, -0.710513115, 0.589847207, -0.400875419, -1.59320593, 0.761381209, -0.714087009, -0.386633068, 0.277693152, -0.341802031, 0.180621013, -0.407044262, 0.40718329, -0.343057722, -0.358702391, -0.242539018, 0.427075744, 0.438927263, 0.677350819, 0.34506014, 0.311973274, 0.431390852, -0.481903553, -0.805651665, 0.652924657, 0.382951111, 0.34651202, 0.547604501, -0.228527293, 0.320236057, 0.505470097, -0.118233278, -0.483198285, -0.175483301, 0.31151852, 0.390251815, 0.294036955, -0.243998915, -0.682308316, 0.409372777, -0.539528608, 1.08507121, 0.392528206, -0.633849263, 0.564027965, -1.2653687, -0.708535314, -0.37867108, 0.462343037, -0.63749373, -0.336225659, -0.354143858, 0.538114786, 0.575526595, -0.513737082, 0.226745903, -0.354042709, 0.321344256, 0.533973157, -1.00941694, -0.384838343, 0.116603948, -0.371144712, 0.309847772, 0.680324495, -0.464205742, 0.382111371, -0.518437624, -0.835754752, 1.296188, -0.719237804, -0.336357653, 0.317768604, -0.37401849, 0.148494884, -0.583994448, 0.362303764, -0.160795614, -0.393341154, -0.592710495, 0.422500819, 0.844100416, 1.22041082, 0.815548182, 0.259628803, 0.518015802, -0.441701949, -1.20411873, 1.26204193, 0.557317436, 0.330148011, 0.305774599, -0.166518152, 0.624247551, 0.459448367, -0.399693191, -1.16738927, -0.503780901, 0.536997199, 0.198219493, 0.41484648, -0.156464636, -0.587040901, 0.381635636, -0.46363765, 0.541935325, 0.447267145, -0.478802979, 0.919147849, -0.607068002, -1.34749579, -0.334636748, 0.49500072, -0.340175569, 0.353704125, 0.101251774, -1.02059579, -0.730872273, 0.478754908, -0.210190028, 0.556650937, -0.0836573839, -0.428684831, 0.475618631, 0.26693821, -0.0365147106, 0.349770874, -0.296871215, -0.461401045, 0.932147861, -0.574303329, 0.337240696, 1.84354556, -0.531826258, 0.684611261, 0.230101213, -0.265553534, 0.351761222, -0.155148238, 0.210944265, -0.266109228, 0.320440918, 0.119257875, 0.288138092, -0.342955351, -0.413885891, -0.525543213, -0.563633621, -0.26180914, -0.464125246, 0.587187707, 0.672474265, -0.593278229, -0.299270064, -0.353163183, -0.463583589, -0.00285831909, -0.251852244, -0.532872677, -0.0746277645, 0.717572629, 0.203225821, -0.289940834, -0.307978928, -0.279727012, 0.257997662, 0.563363969, -0.126924291, 0.392226875, -1.30514491, -0.0880905986, 0.494673967, -0.658143938, 1.59869182, 0.759586871, 0.277507126, -0.217861027, 0.398876876, -0.492357105, -0.282907367, 0.813215792, 0.627021313, -0.321904421, 0.363541245, -0.311341137, 0.114971392, 0.586712539, -0.438207448, -0.291453928, 0.183375284, -0.316651762, 0.33620429, 0.418325275, -0.810234189, 0.564028382, -0.281237781, -1.54698515, 0.64791584, -0.66442287, -0.140249655, 0.357892454, -0.271120518, -0.0289524198, -0.137522936, 0.168941945, -0.435024828, -0.443703264, -0.342307836, 0.250819564, 0.352735728, 0.470329642, 0.484651417, 0.17451258, 0.504986525, -0.489991665, -0.452524006, 0.48424527, 0.453603983, 0.420602649, 0.463263929, -0.239898235, 0.244296864, 0.545481205, -0.197661057, -0.449634731, -0.223071486, 0.32376349, 0.377509594, 0.199731633, -0.298727512, -0.554720581, 0.451484352, -0.285018682, 1.16988611, 0.0934815109, -0.358396918, 0.328986198, -1.4225142, -0.614723146, -0.273198545, 0.22736989, -0.557725787, -0.351461083, -0.262877256, 0.811221361, 0.416087955, -0.510921419, 0.461658508, -0.567678869, 0.33768183, 0.472564608, -0.607918084, -0.25393039, 0.224310562, -0.32430318, 0.35536015, 0.607146919, -0.650484383, 0.625925839, -0.362202227, -0.8074193, 0.735684514, -0.70511049, -0.265186429, 0.325658977, -0.412962407, 0.18513383, -0.42445606, 0.303192258, -0.305631042, -0.355679244, -0.420834124, 0.273631752, 0.425167948, 0.594565034, 0.507372856, 0.183894157, 0.542529643, -0.518569767, -0.60572201, 0.685898781, 0.293093473, 0.42061916, 0.299018055, -0.277766168, 0.450671166, 0.341782182, -0.327823669, -0.508060336, -0.290250212, 0.362154663, 0.246053413, 0.241558269, -0.251524419, -0.508265316, 0.250327438, -0.392809272, 0.668544412, 0.436275512, -0.586359143, 0.622453272, -0.81871587, -0.55931741, -0.30781436, 0.328269511, -0.407830954, -0.387682945, -0.0372718908, 0.546487033, 0.632412314, -0.494615287, 0.484569222, -0.335046232, 0.400614917, 0.409777731, -0.785230041, -0.35260576, 0.146089226, -0.41855368, 0.350596845, 0.767834604, -0.553323448, 0.557047486, -0.474052519, -0.851296663, 1.20988882, -0.479504496, -0.47507292, 0.252668232, -0.0768971816, 0.10374929, -0.491340846, 0.167298138, -0.135968253, -0.237201631, -0.539235413, 0.266471863, 0.764274776, 1.06963873, 0.64189136, 0.258160442, 0.773039699, -0.597770989, -1.18434858, 1.07148314, 0.604650915, 0.436439157, 0.245012432, -0.211310655, 0.393630803, 0.334076166, -0.392476201, -1.0658356, -0.247959822, 0.362116396, 0.347162098, 0.382426381, -0.0759491622, -0.601584256, 0.407191366, -0.328497529, 0.781683564, 0.318506658, -0.326974452, 0.927063286, -0.62534368, -1.00211442, -0.233628362, 0.503780782, -0.579641759, -0.510079503, -0.225645274, 0.714158595, 0.562757492, -0.41103372, 0.357707769, -0.349875361, 0.383057445, 0.474146307, -1.10002911, -0.351130009, 0.233985648, -0.387513161, 0.255342811, 0.734385729, -0.669323981, 0.4122141, -0.628313184, -0.787473977, 1.24135518, -0.668933749, -0.559095502, 0.493527651, -0.325537354, 0.203377366, -0.4349356, 0.218989521, -0.266290963, -0.250037432, -0.707569301, 0.145341069, 0.838765979, 1.36045778, 0.589600563, 0.41397813, 0.701046765, -0.613428831, -1.41070533, 1.2054882, 0.640872717, 0.36385268, 0.334897906, -0.143711925, 0.392348975, 0.496713519, -0.244517505, -1.36358345, -0.466609299, 0.50618273, 0.453114003, 0.209123433, -0.0101209115, -0.494866222, 0.45383361, -0.415456951, 0.557616353, 0.488063991, -0.589736938, 0.964533627, -0.786089599, -1.40910828, -0.219961941, 0.69679755, -0.42304343, -0.0751851201, -0.0158687998, 0.524854839, 0.382059753, -0.380647719, 0.296273112, -0.221393883, 0.295532912, 0.207258373, -1.01958632, -0.419472277, 0.119841956, -0.231918409, 0.127797827, 0.693200946, -0.596327722, 0.273448795, -0.444010764, -0.650002062, 1.56623471, -0.508645296, -0.322794497, 0.232511312, 0.0286838915, 0.123914391, -0.478893369, 0.0807095543, -0.0190814249, -0.138284802, -0.594440401, 0.161965251, 0.646832049, 1.39575422, 0.672821045, 0.266411602, 0.6013605, -0.208654016, -1.19242501, 1.31982136, 0.38568151, 0.303202957, 0.202859864, -0.0928090587, 0.347312659, 0.315423042, -0.12567246, -1.46938014, -0.267662674, 0.402740896, -0.0137400124, 0.0410433933, 0.104746483, -0.513144255, 0.184428141, -0.265233636, 0.507298529, 0.334750563, -0.241917416, 1.19321907, -0.509043217, -1.28002822, -0.154179201, 0.46423164, -0.425630748, -0.377833992, -0.308563799, 0.503439784, 0.566137612, -0.329539478, 0.425764769, -0.447303951, 0.275466025, 0.301733613, -0.909776688, -0.281282872, 0.19528611, -0.443917394, 0.446689099, 0.604748964, -0.472025454, 0.362883776, -0.586260378, -0.786115766, 1.10065484, -0.663078666, -0.53651011, 0.513481915, -0.268212765, 0.135437921, -0.293859124, 0.201443642, -0.263526827, -0.191120133, -0.507800221, 0.197312221, 0.61701107, 1.18685925, 0.58754468, 0.339690387, 0.543017268, -0.573801339, -1.25017965, 1.26668549, 0.644240022, 0.227935314, 0.239973575, -0.0955443829, 0.429756433, 0.310308695, -0.327461034, -1.12692904, -0.343368918, 0.404465795, 0.285750985, 0.347576022, -0.193942234, -0.509978712, 0.299390674, -0.408819109, 0.613180876, 0.50600493, -0.383563101, 0.823956847, -0.557829618, -1.04754567, -0.14566049, 0.683749676, -0.417017907, 0.141781881, 0.0743693039, -0.132111654, -0.194817632, 0.239561945, -0.203357652, 0.129579425, 0.243770778, -0.162329704, -0.120766371, -0.304414809, -0.100198939, 0.306472868, -0.205838069, 0.228253603, 0.0499281138, -0.0701815933, -0.350182891, -0.102613375, 0.308618367, 0.0602031201, -0.356271297, -0.215074703, 0.0202723313, 0.339929104, -0.35398379, -0.0955704078, 0.054202728, 0.199776128, -0.264065534, -0.272960156, 0.252726734, 0.197265312, 0.293150187, 0.241630673, 0.224784866, 0.0434284359, -0.270462722, 0.32273671, 0.330430359, -0.057046663, -0.11925932, 0.302505672, 0.173419356, -0.056487646, -0.131198362, -0.121880151, -0.250820816, 0.220319062, -0.0528289527, -0.267461002, 0.34639132, -0.068936266, -0.145081401, 0.209030926, -0.0336397141, 0.296665043, 0.0556676574, 0.282968313, -0.196078867, -0.392456293, 0.0977721214, 0.126284763, -0.0385491028, -0.536525786, -0.216324195, 0.917357683, 0.536329627, -0.551019132, 0.495584935, -0.356248587, 0.0713457093, 0.452945203, -0.551084518, -0.223783389, 0.23693043, -0.475640595, 0.480812252, 0.483833313, -0.90822643, 0.466743559, -0.492364109, -1.43452275, 0.66220808, -0.800147474, -0.287594885, 0.49357149, -0.400070131, 0.0161626022, -0.284491211, 0.356228054, -0.332562715, -0.46980533, -0.303855091, 0.407975286, 0.441551328, 0.45449084, 0.380961061, 0.376776457, 0.403666914, -0.517319918, -0.723441899, 0.774898529, 0.332766831, 0.347670108, 0.34094736, -0.253277391, 0.293842703, 0.526172578, -0.283712655, -0.712753057, -0.20704098, 0.165279225, 0.358801842, 0.494020849, -0.328629881, -0.772424579, 0.380714238, -0.42599535, 1.14401996, 0.355478346, -0.508070111, 0.439177215, -1.32407653, -0.469580084, -0.414156139, 0.241568148, -0.484124035, -0.276388198, -0.261566132, 0.653547585, 0.59162581, -0.422252506, 0.424493521, -0.599047959, 0.258712322, 0.441181451, -0.53624934, -0.186149001, 0.276645988, -0.383999735, 0.443050385, 0.489643008, -0.733591199, 0.614002407, -0.534607351, -0.705386817, 0.529855013, -0.53553319, -0.261432081, 0.310381442, -0.319335639, 0.267668366, -0.359064192, 0.182456613, -0.20163992, -0.45611757, -0.396166146, 0.226411417, 0.597525537, 0.497735977, 0.519696236, 0.393224806, 0.501320422, -0.6284495, -0.796498358, 0.649134874, 0.404830784, 0.374959826, 0.532537162, -0.0843869746, 0.495871365, 0.55207634, -0.153529882, -0.76127553, -0.440744579, 0.39312306, 0.434141517, 0.313946664, -0.260658473, -0.664929032, 0.20010671, -0.28246513, 0.68965894, 0.159476191, -0.541988015, 0.612759888, -0.686699986, -0.721419275, -0.159214392, 0.563255191, -0.451826155, -0.404601485, -0.129923105, 0.768116534, 0.457714319, -0.282415062, 0.518207252, -0.545926452, 0.202296808, 0.334579706, -0.539969027, -0.0623441637, 0.186650351, -0.314906806, 0.295887321, 0.349980056, -0.642017603, 0.412462145, -0.309073955, -1.63875937, 0.440417379, -0.617059648, -0.303727299, 0.303480119, -0.199189305, -0.0904858708, -0.247963756, 0.236305654, -0.32573244, -0.384526402, -0.379666358, 0.305572599, 0.2990233, 0.532991648, 0.44215709, 0.0943114758, 0.460006803, -0.413071066, -0.602228284, 0.655565858, 0.306779355, 0.375284523, 0.392729402, -0.31339851, 0.310526878, 0.321203232, -0.0857086107, -0.340077549, -0.158091217, 0.276746541, 0.313685209, 0.222494602, -0.0896148905, -0.662942171, 0.40668714, -0.226965919, 1.21436954, 0.116670243, -0.460618585, 0.379437119, -1.43157935, -0.497810781, -0.268609434, 0.2691257, -0.4374744, -0.544128656, -0.153738856, 0.806466758, 0.697766304, -0.308749884, 0.279687375, -0.616335094, 0.0378023386, 0.631812394, -0.61610961, -0.324923128, 0.246356532, -0.479753315, 0.498239189, 0.320099026, -0.879978836, 0.413096756, -0.27323848, -1.64678144, 0.718110323, -0.815286458, -0.438307106, 0.39924106, -0.232177705, -0.013364736, -0.314342916, 0.349587202, -0.35428375, -0.342492789, -0.488959461, 0.243335634, 0.580216885, 0.686432123, 0.512776315, 0.37325263, 0.457635701, -0.666968644, -0.518783569, 0.760379374, 0.273760647, 0.537627399, 0.460816681, -0.324044377, 0.370896131, 0.465907395, -0.0126787117, -0.595686376, -0.374347538, 0.222507402, 0.428265959, 0.479308754, -0.270265073, -0.590712905, 0.396659136, -0.344178051, 1.16334081, 0.384546846, -0.527725339, 0.435495198, -1.30978096, -0.696059883, -0.320203543, 0.229033664, -0.650147617, -0.273492187, -0.164835364, 0.668667018, 0.629295409, -0.522264779, 0.330360919, -0.60428226, 0.169723704, 0.471017838, -0.589739799, -0.172625318, 0.290637463, -0.357112855, 0.482530624, 0.596085727, -0.593576312, 0.496339232, -0.396099567, -0.791489959, 0.523505449, -0.698192954, -0.24262999, 0.361119211, -0.375197023, 0.307743907, -0.457079798, 0.203491971, -0.218809396, -0.207070023, -0.5566383, 0.21313338, 0.587665677, 0.590981603, 0.460330576, 0.381497055, 0.31396991, -0.406499654, -0.646273673, 0.782972097, 0.285102636, 0.433285028, 0.391306609, -0.333679378, 0.320724577, 0.434925884, -0.342287928, -0.727689326, -0.217701256, 0.270231545, 0.473350465, 0.303761214, -0.402583748, -0.546936989, 0.436739236, -0.509154141, 0.763270915, 0.269892544, -0.616448164, 0.659267008, -0.929162681, -0.668321013, -0.337674767, 0.440619588, -0.591116369, -0.563047826, -0.26057142, 0.969926476, 0.607192755, -0.409259439, 0.310617298, -0.471728027, 0.339939326, 0.551383674, -0.62580049, -0.172993213, 0.240941212, -0.26740551, 0.305900991, 0.347701877, -0.878069222, 0.515981078, -0.537627876, -1.17052972, 0.755907178, -0.639583409, -0.47517246, 0.346790433, -0.219063297, 0.0348705351, -0.292179734, 0.474882126, -0.386153251, -0.213677242, -0.456836134, 0.324294567, 0.331846178, 0.537104189, 0.436003745, 0.144273177, 0.530209661, -0.426131099, -0.735307217, 0.718763411, 0.453274429, 0.469704777, 0.321545869, -0.21566245, 0.424108654, 0.344189733, -0.0592800081, -0.521855295, -0.107721195, 0.317939609, 0.430018395, 0.457768142, -0.172899276, -0.612234235, 0.406998247, -0.448220253, 1.11257839, 0.191234738, -0.479058534, 0.481455982, -1.12707865, -0.648124576, -0.194276959, 0.345581084, -0.484572679, -0.343308598, -0.12794216, 0.672531426, 0.424719602, -0.302648067, 0.359854698, -0.400834858, 0.473584592, 0.422555357, -0.678353608, -0.261491418, 0.217765197, -0.171049848, 0.285351127, 0.513761342, -0.658162415, 0.46343568, -0.548393846, -0.617358863, 1.1439836, -0.508872807, -0.538265049, 0.477225065, -0.299464107, 0.22175248, -0.313081294, 0.371365666, -0.230835333, -0.145164087, -0.441226751, 0.414759785, 0.584097981, 1.06914091, 0.552144825, 0.320418417, 0.714488447, -0.354277045, -0.928710818, 1.1338594, 0.36863628, 0.266910672, 0.392667323, -0.0111860326, 0.355612755, 0.278948724, -0.428407669, -0.807357132, -0.262119412, 0.42804426, 0.205490455, 0.33340618, -0.288222104, -0.650719345, 0.412516952, -0.491195202, 0.773645103, 0.364975005, -0.519680321, 0.906551361, -0.524672151, -1.01487565, -0.39606598, 0.405813515, -0.563595951, -0.269886643, -0.350732118, 0.606613576, 0.384260803, -0.376138091, 0.508033037, -0.360961974, 0.466318488, 0.277735382, -0.66640687, -0.35502246, 0.109514922, -0.298087895, 0.355182439, 0.646670938, -0.632044554, 0.439749837, -0.382921994, -0.660431385, 0.893898308, -0.540391684, -0.321551055, 0.221916288, -0.160736755, 0.308179349, -0.26730603, 0.206497774, -0.225358516, -0.351685643, -0.558867693, 0.374778271, 0.612612009, 0.978533804, 0.607411861, 0.285413414, 0.51165098, -0.344507605, -0.921458423, 0.888002694, 0.500364721, 0.202447027, 0.380399704, -0.271877974, 0.380116731, 0.526907861, -0.218600065, -0.825426459, -0.240812227, 0.396916181, 0.264241874, 0.365629554, -0.171145856, -0.403258473, 0.408908993, -0.489471793, 0.606956661, 0.459666014, -0.463012695, 0.852094889, -0.780032933, -0.761940658, -0.291623026, 0.498924643, -0.302560419, -0.171400279, -0.33405292, -0.0493575782, 0.17232205, -0.110599153, 0.329337597, -0.357625425, -0.234940618, 0.152215123, 0.319324821, 0.43764329, 0.386182725, -0.177471906, 0.32160902, -0.474107057, -0.00973141473, 0.0944921076, 0.322700441, 0.0120441252, -0.451121688, -0.0308260825, 0.433692187, 0.224495098, -0.292792976, -0.511347592, 0.473475844, 0.262363851, -0.240330055, -0.421176165, 0.369746774, 0.432316303, -0.436458081, -0.277693868, -0.514254212, -0.520781636, -0.385244131, -0.155822918, 0.358417571, -0.188162878, -0.299654812, 0.237457052, 0.241685927, -0.423709124, -0.283290237, 0.1787242, 0.314056337, 0.152405173, 0.388397336, -0.299144179, 0.190873206, 0.425582856, -0.315479517, -0.129302844, 0.184376732, -0.328748405, -0.127442196, -0.323519915, -0.122181714, -0.446838707, 0.0990149751, 0.233083859, -0.313614875, -0.286455244, -0.108938903, -0.173898384, -0.154455885, 0.608990073, 0.639379859, -0.333209395, 0.214992166, -0.297589988, 0.255593807, 0.415786177, -1.06228507, -0.219749421, 0.0616546981, -0.0850304291, 0.217553958, 0.614582717, -0.527022839, 0.334150106, -0.680784225, -0.861281753, 1.82366407, -0.43191725, -0.372459769, 0.387694806, -0.0302853379, 0.131834209, -0.512922108, 0.107565053, -0.224938229, -0.319808245, -0.549067795, 0.112411819, 0.703112602, 1.82133305, 0.7760638, 0.212270632, 0.559252858, -0.326964855, -1.57775831, 1.69533455, 0.496235013, 0.351062626, 0.150329247, -0.0431579985, 0.518127322, 0.488872588, -0.182545111, -1.98710394, -0.428537518, 0.527171254, 0.13654837, 0.316436887, 0.0261419453, -0.339206904, 0.154128537, -0.293990165, 0.695450902, 0.270007789, -0.371297151, 1.1685667, -0.692904472, -1.70720041, -0.161414593, 0.542755067, -0.368743628, -0.271216959, -0.350861341, 0.879380643, 0.389808565, -0.462255955, 0.25825274, -0.287204325, 0.0223016348, 0.572541773, -0.368543565, -0.262212306, 0.345916182, -0.206542492, 0.198395595, 0.438706398, -0.680423021, 0.421501189, -0.225021601, -1.4016006, 0.453847796, -0.717998624, -0.333025008, 0.322651654, -0.387569427, -0.0341551788, -0.28112945, 0.37996915, -0.186973631, -0.203572124, -0.152209431, 0.34419021, 0.34519434, 0.446676373, 0.446126312, 0.0983296484, 0.314393342, -0.616695642, -0.579172671, 0.402942836, 0.259942979, 0.484394908, 0.313688248, -0.130447447, 0.179317132, 0.490951687, 0.0383905619, -0.331919551, -0.27869752, 0.304098934, 0.407192022, 0.405362815, -0.326767892, -0.457747221, 0.379286647, -0.478376925, 1.23467183, 0.119863309, -0.276864558, 0.246494442, -1.32616842, -0.403463274, -0.377959818, 0.28082931, -0.308996797, -0.425722748, -0.193674147, 0.78785944, 0.508327127, -0.248903885, 0.264103949, -0.357186317, 0.0147308437, 0.409206808, -0.194472671, 0.00276197912, 0.258905709, -0.166197851, 0.420497239, 0.329626769, -0.692572415, 0.47229892, -0.0915081054, -1.23548186, 0.432720244, -0.532778084, -0.293897599, 0.351049364, -0.116568863, -0.0321129113, -0.00978968013, 0.194032043, -0.305195987, -0.331068963, -0.151935816, 0.279666692, 0.18866615, 0.430132568, 0.327653021, 0.187172294, 0.219540179, -0.436067939, -0.488186747, 0.306090027, 0.0649880245, 0.295697391, 0.304286689, -0.220163599, 0.218568921, 0.42988044, 0.083551079, -0.21370098, -0.24988465, 0.119232155, 0.42408514, 0.367069811, -0.316671014, -0.37558344, 0.158022285, -0.264873117, 1.1731286, -0.00102446123, -0.327192366, 0.419644058, -1.28937852, -0.396725744, -0.142590478, 0.174560189, -0.52244091, -0.0736855492, -0.00405138312, 0.502723634, 0.257404685, -0.20088473, 0.338655323, -0.30681926, 0.248688862, 0.340052962, -1.18811226, -0.305723131, 0.132275894, -0.0452247262, 0.171353057, 0.583092511, -0.487280637, 0.196598664, -0.483296543, -0.69260937, 1.35671079, -0.436298639, -0.381194085, 0.213245317, -0.139961824, 0.242243573, -0.332228541, 0.162442148, -0.0164368581, -0.134004563, -0.395557404, 0.153602988, 0.805303276, 1.37767732, 0.616612911, 0.365305662, 0.650224328, -0.22939913, -1.2560699, 1.10163033, 0.357846498, 0.065071173, 0.181495398, -0.0377712026, 0.388611585, 0.213618428, -0.107306898, -1.31008828, -0.177096337, 0.321845561, 0.218017265, 0.206176892, 0.00983442646, -0.525239408, 0.240989879, -0.143164024, 0.669313908, 0.247989461, -0.351266146, 1.11758339, -0.531946778, -1.49604833, 0.02928463, 0.581405699, -0.440303475, -0.385143578, -0.396308482, 0.750951886, 0.57296735, -0.446412802, 0.455750138, -0.418437362, 0.0957896784, 0.501497984, -0.44672817, -0.237872884, 0.274565369, -0.42142725, 0.489412338, 0.56970638, -0.710014164, 0.450249612, -0.278510541, -1.0801419, 0.788323283, -0.569819212, -0.344335169, 0.542477369, -0.337672293, 0.236581355, -0.170987174, 0.246147275, -0.266410828, -0.17478773, -0.250558347, 0.252318501, 0.381735712, 0.602397978, 0.616476417, 0.217723235, 0.384022832, -0.377786189, -0.662218869, 0.57415092, 0.349585682, 0.339607358, 0.465482593, -0.295192808, 0.506696105, 0.317660213, -0.0275208782, -0.636613369, -0.173345938, 0.383084655, 0.39059639, 0.437923908, -0.362441689, -0.492392182, 0.304834664, -0.277102828, 0.780932546, 0.358055443, -0.35449028, 0.648201704, -1.02766812, -0.65746969, -0.290710598, 0.266317517, -0.487403065, -0.342292964, -0.214244977, 0.737149656, 0.448120058, -0.230806604, 0.422618449, -0.292649239, 0.168079019, 0.534740627, -1.16855597, -0.432713687, -0.0108646816, -0.126822308, 0.25649479, 0.770150781, -0.645632446, 0.403120458, -0.724118412, -0.859452844, 2.22503901, -0.64947921, -0.367921531, 0.358518481, -0.155806094, 0.193853229, -0.297354549, 0.120156467, -0.0946324617, -0.243912473, -0.472326577, 0.145495683, 0.832385361, 2.19498634, 0.778509676, 0.342008919, 0.848277271, -0.49624604, -1.69642162, 1.71654153, 0.588248074, 0.33258453, 0.344076008, -0.163638383, 0.56731528, 0.247680068, -0.354752421, -2.37261987, -0.398869097, 0.391421556, 0.352473855, 0.115878321, -0.112021856, -0.472907096, 0.381194562, -0.418286622, 0.543751717, 0.30754447, -0.280784011, 1.41610241, -0.798416913, -2.10225344, -0.185180351, 0.510154903, -0.323697358, -0.458895683, -0.348646909, 0.705939233, 0.538262188, -0.513440371, 0.475339651, -0.328043967, 0.384672582, 0.44323957, -0.761635363, -0.270843118, 0.261911571, -0.252113491, 0.381079525, 0.609498322, -0.450055778, 0.356651932, -0.491022676, -0.810506225, 0.82410872, -0.578057647, -0.521694124, 0.423432797, -0.246942252, 0.291828603, -0.274428874, 0.34558928, -0.163658366, -0.2072023, -0.667214453, 0.331220478, 0.769516528, 0.815972626, 0.761667073, 0.519886792, 0.735126495, -0.363234431, -1.01916885, 0.980866015, 0.465000719, 0.297353357, 0.268718481, -0.133869484, 0.596612692, 0.272900581, -0.374923646, -0.764245868, -0.400829643, 0.387301534, 0.411194116, 0.458122432, -0.0897585005, -0.611259997, 0.396098167, -0.514478326, 0.615652442, 0.469147056, -0.551474094, 0.677580595, -0.723048508, -0.958446622, -0.351297438, 0.5369609, -0.466082484, -0.392684519, -0.140763402, 0.738301575, 0.505346894, -0.551214337, 0.488818526, -0.464140445, 0.197854578, 0.394551396, -0.906450927, -0.236846372, 0.0841318369, -0.367447346, 0.449851722, 0.773675323, -0.738755822, 0.441427588, -0.654032588, -0.711928427, 1.18266237, -0.549853086, -0.460477382, 0.219276875, -0.149520844, 0.179480404, -0.431614518, 0.197724342, -0.272667557, -0.340881646, -0.565278411, 0.232482374, 0.804801285, 1.03302395, 0.805033445, 0.504528701, 0.587796926, -0.4402273, -1.21261656, 1.17494059, 0.443305463, 0.264766097, 0.316561788, -0.138892338, 0.65940237, 0.564585388, -0.31081444, -0.90176338, -0.471996456, 0.371961445, 0.158505559, 0.370738208, -0.0978980586, -0.373646945, 0.392568529, -0.308288038, 0.779628813, 0.232412338, -0.372803688, 0.794813037, -0.738244116, -1.15833187, -0.373204678, 0.6222229, -0.539139509, -0.443403453, -0.290466309, 0.819968641, 0.527707577, -0.413294584, 0.274637192, -0.467576206, 0.0177975688, 0.598754168, -0.495468289, -0.163562313, 0.17254664, -0.416864395, 0.243399248, 0.288690567, -0.750119209, 0.554691315, -0.208583638, -1.92795444, 0.496306002, -0.850651801, -0.344283283, 0.44015038, -0.395032018, -0.0522430316, -0.25097248, 0.401277214, -0.398269415, -0.220324293, -0.422234803, 0.186774373, 0.392636329, 0.649317384, 0.484548628, 0.120573297, 0.480113119, -0.571780026, -0.65580982, 0.513943195, 0.472561806, 0.326867461, 0.286692291, -0.303493977, 0.462431997, 0.504831314, -0.20678623, -0.445540279, -0.0930512697, 0.290064484, 0.194492519, 0.420097232, -0.199875414, -0.649175227, 0.197605386, -0.534060299, 1.32834315, 0.113373868, -0.361338526, 0.44961217, -1.64719367, -0.678484142, -0.303245872, 0.287665248, -0.575748205, -0.336794019, -0.0869292989, 0.432107985, 0.486114502, -0.221369773, 0.288731098, -0.318255961, 0.268310964, 0.240426511, -1.1222862, -0.309996933, -0.0533496514, -0.178539693, 0.306757689, 0.708717108, -0.463632852, 0.213827491, -0.629661322, -0.744728744, 1.77040315, -0.515126169, -0.487291873, 0.264207542, 0.00132249307, 0.323194981, -0.497462869, 0.182954505, -0.23436442, -0.187767476, -0.705290735, 0.164230332, 0.66266185, 2.02163887, 0.588158846, 0.303405881, 0.737843692, -0.390376419, -1.43576646, 1.54322898, 0.434838712, 0.145693526, 0.30881536, -0.0685351416, 0.342455328, 0.24507685, -0.27616778, -2.15865946, -0.287609041, 0.460926324, 0.190310925, 0.0574499927, 0.100047357, -0.557812035, 0.199095517, -0.114541799, 0.670535684, 0.32147494, -0.418899715, 1.15679395, -0.762430549, -1.66618228, -0.093862243, 0.486004472, -0.202861622];
    CONSTANT recurrent_3_r : ARRAY[0..4095] OF REAL := [0.00911375321, -0.00202236348, -0.0237983093, -0.0230638143, 0.0748881623, -0.0255280919, 0.032285504, -0.00382772577, 0.110893279, 0.0975007489, 0.0418522805, 0.0609153658, 0.0313407704, 0.0302556343, 0.0175146423, -0.0281471703, 0.0318852216, 0.0426676609, 0.0123656504, 0.1041703, 0.0541706048, -0.000886218622, 0.197626323, 0.0429425202, -0.0799675807, -0.00761905871, 0.00706546754, -0.0571719408, -0.0689751357, 0.0451986678, 0.0201027133, 0.0631553233, -0.129691571, 0.0320937745, 0.0302708726, 0.121609271, -0.112159126, -0.0793186352, 0.0803062767, 0.0614077896, 0.00459189387, 0.0504808798, -0.125838056, 0.176575303, 0.0082402043, 0.0200517774, 0.0343972668, -0.0574389771, 0.110039622, -0.0383961499, -0.114136584, -0.0274701472, -0.0615831465, 0.0620580614, -0.022973517, -0.00469653029, -0.0329369009, 0.0095978938, -0.056178797, 0.0776937082, 0.0561335124, 0.132600427, -0.100108549, 0.0226371828, 0.0583960861, -0.0655008852, -0.00749516673, -0.0113983564, -0.0423510447, -0.0797068775, -0.0199018288, 0.0782541484, -0.0776402503, -0.0815584138, 0.154344261, 0.116309933, -0.0853010118, 0.0429037586, -0.111408979, 0.0519659445, -0.0714104623, 0.0202703439, 0.0431506336, -0.0217190031, -0.0993405879, -0.0339033231, -0.0319767073, 0.0969930366, -0.0934475288, 0.0431513488, -0.0437430516, 0.0551541001, -0.102149546, -0.0419385284, -0.0510420054, 0.104995966, 0.00981811248, 0.054826092, -0.0460422263, -0.14945735, -0.0887676179, 0.0757255033, -0.0682021081, 0.067138575, 0.0527030081, -0.142467126, 0.00623679161, -0.081650205, -0.0217414498, -0.0519152284, -0.0114929061, -0.0353443436, 0.0697723329, 0.0216454808, -0.147972912, -0.0305027403, 0.00866494142, -0.0361279584, -0.0156128649, 0.0648681819, -0.0711312518, 0.0697998106, -0.0817103982, 0.0791503042, 0.167355821, -0.0372648276, -0.0513354391, 0.120582767, -0.0890771151, 0.0257072933, -0.123685598, 0.0827882737, 0.0198066384, -0.0830840692, -0.0058414354, -0.11684899, 0.11155083, -0.0375803076, -0.0860175788, 0.108100832, 0.00140646752, 0.00455251336, 0.00355935167, 0.104866102, -0.183338359, 0.19762516, -0.02773319, 0.0545151457, -0.0323703475, -0.0841021389, -0.020246096, 0.103897557, 0.0332882218, 0.122344576, 0.0356296748, -0.0390966535, 0.0482734516, -0.0153638236, -0.0705761611, -0.0545569919, 0.0216887072, 0.0146980723, 0.134173021, -0.0277683474, 0.108473256, -0.00895685516, -0.000122845173, -0.148091972, 0.00765258633, 0.112680122, 0.0627765208, -0.0699514449, 0.0579327606, 0.167391047, -0.0206126291, -0.0232587494, -0.0227806028, 0.164959013, 0.017952228, -0.029058177, 0.0931209773, -0.0905666649, 0.0297105536, 0.0643432513, -0.0572242662, 0.00399557408, 0.0640901178, 0.0284853913, -0.0532626435, -0.093953222, -0.116984934, 0.00363150612, 0.0778844729, -0.0534194075, 0.0356680602, -0.0513897985, 0.0127216633, 0.0420455039, -0.026197603, 0.047176417, 0.0816618875, 0.00285134348, 0.0223577488, 0.0966080576, 0.00698447414, 0.0076117944, 0.041453708, -0.0264793001, 0.0078772828, 0.0449370891, -0.114559084, -0.0222518574, -0.0767178088, 0.0344772972, -0.0263515487, 0.00535550434, 0.0400021747, 0.0447246432, -0.0108250044, 0.00396102015, 0.0204284508, 0.071688287, -0.0889900625, -0.0552459359, 0.0875648484, -0.0842856988, -0.0550064743, -0.101071484, 0.0326540209, 0.0544580296, 0.0738798827, 0.00837158598, -0.0739922822, 0.031114623, 0.0112157539, 0.047144495, 0.129318848, -0.037200179, 0.118786499, -0.0740327165, 0.0661123395, -0.0531371832, -0.0284307264, -0.108321421, -0.100672431, -0.029302977, -0.101315923, -0.177598029, -0.092394568, 0.0691574663, -0.0419421941, 0.0279376302, 0.158116013, -0.0253254287, 0.0146561749, -0.047278095, 0.033318989, -0.0360458903, -0.0600628331, 0.0303683579, -0.0589155927, -0.0240204073, 0.0839619339, 0.0034722772, -0.0770511553, 0.0292353425, 0.0550547764, 0.00291131251, -0.0408926569, -0.01090765, -0.0305658355, 0.141737267, 0.021275593, -0.123218119, -0.0334331989, -0.0504225008, 0.0127103962, -0.0695255473, 0.0296204053, 0.0265006982, 0.0580648482, 0.0501579717, -0.0626788139, -0.0789386332, -0.0628380179, -0.0720427558, 0.0320159942, -0.0315630734, -0.10637518, -0.0208138376, 0.00724740699, 0.0239238143, 0.0816971362, -0.0362997353, -0.10336107, -0.00830980577, -0.0301181413, 0.0565131381, 0.0499073453, -0.000258012209, -0.0084053874, -0.0921288431, -0.002275832, -0.114925586, -0.0470449179, -0.106850281, -0.0981545299, 0.0292031579, 0.127993435, 0.023694573, -0.0580891445, -0.108017705, 0.0432504714, 0.0474100932, 0.0421978645, 0.0362437442, 0.00868836232, -0.0331392735, -0.0259158984, -0.0993543863, -0.091642648, -0.0400814563, 0.0184793398, -0.0358050019, 0.143999591, -0.023802178, -0.0589483343, 0.0488821268, -0.0130757075, 0.0715813115, 0.0435160547, 0.0556875393, 0.0652761608, 0.000147297047, 0.0398971811, 0.0967640653, 0.0463042036, 0.00411752611, 0.00755714439, 0.0722247064, 0.0147378575, -0.147983626, -0.0114682335, -0.119335331, -0.0348146968, 0.0757440105, -0.0889739841, -0.171713427, 0.0727809593, -0.109121919, -0.0193136204, 0.107689202, -0.031507574, -0.0489449948, 0.0480983704, -0.0117908092, -0.0625669062, -0.0629829913, -0.0509033576, 0.14963536, -0.101753235, 0.0575250536, 0.0423747487, -0.135954604, 0.00802879781, 0.138046563, 0.203562587, -0.0937730521, -0.043450743, -0.0903653726, 0.0496570095, -0.101320013, -0.0425310731, -0.0388302952, 0.0215265229, -0.0114472369, -0.160118356, -0.0577234179, -0.056208618, -0.159860149, -0.130893126, 0.0153518021, -0.0469167009, 0.0170055293, 0.0609783083, -0.0040185065, 0.0274109729, 0.11365439, 0.00275870599, 0.00512488326, -0.0133355847, 0.094586432, 0.102978855, -0.0182318985, 0.0394562408, 0.024214007, 0.00501166517, 0.146497458, 0.0535710938, -0.167801186, 0.0870854333, -0.0367849171, 0.127105713, -0.0133330319, 0.0571585521, -0.131522089, 0.0820833668, 0.0694639385, -0.00270178728, 0.0746649206, -0.0351437517, 0.0531759933, 0.107341737, -0.0166541357, 0.0899687558, -0.135554671, 0.107365236, -0.0745012611, -0.121961415, 0.00332099153, 0.0623820536, -0.0855424553, -0.144670919, -0.00410610996, 0.018668985, -0.0468354598, 0.104753383, 0.116255291, -0.0909991711, 0.0423864201, -0.0167759657, 0.112893499, 0.0140526397, 0.0157002211, 0.025987532, -0.0515090972, 0.0492114387, 0.0286730602, -0.00728053227, 0.0730762854, -0.0576741025, 0.0987064838, -0.12626642, 0.0363303982, 0.00025613606, -0.0854930282, 0.0409880728, -0.0491628014, -0.0495841466, -0.0832021907, 0.109828413, -0.00949191209, 0.025237117, 0.122777909, 0.0256123319, 0.0638817549, 0.00852558389, 0.0977258906, 0.165678307, 0.0380590409, -0.040783532, -0.0961662456, 0.0668946505, -0.0157988425, -0.0765058249, -0.0761791319, 0.127417073, -0.00562030124, -0.0150924847, 0.0162233636, 0.0635270476, -0.121701874, -0.0227665529, -0.0745811015, 0.00387974456, 0.0041704569, -0.0789878815, -0.0486721024, -0.00843084604, 0.0702937096, 0.030550193, -0.0509378761, -0.0183612444, -0.141379282, 0.118152753, -0.0668954402, -0.0372721925, -0.0300644953, 0.0570926517, -0.0313790515, 0.0383626595, 0.12200132, 0.069827117, 0.0511526726, 0.105546087, 0.111735642, 0.0725364089, -0.0557615533, 0.060444653, -0.0400662571, -0.0745078549, -0.0652316064, -0.0708966032, -0.0220151078, 0.0539559312, 0.0375150554, 0.0141001325, 0.0504179634, -0.0686047524, -0.0137163773, -0.0515023954, 0.0290786456, 0.0783781409, -0.0577777997, 0.013601426, -0.037097238, -0.0802973881, -0.0311410725, 0.000239511253, 0.0391602069, -0.102556601, 0.0228124075, 0.0532910526, 0.00637396704, 0.211682871, -0.0590877682, -0.0185743347, -0.116268821, 0.123046994, 0.0638253465, 0.103012592, -0.0295602046, -0.0184217803, -0.126529723, -0.021587871, 0.0466953442, -0.0207868125, -0.0102520138, 0.0223338567, -0.0615631379, -0.0313155428, 0.0144809857, 0.0701513886, -0.0250683762, 0.0702576339, -0.104813933, 0.0414853878, 0.0486246869, -0.0420227423, 0.0235443022, 0.0312029328, -0.0468768179, -0.0021700263, 0.122100636, 0.0458291471, -0.0841060728, 0.0307521727, 0.120696224, 0.0763218403, 0.124105752, -0.0635750741, 0.0466547534, 0.0204870068, 0.0262179971, 0.00880821981, -0.134466439, 0.0516617745, 0.0791150853, 0.158821866, -0.0417293124, -0.0195431169, -0.0592326075, 0.0584496781, 0.0470124222, -0.0392942876, 0.0094333142, 0.0206860416, 0.160820901, -0.00310400408, 0.0299142431, 0.00139450654, 0.062466152, 0.05967924, -0.0433351211, 0.0331435986, 0.0972179025, 0.105120547, -0.0478204675, 0.0743556842, -0.0672744066, -0.046730414, -0.246408552, -0.0541513227, 0.00750867184, -0.0652973503, 0.0212405361, -0.02554431, 0.00203400478, 0.0351974927, 0.0219492614, -0.0213655662, 0.120339364, 0.0119028874, -0.034202572, -0.00784637406, -0.0541388094, -0.0597577617, 0.0158543289, 0.091164723, -7.52375927e-05, 0.0459715798, 0.0581619553, 0.0518091209, 0.00359082595, -0.0237384886, -0.147958845, 0.0622775517, 0.00865327567, -0.0153832324, -0.00439291075, -0.0402460471, 0.0388767943, 0.0856813192, -0.0089630885, 0.0840314776, 0.0315066054, -0.0487823747, 0.0760353208, -0.0752325878, 0.0017796047, -0.0281302053, 0.0624732561, 0.0957097262, 0.0376511998, -0.0715606511, -0.0852134004, 0.037225768, 0.0122167673, 0.0466136895, 0.038283091, 0.0952630118, 0.0974789783, -0.12276344, 0.00118430168, 0.0302159172, 0.00623338297, 0.018055059, 0.0586414635, 0.0171477292, -0.0526880771, -0.118420757, -0.124844752, 0.0284788664, -0.114810653, 0.0275984257, -0.0696739107, 0.0751996264, 0.095859915, 0.0687997341, -0.0259143673, 0.0121420603, -0.0324660055, 0.0405802354, -0.085328877, 0.119429722, -0.100314185, 0.102070868, -0.0252911821, 0.038893953, 0.0412346721, -0.0210889746, 0.129765391, 0.0169580691, 0.0226371624, -0.00887788087, -0.0572359003, 0.0157009233, 0.0193942357, -0.0108801918, -0.0912810713, -0.0476359725, -0.134074837, 0.0126453936, -0.0825806633, 0.0523258373, -0.0237158537, -0.0808548555, -0.091645591, 0.0902565494, 0.0146779232, 0.0990815386, -0.0994295329, -0.0455697812, 0.0555170365, -0.0137906522, 0.0581970885, -0.0395062715, -0.0858608931, -0.0830656365, 0.154364914, 0.14480707, 0.0541687235, -0.0914984494, 0.0245234314, -0.0803825408, 0.0533412918, 0.0108824316, 0.00130331982, -0.0745498165, 0.0868173093, -0.0637374967, 0.135478705, -0.0230534226, 0.0158655085, 0.0483710021, 0.0841864422, 0.135531038, 0.037712846, -0.0691346228, 0.0643537939, -0.00478052162, 0.111542173, -0.0323873013, -0.0721196979, 0.0629153326, -0.03225936, -0.0202114917, -0.0586395785, 0.0703757331, 0.105001338, -0.0352300443, -0.0207109638, -0.00277804397, -0.088710092, -0.00636978261, 0.0597423539, 0.1233472, -0.0532054417, -0.0184984189, -0.0356769115, -0.106631212, -0.078933306, -0.029100934, -0.0164433196, -0.100324057, 0.00681179203, 0.0538881905, 0.0577190667, 0.0235630125, -0.0408950746, -0.0765696466, 0.0572620928, 0.0715509504, -0.0141098583, -0.14256452, 0.0620078668, 0.0513346642, -0.014593279, -0.000190385617, 0.115069576, -0.00733298063, -0.0381898433, 0.0965593979, -0.082215935, 0.037181966, 0.057968311, -0.0169563778, -0.0351036116, 0.104300693, 0.131403923, -0.0407392234, 0.00248470437, -0.0625106692, 0.0529611409, 0.100966096, 0.0189072099, -0.0458419807, -0.0284237247, 0.0446987785, 0.0183654595, 0.0586776659, -0.0624799319, 0.116953477, 0.090016, 0.0165911783, -0.0229423959, -0.0926959291, 0.0235078447, -0.143053502, 0.0780783594, -0.0424500518, -0.0258744825, -0.13351348, -0.0939254463, -0.0294577107, 0.0331923179, -0.0493002273, 0.0673060417, -0.075317204, 0.0199663527, 0.0166395791, -0.0253233835, 0.0714993253, -0.0840470567, 0.116615638, -0.0817578733, 0.0800578892, 0.0296422839, 0.170557499, -0.1654616, -0.0277361833, -0.0246826354, 0.0284979492, -0.0261004046, -0.0193990432, -0.153675005, -0.000156990252, 0.0446386524, 0.00112404674, 0.00340267271, 0.110186473, -0.129498541, -0.0645064041, 0.0497275293, -0.01430069, -0.0417016521, 0.0662118047, 0.0380283259, 0.088968575, 0.0519468486, 0.0699722841, 0.0985773206, 0.01397039, -0.123004794, 0.050001882, 0.0688602924, 0.0884637237, -0.024484409, 0.0231193155, 0.0867063031, -0.117401488, 0.146742731, -0.0245518778, -0.00049746735, 0.107563034, 0.0153732263, -0.00138764642, 0.00719641149, -0.118613921, -0.0699281916, -0.0448083505, 0.0568592809, -0.03438925, -0.0568434261, 0.128248841, -0.0970832705, -0.131126106, -0.0322123691, 0.0494427308, 0.0349712223, -0.0516956002, -0.0108481338, -0.0205307081, -0.0627812296, -0.094834514, 0.0353070721, -0.0258042347, 0.139962509, 0.171861947, 0.00694552436, 0.0189717431, 0.0562504679, 0.0536639579, -0.012175221, 0.0922481269, -0.00224624015, -0.0172267184, -0.00408977456, -0.0315037183, -0.155455768, -0.0409466997, 0.13185519, 0.0294154324, -0.0134966858, -0.0774052441, -0.0542730987, -0.0419860855, -0.012225043, 0.081311509, 0.158177853, -0.0468696058, -0.0932726637, -0.0693122372, -0.00300208479, 0.0683663636, 0.0593294948, -0.0115551008, 0.179554924, 0.0512919687, -0.00133599411, 0.110675007, -0.0401133969, -0.000876663718, 0.151455745, -0.00121552218, 0.0146848718, -0.00242423825, -0.0363500565, -0.116146825, 0.079527013, 0.0865260661, 0.0545096248, -0.12196292, 0.0208703764, 0.0821463987, -0.0134822782, -0.027833946, 0.010675285, -0.0534569211, -0.15372014, 0.0209434144, 0.00385515532, -0.03036635, 0.0187385231, -0.0500814356, 0.00731410086, -0.0450109951, 0.0475450531, -0.0660711229, -0.0576170869, 0.0392976701, 0.0141733531, 0.105263107, 0.105541557, -0.0835994035, -0.0604783595, 0.0700645596, 0.00952682085, -0.060204614, 0.0383245014, -0.0303084739, 0.0449032895, -0.0314889662, -0.0117235109, -0.0435175374, -0.0120741315, -0.0456162468, -0.0304395314, 0.0392664373, 0.0543761477, -0.0223365463, 0.0479622632, -0.0356663093, -0.0946084857, -0.0987185538, -0.00450733677, -0.0622910261, -0.0854664817, -0.11624071, 0.0300633647, -0.0188361872, -0.196206644, -0.0151952319, 0.0356712975, 0.00420160685, 0.00529858842, -0.0407636985, -0.134199858, 0.0454469286, -0.0514911935, -0.0955984145, 0.0996576995, -0.0216490272, 0.0796884149, -0.0338479728, -0.0541275144, 0.114153914, -0.0927425176, 0.0597409792, 0.0275961626, -0.0266114324, -0.00144245848, -0.0843057185, -0.03371007, -0.000822213478, 0.137287915, 0.00845224597, 0.0294579789, -0.0588286072, -0.00748171657, 0.0366862677, -0.0881185085, -0.181755364, -0.0932161659, -0.0302605592, -0.004988058, -0.0171914734, 0.114152938, -0.0937477127, -0.107621804, 0.0418742374, 0.140122101, -0.109398291, -0.060850732, 0.0686470121, -0.000218321104, -0.0639985651, -0.0357726179, 0.110667303, 0.017532561, 0.0799096227, 0.0709084868, 0.0575583391, -0.0957374871, 0.0288257729, -0.0392640568, -0.124348633, 0.0544305295, 0.0763412863, -0.0880652219, 0.097671628, 0.047271423, -0.053128466, -0.0847817063, 0.0605234578, -0.0322612561, -0.0957455635, 0.163376689, -0.113794908, 0.0213765427, -0.0908470526, -0.0491742082, 0.0226370767, 0.0737887472, -0.0319020078, 0.0486837551, -0.0219347104, 0.0116338525, -0.0391337238, -0.0229025614, -0.055400338, 0.0399981774, -0.161445707, 0.0143578146, 0.108743295, -0.0870562717, -0.0278399661, -0.0423922464, -0.0586773343, -0.0430437848, -0.0837854445, -0.00241982192, 0.0739955232, -0.00983252376, 0.0226107929, -0.0281373821, -0.0663822368, -0.10870792, -0.0264889598, -0.0318740979, 0.0360140987, -0.0275817625, -0.0117399385, -0.0622121133, 0.0386478081, -0.138306975, 0.0722252876, 0.0681583658, 0.0357433297, -0.0503761508, -0.0888322741, 0.00609578472, -0.0550457835, -0.00491966493, 0.0018206574, -0.0777870715, 0.147252217, -0.0580721535, 0.00839607045, -0.0367960967, 0.0526871458, 0.112481609, -0.0370250121, 0.100097127, 0.0684277043, -0.0590134449, -0.000272998586, 0.0157443862, 0.0360369533, -0.00823564827, -0.11443729, -0.0748900771, 0.0570345223, 0.136014342, -0.00862678513, 0.0702614263, 0.0514154285, -0.0681594908, 0.0298552141, 0.00540684536, -0.0526974462, 0.0862854049, 0.0461132079, 0.10347601, 0.0749654993, -0.0231539886, -0.112434372, -0.0588796437, 0.0134588666, -0.131307006, -0.0329538956, 0.0385348871, 0.156908885, -0.0546470098, 0.00706227124, -0.00997575559, 0.0139146633, 0.0237259697, -0.00629263464, -0.0165242497, 0.090869844, 0.0364026949, -0.0375510603, -0.143859923, 0.0524707101, -0.0971896201, 0.00969352759, -0.0669112504, 0.100931376, -0.0398303121, -0.0936012641, -0.056639906, -0.0213063024, 0.175421089, -0.0735043213, -0.0395346321, -0.0607963353, -0.029217504, -0.0229287352, 0.042531345, -0.0905115232, -0.00708591565, -0.137183487, -0.0699275136, 0.107452646, -0.0319059044, -0.00441396236, -0.0106489789, 0.00246873125, 0.0293903332, -0.0112364143, 0.0890116245, -0.0172665641, -0.00711072702, 0.0278019793, 0.051202938, 0.054612495, -0.0475451201, -0.144114584, -0.0397719592, -0.113360614, 0.0785803273, 0.248093903, 0.0131256646, -0.0935446024, -0.0747676492, -0.00567668118, 0.00239985064, 0.0283464417, 0.111431696, -0.0532648116, -0.0453556739, -0.0236246549, -0.0972554907, -0.0118487664, 0.0293593854, -0.0276271068, 0.00488677248, 0.0133009003, 0.041428037, 0.0813874677, -0.00393976644, 0.0840215832, -0.0254320111, -0.0392817594, 0.00961663947, -0.085313648, -0.0234975703, -0.0803359449, 0.103493989, -0.0231693909, -0.0406989381, -0.057833001, -0.0455716588, 0.00552285463, -0.00918115489, -0.0363552719, -0.0460190773, -0.0786511749, -0.111753605, 0.0318435878, -0.0275966488, -0.146628007, -0.0202041827, 0.0246242601, 0.018335212, 0.0525075756, 0.0480933674, 0.015275049, 0.0815747604, 0.0505161509, -0.0541922376, -0.0505428798, 0.111340925, 0.0775246918, -0.0652684048, 0.0497954078, -0.202423543, -0.0580477528, 0.020171009, -0.00113054644, -0.0192843638, 0.0420398563, -0.0225126874, -0.00377615076, -0.0362481251, -0.0177948177, 0.0269957781, -0.00571646122, 0.0753164589, 0.0851424038, 0.0344276242, -0.0110771693, -0.0674054474, 0.0238144211, 0.0722684339, 0.127525941, 0.0353774205, 0.0332326517, 0.0574975386, 0.132011339, -0.021666646, 0.0812211335, -0.0385468937, -0.0912349299, -0.0816484094, 0.0864037871, 0.169749379, 0.0938792005, -0.0426299907, 0.0495092198, 0.044266887, 0.0522757173, 0.0168170929, -0.0512816086, 0.0146380551, 0.0567030497, 0.0319734029, 0.0424369946, 0.0125781037, -0.0639688969, -0.0218270272, -0.00753120333, -0.094087109, 0.0415724069, -0.0458106026, -0.191868842, -0.0353733376, -0.0827914998, 0.0222649202, -0.0110880127, 0.0588395298, -0.00075106509, 0.00630116276, 0.0508419052, -0.0973529369, 0.00889941677, 0.0150931329, -0.0762014017, -0.00210261345, 0.0544563234, -0.0157391671, 0.0114466082, -0.0318201222, -0.00051691226, -0.0407840647, -0.00694661075, 0.137765795, 0.0271868668, 0.0586328693, -0.0419846252, 0.0305384435, 0.0598569289, -0.0171761531, 0.0587193891, 0.0230484381, 0.12882179, 0.0120551828, -0.168238074, 0.0669286475, 0.0403562225, 0.0549735874, 0.066484943, -0.0145690329, 0.0632467121, -0.0359894931, 0.0815353915, -0.0462696441, -0.0617114268, 0.0324998535, 0.104943894, 0.0243134871, 0.0348146185, 0.111343443, 0.0185335688, -0.126225591, 0.0969006494, 0.0387630202, -0.197859943, -0.00749284029, -0.102993302, 0.093429096, -0.130881503, -0.0969738141, 0.159489989, -0.0507350154, -0.0478643775, 0.0019461792, -0.0112797022, -0.112410203, -0.00914694369, -0.0477013178, -0.0175735839, -0.0404180251, -0.0811169967, -0.0171765462, 0.0963852555, 0.114861697, -0.0139015261, -0.100321144, -0.0470585749, -0.0460179895, -0.162901118, -0.0248801392, -0.0205437746, -0.0337562151, 0.0522041097, -0.0410371646, -0.0846687555, -0.0636999235, 0.200840011, 0.0945674181, 0.0910367817, 0.0748383999, -0.140553772, -0.0284785368, -0.0362542495, 0.107232265, -0.0338969082, -0.0610294044, 0.0289454386, 0.0942899287, 0.0331130847, -0.0296364836, -0.0157973766, -0.110053211, -0.0952294171, -0.0308468044, -0.0917455107, -0.012321448, -0.026099572, -0.0903289616, 0.149475008, -0.0356912613, -0.0336054303, -0.0462723821, 0.0410968587, 0.0664142892, -0.0442651771, 0.0419820622, -0.00955121219, -0.0328969583, -0.0133415833, 0.0805753767, -0.0440384522, -0.0572364479, -0.0806434304, -0.199577808, 0.230586052, -0.0350115635, -0.0919062197, -0.142132744, 0.168537289, -0.00562704355, -0.0955159962, 0.0648066252, -0.0613829941, -0.0894394368, -0.0347663015, -0.028064115, 0.0362613648, 0.0463579334, -0.0798790306, -0.0732574761, -0.0253687128, -0.0559770465, 0.0480587594, -0.0656372085, 0.0877685621, -0.0300214272, 0.0177654028, -0.0479325876, -0.04533384, 0.00566974469, -0.160316736, 0.0640275702, 0.0861340314, -0.0507358126, -0.0361745469, 0.0520602651, -0.0654230267, 0.05035422, 0.0391078517, -0.0605994686, -0.0294262469, -0.00314886123, 0.0941899493, -0.0902123451, -0.0473316908, 0.03309476, -0.00887358468, 0.0519970991, -0.0706470236, -0.0585814975, 0.0448119715, 0.0293908119, -0.0922531039, 0.0633407086, -0.164037898, -0.0344860554, 0.0450999252, -0.00827317126, 0.0797850564, 0.0878356174, -0.168259695, -0.111685902, 0.0194611624, -0.0502003171, 0.0400763042, -0.000246921554, 0.0347175598, -0.0578241013, 0.0705874041, -0.0547405779, 0.0456695706, -0.0114778504, 0.00666502118, -0.158520162, 0.0391363762, -0.103737898, -0.0202049147, -0.088732928, -0.0948789492, 0.0870066583, -0.0883992463, 0.0831747726, 0.0661358535, -0.00944175199, -0.194340572, 0.00321928412, 0.0783763677, 0.00112029398, 0.0339062437, -0.0166905355, -0.057094533, -0.0835953802, -0.0406135097, 0.0742160231, -0.044803407, -0.174876824, 0.112007923, 0.147358492, -0.0847913846, 0.0327977575, 0.0154416123, 0.0593767762, -0.00806243159, 0.0516847745, -0.0334345698, -0.00635620393, -0.0670741349, 0.139667913, 0.0469381735, -0.0539213493, -0.0244122203, -0.0659745857, 0.0283477679, -0.0295619257, 0.0378655344, 0.0485721529, -0.0206418131, -0.111100182, -0.0611830056, -0.0195047855, -0.000287644565, 0.0513734743, -0.0807389319, 0.0663611367, 0.0745266005, 0.0250715297, -0.074418515, -0.0920155793, 0.0298504829, -0.0113703683, 0.00965473056, 0.00187846646, -0.138389483, 0.083949022, 0.0813331231, 0.0412819758, -0.0259420518, -0.0780557394, 0.0112823695, 0.0292894877, -0.121571183, -0.171000004, -0.082161963, -0.0934179276, 0.032158263, -0.0429277867, 0.0859632492, 0.143906415, 0.0723193884, 0.1921767, 0.0211715698, -0.119239479, 0.00303502637, 0.0327959321, -0.0355542824, -0.0364986621, 0.014449208, 0.0821491703, -0.0108046737, -0.09774068, -0.0262510162, -0.0463821851, -0.025814116, -0.113182858, -0.0296528637, 0.141963795, 0.069177866, 0.011556413, 0.00709964149, 0.0644153059, -0.0336896852, 0.0873855054, -0.0798419714, -0.0273210257, -0.117931627, -0.0242039915, -0.0473055542, -0.049700819, 0.0279959533, 0.120111533, -0.0517931357, -0.0758071691, 0.0162475444, 0.0594417267, -0.165750802, -0.0595090389, 0.024117101, -0.00721539045, 0.02062824, -0.0610174797, -0.047291778, 0.0229518041, -0.0178083591, 0.0143660717, 0.107656598, 0.0646652132, 0.0129710324, -0.0765416026, -0.0067758821, 0.071242258, -0.0673705488, -0.196762294, -0.0317336246, 0.0874641016, -0.0363835618, -0.0167499296, 0.0126019027, 0.0590260327, -0.0619911924, 0.125976726, 0.0454879105, -0.0814923048, -0.160627574, 0.0401536077, 0.11946094, -0.00205735117, 0.0649667308, 0.119357049, -0.0163080599, -0.0327946432, -0.0541737825, 0.103204623, -0.0368971452, -0.00818765908, -0.0605907142, 0.0254717674, -0.0940710902, -0.190521747, -0.102423266, -0.0435902327, -0.0440872647, 0.0942212269, -0.00657942891, 0.00986169092, 0.0419842377, -0.0898573399, -0.13850674, 0.0310922042, 0.110772438, 0.128877789, -0.0391735509, -0.0354640856, -0.0221875757, -0.109102696, -0.131654769, -0.00299015827, -0.0143673187, -0.0724790767, -0.0387414917, -0.0553217307, -0.0794467032, 0.0357225388, -0.0577824861, 0.127521515, 0.030323673, -0.0575866997, 0.0470415689, -0.02680251, -0.13124375, 0.14153403, 0.0602536276, -0.0151671181, -0.0162680708, 0.0525177345, 0.0274184011, 0.0358750187, -0.119836435, 0.0613141358, 0.0407154448, -0.0118777975, -0.0230017081, -0.00926114991, -0.0414987132, -0.0842045993, -0.00167208165, -0.0925509632, 0.0421595834, 0.0608234778, -0.130276754, 0.0267832708, 0.100988097, 0.0781755894, -0.0390111469, 0.0901702121, -0.057276465, 0.0248767994, 0.172336698, -0.020048501, 0.0744086504, -0.0542870872, 0.0197537728, 0.0848038197, -0.0120387282, -0.0234180801, -0.0143575976, -0.0196826849, -0.0373380929, 0.0507742353, 0.0573016703, -0.105674788, -0.0482716076, 0.0154178804, 0.0567820966, 0.0546647832, -0.077160351, -0.0974433571, 0.0261986218, 0.0682947934, 0.142600715, -0.0821557045, -0.0264292788, 0.0293401107, -0.141429424, 0.0557237118, 0.00814896636, -0.0856773034, -0.0153672369, -0.0419892743, -0.0394244827, 0.0818297863, -0.0586152971, -0.0249222666, 0.0107620507, 0.0225159116, 0.0488754958, 0.0784658343, 0.158379465, -0.00325796939, 0.0975780785, -0.0909784883, -0.00240113959, 0.028311016, -0.0576878339, -0.107952863, 0.0455746762, 0.0782887936, -0.0428143069, -0.0966097116, 0.0105752349, 0.147920817, 0.0276091732, 0.0509470589, 0.0948298052, -0.115800686, -0.0791827589, -0.0415750258, -0.0642590597, 0.051787965, -0.0664690211, 0.135570541, 6.43308667e-05, -0.0391023755, -0.0508662984, 0.0224460736, 0.0564484969, 0.053764686, -0.107197657, -0.00115409866, 0.0311301108, 0.0211292151, -0.0459631011, 0.0348635539, -0.0117480159, -0.0270452388, -0.00449803099, 0.109037757, 0.155846879, -0.0825168863, 0.122937411, 0.0165575948, 0.0443798937, 0.0524557307, 0.0123378197, 0.230386585, 0.00925843418, -0.147435188, 0.0187123716, 0.0921274424, 0.0463036858, 0.0319886357, 0.00493047945, -0.0185778253, 0.0484505594, 0.134464771, -0.0519553833, -0.0243367665, 0.106514797, 0.0361147523, 0.0137277758, 0.00527644157, 0.0497434065, -0.00503639504, -0.0432905667, 0.0993102491, 0.136526898, -0.0145881996, 0.130319893, -0.132631332, -0.066883117, 0.0614537522, -0.146018207, -0.0854729265, -0.0106974319, -0.0684075132, 0.000379471108, -0.0152550749, 0.0307253655, -0.0415801778, 0.0565482304, 0.0613053888, 0.0351135246, -0.00204717368, -0.0194362011, 0.119199343, -0.10788542, -0.121140428, -0.0756799057, 0.0656082779, 0.0473917872, 0.110425636, -0.10782776, 0.0833447948, 0.0206291992, -0.0329098925, 0.105064832, -0.027444927, 0.00177714229, 0.0579485819, 0.0476972051, 0.0915832892, -0.0460004956, -0.0286061596, -0.0868751183, -0.00388204306, -0.122030437, 0.0168477185, 0.0854151845, 0.0344677158, -0.109319732, -0.0454696715, -0.0337420478, 0.0016348036, 0.116318591, 0.091471374, -0.0618529841, 0.00717924815, 0.0219491664, 0.027185725, -0.0214611832, 0.00936102122, -0.0100392811, -0.122589931, 0.0584963523, -0.0140657034, -0.0762873739, 0.0760588795, 0.0238103811, -0.0771279335, -0.0201385953, 0.0819055736, 0.0235249512, -0.0114337914, 0.0701106191, 0.0395762213, 0.0140983667, 0.0242828913, 0.0286869016, 0.0211825147, -0.0424613357, 0.0431166589, -0.097460188, -0.00259585679, 0.0190237854, 0.0898538753, -0.0310720168, 0.0507076494, -0.0149203688, -0.0873094648, 0.0690678656, -0.0789354071, -0.0375652462, 0.013849549, 0.0499016792, 0.0156347491, 0.0342558399, 0.0526852161, 0.115731694, 0.113165185, -0.0557963699, 0.0368037485, 0.0216162018, 0.214696974, 0.000794485211, -0.0406426713, -0.0198553521, 0.0373584591, -0.0704259425, 0.029388763, 0.082738027, -0.0326178819, 0.09166722, -0.0369430296, 0.00916040316, -0.0170614962, 0.0870813802, -0.0095146168, -0.065076001, -0.102999263, -0.045840688, 0.0162314083, -0.0649379268, 0.0297924839, -0.0204978622, -0.0241616368, 0.0600432009, 0.159195215, 0.143640861, 0.0745456144, 0.0539212152, 0.00271478156, -0.0936590433, 0.0323141217, 0.0196025074, -0.000803589821, 0.0519903377, -0.120891005, 0.0062912032, 0.0357041061, 0.0307115577, 0.0233878214, 0.0397786349, -0.0911078379, 0.00382280257, 0.0125010032, -0.0251113549, 0.0125831477, 0.0556067452, 0.0666292682, 0.0994372368, 0.0410823897, 0.0671635717, -0.0785583779, 0.0100541897, -0.0105275586, 0.100008905, 0.00607637689, 0.119727626, 0.06037727, -0.0570261627, -0.0179527644, 0.0237348266, 0.0198590662, 0.097318396, -0.0709325224, -0.150020763, -0.0541847646, -0.00585578289, 0.00333797373, -0.028236445, -0.00830273796, 0.0893258899, 0.136049345, 0.0833097324, 0.00150818564, 0.0841375962, 0.044127617, 0.0420588702, 0.0320436023, 0.0824125558, -0.0333235189, -0.0897977799, 0.0601325929, -0.0908033848, -0.0204037391, -0.103487767, 0.084499523, 0.0478009656, -0.0516456328, 0.0319618322, -0.0162731893, -0.0307973847, -0.0242388286, -0.0598752722, 0.0676786974, -0.0532381423, 0.0455306582, -0.0513714179, -0.0223139729, -0.0721026957, -0.0332549997, 0.0154482415, 0.00276384782, -0.00769143552, -0.135057539, 0.0194987282, -0.0791820884, 0.027593242, 0.0468132161, 0.0648820028, 0.141864702, 0.0540276431, -0.0930785388, -0.0342094153, -0.0712071806, 0.0516552515, -0.0519339666, 0.141384766, -0.115820587, -0.0578783303, 0.0993592069, -0.0826922432, -0.0402599946, 0.0600859299, 0.052808255, 0.062896654, -0.0991227105, -0.0308523662, 0.0058810655, 0.0195116568, -0.176231444, -0.0120743476, 0.0466277748, -0.00479177758, 0.132687926, 0.0372997411, -0.0698493868, -0.114647776, 0.0988531783, -0.00462367944, 0.0126146749, 0.0215533301, -0.0302089714, 0.111634687, 0.0171016511, 0.0716648474, 0.0292715598, -0.0343657285, 0.0722840428, 0.00431878865, 0.169528246, -0.0553757697, 0.0625901446, 0.129925251, 0.0075961519, 0.0814568102, -0.000654119998, -0.0866291448, 0.122778445, 0.0197446793, -0.0894370601, -0.0221604332, -0.0719681457, -0.000667473301, 0.0250691995, 0.0285977963, -0.0907365084, 0.07515008, -0.165994599, 0.168218225, -0.137749895, 0.106884032, -0.129251719, 0.0266259871, 0.0769484565, -0.0372937955, 0.0479861833, -0.0484450944, 0.0363472104, -0.0782243684, -0.0511998497, -0.013238335, -0.0329197496, 0.0104758553, -0.0709497258, 0.0391665697, -0.127216831, -0.0404612347, -0.0867774114, -0.046600692, 0.00418355316, -0.0633166507, -0.0414735936, 0.0236057006, -0.0258368962, 0.0678422004, 0.112647943, -0.0324306339, -0.00988782942, 0.0839368254, 0.0120457122, -0.0703958571, -0.0518545657, -0.0366280451, -0.0344718434, -0.0195410885, 0.140279353, 0.0287122019, 0.034899421, -0.0190885291, -0.0903406516, 0.0937678069, 0.0595882423, 0.0444250442, 0.02489971, -0.0289831776, 0.0477713309, 0.160236746, -0.0507163815, -0.02798298, 0.0835297853, -0.145065278, 0.110856101, -0.0219675228, -0.09635894, 0.139262006, -0.0428989083, 0.006609309, -0.0212683361, -0.0233980827, 0.00470141508, 0.0974960998, 0.104721539, 0.0269472525, 0.0124460198, -0.0666405708, 0.00455601886, 0.0233568326, -0.140762657, 0.0594203956, 0.00405210583, -0.180983603, 0.0104133934, 0.00331818778, -0.0334692076, 0.0713636801, 0.0462374873, 0.0826871693, 0.0863402188, 0.134145707, -0.0676784068, 0.0348382145, -0.0834512562, 0.0684894025, 0.0506787188, -0.0485029928, 0.0136228791, 0.164052099, 0.0657436177, -0.000161466189, 0.00585474214, -0.00230954075, -0.0957160294, 0.0718223453, 0.0585715473, -0.0631539151, 0.0948207974, -0.0422124118, -0.0262737256, -0.0412255339, 0.0186428111, -0.13579911, -0.183053255, 0.00305974856, -0.024856139, -0.0873593986, 0.100135244, -0.0249364562, -0.0182432774, -0.0374694169, 0.112602696, 0.0115270391, 0.00774586573, 0.00832534954, -0.0187189281, -0.0247038193, -0.072468698, -0.0127941612, 0.0929326862, 0.0153889861, 0.0401442125, -0.105329812, -0.041904889, 0.0746989921, -0.0426267236, 0.096574001, 0.0588563308, -0.0723425001, 0.0519671626, -0.110282645, 0.023782514, -0.0220482349, 0.0455567315, 0.00126918801, 0.0148957735, -0.0828897879, 0.0330617018, -0.0603466406, -0.0312512703, 0.158161759, -0.064591296, -0.0302896984, -0.0546595864, 0.041126214, -0.0834092349, -0.0379186906, 0.159711421, -0.080117397, -0.0189905092, -0.0189962052, 0.0377800204, 0.0824783742, 0.0999648273, -0.030885186, 0.0940911844, -0.0122155016, -0.0698266551, -0.0508394614, 0.0794238448, 0.0523062013, -0.0470671318, 0.0817164108, 0.0626662672, 0.0733318478, 0.104500718, 0.0606436543, -0.0396260135, 0.0492423661, 0.0252361633, -0.053880997, -0.0710671544, -0.034930598, 0.0249724053, 0.039634496, 0.00128793344, -0.0316855088, -0.0832425132, 0.128735602, -0.107892126, 0.189235479, 0.114530109, -0.0733102486, 0.0611379035, -0.0727086216, -0.00784323364, 0.0649280772, 0.078512989, -0.0140992254, 0.0500521399, 0.0546547771, 0.032995224, -0.0924386531, 0.0342714824, -0.0288704298, -0.0537729412, 0.0160043482, -0.0571973547, -0.0930881575, -0.0060783294, 0.00658744713, -0.00991571881, 0.0334253199, -0.0391148813, -0.0716266036, 0.0784005821, 0.100003406, -0.049674537, -0.136607498, 0.0599353202, 0.00876861438, 0.123580955, 0.11543794, 0.027512813, 0.0601726808, 0.0825635195, 0.0102091115, -0.0660458058, 0.0296149608, 0.00901784003, 0.140400052, -0.140364692, -0.0125178769, 0.0600770488, 0.0589169003, 0.0683401376, 0.0202003792, -0.0620686933, -0.112169608, 0.0258502401, 0.112197705, 0.0135365054, 0.0189605858, -0.086132735, -0.169402003, 0.0953313708, 0.00955498405, -0.0141711263, 0.0974058509, -0.0825876519, 0.0700342059, 0.0554787591, 0.0475979745, 0.113273486, 0.0469833612, -0.095944792, -0.00116587523, 0.107693441, -0.0434525535, 0.0535380021, 0.00395460706, -0.0444919243, 0.109183334, 0.147456348, 0.0826073885, 0.134649783, -0.0860900283, -0.0745515525, 0.0465153717, -0.122678399, 0.0569026023, -0.0684145316, -0.0305911433, -0.0619250238, -0.0482132137, -0.0189730283, -0.0551335625, -0.116009459, 0.02166228, -0.0904422402, -0.0962748304, 0.0397973061, 0.0565618835, -0.0541109219, 0.00912805088, 0.00842884742, -0.00535425078, -0.0266479701, -0.0859368294, 0.0233013704, 0.042687472, -0.018398555, -0.0481752902, 0.0822771192, -0.022317227, -0.118334077, 0.095822528, 0.139224648, 0.0195650458, 0.0683586597, 0.0631345958, -0.0373875722, 0.00341564603, 0.107133001, -0.0751987696, 0.00454649981, -0.0362539589, 0.026337428, -0.0179972276, 6.35553151e-05, -0.0705527738, 0.0230018832, 0.0606943443, -0.038967438, -0.0266847778, 0.0172603615, 0.0308038648, 0.022909835, -0.0310519468, 0.0154562201, 0.0787664652, -0.121662647, -0.0801561549, -0.00359021639, -0.0524999462, -0.00503655523, -0.0436337888, -0.0619397163, 0.0351424366, 0.0792855993, -0.0914481431, 0.054709658, 0.0170378536, 0.0350544453, -0.0636989996, 0.0668064356, 0.0525544137, 0.0519481078, 0.0748329982, -0.0683197007, -0.110261567, -0.0808580518, 0.0433228835, 0.0686655864, 0.0811156705, 0.156877279, 0.0324891731, 0.025431687, 0.102199338, 0.0574450791, 0.141714647, 0.111159399, 0.0125291236, -0.0447607189, 0.130543992, -0.0637754649, -0.0112033971, 0.0106440624, -0.0678310171, 0.0161886699, 0.033586964, -0.0785687715, -0.000732215121, -0.100033045, -0.00619979948, 0.0352816507, 0.00844343752, -0.0454045013, -0.101458229, -0.119886011, -0.0570310503, 0.00495114177, 0.0789650828, -0.0153123513, 0.07088162, 0.00860105455, -0.0862798318, -0.0800941512, 0.0199356303, 0.0428098105, 0.0869083628, 0.0312335305, -0.0582196042, 0.110067889, 0.0443210714, 0.0505822003, -0.0973165855, -0.0469971225, -0.0390720591, 0.151471704, 0.127615348, -0.105041966, -0.164652064, 0.0131918658, 0.029172156, 0.00465614349, -0.0354489461, 0.0173196532, 0.0124960765, -0.200602576, 0.00305063999, -0.011325432, -0.0427099168, -0.0469666794, -0.0288568828, -0.0726884678, -0.00320445118, -0.020172514, 0.0339836776, -0.0170585364, -0.0856021419, 0.000350127928, -0.00189465168, 0.0373253897, -0.0414954796, 0.073211439, -0.0566916279, -0.012231566, 0.0222783666, 0.0329278037, -0.115158595, -0.138853624, -0.0693328455, -0.0101504438, 0.0382712074, -0.00926143676, 0.0709851384, 0.0712291747, 0.0422781147, 0.053045772, 0.054939948, 0.0537798926, 0.0823203847, -0.0454094484, 0.124955572, 0.0222275015, -0.0329840928, -0.097050406, -0.0406842232, -0.0315937251, -0.0451682471, 0.0331139192, -0.111749321, 0.0606486052, -0.076717943, 0.0591437481, 0.0165941566, -0.158840597, -0.00306601822, 0.0333832949, -0.0355267599, 0.111018218, -0.0104070455, 0.0489391163, -0.00862740353, -0.0600290075, -0.0773975477, -0.0431323797, 0.0192667395, 0.105983481, 0.0561273359, -0.091204077, -0.114225745, 0.103793919, 0.012235254, -0.115128316, -0.0581305996, 0.0234019887, 0.0715955943, -0.0840854943, -0.102567874, -0.0818333924, 0.0280918758, -0.0301763713, 0.0228692051, -0.0594820604, 0.0897795111, 0.106658682, 0.0206690338, 0.0726500899, -0.000891397242, 0.0139189754, -0.054154858, -0.0630462244, -0.108763322, 0.126787513, 0.00294042518, 0.0292959437, -0.0553980321, 0.0807077736, -0.0965617076, -0.0890631229, 0.0466582552, -0.00911538024, 0.156839207, -0.0626729354, -0.0245680921, -0.00179294869, -0.056965515, -0.0199423786, -0.115498662, 0.0221503396, 0.0872155279, 0.119776607, 0.0166656077, -0.0399951339, -0.0429340228, -0.0653482974, -0.033989653, -0.0458589531, -0.0407891795, -0.0253337026, -0.0725796819, -0.0302919783, 0.00206887163, -0.100360379, -0.071315363, -0.017575983, 0.0177510977, 0.0351644121, 0.0383973196, -0.0745397806, -0.0709501654, 0.195765108, -0.0271085314, 0.0249852221, -0.0700546056, 0.184820786, 0.158069536, -0.0409562513, -0.0287105516, -0.0858581439, 0.0129066352, -0.030616425, -0.0372961275, 0.0750120357, -0.00228865957, 0.000365508662, -0.0622223467, 0.102390289, 0.0501865447, -0.0586910993, -0.0958363265, 0.0167813376, -0.0460788198, 0.0475374013, 0.073757261, 0.0686880201, -0.016310079, -0.0307487864, 0.012816906, -0.0567861497, 0.117383681, 0.0600756668, -0.0127716083, -0.0240453258, -0.0374855399, -0.032605987, 0.0901284069, -0.133627295, 0.0372318402, 0.180233389, -0.042641554, -0.0745786205, 0.102745302, 0.0446086749, 0.141644612, 0.0281131864, -0.0547536165, -0.0813148469, -0.0966759175, 0.0440410338, 0.0347155966, -0.0452661924, 0.00467441976, 0.143894181, 0.0984901041, 0.000415101647, -0.0614643805, 0.00953144394, 0.0880256295, 0.0648551509, 0.0617447086, 0.152493358, -0.0478570797, 0.104216434, 0.0910557956, -0.065354012, 0.0716719031, 0.0858117864, -0.0790668055, 0.100356698, 0.125176936, 0.00570722762, 0.0199908521, -0.0199188571, 0.0151966773, -0.0859806389, 0.0459887758, 0.229563281, -0.055340413, 0.0785515308, -0.0705481991, -0.0218721218, -0.0860364884, 0.0521545634, -0.0791168362, 0.092071332, 0.0687095225, -0.0352584347, 0.0084028868, -0.0515908487, 0.067410484, -0.0238079429, 0.0491214432, 0.0763769448, 0.0616733208, -0.10592977, 0.0577273741, 0.0236162581, 0.0179329254, -0.0668587163, -0.000917315483, 0.100958973, -0.136879578, 0.0519942529, 0.0552516207, -0.117933288, -0.0284534171, 0.0147698354, 0.0290891677, -0.0483859926, -0.00171393529, 0.0671777129, 0.0262195617, 0.0175